(* IEC 61131-3 sources: PLC_FIFO_Optimization/build/OpenPLC Runtime v4/src, 1 file *)

(* ---- program.st ---- *)
FUNCTION_BLOCK Circular_queue
  VAR_INPUT
    XPush : BOOL;
    XPop : BOOL;
    iInputVal : INT;
  END_VAR
  VAR_OUTPUT
    iOutputVal : INT;
    iCount : INT;
    Operation_Cost : INT;
  END_VAR
  VAR
    Buffer : ARRAY [0..4999] OF INT;
    Head : INT;
    Tail : INT;
    MaxLen : INT;
    R_Trig_Push : R_TRIG;
    R_Trig_Pop : R_TRIG;
  END_VAR

  (* Edge Detection *)
  R_Trig_Push(CLK := xPush);
  R_Trig_Pop(CLK := xPop);

  (* initialize MaxLen if 0 (safety check) *)
  MaxLen := 5000;

  (* --- PUSH (Enqueue) --- *)
  IF R_Trig_Push.Q THEN
      (* Only push if not full (Optional safety, but good practice) *)
      IF iCount < MaxLen THEN
          Buffer[Head] := iInputVal;
          Head := Head + 1;
          IF Head >= MaxLen THEN Head := 0; END_IF;

          (* DIRECT COUNTING - The Fix *)
          iCount := iCount + 1;
      END_IF;
  END_IF;

  (* --- POP (Dequeue) --- *)
  IF R_Trig_Pop.Q AND iCount > 0 THEN
      iOutputVal := Buffer[Tail];
      Tail := Tail + 1;
      IF Tail >= MaxLen THEN Tail := 0; END_IF;

      (* DIRECT COUNTING - The Fix *)
      iCount := iCount - 1;
      Operation_Cost := 0;
  END_IF;
END_FUNCTION_BLOCK

FUNCTION_BLOCK FB_FIFO
  VAR_INPUT
    XPush : BOOL;
    XPop : BOOL;
    iInputVal : INT;
  END_VAR
  VAR_OUTPUT
    iOutputVal : INT;
    iCount : INT;
    Operation_Cost : INT;
  END_VAR
  VAR
    Buffer : ARRAY [0..4999] OF INT;
    i : INT;
    R_Trig_Push : R_TRIG;
    R_Trig_Pop : R_TRIG;
  END_VAR

  (* Edge Detection *)
  R_Trig_Push(CLK := xPush);
  R_Trig_Pop(CLK := xPop);

  (* --- PUSH (FFL) --- *)
  (* Simply add to the end. This part is actually fast (O(1)) *)
  IF R_Trig_Push.Q AND iCount < 5000 THEN
      Buffer[iCount] := iInputVal;
      iCount := iCount + 1;
  END_IF;

  (* --- POP (FFU) - THE EXPENSIVE PART --- *)
  (* This simulates the AB FFU shifting mechanism *)
  IF R_Trig_Pop.Q AND iCount > 0 THEN

      (* 1. Grab the value at Head (Index 0) *)
      iOutputVal := Buffer[0];

      (* 2. THE SHIFT LOOP (The "Bad" Part) *)
      (* We must physically move every item down one slot *)
      (* If you have 50 items, this loop runs 49 times! *)

      FOR i := 0 TO iCount - 2 DO
          Buffer[i] := Buffer[i+1]; (* Move data from i+1 to i *)

          (* Increment the "Cost" Counter to visualize the inefficiency *)
          Operation_Cost := Operation_Cost + 1;
      END_FOR;

      (* 3. Clear the last slot (optional, but clean) *)
      Buffer[iCount - 1] := 0;

      (* 4. Decrement Count *)
      iCount := iCount - 1;

  END_IF;
END_FUNCTION_BLOCK

PROGRAM main
  VAR
    My_Bad_FIFO : FB_FIFO;
    My_Good_FIFO : CIRCULAR_QUEUE;
    pb_Push : BOOL;
    pb_Pop : BOOL;
    Input_Data : INT;
    Auto_TImer : TON;
    Test_Step : INT := 0;
    Auto_Start : BOOL := FALSE;
    Fill_Queue_Now : BOOL := FALSE;
    i : INT := 0;
    Queue_Count_Good : INT := 0;
  END_VAR
  VAR
    Output_Bad AT %QW1 : INT;
    Output_Good AT %QW4 : INT;
    Test_value AT %QW5 : INT;
    Queue_Count AT %QW0 : INT;
    Shift_Counter AT %QW3 : INT;
    Shift_Counter_Good AT %QW2 : INT;
  END_VAR

  (* ============================================================= *)
  (* ZONE 1: THE STRESS TEST LOADER (Instant Fill) *)
  (* ============================================================= *)
  (* This logic only runs ONCE when you force 'Fill_Queue_Now' to TRUE. *)
  (* It pauses the scan cycle, stuffs 5,000 items into the queues, *)
  (* and then releases the PLC back to normal operation. *)

  IF Fill_Queue_Now THEN

      (* Loop from 1 to 5000 to fill the array completely *)
      FOR i := 1 TO 5000 DO

          (* 1. SIMULATE RISING EDGE (Push Button Press) *)
          (* We call the FBs directly here to force the data in *)
          My_Bad_FIFO(xPush := TRUE, xPop := FALSE, iInputVal := i);
          My_Good_FIFO(xPush := TRUE, xPop := FALSE, iInputVal := i);

          (* 2. SIMULATE FALLING EDGE (Push Button Release) *)
          (* We must call them again with FALSE to reset the trigger for the next loop iteration *)
          My_Bad_FIFO(xPush := FALSE, xPop := FALSE, iInputVal := i);
          My_Good_FIFO(xPush := FALSE, xPop := FALSE, iInputVal := i);

      END_FOR;

      (* Reset the trigger so it doesn't run forever *)
      Fill_Queue_Now := FALSE;

  END_IF;

  (* ============================================================= *)
  (* ZONE 2: NORMAL OPERATION (Manual Pop) *)
  (* ============================================================= *)
  (* This runs every single scan cycle. It listens to your manual *)
  (* 'pb_Pop' button so you can trigger the unloads when ready. *)

  (* Call the Bad FIFO (Linear Shift) *)
  My_Bad_FIFO(
      xPush := pb_Push,      (* Normal button control *)
      xPop := pb_Pop,        (* Normal button control *)
      iInputVal := Input_Data,
      iOutputVal => Output_Bad,
      iCount => Queue_Count,
      Operation_Cost => Shift_Counter
  );

  (* Call the Good FIFO (Circular Buffer) *)
  My_Good_FIFO(
      xPush := pb_Push,
      xPop := pb_Pop,
      iInputVal := Input_Data,
      iOutputVal => Output_Good,
      iCount => Queue_Count_Good,
      Operation_Cost => Shift_Counter_Good
  );
END_PROGRAM

CONFIGURATION Config0

  RESOURCE Res0 ON PLC
    TASK task0(INTERVAL := T#20ms,PRIORITY := 1);
    PROGRAM instance0 WITH task0 : main;
  END_RESOURCE
END_CONFIGURATION

(*DBG:char md5[] = "892a26d77c3caac8eb1d182cbc9cad2f";*)
(*DBG:/**)
(*DBG: * This file is part of OpenPLC Runtime*)
(*DBG: **)
(*DBG: * Copyright (C) 2023 Autonomy, GP Orcullo*)
(*DBG: * Based on the work by GP Orcullo on Beremiz for uC*)
(*DBG: **)
(*DBG: * This program is free software; you can redistribute it and/or*)
(*DBG: * modify it under the terms of the GNU General Public License*)
(*DBG: * as published by the Free Software Foundation; either version 2*)
(*DBG: * of the License, or (at your option) any later version.*)
(*DBG: **)
(*DBG: * This program is distributed in the hope that it will be useful,*)
(*DBG: * but WITHOUT ANY WARRANTY; without even the implied warranty of*)
(*DBG: * MERCHANTABILITY or FITNESS FOR A PARTICULAR PURPOSE.  See the*)
(*DBG: * GNU General Public License for more details.*)
(*DBG: **)
(*DBG: * You should have received a copy of the GNU General Public License*)
(*DBG: * along with this program; If not, see <http://www.gnu.org/licenses/>.*)
(*DBG: **)
(*DBG: */*)
(*DBG:*)
(*DBG:#include <stdbool.h>*)
(*DBG:*)
(*DBG:#include "iec_types_all.h"*)
(*DBG:#include "POUS.h"*)
(*DBG:*)
(*DBG:#define SAME_ENDIANNESS      0*)
(*DBG:#define REVERSE_ENDIANNESS   1*)
(*DBG:*)
(*DBG:char plc_program_md5[] = "892a26d77c3caac8eb1d182cbc9cad2f";*)
(*DBG:*)
(*DBG:uint8_t endianness;*)
(*DBG:*)
(*DBG:*)
(*DBG:extern MAIN RES0__INSTANCE0;*)
(*DBG:*)
(*DBG:static const struct {*)
(*DBG:    void *ptr;*)
(*DBG:    __IEC_types_enum type;*)
(*DBG:} debug_vars[] = {*)
(*DBG:    {&(RES0__INSTANCE0.MY_BAD_FIFO.EN), BOOL_ENUM},*)
(*DBG:    {&(RES0__INSTANCE0.MY_BAD_FIFO.ENO), BOOL_ENUM},*)
(*DBG:    {&(RES0__INSTANCE0.MY_BAD_FIFO.XPUSH), BOOL_ENUM},*)
(*DBG:    {&(RES0__INSTANCE0.MY_BAD_FIFO.XPOP), BOOL_ENUM},*)
(*DBG:    {&(RES0__INSTANCE0.MY_BAD_FIFO.IINPUTVAL), INT_ENUM},*)
(*DBG:    {&(RES0__INSTANCE0.MY_BAD_FIFO.IOUTPUTVAL), INT_ENUM},*)
(*DBG:    {&(RES0__INSTANCE0.MY_BAD_FIFO.ICOUNT), INT_ENUM},*)
(*DBG:    {&(RES0__INSTANCE0.MY_BAD_FIFO.OPERATION_COST), INT_ENUM},*)
(*DBG:    {&(RES0__INSTANCE0.MY_BAD_FIFO.BUFFER.value.table[0]), INT_ENUM},*)
(*DBG:    {&(RES0__INSTANCE0.MY_BAD_FIFO.BUFFER.value.table[1]), INT_ENUM},*)
(*DBG:    {&(RES0__INSTANCE0.MY_BAD_FIFO.BUFFER.value.table[2]), INT_ENUM},*)
(*DBG:    {&(RES0__INSTANCE0.MY_BAD_FIFO.BUFFER.value.table[3]), INT_ENUM},*)
(*DBG:    {&(RES0__INSTANCE0.MY_BAD_FIFO.BUFFER.value.table[4]), INT_ENUM},*)
(*DBG:    {&(RES0__INSTANCE0.MY_BAD_FIFO.BUFFER.value.table[5]), INT_ENUM},*)
(*DBG:    {&(RES0__INSTANCE0.MY_BAD_FIFO.BUFFER.value.table[6]), INT_ENUM},*)
(*DBG:    {&(RES0__INSTANCE0.MY_BAD_FIFO.BUFFER.value.table[7]), INT_ENUM},*)
(*DBG:    {&(RES0__INSTANCE0.MY_BAD_FIFO.BUFFER.value.table[8]), INT_ENUM},*)
(*DBG:    {&(RES0__INSTANCE0.MY_BAD_FIFO.BUFFER.value.table[9]), INT_ENUM},*)
(*DBG:    {&(RES0__INSTANCE0.MY_BAD_FIFO.BUFFER.value.table[10]), INT_ENUM},*)
(*DBG:    {&(RES0__INSTANCE0.MY_BAD_FIFO.BUFFER.value.table[11]), INT_ENUM},*)
(*DBG:    {&(RES0__INSTANCE0.MY_BAD_FIFO.BUFFER.value.table[12]), INT_ENUM},*)
(*DBG:    {&(RES0__INSTANCE0.MY_BAD_FIFO.BUFFER.value.table[13]), INT_ENUM},*)
(*DBG:    {&(RES0__INSTANCE0.MY_BAD_FIFO.BUFFER.value.table[14]), INT_ENUM},*)
(*DBG:    {&(RES0__INSTANCE0.MY_BAD_FIFO.BUFFER.value.table[15]), INT_ENUM},*)
(*DBG:    {&(RES0__INSTANCE0.MY_BAD_FIFO.BUFFER.value.table[16]), INT_ENUM},*)
(*DBG:    {&(RES0__INSTANCE0.MY_BAD_FIFO.BUFFER.value.table[17]), INT_ENUM},*)
(*DBG:    {&(RES0__INSTANCE0.MY_BAD_FIFO.BUFFER.value.table[18]), INT_ENUM},*)
(*DBG:    {&(RES0__INSTANCE0.MY_BAD_FIFO.BUFFER.value.table[19]), INT_ENUM},*)
(*DBG:    {&(RES0__INSTANCE0.MY_BAD_FIFO.BUFFER.value.table[20]), INT_ENUM},*)
(*DBG:    {&(RES0__INSTANCE0.MY_BAD_FIFO.BUFFER.value.table[21]), INT_ENUM},*)
(*DBG:    {&(RES0__INSTANCE0.MY_BAD_FIFO.BUFFER.value.table[22]), INT_ENUM},*)
(*DBG:    {&(RES0__INSTANCE0.MY_BAD_FIFO.BUFFER.value.table[23]), INT_ENUM},*)
(*DBG:    {&(RES0__INSTANCE0.MY_BAD_FIFO.BUFFER.value.table[24]), INT_ENUM},*)
(*DBG:    {&(RES0__INSTANCE0.MY_BAD_FIFO.BUFFER.value.table[25]), INT_ENUM},*)
(*DBG:    {&(RES0__INSTANCE0.MY_BAD_FIFO.BUFFER.value.table[26]), INT_ENUM},*)
(*DBG:    {&(RES0__INSTANCE0.MY_BAD_FIFO.BUFFER.value.table[27]), INT_ENUM},*)
(*DBG:    {&(RES0__INSTANCE0.MY_BAD_FIFO.BUFFER.value.table[28]), INT_ENUM},*)
(*DBG:    {&(RES0__INSTANCE0.MY_BAD_FIFO.BUFFER.value.table[29]), INT_ENUM},*)
(*DBG:    {&(RES0__INSTANCE0.MY_BAD_FIFO.BUFFER.value.table[30]), INT_ENUM},*)
(*DBG:    {&(RES0__INSTANCE0.MY_BAD_FIFO.BUFFER.value.table[31]), INT_ENUM},*)
(*DBG:    {&(RES0__INSTANCE0.MY_BAD_FIFO.BUFFER.value.table[32]), INT_ENUM},*)
(*DBG:    {&(RES0__INSTANCE0.MY_BAD_FIFO.BUFFER.value.table[33]), INT_ENUM},*)
(*DBG:    {&(RES0__INSTANCE0.MY_BAD_FIFO.BUFFER.value.table[34]), INT_ENUM},*)
(*DBG:    {&(RES0__INSTANCE0.MY_BAD_FIFO.BUFFER.value.table[35]), INT_ENUM},*)
(*DBG:    {&(RES0__INSTANCE0.MY_BAD_FIFO.BUFFER.value.table[36]), INT_ENUM},*)
(*DBG:    {&(RES0__INSTANCE0.MY_BAD_FIFO.BUFFER.value.table[37]), INT_ENUM},*)
(*DBG:    {&(RES0__INSTANCE0.MY_BAD_FIFO.BUFFER.value.table[38]), INT_ENUM},*)
(*DBG:    {&(RES0__INSTANCE0.MY_BAD_FIFO.BUFFER.value.table[39]), INT_ENUM},*)
(*DBG:    {&(RES0__INSTANCE0.MY_BAD_FIFO.BUFFER.value.table[40]), INT_ENUM},*)
(*DBG:    {&(RES0__INSTANCE0.MY_BAD_FIFO.BUFFER.value.table[41]), INT_ENUM},*)
(*DBG:    {&(RES0__INSTANCE0.MY_BAD_FIFO.BUFFER.value.table[42]), INT_ENUM},*)
(*DBG:    {&(RES0__INSTANCE0.MY_BAD_FIFO.BUFFER.value.table[43]), INT_ENUM},*)
(*DBG:    {&(RES0__INSTANCE0.MY_BAD_FIFO.BUFFER.value.table[44]), INT_ENUM},*)
(*DBG:    {&(RES0__INSTANCE0.MY_BAD_FIFO.BUFFER.value.table[45]), INT_ENUM},*)
(*DBG:    {&(RES0__INSTANCE0.MY_BAD_FIFO.BUFFER.value.table[46]), INT_ENUM},*)
(*DBG:    {&(RES0__INSTANCE0.MY_BAD_FIFO.BUFFER.value.table[47]), INT_ENUM},*)
(*DBG:    {&(RES0__INSTANCE0.MY_BAD_FIFO.BUFFER.value.table[48]), INT_ENUM},*)
(*DBG:    {&(RES0__INSTANCE0.MY_BAD_FIFO.BUFFER.value.table[49]), INT_ENUM},*)
(*DBG:    {&(RES0__INSTANCE0.MY_BAD_FIFO.BUFFER.value.table[50]), INT_ENUM},*)
(*DBG:    {&(RES0__INSTANCE0.MY_BAD_FIFO.BUFFER.value.table[51]), INT_ENUM},*)
(*DBG:    {&(RES0__INSTANCE0.MY_BAD_FIFO.BUFFER.value.table[52]), INT_ENUM},*)
(*DBG:    {&(RES0__INSTANCE0.MY_BAD_FIFO.BUFFER.value.table[53]), INT_ENUM},*)
(*DBG:    {&(RES0__INSTANCE0.MY_BAD_FIFO.BUFFER.value.table[54]), INT_ENUM},*)
(*DBG:    {&(RES0__INSTANCE0.MY_BAD_FIFO.BUFFER.value.table[55]), INT_ENUM},*)
(*DBG:    {&(RES0__INSTANCE0.MY_BAD_FIFO.BUFFER.value.table[56]), INT_ENUM},*)
(*DBG:    {&(RES0__INSTANCE0.MY_BAD_FIFO.BUFFER.value.table[57]), INT_ENUM},*)
(*DBG:    {&(RES0__INSTANCE0.MY_BAD_FIFO.BUFFER.value.table[58]), INT_ENUM},*)
(*DBG:    {&(RES0__INSTANCE0.MY_BAD_FIFO.BUFFER.value.table[59]), INT_ENUM},*)
(*DBG:    {&(RES0__INSTANCE0.MY_BAD_FIFO.BUFFER.value.table[60]), INT_ENUM},*)
(*DBG:    {&(RES0__INSTANCE0.MY_BAD_FIFO.BUFFER.value.table[61]), INT_ENUM},*)
(*DBG:    {&(RES0__INSTANCE0.MY_BAD_FIFO.BUFFER.value.table[62]), INT_ENUM},*)
(*DBG:    {&(RES0__INSTANCE0.MY_BAD_FIFO.BUFFER.value.table[63]), INT_ENUM},*)
(*DBG:    {&(RES0__INSTANCE0.MY_BAD_FIFO.BUFFER.value.table[64]), INT_ENUM},*)
(*DBG:    {&(RES0__INSTANCE0.MY_BAD_FIFO.BUFFER.value.table[65]), INT_ENUM},*)
(*DBG:    {&(RES0__INSTANCE0.MY_BAD_FIFO.BUFFER.value.table[66]), INT_ENUM},*)
(*DBG:    {&(RES0__INSTANCE0.MY_BAD_FIFO.BUFFER.value.table[67]), INT_ENUM},*)
(*DBG:    {&(RES0__INSTANCE0.MY_BAD_FIFO.BUFFER.value.table[68]), INT_ENUM},*)
(*DBG:    {&(RES0__INSTANCE0.MY_BAD_FIFO.BUFFER.value.table[69]), INT_ENUM},*)
(*DBG:    {&(RES0__INSTANCE0.MY_BAD_FIFO.BUFFER.value.table[70]), INT_ENUM},*)
(*DBG:    {&(RES0__INSTANCE0.MY_BAD_FIFO.BUFFER.value.table[71]), INT_ENUM},*)
(*DBG:    {&(RES0__INSTANCE0.MY_BAD_FIFO.BUFFER.value.table[72]), INT_ENUM},*)
(*DBG:    {&(RES0__INSTANCE0.MY_BAD_FIFO.BUFFER.value.table[73]), INT_ENUM},*)
(*DBG:    {&(RES0__INSTANCE0.MY_BAD_FIFO.BUFFER.value.table[74]), INT_ENUM},*)
(*DBG:    {&(RES0__INSTANCE0.MY_BAD_FIFO.BUFFER.value.table[75]), INT_ENUM},*)
(*DBG:    {&(RES0__INSTANCE0.MY_BAD_FIFO.BUFFER.value.table[76]), INT_ENUM},*)
(*DBG:    {&(RES0__INSTANCE0.MY_BAD_FIFO.BUFFER.value.table[77]), INT_ENUM},*)
(*DBG:    {&(RES0__INSTANCE0.MY_BAD_FIFO.BUFFER.value.table[78]), INT_ENUM},*)
(*DBG:    {&(RES0__INSTANCE0.MY_BAD_FIFO.BUFFER.value.table[79]), INT_ENUM},*)
(*DBG:    {&(RES0__INSTANCE0.MY_BAD_FIFO.BUFFER.value.table[80]), INT_ENUM},*)
(*DBG:    {&(RES0__INSTANCE0.MY_BAD_FIFO.BUFFER.value.table[81]), INT_ENUM},*)
(*DBG:    {&(RES0__INSTANCE0.MY_BAD_FIFO.BUFFER.value.table[82]), INT_ENUM},*)
(*DBG:    {&(RES0__INSTANCE0.MY_BAD_FIFO.BUFFER.value.table[83]), INT_ENUM},*)
(*DBG:    {&(RES0__INSTANCE0.MY_BAD_FIFO.BUFFER.value.table[84]), INT_ENUM},*)
(*DBG:    {&(RES0__INSTANCE0.MY_BAD_FIFO.BUFFER.value.table[85]), INT_ENUM},*)
(*DBG:    {&(RES0__INSTANCE0.MY_BAD_FIFO.BUFFER.value.table[86]), INT_ENUM},*)
(*DBG:    {&(RES0__INSTANCE0.MY_BAD_FIFO.BUFFER.value.table[87]), INT_ENUM},*)
(*DBG:    {&(RES0__INSTANCE0.MY_BAD_FIFO.BUFFER.value.table[88]), INT_ENUM},*)
(*DBG:    {&(RES0__INSTANCE0.MY_BAD_FIFO.BUFFER.value.table[89]), INT_ENUM},*)
(*DBG:    {&(RES0__INSTANCE0.MY_BAD_FIFO.BUFFER.value.table[90]), INT_ENUM},*)
(*DBG:    {&(RES0__INSTANCE0.MY_BAD_FIFO.BUFFER.value.table[91]), INT_ENUM},*)
(*DBG:    {&(RES0__INSTANCE0.MY_BAD_FIFO.BUFFER.value.table[92]), INT_ENUM},*)
(*DBG:    {&(RES0__INSTANCE0.MY_BAD_FIFO.BUFFER.value.table[93]), INT_ENUM},*)
(*DBG:    {&(RES0__INSTANCE0.MY_BAD_FIFO.BUFFER.value.table[94]), INT_ENUM},*)
(*DBG:    {&(RES0__INSTANCE0.MY_BAD_FIFO.BUFFER.value.table[95]), INT_ENUM},*)
(*DBG:    {&(RES0__INSTANCE0.MY_BAD_FIFO.BUFFER.value.table[96]), INT_ENUM},*)
(*DBG:    {&(RES0__INSTANCE0.MY_BAD_FIFO.BUFFER.value.table[97]), INT_ENUM},*)
(*DBG:    {&(RES0__INSTANCE0.MY_BAD_FIFO.BUFFER.value.table[98]), INT_ENUM},*)
(*DBG:    {&(RES0__INSTANCE0.MY_BAD_FIFO.BUFFER.value.table[99]), INT_ENUM},*)
(*DBG:    {&(RES0__INSTANCE0.MY_BAD_FIFO.BUFFER.value.table[100]), INT_ENUM},*)
(*DBG:    {&(RES0__INSTANCE0.MY_BAD_FIFO.BUFFER.value.table[101]), INT_ENUM},*)
(*DBG:    {&(RES0__INSTANCE0.MY_BAD_FIFO.BUFFER.value.table[102]), INT_ENUM},*)
(*DBG:    {&(RES0__INSTANCE0.MY_BAD_FIFO.BUFFER.value.table[103]), INT_ENUM},*)
(*DBG:    {&(RES0__INSTANCE0.MY_BAD_FIFO.BUFFER.value.table[104]), INT_ENUM},*)
(*DBG:    {&(RES0__INSTANCE0.MY_BAD_FIFO.BUFFER.value.table[105]), INT_ENUM},*)
(*DBG:    {&(RES0__INSTANCE0.MY_BAD_FIFO.BUFFER.value.table[106]), INT_ENUM},*)
(*DBG:    {&(RES0__INSTANCE0.MY_BAD_FIFO.BUFFER.value.table[107]), INT_ENUM},*)
(*DBG:    {&(RES0__INSTANCE0.MY_BAD_FIFO.BUFFER.value.table[108]), INT_ENUM},*)
(*DBG:    {&(RES0__INSTANCE0.MY_BAD_FIFO.BUFFER.value.table[109]), INT_ENUM},*)
(*DBG:    {&(RES0__INSTANCE0.MY_BAD_FIFO.BUFFER.value.table[110]), INT_ENUM},*)
(*DBG:    {&(RES0__INSTANCE0.MY_BAD_FIFO.BUFFER.value.table[111]), INT_ENUM},*)
(*DBG:    {&(RES0__INSTANCE0.MY_BAD_FIFO.BUFFER.value.table[112]), INT_ENUM},*)
(*DBG:    {&(RES0__INSTANCE0.MY_BAD_FIFO.BUFFER.value.table[113]), INT_ENUM},*)
(*DBG:    {&(RES0__INSTANCE0.MY_BAD_FIFO.BUFFER.value.table[114]), INT_ENUM},*)
(*DBG:    {&(RES0__INSTANCE0.MY_BAD_FIFO.BUFFER.value.table[115]), INT_ENUM},*)
(*DBG:    {&(RES0__INSTANCE0.MY_BAD_FIFO.BUFFER.value.table[116]), INT_ENUM},*)
(*DBG:    {&(RES0__INSTANCE0.MY_BAD_FIFO.BUFFER.value.table[117]), INT_ENUM},*)
(*DBG:    {&(RES0__INSTANCE0.MY_BAD_FIFO.BUFFER.value.table[118]), INT_ENUM},*)
(*DBG:    {&(RES0__INSTANCE0.MY_BAD_FIFO.BUFFER.value.table[119]), INT_ENUM},*)
(*DBG:    {&(RES0__INSTANCE0.MY_BAD_FIFO.BUFFER.value.table[120]), INT_ENUM},*)
(*DBG:    {&(RES0__INSTANCE0.MY_BAD_FIFO.BUFFER.value.table[121]), INT_ENUM},*)
(*DBG:    {&(RES0__INSTANCE0.MY_BAD_FIFO.BUFFER.value.table[122]), INT_ENUM},*)
(*DBG:    {&(RES0__INSTANCE0.MY_BAD_FIFO.BUFFER.value.table[123]), INT_ENUM},*)
(*DBG:    {&(RES0__INSTANCE0.MY_BAD_FIFO.BUFFER.value.table[124]), INT_ENUM},*)
(*DBG:    {&(RES0__INSTANCE0.MY_BAD_FIFO.BUFFER.value.table[125]), INT_ENUM},*)
(*DBG:    {&(RES0__INSTANCE0.MY_BAD_FIFO.BUFFER.value.table[126]), INT_ENUM},*)
(*DBG:    {&(RES0__INSTANCE0.MY_BAD_FIFO.BUFFER.value.table[127]), INT_ENUM},*)
(*DBG:    {&(RES0__INSTANCE0.MY_BAD_FIFO.BUFFER.value.table[128]), INT_ENUM},*)
(*DBG:    {&(RES0__INSTANCE0.MY_BAD_FIFO.BUFFER.value.table[129]), INT_ENUM},*)
(*DBG:    {&(RES0__INSTANCE0.MY_BAD_FIFO.BUFFER.value.table[130]), INT_ENUM},*)
(*DBG:    {&(RES0__INSTANCE0.MY_BAD_FIFO.BUFFER.value.table[131]), INT_ENUM},*)
(*DBG:    {&(RES0__INSTANCE0.MY_BAD_FIFO.BUFFER.value.table[132]), INT_ENUM},*)
(*DBG:    {&(RES0__INSTANCE0.MY_BAD_FIFO.BUFFER.value.table[133]), INT_ENUM},*)
(*DBG:    {&(RES0__INSTANCE0.MY_BAD_FIFO.BUFFER.value.table[134]), INT_ENUM},*)
(*DBG:    {&(RES0__INSTANCE0.MY_BAD_FIFO.BUFFER.value.table[135]), INT_ENUM},*)
(*DBG:    {&(RES0__INSTANCE0.MY_BAD_FIFO.BUFFER.value.table[136]), INT_ENUM},*)
(*DBG:    {&(RES0__INSTANCE0.MY_BAD_FIFO.BUFFER.value.table[137]), INT_ENUM},*)
(*DBG:    {&(RES0__INSTANCE0.MY_BAD_FIFO.BUFFER.value.table[138]), INT_ENUM},*)
(*DBG:    {&(RES0__INSTANCE0.MY_BAD_FIFO.BUFFER.value.table[139]), INT_ENUM},*)
(*DBG:    {&(RES0__INSTANCE0.MY_BAD_FIFO.BUFFER.value.table[140]), INT_ENUM},*)
(*DBG:    {&(RES0__INSTANCE0.MY_BAD_FIFO.BUFFER.value.table[141]), INT_ENUM},*)
(*DBG:    {&(RES0__INSTANCE0.MY_BAD_FIFO.BUFFER.value.table[142]), INT_ENUM},*)
(*DBG:    {&(RES0__INSTANCE0.MY_BAD_FIFO.BUFFER.value.table[143]), INT_ENUM},*)
(*DBG:    {&(RES0__INSTANCE0.MY_BAD_FIFO.BUFFER.value.table[144]), INT_ENUM},*)
(*DBG:    {&(RES0__INSTANCE0.MY_BAD_FIFO.BUFFER.value.table[145]), INT_ENUM},*)
(*DBG:    {&(RES0__INSTANCE0.MY_BAD_FIFO.BUFFER.value.table[146]), INT_ENUM},*)
(*DBG:    {&(RES0__INSTANCE0.MY_BAD_FIFO.BUFFER.value.table[147]), INT_ENUM},*)
(*DBG:    {&(RES0__INSTANCE0.MY_BAD_FIFO.BUFFER.value.table[148]), INT_ENUM},*)
(*DBG:    {&(RES0__INSTANCE0.MY_BAD_FIFO.BUFFER.value.table[149]), INT_ENUM},*)
(*DBG:    {&(RES0__INSTANCE0.MY_BAD_FIFO.BUFFER.value.table[150]), INT_ENUM},*)
(*DBG:    {&(RES0__INSTANCE0.MY_BAD_FIFO.BUFFER.value.table[151]), INT_ENUM},*)
(*DBG:    {&(RES0__INSTANCE0.MY_BAD_FIFO.BUFFER.value.table[152]), INT_ENUM},*)
(*DBG:    {&(RES0__INSTANCE0.MY_BAD_FIFO.BUFFER.value.table[153]), INT_ENUM},*)
(*DBG:    {&(RES0__INSTANCE0.MY_BAD_FIFO.BUFFER.value.table[154]), INT_ENUM},*)
(*DBG:    {&(RES0__INSTANCE0.MY_BAD_FIFO.BUFFER.value.table[155]), INT_ENUM},*)
(*DBG:    {&(RES0__INSTANCE0.MY_BAD_FIFO.BUFFER.value.table[156]), INT_ENUM},*)
(*DBG:    {&(RES0__INSTANCE0.MY_BAD_FIFO.BUFFER.value.table[157]), INT_ENUM},*)
(*DBG:    {&(RES0__INSTANCE0.MY_BAD_FIFO.BUFFER.value.table[158]), INT_ENUM},*)
(*DBG:    {&(RES0__INSTANCE0.MY_BAD_FIFO.BUFFER.value.table[159]), INT_ENUM},*)
(*DBG:    {&(RES0__INSTANCE0.MY_BAD_FIFO.BUFFER.value.table[160]), INT_ENUM},*)
(*DBG:    {&(RES0__INSTANCE0.MY_BAD_FIFO.BUFFER.value.table[161]), INT_ENUM},*)
(*DBG:    {&(RES0__INSTANCE0.MY_BAD_FIFO.BUFFER.value.table[162]), INT_ENUM},*)
(*DBG:    {&(RES0__INSTANCE0.MY_BAD_FIFO.BUFFER.value.table[163]), INT_ENUM},*)
(*DBG:    {&(RES0__INSTANCE0.MY_BAD_FIFO.BUFFER.value.table[164]), INT_ENUM},*)
(*DBG:    {&(RES0__INSTANCE0.MY_BAD_FIFO.BUFFER.value.table[165]), INT_ENUM},*)
(*DBG:    {&(RES0__INSTANCE0.MY_BAD_FIFO.BUFFER.value.table[166]), INT_ENUM},*)
(*DBG:    {&(RES0__INSTANCE0.MY_BAD_FIFO.BUFFER.value.table[167]), INT_ENUM},*)
(*DBG:    {&(RES0__INSTANCE0.MY_BAD_FIFO.BUFFER.value.table[168]), INT_ENUM},*)
(*DBG:    {&(RES0__INSTANCE0.MY_BAD_FIFO.BUFFER.value.table[169]), INT_ENUM},*)
(*DBG:    {&(RES0__INSTANCE0.MY_BAD_FIFO.BUFFER.value.table[170]), INT_ENUM},*)
(*DBG:    {&(RES0__INSTANCE0.MY_BAD_FIFO.BUFFER.value.table[171]), INT_ENUM},*)
(*DBG:    {&(RES0__INSTANCE0.MY_BAD_FIFO.BUFFER.value.table[172]), INT_ENUM},*)
(*DBG:    {&(RES0__INSTANCE0.MY_BAD_FIFO.BUFFER.value.table[173]), INT_ENUM},*)
(*DBG:    {&(RES0__INSTANCE0.MY_BAD_FIFO.BUFFER.value.table[174]), INT_ENUM},*)
(*DBG:    {&(RES0__INSTANCE0.MY_BAD_FIFO.BUFFER.value.table[175]), INT_ENUM},*)
(*DBG:    {&(RES0__INSTANCE0.MY_BAD_FIFO.BUFFER.value.table[176]), INT_ENUM},*)
(*DBG:    {&(RES0__INSTANCE0.MY_BAD_FIFO.BUFFER.value.table[177]), INT_ENUM},*)
(*DBG:    {&(RES0__INSTANCE0.MY_BAD_FIFO.BUFFER.value.table[178]), INT_ENUM},*)
(*DBG:    {&(RES0__INSTANCE0.MY_BAD_FIFO.BUFFER.value.table[179]), INT_ENUM},*)
(*DBG:    {&(RES0__INSTANCE0.MY_BAD_FIFO.BUFFER.value.table[180]), INT_ENUM},*)
(*DBG:    {&(RES0__INSTANCE0.MY_BAD_FIFO.BUFFER.value.table[181]), INT_ENUM},*)
(*DBG:    {&(RES0__INSTANCE0.MY_BAD_FIFO.BUFFER.value.table[182]), INT_ENUM},*)
(*DBG:    {&(RES0__INSTANCE0.MY_BAD_FIFO.BUFFER.value.table[183]), INT_ENUM},*)
(*DBG:    {&(RES0__INSTANCE0.MY_BAD_FIFO.BUFFER.value.table[184]), INT_ENUM},*)
(*DBG:    {&(RES0__INSTANCE0.MY_BAD_FIFO.BUFFER.value.table[185]), INT_ENUM},*)
(*DBG:    {&(RES0__INSTANCE0.MY_BAD_FIFO.BUFFER.value.table[186]), INT_ENUM},*)
(*DBG:    {&(RES0__INSTANCE0.MY_BAD_FIFO.BUFFER.value.table[187]), INT_ENUM},*)
(*DBG:    {&(RES0__INSTANCE0.MY_BAD_FIFO.BUFFER.value.table[188]), INT_ENUM},*)
(*DBG:    {&(RES0__INSTANCE0.MY_BAD_FIFO.BUFFER.value.table[189]), INT_ENUM},*)
(*DBG:    {&(RES0__INSTANCE0.MY_BAD_FIFO.BUFFER.value.table[190]), INT_ENUM},*)
(*DBG:    {&(RES0__INSTANCE0.MY_BAD_FIFO.BUFFER.value.table[191]), INT_ENUM},*)
(*DBG:    {&(RES0__INSTANCE0.MY_BAD_FIFO.BUFFER.value.table[192]), INT_ENUM},*)
(*DBG:    {&(RES0__INSTANCE0.MY_BAD_FIFO.BUFFER.value.table[193]), INT_ENUM},*)
(*DBG:    {&(RES0__INSTANCE0.MY_BAD_FIFO.BUFFER.value.table[194]), INT_ENUM},*)
(*DBG:    {&(RES0__INSTANCE0.MY_BAD_FIFO.BUFFER.value.table[195]), INT_ENUM},*)
(*DBG:    {&(RES0__INSTANCE0.MY_BAD_FIFO.BUFFER.value.table[196]), INT_ENUM},*)
(*DBG:    {&(RES0__INSTANCE0.MY_BAD_FIFO.BUFFER.value.table[197]), INT_ENUM},*)
(*DBG:    {&(RES0__INSTANCE0.MY_BAD_FIFO.BUFFER.value.table[198]), INT_ENUM},*)
(*DBG:    {&(RES0__INSTANCE0.MY_BAD_FIFO.BUFFER.value.table[199]), INT_ENUM},*)
(*DBG:    {&(RES0__INSTANCE0.MY_BAD_FIFO.BUFFER.value.table[200]), INT_ENUM},*)
(*DBG:    {&(RES0__INSTANCE0.MY_BAD_FIFO.BUFFER.value.table[201]), INT_ENUM},*)
(*DBG:    {&(RES0__INSTANCE0.MY_BAD_FIFO.BUFFER.value.table[202]), INT_ENUM},*)
(*DBG:    {&(RES0__INSTANCE0.MY_BAD_FIFO.BUFFER.value.table[203]), INT_ENUM},*)
(*DBG:    {&(RES0__INSTANCE0.MY_BAD_FIFO.BUFFER.value.table[204]), INT_ENUM},*)
(*DBG:    {&(RES0__INSTANCE0.MY_BAD_FIFO.BUFFER.value.table[205]), INT_ENUM},*)
(*DBG:    {&(RES0__INSTANCE0.MY_BAD_FIFO.BUFFER.value.table[206]), INT_ENUM},*)
(*DBG:    {&(RES0__INSTANCE0.MY_BAD_FIFO.BUFFER.value.table[207]), INT_ENUM},*)
(*DBG:    {&(RES0__INSTANCE0.MY_BAD_FIFO.BUFFER.value.table[208]), INT_ENUM},*)
(*DBG:    {&(RES0__INSTANCE0.MY_BAD_FIFO.BUFFER.value.table[209]), INT_ENUM},*)
(*DBG:    {&(RES0__INSTANCE0.MY_BAD_FIFO.BUFFER.value.table[210]), INT_ENUM},*)
(*DBG:    {&(RES0__INSTANCE0.MY_BAD_FIFO.BUFFER.value.table[211]), INT_ENUM},*)
(*DBG:    {&(RES0__INSTANCE0.MY_BAD_FIFO.BUFFER.value.table[212]), INT_ENUM},*)
(*DBG:    {&(RES0__INSTANCE0.MY_BAD_FIFO.BUFFER.value.table[213]), INT_ENUM},*)
(*DBG:    {&(RES0__INSTANCE0.MY_BAD_FIFO.BUFFER.value.table[214]), INT_ENUM},*)
(*DBG:    {&(RES0__INSTANCE0.MY_BAD_FIFO.BUFFER.value.table[215]), INT_ENUM},*)
(*DBG:    {&(RES0__INSTANCE0.MY_BAD_FIFO.BUFFER.value.table[216]), INT_ENUM},*)
(*DBG:    {&(RES0__INSTANCE0.MY_BAD_FIFO.BUFFER.value.table[217]), INT_ENUM},*)
(*DBG:    {&(RES0__INSTANCE0.MY_BAD_FIFO.BUFFER.value.table[218]), INT_ENUM},*)
(*DBG:    {&(RES0__INSTANCE0.MY_BAD_FIFO.BUFFER.value.table[219]), INT_ENUM},*)
(*DBG:    {&(RES0__INSTANCE0.MY_BAD_FIFO.BUFFER.value.table[220]), INT_ENUM},*)
(*DBG:    {&(RES0__INSTANCE0.MY_BAD_FIFO.BUFFER.value.table[221]), INT_ENUM},*)
(*DBG:    {&(RES0__INSTANCE0.MY_BAD_FIFO.BUFFER.value.table[222]), INT_ENUM},*)
(*DBG:    {&(RES0__INSTANCE0.MY_BAD_FIFO.BUFFER.value.table[223]), INT_ENUM},*)
(*DBG:    {&(RES0__INSTANCE0.MY_BAD_FIFO.BUFFER.value.table[224]), INT_ENUM},*)
(*DBG:    {&(RES0__INSTANCE0.MY_BAD_FIFO.BUFFER.value.table[225]), INT_ENUM},*)
(*DBG:    {&(RES0__INSTANCE0.MY_BAD_FIFO.BUFFER.value.table[226]), INT_ENUM},*)
(*DBG:    {&(RES0__INSTANCE0.MY_BAD_FIFO.BUFFER.value.table[227]), INT_ENUM},*)
(*DBG:    {&(RES0__INSTANCE0.MY_BAD_FIFO.BUFFER.value.table[228]), INT_ENUM},*)
(*DBG:    {&(RES0__INSTANCE0.MY_BAD_FIFO.BUFFER.value.table[229]), INT_ENUM},*)
(*DBG:    {&(RES0__INSTANCE0.MY_BAD_FIFO.BUFFER.value.table[230]), INT_ENUM},*)
(*DBG:    {&(RES0__INSTANCE0.MY_BAD_FIFO.BUFFER.value.table[231]), INT_ENUM},*)
(*DBG:    {&(RES0__INSTANCE0.MY_BAD_FIFO.BUFFER.value.table[232]), INT_ENUM},*)
(*DBG:    {&(RES0__INSTANCE0.MY_BAD_FIFO.BUFFER.value.table[233]), INT_ENUM},*)
(*DBG:    {&(RES0__INSTANCE0.MY_BAD_FIFO.BUFFER.value.table[234]), INT_ENUM},*)
(*DBG:    {&(RES0__INSTANCE0.MY_BAD_FIFO.BUFFER.value.table[235]), INT_ENUM},*)
(*DBG:    {&(RES0__INSTANCE0.MY_BAD_FIFO.BUFFER.value.table[236]), INT_ENUM},*)
(*DBG:    {&(RES0__INSTANCE0.MY_BAD_FIFO.BUFFER.value.table[237]), INT_ENUM},*)
(*DBG:    {&(RES0__INSTANCE0.MY_BAD_FIFO.BUFFER.value.table[238]), INT_ENUM},*)
(*DBG:    {&(RES0__INSTANCE0.MY_BAD_FIFO.BUFFER.value.table[239]), INT_ENUM},*)
(*DBG:    {&(RES0__INSTANCE0.MY_BAD_FIFO.BUFFER.value.table[240]), INT_ENUM},*)
(*DBG:    {&(RES0__INSTANCE0.MY_BAD_FIFO.BUFFER.value.table[241]), INT_ENUM},*)
(*DBG:    {&(RES0__INSTANCE0.MY_BAD_FIFO.BUFFER.value.table[242]), INT_ENUM},*)
(*DBG:    {&(RES0__INSTANCE0.MY_BAD_FIFO.BUFFER.value.table[243]), INT_ENUM},*)
(*DBG:    {&(RES0__INSTANCE0.MY_BAD_FIFO.BUFFER.value.table[244]), INT_ENUM},*)
(*DBG:    {&(RES0__INSTANCE0.MY_BAD_FIFO.BUFFER.value.table[245]), INT_ENUM},*)
(*DBG:    {&(RES0__INSTANCE0.MY_BAD_FIFO.BUFFER.value.table[246]), INT_ENUM},*)
(*DBG:    {&(RES0__INSTANCE0.MY_BAD_FIFO.BUFFER.value.table[247]), INT_ENUM},*)
(*DBG:    {&(RES0__INSTANCE0.MY_BAD_FIFO.BUFFER.value.table[248]), INT_ENUM},*)
(*DBG:    {&(RES0__INSTANCE0.MY_BAD_FIFO.BUFFER.value.table[249]), INT_ENUM},*)
(*DBG:    {&(RES0__INSTANCE0.MY_BAD_FIFO.BUFFER.value.table[250]), INT_ENUM},*)
(*DBG:    {&(RES0__INSTANCE0.MY_BAD_FIFO.BUFFER.value.table[251]), INT_ENUM},*)
(*DBG:    {&(RES0__INSTANCE0.MY_BAD_FIFO.BUFFER.value.table[252]), INT_ENUM},*)
(*DBG:    {&(RES0__INSTANCE0.MY_BAD_FIFO.BUFFER.value.table[253]), INT_ENUM},*)
(*DBG:    {&(RES0__INSTANCE0.MY_BAD_FIFO.BUFFER.value.table[254]), INT_ENUM},*)
(*DBG:    {&(RES0__INSTANCE0.MY_BAD_FIFO.BUFFER.value.table[255]), INT_ENUM},*)
(*DBG:    {&(RES0__INSTANCE0.MY_BAD_FIFO.BUFFER.value.table[256]), INT_ENUM},*)
(*DBG:    {&(RES0__INSTANCE0.MY_BAD_FIFO.BUFFER.value.table[257]), INT_ENUM},*)
(*DBG:    {&(RES0__INSTANCE0.MY_BAD_FIFO.BUFFER.value.table[258]), INT_ENUM},*)
(*DBG:    {&(RES0__INSTANCE0.MY_BAD_FIFO.BUFFER.value.table[259]), INT_ENUM},*)
(*DBG:    {&(RES0__INSTANCE0.MY_BAD_FIFO.BUFFER.value.table[260]), INT_ENUM},*)
(*DBG:    {&(RES0__INSTANCE0.MY_BAD_FIFO.BUFFER.value.table[261]), INT_ENUM},*)
(*DBG:    {&(RES0__INSTANCE0.MY_BAD_FIFO.BUFFER.value.table[262]), INT_ENUM},*)
(*DBG:    {&(RES0__INSTANCE0.MY_BAD_FIFO.BUFFER.value.table[263]), INT_ENUM},*)
(*DBG:    {&(RES0__INSTANCE0.MY_BAD_FIFO.BUFFER.value.table[264]), INT_ENUM},*)
(*DBG:    {&(RES0__INSTANCE0.MY_BAD_FIFO.BUFFER.value.table[265]), INT_ENUM},*)
(*DBG:    {&(RES0__INSTANCE0.MY_BAD_FIFO.BUFFER.value.table[266]), INT_ENUM},*)
(*DBG:    {&(RES0__INSTANCE0.MY_BAD_FIFO.BUFFER.value.table[267]), INT_ENUM},*)
(*DBG:    {&(RES0__INSTANCE0.MY_BAD_FIFO.BUFFER.value.table[268]), INT_ENUM},*)
(*DBG:    {&(RES0__INSTANCE0.MY_BAD_FIFO.BUFFER.value.table[269]), INT_ENUM},*)
(*DBG:    {&(RES0__INSTANCE0.MY_BAD_FIFO.BUFFER.value.table[270]), INT_ENUM},*)
(*DBG:    {&(RES0__INSTANCE0.MY_BAD_FIFO.BUFFER.value.table[271]), INT_ENUM},*)
(*DBG:    {&(RES0__INSTANCE0.MY_BAD_FIFO.BUFFER.value.table[272]), INT_ENUM},*)
(*DBG:    {&(RES0__INSTANCE0.MY_BAD_FIFO.BUFFER.value.table[273]), INT_ENUM},*)
(*DBG:    {&(RES0__INSTANCE0.MY_BAD_FIFO.BUFFER.value.table[274]), INT_ENUM},*)
(*DBG:    {&(RES0__INSTANCE0.MY_BAD_FIFO.BUFFER.value.table[275]), INT_ENUM},*)
(*DBG:    {&(RES0__INSTANCE0.MY_BAD_FIFO.BUFFER.value.table[276]), INT_ENUM},*)
(*DBG:    {&(RES0__INSTANCE0.MY_BAD_FIFO.BUFFER.value.table[277]), INT_ENUM},*)
(*DBG:    {&(RES0__INSTANCE0.MY_BAD_FIFO.BUFFER.value.table[278]), INT_ENUM},*)
(*DBG:    {&(RES0__INSTANCE0.MY_BAD_FIFO.BUFFER.value.table[279]), INT_ENUM},*)
(*DBG:    {&(RES0__INSTANCE0.MY_BAD_FIFO.BUFFER.value.table[280]), INT_ENUM},*)
(*DBG:    {&(RES0__INSTANCE0.MY_BAD_FIFO.BUFFER.value.table[281]), INT_ENUM},*)
(*DBG:    {&(RES0__INSTANCE0.MY_BAD_FIFO.BUFFER.value.table[282]), INT_ENUM},*)
(*DBG:    {&(RES0__INSTANCE0.MY_BAD_FIFO.BUFFER.value.table[283]), INT_ENUM},*)
(*DBG:    {&(RES0__INSTANCE0.MY_BAD_FIFO.BUFFER.value.table[284]), INT_ENUM},*)
(*DBG:    {&(RES0__INSTANCE0.MY_BAD_FIFO.BUFFER.value.table[285]), INT_ENUM},*)
(*DBG:    {&(RES0__INSTANCE0.MY_BAD_FIFO.BUFFER.value.table[286]), INT_ENUM},*)
(*DBG:    {&(RES0__INSTANCE0.MY_BAD_FIFO.BUFFER.value.table[287]), INT_ENUM},*)
(*DBG:    {&(RES0__INSTANCE0.MY_BAD_FIFO.BUFFER.value.table[288]), INT_ENUM},*)
(*DBG:    {&(RES0__INSTANCE0.MY_BAD_FIFO.BUFFER.value.table[289]), INT_ENUM},*)
(*DBG:    {&(RES0__INSTANCE0.MY_BAD_FIFO.BUFFER.value.table[290]), INT_ENUM},*)
(*DBG:    {&(RES0__INSTANCE0.MY_BAD_FIFO.BUFFER.value.table[291]), INT_ENUM},*)
(*DBG:    {&(RES0__INSTANCE0.MY_BAD_FIFO.BUFFER.value.table[292]), INT_ENUM},*)
(*DBG:    {&(RES0__INSTANCE0.MY_BAD_FIFO.BUFFER.value.table[293]), INT_ENUM},*)
(*DBG:    {&(RES0__INSTANCE0.MY_BAD_FIFO.BUFFER.value.table[294]), INT_ENUM},*)
(*DBG:    {&(RES0__INSTANCE0.MY_BAD_FIFO.BUFFER.value.table[295]), INT_ENUM},*)
(*DBG:    {&(RES0__INSTANCE0.MY_BAD_FIFO.BUFFER.value.table[296]), INT_ENUM},*)
(*DBG:    {&(RES0__INSTANCE0.MY_BAD_FIFO.BUFFER.value.table[297]), INT_ENUM},*)
(*DBG:    {&(RES0__INSTANCE0.MY_BAD_FIFO.BUFFER.value.table[298]), INT_ENUM},*)
(*DBG:    {&(RES0__INSTANCE0.MY_BAD_FIFO.BUFFER.value.table[299]), INT_ENUM},*)
(*DBG:    {&(RES0__INSTANCE0.MY_BAD_FIFO.BUFFER.value.table[300]), INT_ENUM},*)
(*DBG:    {&(RES0__INSTANCE0.MY_BAD_FIFO.BUFFER.value.table[301]), INT_ENUM},*)
(*DBG:    {&(RES0__INSTANCE0.MY_BAD_FIFO.BUFFER.value.table[302]), INT_ENUM},*)
(*DBG:    {&(RES0__INSTANCE0.MY_BAD_FIFO.BUFFER.value.table[303]), INT_ENUM},*)
(*DBG:    {&(RES0__INSTANCE0.MY_BAD_FIFO.BUFFER.value.table[304]), INT_ENUM},*)
(*DBG:    {&(RES0__INSTANCE0.MY_BAD_FIFO.BUFFER.value.table[305]), INT_ENUM},*)
(*DBG:    {&(RES0__INSTANCE0.MY_BAD_FIFO.BUFFER.value.table[306]), INT_ENUM},*)
(*DBG:    {&(RES0__INSTANCE0.MY_BAD_FIFO.BUFFER.value.table[307]), INT_ENUM},*)
(*DBG:    {&(RES0__INSTANCE0.MY_BAD_FIFO.BUFFER.value.table[308]), INT_ENUM},*)
(*DBG:    {&(RES0__INSTANCE0.MY_BAD_FIFO.BUFFER.value.table[309]), INT_ENUM},*)
(*DBG:    {&(RES0__INSTANCE0.MY_BAD_FIFO.BUFFER.value.table[310]), INT_ENUM},*)
(*DBG:    {&(RES0__INSTANCE0.MY_BAD_FIFO.BUFFER.value.table[311]), INT_ENUM},*)
(*DBG:    {&(RES0__INSTANCE0.MY_BAD_FIFO.BUFFER.value.table[312]), INT_ENUM},*)
(*DBG:    {&(RES0__INSTANCE0.MY_BAD_FIFO.BUFFER.value.table[313]), INT_ENUM},*)
(*DBG:    {&(RES0__INSTANCE0.MY_BAD_FIFO.BUFFER.value.table[314]), INT_ENUM},*)
(*DBG:    {&(RES0__INSTANCE0.MY_BAD_FIFO.BUFFER.value.table[315]), INT_ENUM},*)
(*DBG:    {&(RES0__INSTANCE0.MY_BAD_FIFO.BUFFER.value.table[316]), INT_ENUM},*)
(*DBG:    {&(RES0__INSTANCE0.MY_BAD_FIFO.BUFFER.value.table[317]), INT_ENUM},*)
(*DBG:    {&(RES0__INSTANCE0.MY_BAD_FIFO.BUFFER.value.table[318]), INT_ENUM},*)
(*DBG:    {&(RES0__INSTANCE0.MY_BAD_FIFO.BUFFER.value.table[319]), INT_ENUM},*)
(*DBG:    {&(RES0__INSTANCE0.MY_BAD_FIFO.BUFFER.value.table[320]), INT_ENUM},*)
(*DBG:    {&(RES0__INSTANCE0.MY_BAD_FIFO.BUFFER.value.table[321]), INT_ENUM},*)
(*DBG:    {&(RES0__INSTANCE0.MY_BAD_FIFO.BUFFER.value.table[322]), INT_ENUM},*)
(*DBG:    {&(RES0__INSTANCE0.MY_BAD_FIFO.BUFFER.value.table[323]), INT_ENUM},*)
(*DBG:    {&(RES0__INSTANCE0.MY_BAD_FIFO.BUFFER.value.table[324]), INT_ENUM},*)
(*DBG:    {&(RES0__INSTANCE0.MY_BAD_FIFO.BUFFER.value.table[325]), INT_ENUM},*)
(*DBG:    {&(RES0__INSTANCE0.MY_BAD_FIFO.BUFFER.value.table[326]), INT_ENUM},*)
(*DBG:    {&(RES0__INSTANCE0.MY_BAD_FIFO.BUFFER.value.table[327]), INT_ENUM},*)
(*DBG:    {&(RES0__INSTANCE0.MY_BAD_FIFO.BUFFER.value.table[328]), INT_ENUM},*)
(*DBG:    {&(RES0__INSTANCE0.MY_BAD_FIFO.BUFFER.value.table[329]), INT_ENUM},*)
(*DBG:    {&(RES0__INSTANCE0.MY_BAD_FIFO.BUFFER.value.table[330]), INT_ENUM},*)
(*DBG:    {&(RES0__INSTANCE0.MY_BAD_FIFO.BUFFER.value.table[331]), INT_ENUM},*)
(*DBG:    {&(RES0__INSTANCE0.MY_BAD_FIFO.BUFFER.value.table[332]), INT_ENUM},*)
(*DBG:    {&(RES0__INSTANCE0.MY_BAD_FIFO.BUFFER.value.table[333]), INT_ENUM},*)
(*DBG:    {&(RES0__INSTANCE0.MY_BAD_FIFO.BUFFER.value.table[334]), INT_ENUM},*)
(*DBG:    {&(RES0__INSTANCE0.MY_BAD_FIFO.BUFFER.value.table[335]), INT_ENUM},*)
(*DBG:    {&(RES0__INSTANCE0.MY_BAD_FIFO.BUFFER.value.table[336]), INT_ENUM},*)
(*DBG:    {&(RES0__INSTANCE0.MY_BAD_FIFO.BUFFER.value.table[337]), INT_ENUM},*)
(*DBG:    {&(RES0__INSTANCE0.MY_BAD_FIFO.BUFFER.value.table[338]), INT_ENUM},*)
(*DBG:    {&(RES0__INSTANCE0.MY_BAD_FIFO.BUFFER.value.table[339]), INT_ENUM},*)
(*DBG:    {&(RES0__INSTANCE0.MY_BAD_FIFO.BUFFER.value.table[340]), INT_ENUM},*)
(*DBG:    {&(RES0__INSTANCE0.MY_BAD_FIFO.BUFFER.value.table[341]), INT_ENUM},*)
(*DBG:    {&(RES0__INSTANCE0.MY_BAD_FIFO.BUFFER.value.table[342]), INT_ENUM},*)
(*DBG:    {&(RES0__INSTANCE0.MY_BAD_FIFO.BUFFER.value.table[343]), INT_ENUM},*)
(*DBG:    {&(RES0__INSTANCE0.MY_BAD_FIFO.BUFFER.value.table[344]), INT_ENUM},*)
(*DBG:    {&(RES0__INSTANCE0.MY_BAD_FIFO.BUFFER.value.table[345]), INT_ENUM},*)
(*DBG:    {&(RES0__INSTANCE0.MY_BAD_FIFO.BUFFER.value.table[346]), INT_ENUM},*)
(*DBG:    {&(RES0__INSTANCE0.MY_BAD_FIFO.BUFFER.value.table[347]), INT_ENUM},*)
(*DBG:    {&(RES0__INSTANCE0.MY_BAD_FIFO.BUFFER.value.table[348]), INT_ENUM},*)
(*DBG:    {&(RES0__INSTANCE0.MY_BAD_FIFO.BUFFER.value.table[349]), INT_ENUM},*)
(*DBG:    {&(RES0__INSTANCE0.MY_BAD_FIFO.BUFFER.value.table[350]), INT_ENUM},*)
(*DBG:    {&(RES0__INSTANCE0.MY_BAD_FIFO.BUFFER.value.table[351]), INT_ENUM},*)
(*DBG:    {&(RES0__INSTANCE0.MY_BAD_FIFO.BUFFER.value.table[352]), INT_ENUM},*)
(*DBG:    {&(RES0__INSTANCE0.MY_BAD_FIFO.BUFFER.value.table[353]), INT_ENUM},*)
(*DBG:    {&(RES0__INSTANCE0.MY_BAD_FIFO.BUFFER.value.table[354]), INT_ENUM},*)
(*DBG:    {&(RES0__INSTANCE0.MY_BAD_FIFO.BUFFER.value.table[355]), INT_ENUM},*)
(*DBG:    {&(RES0__INSTANCE0.MY_BAD_FIFO.BUFFER.value.table[356]), INT_ENUM},*)
(*DBG:    {&(RES0__INSTANCE0.MY_BAD_FIFO.BUFFER.value.table[357]), INT_ENUM},*)
(*DBG:    {&(RES0__INSTANCE0.MY_BAD_FIFO.BUFFER.value.table[358]), INT_ENUM},*)
(*DBG:    {&(RES0__INSTANCE0.MY_BAD_FIFO.BUFFER.value.table[359]), INT_ENUM},*)
(*DBG:    {&(RES0__INSTANCE0.MY_BAD_FIFO.BUFFER.value.table[360]), INT_ENUM},*)
(*DBG:    {&(RES0__INSTANCE0.MY_BAD_FIFO.BUFFER.value.table[361]), INT_ENUM},*)
(*DBG:    {&(RES0__INSTANCE0.MY_BAD_FIFO.BUFFER.value.table[362]), INT_ENUM},*)
(*DBG:    {&(RES0__INSTANCE0.MY_BAD_FIFO.BUFFER.value.table[363]), INT_ENUM},*)
(*DBG:    {&(RES0__INSTANCE0.MY_BAD_FIFO.BUFFER.value.table[364]), INT_ENUM},*)
(*DBG:    {&(RES0__INSTANCE0.MY_BAD_FIFO.BUFFER.value.table[365]), INT_ENUM},*)
(*DBG:    {&(RES0__INSTANCE0.MY_BAD_FIFO.BUFFER.value.table[366]), INT_ENUM},*)
(*DBG:    {&(RES0__INSTANCE0.MY_BAD_FIFO.BUFFER.value.table[367]), INT_ENUM},*)
(*DBG:    {&(RES0__INSTANCE0.MY_BAD_FIFO.BUFFER.value.table[368]), INT_ENUM},*)
(*DBG:    {&(RES0__INSTANCE0.MY_BAD_FIFO.BUFFER.value.table[369]), INT_ENUM},*)
(*DBG:    {&(RES0__INSTANCE0.MY_BAD_FIFO.BUFFER.value.table[370]), INT_ENUM},*)
(*DBG:    {&(RES0__INSTANCE0.MY_BAD_FIFO.BUFFER.value.table[371]), INT_ENUM},*)
(*DBG:    {&(RES0__INSTANCE0.MY_BAD_FIFO.BUFFER.value.table[372]), INT_ENUM},*)
(*DBG:    {&(RES0__INSTANCE0.MY_BAD_FIFO.BUFFER.value.table[373]), INT_ENUM},*)
(*DBG:    {&(RES0__INSTANCE0.MY_BAD_FIFO.BUFFER.value.table[374]), INT_ENUM},*)
(*DBG:    {&(RES0__INSTANCE0.MY_BAD_FIFO.BUFFER.value.table[375]), INT_ENUM},*)
(*DBG:    {&(RES0__INSTANCE0.MY_BAD_FIFO.BUFFER.value.table[376]), INT_ENUM},*)
(*DBG:    {&(RES0__INSTANCE0.MY_BAD_FIFO.BUFFER.value.table[377]), INT_ENUM},*)
(*DBG:    {&(RES0__INSTANCE0.MY_BAD_FIFO.BUFFER.value.table[378]), INT_ENUM},*)
(*DBG:    {&(RES0__INSTANCE0.MY_BAD_FIFO.BUFFER.value.table[379]), INT_ENUM},*)
(*DBG:    {&(RES0__INSTANCE0.MY_BAD_FIFO.BUFFER.value.table[380]), INT_ENUM},*)
(*DBG:    {&(RES0__INSTANCE0.MY_BAD_FIFO.BUFFER.value.table[381]), INT_ENUM},*)
(*DBG:    {&(RES0__INSTANCE0.MY_BAD_FIFO.BUFFER.value.table[382]), INT_ENUM},*)
(*DBG:    {&(RES0__INSTANCE0.MY_BAD_FIFO.BUFFER.value.table[383]), INT_ENUM},*)
(*DBG:    {&(RES0__INSTANCE0.MY_BAD_FIFO.BUFFER.value.table[384]), INT_ENUM},*)
(*DBG:    {&(RES0__INSTANCE0.MY_BAD_FIFO.BUFFER.value.table[385]), INT_ENUM},*)
(*DBG:    {&(RES0__INSTANCE0.MY_BAD_FIFO.BUFFER.value.table[386]), INT_ENUM},*)
(*DBG:    {&(RES0__INSTANCE0.MY_BAD_FIFO.BUFFER.value.table[387]), INT_ENUM},*)
(*DBG:    {&(RES0__INSTANCE0.MY_BAD_FIFO.BUFFER.value.table[388]), INT_ENUM},*)
(*DBG:    {&(RES0__INSTANCE0.MY_BAD_FIFO.BUFFER.value.table[389]), INT_ENUM},*)
(*DBG:    {&(RES0__INSTANCE0.MY_BAD_FIFO.BUFFER.value.table[390]), INT_ENUM},*)
(*DBG:    {&(RES0__INSTANCE0.MY_BAD_FIFO.BUFFER.value.table[391]), INT_ENUM},*)
(*DBG:    {&(RES0__INSTANCE0.MY_BAD_FIFO.BUFFER.value.table[392]), INT_ENUM},*)
(*DBG:    {&(RES0__INSTANCE0.MY_BAD_FIFO.BUFFER.value.table[393]), INT_ENUM},*)
(*DBG:    {&(RES0__INSTANCE0.MY_BAD_FIFO.BUFFER.value.table[394]), INT_ENUM},*)
(*DBG:    {&(RES0__INSTANCE0.MY_BAD_FIFO.BUFFER.value.table[395]), INT_ENUM},*)
(*DBG:    {&(RES0__INSTANCE0.MY_BAD_FIFO.BUFFER.value.table[396]), INT_ENUM},*)
(*DBG:    {&(RES0__INSTANCE0.MY_BAD_FIFO.BUFFER.value.table[397]), INT_ENUM},*)
(*DBG:    {&(RES0__INSTANCE0.MY_BAD_FIFO.BUFFER.value.table[398]), INT_ENUM},*)
(*DBG:    {&(RES0__INSTANCE0.MY_BAD_FIFO.BUFFER.value.table[399]), INT_ENUM},*)
(*DBG:    {&(RES0__INSTANCE0.MY_BAD_FIFO.BUFFER.value.table[400]), INT_ENUM},*)
(*DBG:    {&(RES0__INSTANCE0.MY_BAD_FIFO.BUFFER.value.table[401]), INT_ENUM},*)
(*DBG:    {&(RES0__INSTANCE0.MY_BAD_FIFO.BUFFER.value.table[402]), INT_ENUM},*)
(*DBG:    {&(RES0__INSTANCE0.MY_BAD_FIFO.BUFFER.value.table[403]), INT_ENUM},*)
(*DBG:    {&(RES0__INSTANCE0.MY_BAD_FIFO.BUFFER.value.table[404]), INT_ENUM},*)
(*DBG:    {&(RES0__INSTANCE0.MY_BAD_FIFO.BUFFER.value.table[405]), INT_ENUM},*)
(*DBG:    {&(RES0__INSTANCE0.MY_BAD_FIFO.BUFFER.value.table[406]), INT_ENUM},*)
(*DBG:    {&(RES0__INSTANCE0.MY_BAD_FIFO.BUFFER.value.table[407]), INT_ENUM},*)
(*DBG:    {&(RES0__INSTANCE0.MY_BAD_FIFO.BUFFER.value.table[408]), INT_ENUM},*)
(*DBG:    {&(RES0__INSTANCE0.MY_BAD_FIFO.BUFFER.value.table[409]), INT_ENUM},*)
(*DBG:    {&(RES0__INSTANCE0.MY_BAD_FIFO.BUFFER.value.table[410]), INT_ENUM},*)
(*DBG:    {&(RES0__INSTANCE0.MY_BAD_FIFO.BUFFER.value.table[411]), INT_ENUM},*)
(*DBG:    {&(RES0__INSTANCE0.MY_BAD_FIFO.BUFFER.value.table[412]), INT_ENUM},*)
(*DBG:    {&(RES0__INSTANCE0.MY_BAD_FIFO.BUFFER.value.table[413]), INT_ENUM},*)
(*DBG:    {&(RES0__INSTANCE0.MY_BAD_FIFO.BUFFER.value.table[414]), INT_ENUM},*)
(*DBG:    {&(RES0__INSTANCE0.MY_BAD_FIFO.BUFFER.value.table[415]), INT_ENUM},*)
(*DBG:    {&(RES0__INSTANCE0.MY_BAD_FIFO.BUFFER.value.table[416]), INT_ENUM},*)
(*DBG:    {&(RES0__INSTANCE0.MY_BAD_FIFO.BUFFER.value.table[417]), INT_ENUM},*)
(*DBG:    {&(RES0__INSTANCE0.MY_BAD_FIFO.BUFFER.value.table[418]), INT_ENUM},*)
(*DBG:    {&(RES0__INSTANCE0.MY_BAD_FIFO.BUFFER.value.table[419]), INT_ENUM},*)
(*DBG:    {&(RES0__INSTANCE0.MY_BAD_FIFO.BUFFER.value.table[420]), INT_ENUM},*)
(*DBG:    {&(RES0__INSTANCE0.MY_BAD_FIFO.BUFFER.value.table[421]), INT_ENUM},*)
(*DBG:    {&(RES0__INSTANCE0.MY_BAD_FIFO.BUFFER.value.table[422]), INT_ENUM},*)
(*DBG:    {&(RES0__INSTANCE0.MY_BAD_FIFO.BUFFER.value.table[423]), INT_ENUM},*)
(*DBG:    {&(RES0__INSTANCE0.MY_BAD_FIFO.BUFFER.value.table[424]), INT_ENUM},*)
(*DBG:    {&(RES0__INSTANCE0.MY_BAD_FIFO.BUFFER.value.table[425]), INT_ENUM},*)
(*DBG:    {&(RES0__INSTANCE0.MY_BAD_FIFO.BUFFER.value.table[426]), INT_ENUM},*)
(*DBG:    {&(RES0__INSTANCE0.MY_BAD_FIFO.BUFFER.value.table[427]), INT_ENUM},*)
(*DBG:    {&(RES0__INSTANCE0.MY_BAD_FIFO.BUFFER.value.table[428]), INT_ENUM},*)
(*DBG:    {&(RES0__INSTANCE0.MY_BAD_FIFO.BUFFER.value.table[429]), INT_ENUM},*)
(*DBG:    {&(RES0__INSTANCE0.MY_BAD_FIFO.BUFFER.value.table[430]), INT_ENUM},*)
(*DBG:    {&(RES0__INSTANCE0.MY_BAD_FIFO.BUFFER.value.table[431]), INT_ENUM},*)
(*DBG:    {&(RES0__INSTANCE0.MY_BAD_FIFO.BUFFER.value.table[432]), INT_ENUM},*)
(*DBG:    {&(RES0__INSTANCE0.MY_BAD_FIFO.BUFFER.value.table[433]), INT_ENUM},*)
(*DBG:    {&(RES0__INSTANCE0.MY_BAD_FIFO.BUFFER.value.table[434]), INT_ENUM},*)
(*DBG:    {&(RES0__INSTANCE0.MY_BAD_FIFO.BUFFER.value.table[435]), INT_ENUM},*)
(*DBG:    {&(RES0__INSTANCE0.MY_BAD_FIFO.BUFFER.value.table[436]), INT_ENUM},*)
(*DBG:    {&(RES0__INSTANCE0.MY_BAD_FIFO.BUFFER.value.table[437]), INT_ENUM},*)
(*DBG:    {&(RES0__INSTANCE0.MY_BAD_FIFO.BUFFER.value.table[438]), INT_ENUM},*)
(*DBG:    {&(RES0__INSTANCE0.MY_BAD_FIFO.BUFFER.value.table[439]), INT_ENUM},*)
(*DBG:    {&(RES0__INSTANCE0.MY_BAD_FIFO.BUFFER.value.table[440]), INT_ENUM},*)
(*DBG:    {&(RES0__INSTANCE0.MY_BAD_FIFO.BUFFER.value.table[441]), INT_ENUM},*)
(*DBG:    {&(RES0__INSTANCE0.MY_BAD_FIFO.BUFFER.value.table[442]), INT_ENUM},*)
(*DBG:    {&(RES0__INSTANCE0.MY_BAD_FIFO.BUFFER.value.table[443]), INT_ENUM},*)
(*DBG:    {&(RES0__INSTANCE0.MY_BAD_FIFO.BUFFER.value.table[444]), INT_ENUM},*)
(*DBG:    {&(RES0__INSTANCE0.MY_BAD_FIFO.BUFFER.value.table[445]), INT_ENUM},*)
(*DBG:    {&(RES0__INSTANCE0.MY_BAD_FIFO.BUFFER.value.table[446]), INT_ENUM},*)
(*DBG:    {&(RES0__INSTANCE0.MY_BAD_FIFO.BUFFER.value.table[447]), INT_ENUM},*)
(*DBG:    {&(RES0__INSTANCE0.MY_BAD_FIFO.BUFFER.value.table[448]), INT_ENUM},*)
(*DBG:    {&(RES0__INSTANCE0.MY_BAD_FIFO.BUFFER.value.table[449]), INT_ENUM},*)
(*DBG:    {&(RES0__INSTANCE0.MY_BAD_FIFO.BUFFER.value.table[450]), INT_ENUM},*)
(*DBG:    {&(RES0__INSTANCE0.MY_BAD_FIFO.BUFFER.value.table[451]), INT_ENUM},*)
(*DBG:    {&(RES0__INSTANCE0.MY_BAD_FIFO.BUFFER.value.table[452]), INT_ENUM},*)
(*DBG:    {&(RES0__INSTANCE0.MY_BAD_FIFO.BUFFER.value.table[453]), INT_ENUM},*)
(*DBG:    {&(RES0__INSTANCE0.MY_BAD_FIFO.BUFFER.value.table[454]), INT_ENUM},*)
(*DBG:    {&(RES0__INSTANCE0.MY_BAD_FIFO.BUFFER.value.table[455]), INT_ENUM},*)
(*DBG:    {&(RES0__INSTANCE0.MY_BAD_FIFO.BUFFER.value.table[456]), INT_ENUM},*)
(*DBG:    {&(RES0__INSTANCE0.MY_BAD_FIFO.BUFFER.value.table[457]), INT_ENUM},*)
(*DBG:    {&(RES0__INSTANCE0.MY_BAD_FIFO.BUFFER.value.table[458]), INT_ENUM},*)
(*DBG:    {&(RES0__INSTANCE0.MY_BAD_FIFO.BUFFER.value.table[459]), INT_ENUM},*)
(*DBG:    {&(RES0__INSTANCE0.MY_BAD_FIFO.BUFFER.value.table[460]), INT_ENUM},*)
(*DBG:    {&(RES0__INSTANCE0.MY_BAD_FIFO.BUFFER.value.table[461]), INT_ENUM},*)
(*DBG:    {&(RES0__INSTANCE0.MY_BAD_FIFO.BUFFER.value.table[462]), INT_ENUM},*)
(*DBG:    {&(RES0__INSTANCE0.MY_BAD_FIFO.BUFFER.value.table[463]), INT_ENUM},*)
(*DBG:    {&(RES0__INSTANCE0.MY_BAD_FIFO.BUFFER.value.table[464]), INT_ENUM},*)
(*DBG:    {&(RES0__INSTANCE0.MY_BAD_FIFO.BUFFER.value.table[465]), INT_ENUM},*)
(*DBG:    {&(RES0__INSTANCE0.MY_BAD_FIFO.BUFFER.value.table[466]), INT_ENUM},*)
(*DBG:    {&(RES0__INSTANCE0.MY_BAD_FIFO.BUFFER.value.table[467]), INT_ENUM},*)
(*DBG:    {&(RES0__INSTANCE0.MY_BAD_FIFO.BUFFER.value.table[468]), INT_ENUM},*)
(*DBG:    {&(RES0__INSTANCE0.MY_BAD_FIFO.BUFFER.value.table[469]), INT_ENUM},*)
(*DBG:    {&(RES0__INSTANCE0.MY_BAD_FIFO.BUFFER.value.table[470]), INT_ENUM},*)
(*DBG:    {&(RES0__INSTANCE0.MY_BAD_FIFO.BUFFER.value.table[471]), INT_ENUM},*)
(*DBG:    {&(RES0__INSTANCE0.MY_BAD_FIFO.BUFFER.value.table[472]), INT_ENUM},*)
(*DBG:    {&(RES0__INSTANCE0.MY_BAD_FIFO.BUFFER.value.table[473]), INT_ENUM},*)
(*DBG:    {&(RES0__INSTANCE0.MY_BAD_FIFO.BUFFER.value.table[474]), INT_ENUM},*)
(*DBG:    {&(RES0__INSTANCE0.MY_BAD_FIFO.BUFFER.value.table[475]), INT_ENUM},*)
(*DBG:    {&(RES0__INSTANCE0.MY_BAD_FIFO.BUFFER.value.table[476]), INT_ENUM},*)
(*DBG:    {&(RES0__INSTANCE0.MY_BAD_FIFO.BUFFER.value.table[477]), INT_ENUM},*)
(*DBG:    {&(RES0__INSTANCE0.MY_BAD_FIFO.BUFFER.value.table[478]), INT_ENUM},*)
(*DBG:    {&(RES0__INSTANCE0.MY_BAD_FIFO.BUFFER.value.table[479]), INT_ENUM},*)
(*DBG:    {&(RES0__INSTANCE0.MY_BAD_FIFO.BUFFER.value.table[480]), INT_ENUM},*)
(*DBG:    {&(RES0__INSTANCE0.MY_BAD_FIFO.BUFFER.value.table[481]), INT_ENUM},*)
(*DBG:    {&(RES0__INSTANCE0.MY_BAD_FIFO.BUFFER.value.table[482]), INT_ENUM},*)
(*DBG:    {&(RES0__INSTANCE0.MY_BAD_FIFO.BUFFER.value.table[483]), INT_ENUM},*)
(*DBG:    {&(RES0__INSTANCE0.MY_BAD_FIFO.BUFFER.value.table[484]), INT_ENUM},*)
(*DBG:    {&(RES0__INSTANCE0.MY_BAD_FIFO.BUFFER.value.table[485]), INT_ENUM},*)
(*DBG:    {&(RES0__INSTANCE0.MY_BAD_FIFO.BUFFER.value.table[486]), INT_ENUM},*)
(*DBG:    {&(RES0__INSTANCE0.MY_BAD_FIFO.BUFFER.value.table[487]), INT_ENUM},*)
(*DBG:    {&(RES0__INSTANCE0.MY_BAD_FIFO.BUFFER.value.table[488]), INT_ENUM},*)
(*DBG:    {&(RES0__INSTANCE0.MY_BAD_FIFO.BUFFER.value.table[489]), INT_ENUM},*)
(*DBG:    {&(RES0__INSTANCE0.MY_BAD_FIFO.BUFFER.value.table[490]), INT_ENUM},*)
(*DBG:    {&(RES0__INSTANCE0.MY_BAD_FIFO.BUFFER.value.table[491]), INT_ENUM},*)
(*DBG:    {&(RES0__INSTANCE0.MY_BAD_FIFO.BUFFER.value.table[492]), INT_ENUM},*)
(*DBG:    {&(RES0__INSTANCE0.MY_BAD_FIFO.BUFFER.value.table[493]), INT_ENUM},*)
(*DBG:    {&(RES0__INSTANCE0.MY_BAD_FIFO.BUFFER.value.table[494]), INT_ENUM},*)
(*DBG:    {&(RES0__INSTANCE0.MY_BAD_FIFO.BUFFER.value.table[495]), INT_ENUM},*)
(*DBG:    {&(RES0__INSTANCE0.MY_BAD_FIFO.BUFFER.value.table[496]), INT_ENUM},*)
(*DBG:    {&(RES0__INSTANCE0.MY_BAD_FIFO.BUFFER.value.table[497]), INT_ENUM},*)
(*DBG:    {&(RES0__INSTANCE0.MY_BAD_FIFO.BUFFER.value.table[498]), INT_ENUM},*)
(*DBG:    {&(RES0__INSTANCE0.MY_BAD_FIFO.BUFFER.value.table[499]), INT_ENUM},*)
(*DBG:    {&(RES0__INSTANCE0.MY_BAD_FIFO.BUFFER.value.table[500]), INT_ENUM},*)
(*DBG:    {&(RES0__INSTANCE0.MY_BAD_FIFO.BUFFER.value.table[501]), INT_ENUM},*)
(*DBG:    {&(RES0__INSTANCE0.MY_BAD_FIFO.BUFFER.value.table[502]), INT_ENUM},*)
(*DBG:    {&(RES0__INSTANCE0.MY_BAD_FIFO.BUFFER.value.table[503]), INT_ENUM},*)
(*DBG:    {&(RES0__INSTANCE0.MY_BAD_FIFO.BUFFER.value.table[504]), INT_ENUM},*)
(*DBG:    {&(RES0__INSTANCE0.MY_BAD_FIFO.BUFFER.value.table[505]), INT_ENUM},*)
(*DBG:    {&(RES0__INSTANCE0.MY_BAD_FIFO.BUFFER.value.table[506]), INT_ENUM},*)
(*DBG:    {&(RES0__INSTANCE0.MY_BAD_FIFO.BUFFER.value.table[507]), INT_ENUM},*)
(*DBG:    {&(RES0__INSTANCE0.MY_BAD_FIFO.BUFFER.value.table[508]), INT_ENUM},*)
(*DBG:    {&(RES0__INSTANCE0.MY_BAD_FIFO.BUFFER.value.table[509]), INT_ENUM},*)
(*DBG:    {&(RES0__INSTANCE0.MY_BAD_FIFO.BUFFER.value.table[510]), INT_ENUM},*)
(*DBG:    {&(RES0__INSTANCE0.MY_BAD_FIFO.BUFFER.value.table[511]), INT_ENUM},*)
(*DBG:    {&(RES0__INSTANCE0.MY_BAD_FIFO.BUFFER.value.table[512]), INT_ENUM},*)
(*DBG:    {&(RES0__INSTANCE0.MY_BAD_FIFO.BUFFER.value.table[513]), INT_ENUM},*)
(*DBG:    {&(RES0__INSTANCE0.MY_BAD_FIFO.BUFFER.value.table[514]), INT_ENUM},*)
(*DBG:    {&(RES0__INSTANCE0.MY_BAD_FIFO.BUFFER.value.table[515]), INT_ENUM},*)
(*DBG:    {&(RES0__INSTANCE0.MY_BAD_FIFO.BUFFER.value.table[516]), INT_ENUM},*)
(*DBG:    {&(RES0__INSTANCE0.MY_BAD_FIFO.BUFFER.value.table[517]), INT_ENUM},*)
(*DBG:    {&(RES0__INSTANCE0.MY_BAD_FIFO.BUFFER.value.table[518]), INT_ENUM},*)
(*DBG:    {&(RES0__INSTANCE0.MY_BAD_FIFO.BUFFER.value.table[519]), INT_ENUM},*)
(*DBG:    {&(RES0__INSTANCE0.MY_BAD_FIFO.BUFFER.value.table[520]), INT_ENUM},*)
(*DBG:    {&(RES0__INSTANCE0.MY_BAD_FIFO.BUFFER.value.table[521]), INT_ENUM},*)
(*DBG:    {&(RES0__INSTANCE0.MY_BAD_FIFO.BUFFER.value.table[522]), INT_ENUM},*)
(*DBG:    {&(RES0__INSTANCE0.MY_BAD_FIFO.BUFFER.value.table[523]), INT_ENUM},*)
(*DBG:    {&(RES0__INSTANCE0.MY_BAD_FIFO.BUFFER.value.table[524]), INT_ENUM},*)
(*DBG:    {&(RES0__INSTANCE0.MY_BAD_FIFO.BUFFER.value.table[525]), INT_ENUM},*)
(*DBG:    {&(RES0__INSTANCE0.MY_BAD_FIFO.BUFFER.value.table[526]), INT_ENUM},*)
(*DBG:    {&(RES0__INSTANCE0.MY_BAD_FIFO.BUFFER.value.table[527]), INT_ENUM},*)
(*DBG:    {&(RES0__INSTANCE0.MY_BAD_FIFO.BUFFER.value.table[528]), INT_ENUM},*)
(*DBG:    {&(RES0__INSTANCE0.MY_BAD_FIFO.BUFFER.value.table[529]), INT_ENUM},*)
(*DBG:    {&(RES0__INSTANCE0.MY_BAD_FIFO.BUFFER.value.table[530]), INT_ENUM},*)
(*DBG:    {&(RES0__INSTANCE0.MY_BAD_FIFO.BUFFER.value.table[531]), INT_ENUM},*)
(*DBG:    {&(RES0__INSTANCE0.MY_BAD_FIFO.BUFFER.value.table[532]), INT_ENUM},*)
(*DBG:    {&(RES0__INSTANCE0.MY_BAD_FIFO.BUFFER.value.table[533]), INT_ENUM},*)
(*DBG:    {&(RES0__INSTANCE0.MY_BAD_FIFO.BUFFER.value.table[534]), INT_ENUM},*)
(*DBG:    {&(RES0__INSTANCE0.MY_BAD_FIFO.BUFFER.value.table[535]), INT_ENUM},*)
(*DBG:    {&(RES0__INSTANCE0.MY_BAD_FIFO.BUFFER.value.table[536]), INT_ENUM},*)
(*DBG:    {&(RES0__INSTANCE0.MY_BAD_FIFO.BUFFER.value.table[537]), INT_ENUM},*)
(*DBG:    {&(RES0__INSTANCE0.MY_BAD_FIFO.BUFFER.value.table[538]), INT_ENUM},*)
(*DBG:    {&(RES0__INSTANCE0.MY_BAD_FIFO.BUFFER.value.table[539]), INT_ENUM},*)
(*DBG:    {&(RES0__INSTANCE0.MY_BAD_FIFO.BUFFER.value.table[540]), INT_ENUM},*)
(*DBG:    {&(RES0__INSTANCE0.MY_BAD_FIFO.BUFFER.value.table[541]), INT_ENUM},*)
(*DBG:    {&(RES0__INSTANCE0.MY_BAD_FIFO.BUFFER.value.table[542]), INT_ENUM},*)
(*DBG:    {&(RES0__INSTANCE0.MY_BAD_FIFO.BUFFER.value.table[543]), INT_ENUM},*)
(*DBG:    {&(RES0__INSTANCE0.MY_BAD_FIFO.BUFFER.value.table[544]), INT_ENUM},*)
(*DBG:    {&(RES0__INSTANCE0.MY_BAD_FIFO.BUFFER.value.table[545]), INT_ENUM},*)
(*DBG:    {&(RES0__INSTANCE0.MY_BAD_FIFO.BUFFER.value.table[546]), INT_ENUM},*)
(*DBG:    {&(RES0__INSTANCE0.MY_BAD_FIFO.BUFFER.value.table[547]), INT_ENUM},*)
(*DBG:    {&(RES0__INSTANCE0.MY_BAD_FIFO.BUFFER.value.table[548]), INT_ENUM},*)
(*DBG:    {&(RES0__INSTANCE0.MY_BAD_FIFO.BUFFER.value.table[549]), INT_ENUM},*)
(*DBG:    {&(RES0__INSTANCE0.MY_BAD_FIFO.BUFFER.value.table[550]), INT_ENUM},*)
(*DBG:    {&(RES0__INSTANCE0.MY_BAD_FIFO.BUFFER.value.table[551]), INT_ENUM},*)
(*DBG:    {&(RES0__INSTANCE0.MY_BAD_FIFO.BUFFER.value.table[552]), INT_ENUM},*)
(*DBG:    {&(RES0__INSTANCE0.MY_BAD_FIFO.BUFFER.value.table[553]), INT_ENUM},*)
(*DBG:    {&(RES0__INSTANCE0.MY_BAD_FIFO.BUFFER.value.table[554]), INT_ENUM},*)
(*DBG:    {&(RES0__INSTANCE0.MY_BAD_FIFO.BUFFER.value.table[555]), INT_ENUM},*)
(*DBG:    {&(RES0__INSTANCE0.MY_BAD_FIFO.BUFFER.value.table[556]), INT_ENUM},*)
(*DBG:    {&(RES0__INSTANCE0.MY_BAD_FIFO.BUFFER.value.table[557]), INT_ENUM},*)
(*DBG:    {&(RES0__INSTANCE0.MY_BAD_FIFO.BUFFER.value.table[558]), INT_ENUM},*)
(*DBG:    {&(RES0__INSTANCE0.MY_BAD_FIFO.BUFFER.value.table[559]), INT_ENUM},*)
(*DBG:    {&(RES0__INSTANCE0.MY_BAD_FIFO.BUFFER.value.table[560]), INT_ENUM},*)
(*DBG:    {&(RES0__INSTANCE0.MY_BAD_FIFO.BUFFER.value.table[561]), INT_ENUM},*)
(*DBG:    {&(RES0__INSTANCE0.MY_BAD_FIFO.BUFFER.value.table[562]), INT_ENUM},*)
(*DBG:    {&(RES0__INSTANCE0.MY_BAD_FIFO.BUFFER.value.table[563]), INT_ENUM},*)
(*DBG:    {&(RES0__INSTANCE0.MY_BAD_FIFO.BUFFER.value.table[564]), INT_ENUM},*)
(*DBG:    {&(RES0__INSTANCE0.MY_BAD_FIFO.BUFFER.value.table[565]), INT_ENUM},*)
(*DBG:    {&(RES0__INSTANCE0.MY_BAD_FIFO.BUFFER.value.table[566]), INT_ENUM},*)
(*DBG:    {&(RES0__INSTANCE0.MY_BAD_FIFO.BUFFER.value.table[567]), INT_ENUM},*)
(*DBG:    {&(RES0__INSTANCE0.MY_BAD_FIFO.BUFFER.value.table[568]), INT_ENUM},*)
(*DBG:    {&(RES0__INSTANCE0.MY_BAD_FIFO.BUFFER.value.table[569]), INT_ENUM},*)
(*DBG:    {&(RES0__INSTANCE0.MY_BAD_FIFO.BUFFER.value.table[570]), INT_ENUM},*)
(*DBG:    {&(RES0__INSTANCE0.MY_BAD_FIFO.BUFFER.value.table[571]), INT_ENUM},*)
(*DBG:    {&(RES0__INSTANCE0.MY_BAD_FIFO.BUFFER.value.table[572]), INT_ENUM},*)
(*DBG:    {&(RES0__INSTANCE0.MY_BAD_FIFO.BUFFER.value.table[573]), INT_ENUM},*)
(*DBG:    {&(RES0__INSTANCE0.MY_BAD_FIFO.BUFFER.value.table[574]), INT_ENUM},*)
(*DBG:    {&(RES0__INSTANCE0.MY_BAD_FIFO.BUFFER.value.table[575]), INT_ENUM},*)
(*DBG:    {&(RES0__INSTANCE0.MY_BAD_FIFO.BUFFER.value.table[576]), INT_ENUM},*)
(*DBG:    {&(RES0__INSTANCE0.MY_BAD_FIFO.BUFFER.value.table[577]), INT_ENUM},*)
(*DBG:    {&(RES0__INSTANCE0.MY_BAD_FIFO.BUFFER.value.table[578]), INT_ENUM},*)
(*DBG:    {&(RES0__INSTANCE0.MY_BAD_FIFO.BUFFER.value.table[579]), INT_ENUM},*)
(*DBG:    {&(RES0__INSTANCE0.MY_BAD_FIFO.BUFFER.value.table[580]), INT_ENUM},*)
(*DBG:    {&(RES0__INSTANCE0.MY_BAD_FIFO.BUFFER.value.table[581]), INT_ENUM},*)
(*DBG:    {&(RES0__INSTANCE0.MY_BAD_FIFO.BUFFER.value.table[582]), INT_ENUM},*)
(*DBG:    {&(RES0__INSTANCE0.MY_BAD_FIFO.BUFFER.value.table[583]), INT_ENUM},*)
(*DBG:    {&(RES0__INSTANCE0.MY_BAD_FIFO.BUFFER.value.table[584]), INT_ENUM},*)
(*DBG:    {&(RES0__INSTANCE0.MY_BAD_FIFO.BUFFER.value.table[585]), INT_ENUM},*)
(*DBG:    {&(RES0__INSTANCE0.MY_BAD_FIFO.BUFFER.value.table[586]), INT_ENUM},*)
(*DBG:    {&(RES0__INSTANCE0.MY_BAD_FIFO.BUFFER.value.table[587]), INT_ENUM},*)
(*DBG:    {&(RES0__INSTANCE0.MY_BAD_FIFO.BUFFER.value.table[588]), INT_ENUM},*)
(*DBG:    {&(RES0__INSTANCE0.MY_BAD_FIFO.BUFFER.value.table[589]), INT_ENUM},*)
(*DBG:    {&(RES0__INSTANCE0.MY_BAD_FIFO.BUFFER.value.table[590]), INT_ENUM},*)
(*DBG:    {&(RES0__INSTANCE0.MY_BAD_FIFO.BUFFER.value.table[591]), INT_ENUM},*)
(*DBG:    {&(RES0__INSTANCE0.MY_BAD_FIFO.BUFFER.value.table[592]), INT_ENUM},*)
(*DBG:    {&(RES0__INSTANCE0.MY_BAD_FIFO.BUFFER.value.table[593]), INT_ENUM},*)
(*DBG:    {&(RES0__INSTANCE0.MY_BAD_FIFO.BUFFER.value.table[594]), INT_ENUM},*)
(*DBG:    {&(RES0__INSTANCE0.MY_BAD_FIFO.BUFFER.value.table[595]), INT_ENUM},*)
(*DBG:    {&(RES0__INSTANCE0.MY_BAD_FIFO.BUFFER.value.table[596]), INT_ENUM},*)
(*DBG:    {&(RES0__INSTANCE0.MY_BAD_FIFO.BUFFER.value.table[597]), INT_ENUM},*)
(*DBG:    {&(RES0__INSTANCE0.MY_BAD_FIFO.BUFFER.value.table[598]), INT_ENUM},*)
(*DBG:    {&(RES0__INSTANCE0.MY_BAD_FIFO.BUFFER.value.table[599]), INT_ENUM},*)
(*DBG:    {&(RES0__INSTANCE0.MY_BAD_FIFO.BUFFER.value.table[600]), INT_ENUM},*)
(*DBG:    {&(RES0__INSTANCE0.MY_BAD_FIFO.BUFFER.value.table[601]), INT_ENUM},*)
(*DBG:    {&(RES0__INSTANCE0.MY_BAD_FIFO.BUFFER.value.table[602]), INT_ENUM},*)
(*DBG:    {&(RES0__INSTANCE0.MY_BAD_FIFO.BUFFER.value.table[603]), INT_ENUM},*)
(*DBG:    {&(RES0__INSTANCE0.MY_BAD_FIFO.BUFFER.value.table[604]), INT_ENUM},*)
(*DBG:    {&(RES0__INSTANCE0.MY_BAD_FIFO.BUFFER.value.table[605]), INT_ENUM},*)
(*DBG:    {&(RES0__INSTANCE0.MY_BAD_FIFO.BUFFER.value.table[606]), INT_ENUM},*)
(*DBG:    {&(RES0__INSTANCE0.MY_BAD_FIFO.BUFFER.value.table[607]), INT_ENUM},*)
(*DBG:    {&(RES0__INSTANCE0.MY_BAD_FIFO.BUFFER.value.table[608]), INT_ENUM},*)
(*DBG:    {&(RES0__INSTANCE0.MY_BAD_FIFO.BUFFER.value.table[609]), INT_ENUM},*)
(*DBG:    {&(RES0__INSTANCE0.MY_BAD_FIFO.BUFFER.value.table[610]), INT_ENUM},*)
(*DBG:    {&(RES0__INSTANCE0.MY_BAD_FIFO.BUFFER.value.table[611]), INT_ENUM},*)
(*DBG:    {&(RES0__INSTANCE0.MY_BAD_FIFO.BUFFER.value.table[612]), INT_ENUM},*)
(*DBG:    {&(RES0__INSTANCE0.MY_BAD_FIFO.BUFFER.value.table[613]), INT_ENUM},*)
(*DBG:    {&(RES0__INSTANCE0.MY_BAD_FIFO.BUFFER.value.table[614]), INT_ENUM},*)
(*DBG:    {&(RES0__INSTANCE0.MY_BAD_FIFO.BUFFER.value.table[615]), INT_ENUM},*)
(*DBG:    {&(RES0__INSTANCE0.MY_BAD_FIFO.BUFFER.value.table[616]), INT_ENUM},*)
(*DBG:    {&(RES0__INSTANCE0.MY_BAD_FIFO.BUFFER.value.table[617]), INT_ENUM},*)
(*DBG:    {&(RES0__INSTANCE0.MY_BAD_FIFO.BUFFER.value.table[618]), INT_ENUM},*)
(*DBG:    {&(RES0__INSTANCE0.MY_BAD_FIFO.BUFFER.value.table[619]), INT_ENUM},*)
(*DBG:    {&(RES0__INSTANCE0.MY_BAD_FIFO.BUFFER.value.table[620]), INT_ENUM},*)
(*DBG:    {&(RES0__INSTANCE0.MY_BAD_FIFO.BUFFER.value.table[621]), INT_ENUM},*)
(*DBG:    {&(RES0__INSTANCE0.MY_BAD_FIFO.BUFFER.value.table[622]), INT_ENUM},*)
(*DBG:    {&(RES0__INSTANCE0.MY_BAD_FIFO.BUFFER.value.table[623]), INT_ENUM},*)
(*DBG:    {&(RES0__INSTANCE0.MY_BAD_FIFO.BUFFER.value.table[624]), INT_ENUM},*)
(*DBG:    {&(RES0__INSTANCE0.MY_BAD_FIFO.BUFFER.value.table[625]), INT_ENUM},*)
(*DBG:    {&(RES0__INSTANCE0.MY_BAD_FIFO.BUFFER.value.table[626]), INT_ENUM},*)
(*DBG:    {&(RES0__INSTANCE0.MY_BAD_FIFO.BUFFER.value.table[627]), INT_ENUM},*)
(*DBG:    {&(RES0__INSTANCE0.MY_BAD_FIFO.BUFFER.value.table[628]), INT_ENUM},*)
(*DBG:    {&(RES0__INSTANCE0.MY_BAD_FIFO.BUFFER.value.table[629]), INT_ENUM},*)
(*DBG:    {&(RES0__INSTANCE0.MY_BAD_FIFO.BUFFER.value.table[630]), INT_ENUM},*)
(*DBG:    {&(RES0__INSTANCE0.MY_BAD_FIFO.BUFFER.value.table[631]), INT_ENUM},*)
(*DBG:    {&(RES0__INSTANCE0.MY_BAD_FIFO.BUFFER.value.table[632]), INT_ENUM},*)
(*DBG:    {&(RES0__INSTANCE0.MY_BAD_FIFO.BUFFER.value.table[633]), INT_ENUM},*)
(*DBG:    {&(RES0__INSTANCE0.MY_BAD_FIFO.BUFFER.value.table[634]), INT_ENUM},*)
(*DBG:    {&(RES0__INSTANCE0.MY_BAD_FIFO.BUFFER.value.table[635]), INT_ENUM},*)
(*DBG:    {&(RES0__INSTANCE0.MY_BAD_FIFO.BUFFER.value.table[636]), INT_ENUM},*)
(*DBG:    {&(RES0__INSTANCE0.MY_BAD_FIFO.BUFFER.value.table[637]), INT_ENUM},*)
(*DBG:    {&(RES0__INSTANCE0.MY_BAD_FIFO.BUFFER.value.table[638]), INT_ENUM},*)
(*DBG:    {&(RES0__INSTANCE0.MY_BAD_FIFO.BUFFER.value.table[639]), INT_ENUM},*)
(*DBG:    {&(RES0__INSTANCE0.MY_BAD_FIFO.BUFFER.value.table[640]), INT_ENUM},*)
(*DBG:    {&(RES0__INSTANCE0.MY_BAD_FIFO.BUFFER.value.table[641]), INT_ENUM},*)
(*DBG:    {&(RES0__INSTANCE0.MY_BAD_FIFO.BUFFER.value.table[642]), INT_ENUM},*)
(*DBG:    {&(RES0__INSTANCE0.MY_BAD_FIFO.BUFFER.value.table[643]), INT_ENUM},*)
(*DBG:    {&(RES0__INSTANCE0.MY_BAD_FIFO.BUFFER.value.table[644]), INT_ENUM},*)
(*DBG:    {&(RES0__INSTANCE0.MY_BAD_FIFO.BUFFER.value.table[645]), INT_ENUM},*)
(*DBG:    {&(RES0__INSTANCE0.MY_BAD_FIFO.BUFFER.value.table[646]), INT_ENUM},*)
(*DBG:    {&(RES0__INSTANCE0.MY_BAD_FIFO.BUFFER.value.table[647]), INT_ENUM},*)
(*DBG:    {&(RES0__INSTANCE0.MY_BAD_FIFO.BUFFER.value.table[648]), INT_ENUM},*)
(*DBG:    {&(RES0__INSTANCE0.MY_BAD_FIFO.BUFFER.value.table[649]), INT_ENUM},*)
(*DBG:    {&(RES0__INSTANCE0.MY_BAD_FIFO.BUFFER.value.table[650]), INT_ENUM},*)
(*DBG:    {&(RES0__INSTANCE0.MY_BAD_FIFO.BUFFER.value.table[651]), INT_ENUM},*)
(*DBG:    {&(RES0__INSTANCE0.MY_BAD_FIFO.BUFFER.value.table[652]), INT_ENUM},*)
(*DBG:    {&(RES0__INSTANCE0.MY_BAD_FIFO.BUFFER.value.table[653]), INT_ENUM},*)
(*DBG:    {&(RES0__INSTANCE0.MY_BAD_FIFO.BUFFER.value.table[654]), INT_ENUM},*)
(*DBG:    {&(RES0__INSTANCE0.MY_BAD_FIFO.BUFFER.value.table[655]), INT_ENUM},*)
(*DBG:    {&(RES0__INSTANCE0.MY_BAD_FIFO.BUFFER.value.table[656]), INT_ENUM},*)
(*DBG:    {&(RES0__INSTANCE0.MY_BAD_FIFO.BUFFER.value.table[657]), INT_ENUM},*)
(*DBG:    {&(RES0__INSTANCE0.MY_BAD_FIFO.BUFFER.value.table[658]), INT_ENUM},*)
(*DBG:    {&(RES0__INSTANCE0.MY_BAD_FIFO.BUFFER.value.table[659]), INT_ENUM},*)
(*DBG:    {&(RES0__INSTANCE0.MY_BAD_FIFO.BUFFER.value.table[660]), INT_ENUM},*)
(*DBG:    {&(RES0__INSTANCE0.MY_BAD_FIFO.BUFFER.value.table[661]), INT_ENUM},*)
(*DBG:    {&(RES0__INSTANCE0.MY_BAD_FIFO.BUFFER.value.table[662]), INT_ENUM},*)
(*DBG:    {&(RES0__INSTANCE0.MY_BAD_FIFO.BUFFER.value.table[663]), INT_ENUM},*)
(*DBG:    {&(RES0__INSTANCE0.MY_BAD_FIFO.BUFFER.value.table[664]), INT_ENUM},*)
(*DBG:    {&(RES0__INSTANCE0.MY_BAD_FIFO.BUFFER.value.table[665]), INT_ENUM},*)
(*DBG:    {&(RES0__INSTANCE0.MY_BAD_FIFO.BUFFER.value.table[666]), INT_ENUM},*)
(*DBG:    {&(RES0__INSTANCE0.MY_BAD_FIFO.BUFFER.value.table[667]), INT_ENUM},*)
(*DBG:    {&(RES0__INSTANCE0.MY_BAD_FIFO.BUFFER.value.table[668]), INT_ENUM},*)
(*DBG:    {&(RES0__INSTANCE0.MY_BAD_FIFO.BUFFER.value.table[669]), INT_ENUM},*)
(*DBG:    {&(RES0__INSTANCE0.MY_BAD_FIFO.BUFFER.value.table[670]), INT_ENUM},*)
(*DBG:    {&(RES0__INSTANCE0.MY_BAD_FIFO.BUFFER.value.table[671]), INT_ENUM},*)
(*DBG:    {&(RES0__INSTANCE0.MY_BAD_FIFO.BUFFER.value.table[672]), INT_ENUM},*)
(*DBG:    {&(RES0__INSTANCE0.MY_BAD_FIFO.BUFFER.value.table[673]), INT_ENUM},*)
(*DBG:    {&(RES0__INSTANCE0.MY_BAD_FIFO.BUFFER.value.table[674]), INT_ENUM},*)
(*DBG:    {&(RES0__INSTANCE0.MY_BAD_FIFO.BUFFER.value.table[675]), INT_ENUM},*)
(*DBG:    {&(RES0__INSTANCE0.MY_BAD_FIFO.BUFFER.value.table[676]), INT_ENUM},*)
(*DBG:    {&(RES0__INSTANCE0.MY_BAD_FIFO.BUFFER.value.table[677]), INT_ENUM},*)
(*DBG:    {&(RES0__INSTANCE0.MY_BAD_FIFO.BUFFER.value.table[678]), INT_ENUM},*)
(*DBG:    {&(RES0__INSTANCE0.MY_BAD_FIFO.BUFFER.value.table[679]), INT_ENUM},*)
(*DBG:    {&(RES0__INSTANCE0.MY_BAD_FIFO.BUFFER.value.table[680]), INT_ENUM},*)
(*DBG:    {&(RES0__INSTANCE0.MY_BAD_FIFO.BUFFER.value.table[681]), INT_ENUM},*)
(*DBG:    {&(RES0__INSTANCE0.MY_BAD_FIFO.BUFFER.value.table[682]), INT_ENUM},*)
(*DBG:    {&(RES0__INSTANCE0.MY_BAD_FIFO.BUFFER.value.table[683]), INT_ENUM},*)
(*DBG:    {&(RES0__INSTANCE0.MY_BAD_FIFO.BUFFER.value.table[684]), INT_ENUM},*)
(*DBG:    {&(RES0__INSTANCE0.MY_BAD_FIFO.BUFFER.value.table[685]), INT_ENUM},*)
(*DBG:    {&(RES0__INSTANCE0.MY_BAD_FIFO.BUFFER.value.table[686]), INT_ENUM},*)
(*DBG:    {&(RES0__INSTANCE0.MY_BAD_FIFO.BUFFER.value.table[687]), INT_ENUM},*)
(*DBG:    {&(RES0__INSTANCE0.MY_BAD_FIFO.BUFFER.value.table[688]), INT_ENUM},*)
(*DBG:    {&(RES0__INSTANCE0.MY_BAD_FIFO.BUFFER.value.table[689]), INT_ENUM},*)
(*DBG:    {&(RES0__INSTANCE0.MY_BAD_FIFO.BUFFER.value.table[690]), INT_ENUM},*)
(*DBG:    {&(RES0__INSTANCE0.MY_BAD_FIFO.BUFFER.value.table[691]), INT_ENUM},*)
(*DBG:    {&(RES0__INSTANCE0.MY_BAD_FIFO.BUFFER.value.table[692]), INT_ENUM},*)
(*DBG:    {&(RES0__INSTANCE0.MY_BAD_FIFO.BUFFER.value.table[693]), INT_ENUM},*)
(*DBG:    {&(RES0__INSTANCE0.MY_BAD_FIFO.BUFFER.value.table[694]), INT_ENUM},*)
(*DBG:    {&(RES0__INSTANCE0.MY_BAD_FIFO.BUFFER.value.table[695]), INT_ENUM},*)
(*DBG:    {&(RES0__INSTANCE0.MY_BAD_FIFO.BUFFER.value.table[696]), INT_ENUM},*)
(*DBG:    {&(RES0__INSTANCE0.MY_BAD_FIFO.BUFFER.value.table[697]), INT_ENUM},*)
(*DBG:    {&(RES0__INSTANCE0.MY_BAD_FIFO.BUFFER.value.table[698]), INT_ENUM},*)
(*DBG:    {&(RES0__INSTANCE0.MY_BAD_FIFO.BUFFER.value.table[699]), INT_ENUM},*)
(*DBG:    {&(RES0__INSTANCE0.MY_BAD_FIFO.BUFFER.value.table[700]), INT_ENUM},*)
(*DBG:    {&(RES0__INSTANCE0.MY_BAD_FIFO.BUFFER.value.table[701]), INT_ENUM},*)
(*DBG:    {&(RES0__INSTANCE0.MY_BAD_FIFO.BUFFER.value.table[702]), INT_ENUM},*)
(*DBG:    {&(RES0__INSTANCE0.MY_BAD_FIFO.BUFFER.value.table[703]), INT_ENUM},*)
(*DBG:    {&(RES0__INSTANCE0.MY_BAD_FIFO.BUFFER.value.table[704]), INT_ENUM},*)
(*DBG:    {&(RES0__INSTANCE0.MY_BAD_FIFO.BUFFER.value.table[705]), INT_ENUM},*)
(*DBG:    {&(RES0__INSTANCE0.MY_BAD_FIFO.BUFFER.value.table[706]), INT_ENUM},*)
(*DBG:    {&(RES0__INSTANCE0.MY_BAD_FIFO.BUFFER.value.table[707]), INT_ENUM},*)
(*DBG:    {&(RES0__INSTANCE0.MY_BAD_FIFO.BUFFER.value.table[708]), INT_ENUM},*)
(*DBG:    {&(RES0__INSTANCE0.MY_BAD_FIFO.BUFFER.value.table[709]), INT_ENUM},*)
(*DBG:    {&(RES0__INSTANCE0.MY_BAD_FIFO.BUFFER.value.table[710]), INT_ENUM},*)
(*DBG:    {&(RES0__INSTANCE0.MY_BAD_FIFO.BUFFER.value.table[711]), INT_ENUM},*)
(*DBG:    {&(RES0__INSTANCE0.MY_BAD_FIFO.BUFFER.value.table[712]), INT_ENUM},*)
(*DBG:    {&(RES0__INSTANCE0.MY_BAD_FIFO.BUFFER.value.table[713]), INT_ENUM},*)
(*DBG:    {&(RES0__INSTANCE0.MY_BAD_FIFO.BUFFER.value.table[714]), INT_ENUM},*)
(*DBG:    {&(RES0__INSTANCE0.MY_BAD_FIFO.BUFFER.value.table[715]), INT_ENUM},*)
(*DBG:    {&(RES0__INSTANCE0.MY_BAD_FIFO.BUFFER.value.table[716]), INT_ENUM},*)
(*DBG:    {&(RES0__INSTANCE0.MY_BAD_FIFO.BUFFER.value.table[717]), INT_ENUM},*)
(*DBG:    {&(RES0__INSTANCE0.MY_BAD_FIFO.BUFFER.value.table[718]), INT_ENUM},*)
(*DBG:    {&(RES0__INSTANCE0.MY_BAD_FIFO.BUFFER.value.table[719]), INT_ENUM},*)
(*DBG:    {&(RES0__INSTANCE0.MY_BAD_FIFO.BUFFER.value.table[720]), INT_ENUM},*)
(*DBG:    {&(RES0__INSTANCE0.MY_BAD_FIFO.BUFFER.value.table[721]), INT_ENUM},*)
(*DBG:    {&(RES0__INSTANCE0.MY_BAD_FIFO.BUFFER.value.table[722]), INT_ENUM},*)
(*DBG:    {&(RES0__INSTANCE0.MY_BAD_FIFO.BUFFER.value.table[723]), INT_ENUM},*)
(*DBG:    {&(RES0__INSTANCE0.MY_BAD_FIFO.BUFFER.value.table[724]), INT_ENUM},*)
(*DBG:    {&(RES0__INSTANCE0.MY_BAD_FIFO.BUFFER.value.table[725]), INT_ENUM},*)
(*DBG:    {&(RES0__INSTANCE0.MY_BAD_FIFO.BUFFER.value.table[726]), INT_ENUM},*)
(*DBG:    {&(RES0__INSTANCE0.MY_BAD_FIFO.BUFFER.value.table[727]), INT_ENUM},*)
(*DBG:    {&(RES0__INSTANCE0.MY_BAD_FIFO.BUFFER.value.table[728]), INT_ENUM},*)
(*DBG:    {&(RES0__INSTANCE0.MY_BAD_FIFO.BUFFER.value.table[729]), INT_ENUM},*)
(*DBG:    {&(RES0__INSTANCE0.MY_BAD_FIFO.BUFFER.value.table[730]), INT_ENUM},*)
(*DBG:    {&(RES0__INSTANCE0.MY_BAD_FIFO.BUFFER.value.table[731]), INT_ENUM},*)
(*DBG:    {&(RES0__INSTANCE0.MY_BAD_FIFO.BUFFER.value.table[732]), INT_ENUM},*)
(*DBG:    {&(RES0__INSTANCE0.MY_BAD_FIFO.BUFFER.value.table[733]), INT_ENUM},*)
(*DBG:    {&(RES0__INSTANCE0.MY_BAD_FIFO.BUFFER.value.table[734]), INT_ENUM},*)
(*DBG:    {&(RES0__INSTANCE0.MY_BAD_FIFO.BUFFER.value.table[735]), INT_ENUM},*)
(*DBG:    {&(RES0__INSTANCE0.MY_BAD_FIFO.BUFFER.value.table[736]), INT_ENUM},*)
(*DBG:    {&(RES0__INSTANCE0.MY_BAD_FIFO.BUFFER.value.table[737]), INT_ENUM},*)
(*DBG:    {&(RES0__INSTANCE0.MY_BAD_FIFO.BUFFER.value.table[738]), INT_ENUM},*)
(*DBG:    {&(RES0__INSTANCE0.MY_BAD_FIFO.BUFFER.value.table[739]), INT_ENUM},*)
(*DBG:    {&(RES0__INSTANCE0.MY_BAD_FIFO.BUFFER.value.table[740]), INT_ENUM},*)
(*DBG:    {&(RES0__INSTANCE0.MY_BAD_FIFO.BUFFER.value.table[741]), INT_ENUM},*)
(*DBG:    {&(RES0__INSTANCE0.MY_BAD_FIFO.BUFFER.value.table[742]), INT_ENUM},*)
(*DBG:    {&(RES0__INSTANCE0.MY_BAD_FIFO.BUFFER.value.table[743]), INT_ENUM},*)
(*DBG:    {&(RES0__INSTANCE0.MY_BAD_FIFO.BUFFER.value.table[744]), INT_ENUM},*)
(*DBG:    {&(RES0__INSTANCE0.MY_BAD_FIFO.BUFFER.value.table[745]), INT_ENUM},*)
(*DBG:    {&(RES0__INSTANCE0.MY_BAD_FIFO.BUFFER.value.table[746]), INT_ENUM},*)
(*DBG:    {&(RES0__INSTANCE0.MY_BAD_FIFO.BUFFER.value.table[747]), INT_ENUM},*)
(*DBG:    {&(RES0__INSTANCE0.MY_BAD_FIFO.BUFFER.value.table[748]), INT_ENUM},*)
(*DBG:    {&(RES0__INSTANCE0.MY_BAD_FIFO.BUFFER.value.table[749]), INT_ENUM},*)
(*DBG:    {&(RES0__INSTANCE0.MY_BAD_FIFO.BUFFER.value.table[750]), INT_ENUM},*)
(*DBG:    {&(RES0__INSTANCE0.MY_BAD_FIFO.BUFFER.value.table[751]), INT_ENUM},*)
(*DBG:    {&(RES0__INSTANCE0.MY_BAD_FIFO.BUFFER.value.table[752]), INT_ENUM},*)
(*DBG:    {&(RES0__INSTANCE0.MY_BAD_FIFO.BUFFER.value.table[753]), INT_ENUM},*)
(*DBG:    {&(RES0__INSTANCE0.MY_BAD_FIFO.BUFFER.value.table[754]), INT_ENUM},*)
(*DBG:    {&(RES0__INSTANCE0.MY_BAD_FIFO.BUFFER.value.table[755]), INT_ENUM},*)
(*DBG:    {&(RES0__INSTANCE0.MY_BAD_FIFO.BUFFER.value.table[756]), INT_ENUM},*)
(*DBG:    {&(RES0__INSTANCE0.MY_BAD_FIFO.BUFFER.value.table[757]), INT_ENUM},*)
(*DBG:    {&(RES0__INSTANCE0.MY_BAD_FIFO.BUFFER.value.table[758]), INT_ENUM},*)
(*DBG:    {&(RES0__INSTANCE0.MY_BAD_FIFO.BUFFER.value.table[759]), INT_ENUM},*)
(*DBG:    {&(RES0__INSTANCE0.MY_BAD_FIFO.BUFFER.value.table[760]), INT_ENUM},*)
(*DBG:    {&(RES0__INSTANCE0.MY_BAD_FIFO.BUFFER.value.table[761]), INT_ENUM},*)
(*DBG:    {&(RES0__INSTANCE0.MY_BAD_FIFO.BUFFER.value.table[762]), INT_ENUM},*)
(*DBG:    {&(RES0__INSTANCE0.MY_BAD_FIFO.BUFFER.value.table[763]), INT_ENUM},*)
(*DBG:    {&(RES0__INSTANCE0.MY_BAD_FIFO.BUFFER.value.table[764]), INT_ENUM},*)
(*DBG:    {&(RES0__INSTANCE0.MY_BAD_FIFO.BUFFER.value.table[765]), INT_ENUM},*)
(*DBG:    {&(RES0__INSTANCE0.MY_BAD_FIFO.BUFFER.value.table[766]), INT_ENUM},*)
(*DBG:    {&(RES0__INSTANCE0.MY_BAD_FIFO.BUFFER.value.table[767]), INT_ENUM},*)
(*DBG:    {&(RES0__INSTANCE0.MY_BAD_FIFO.BUFFER.value.table[768]), INT_ENUM},*)
(*DBG:    {&(RES0__INSTANCE0.MY_BAD_FIFO.BUFFER.value.table[769]), INT_ENUM},*)
(*DBG:    {&(RES0__INSTANCE0.MY_BAD_FIFO.BUFFER.value.table[770]), INT_ENUM},*)
(*DBG:    {&(RES0__INSTANCE0.MY_BAD_FIFO.BUFFER.value.table[771]), INT_ENUM},*)
(*DBG:    {&(RES0__INSTANCE0.MY_BAD_FIFO.BUFFER.value.table[772]), INT_ENUM},*)
(*DBG:    {&(RES0__INSTANCE0.MY_BAD_FIFO.BUFFER.value.table[773]), INT_ENUM},*)
(*DBG:    {&(RES0__INSTANCE0.MY_BAD_FIFO.BUFFER.value.table[774]), INT_ENUM},*)
(*DBG:    {&(RES0__INSTANCE0.MY_BAD_FIFO.BUFFER.value.table[775]), INT_ENUM},*)
(*DBG:    {&(RES0__INSTANCE0.MY_BAD_FIFO.BUFFER.value.table[776]), INT_ENUM},*)
(*DBG:    {&(RES0__INSTANCE0.MY_BAD_FIFO.BUFFER.value.table[777]), INT_ENUM},*)
(*DBG:    {&(RES0__INSTANCE0.MY_BAD_FIFO.BUFFER.value.table[778]), INT_ENUM},*)
(*DBG:    {&(RES0__INSTANCE0.MY_BAD_FIFO.BUFFER.value.table[779]), INT_ENUM},*)
(*DBG:    {&(RES0__INSTANCE0.MY_BAD_FIFO.BUFFER.value.table[780]), INT_ENUM},*)
(*DBG:    {&(RES0__INSTANCE0.MY_BAD_FIFO.BUFFER.value.table[781]), INT_ENUM},*)
(*DBG:    {&(RES0__INSTANCE0.MY_BAD_FIFO.BUFFER.value.table[782]), INT_ENUM},*)
(*DBG:    {&(RES0__INSTANCE0.MY_BAD_FIFO.BUFFER.value.table[783]), INT_ENUM},*)
(*DBG:    {&(RES0__INSTANCE0.MY_BAD_FIFO.BUFFER.value.table[784]), INT_ENUM},*)
(*DBG:    {&(RES0__INSTANCE0.MY_BAD_FIFO.BUFFER.value.table[785]), INT_ENUM},*)
(*DBG:    {&(RES0__INSTANCE0.MY_BAD_FIFO.BUFFER.value.table[786]), INT_ENUM},*)
(*DBG:    {&(RES0__INSTANCE0.MY_BAD_FIFO.BUFFER.value.table[787]), INT_ENUM},*)
(*DBG:    {&(RES0__INSTANCE0.MY_BAD_FIFO.BUFFER.value.table[788]), INT_ENUM},*)
(*DBG:    {&(RES0__INSTANCE0.MY_BAD_FIFO.BUFFER.value.table[789]), INT_ENUM},*)
(*DBG:    {&(RES0__INSTANCE0.MY_BAD_FIFO.BUFFER.value.table[790]), INT_ENUM},*)
(*DBG:    {&(RES0__INSTANCE0.MY_BAD_FIFO.BUFFER.value.table[791]), INT_ENUM},*)
(*DBG:    {&(RES0__INSTANCE0.MY_BAD_FIFO.BUFFER.value.table[792]), INT_ENUM},*)
(*DBG:    {&(RES0__INSTANCE0.MY_BAD_FIFO.BUFFER.value.table[793]), INT_ENUM},*)
(*DBG:    {&(RES0__INSTANCE0.MY_BAD_FIFO.BUFFER.value.table[794]), INT_ENUM},*)
(*DBG:    {&(RES0__INSTANCE0.MY_BAD_FIFO.BUFFER.value.table[795]), INT_ENUM},*)
(*DBG:    {&(RES0__INSTANCE0.MY_BAD_FIFO.BUFFER.value.table[796]), INT_ENUM},*)
(*DBG:    {&(RES0__INSTANCE0.MY_BAD_FIFO.BUFFER.value.table[797]), INT_ENUM},*)
(*DBG:    {&(RES0__INSTANCE0.MY_BAD_FIFO.BUFFER.value.table[798]), INT_ENUM},*)
(*DBG:    {&(RES0__INSTANCE0.MY_BAD_FIFO.BUFFER.value.table[799]), INT_ENUM},*)
(*DBG:    {&(RES0__INSTANCE0.MY_BAD_FIFO.BUFFER.value.table[800]), INT_ENUM},*)
(*DBG:    {&(RES0__INSTANCE0.MY_BAD_FIFO.BUFFER.value.table[801]), INT_ENUM},*)
(*DBG:    {&(RES0__INSTANCE0.MY_BAD_FIFO.BUFFER.value.table[802]), INT_ENUM},*)
(*DBG:    {&(RES0__INSTANCE0.MY_BAD_FIFO.BUFFER.value.table[803]), INT_ENUM},*)
(*DBG:    {&(RES0__INSTANCE0.MY_BAD_FIFO.BUFFER.value.table[804]), INT_ENUM},*)
(*DBG:    {&(RES0__INSTANCE0.MY_BAD_FIFO.BUFFER.value.table[805]), INT_ENUM},*)
(*DBG:    {&(RES0__INSTANCE0.MY_BAD_FIFO.BUFFER.value.table[806]), INT_ENUM},*)
(*DBG:    {&(RES0__INSTANCE0.MY_BAD_FIFO.BUFFER.value.table[807]), INT_ENUM},*)
(*DBG:    {&(RES0__INSTANCE0.MY_BAD_FIFO.BUFFER.value.table[808]), INT_ENUM},*)
(*DBG:    {&(RES0__INSTANCE0.MY_BAD_FIFO.BUFFER.value.table[809]), INT_ENUM},*)
(*DBG:    {&(RES0__INSTANCE0.MY_BAD_FIFO.BUFFER.value.table[810]), INT_ENUM},*)
(*DBG:    {&(RES0__INSTANCE0.MY_BAD_FIFO.BUFFER.value.table[811]), INT_ENUM},*)
(*DBG:    {&(RES0__INSTANCE0.MY_BAD_FIFO.BUFFER.value.table[812]), INT_ENUM},*)
(*DBG:    {&(RES0__INSTANCE0.MY_BAD_FIFO.BUFFER.value.table[813]), INT_ENUM},*)
(*DBG:    {&(RES0__INSTANCE0.MY_BAD_FIFO.BUFFER.value.table[814]), INT_ENUM},*)
(*DBG:    {&(RES0__INSTANCE0.MY_BAD_FIFO.BUFFER.value.table[815]), INT_ENUM},*)
(*DBG:    {&(RES0__INSTANCE0.MY_BAD_FIFO.BUFFER.value.table[816]), INT_ENUM},*)
(*DBG:    {&(RES0__INSTANCE0.MY_BAD_FIFO.BUFFER.value.table[817]), INT_ENUM},*)
(*DBG:    {&(RES0__INSTANCE0.MY_BAD_FIFO.BUFFER.value.table[818]), INT_ENUM},*)
(*DBG:    {&(RES0__INSTANCE0.MY_BAD_FIFO.BUFFER.value.table[819]), INT_ENUM},*)
(*DBG:    {&(RES0__INSTANCE0.MY_BAD_FIFO.BUFFER.value.table[820]), INT_ENUM},*)
(*DBG:    {&(RES0__INSTANCE0.MY_BAD_FIFO.BUFFER.value.table[821]), INT_ENUM},*)
(*DBG:    {&(RES0__INSTANCE0.MY_BAD_FIFO.BUFFER.value.table[822]), INT_ENUM},*)
(*DBG:    {&(RES0__INSTANCE0.MY_BAD_FIFO.BUFFER.value.table[823]), INT_ENUM},*)
(*DBG:    {&(RES0__INSTANCE0.MY_BAD_FIFO.BUFFER.value.table[824]), INT_ENUM},*)
(*DBG:    {&(RES0__INSTANCE0.MY_BAD_FIFO.BUFFER.value.table[825]), INT_ENUM},*)
(*DBG:    {&(RES0__INSTANCE0.MY_BAD_FIFO.BUFFER.value.table[826]), INT_ENUM},*)
(*DBG:    {&(RES0__INSTANCE0.MY_BAD_FIFO.BUFFER.value.table[827]), INT_ENUM},*)
(*DBG:    {&(RES0__INSTANCE0.MY_BAD_FIFO.BUFFER.value.table[828]), INT_ENUM},*)
(*DBG:    {&(RES0__INSTANCE0.MY_BAD_FIFO.BUFFER.value.table[829]), INT_ENUM},*)
(*DBG:    {&(RES0__INSTANCE0.MY_BAD_FIFO.BUFFER.value.table[830]), INT_ENUM},*)
(*DBG:    {&(RES0__INSTANCE0.MY_BAD_FIFO.BUFFER.value.table[831]), INT_ENUM},*)
(*DBG:    {&(RES0__INSTANCE0.MY_BAD_FIFO.BUFFER.value.table[832]), INT_ENUM},*)
(*DBG:    {&(RES0__INSTANCE0.MY_BAD_FIFO.BUFFER.value.table[833]), INT_ENUM},*)
(*DBG:    {&(RES0__INSTANCE0.MY_BAD_FIFO.BUFFER.value.table[834]), INT_ENUM},*)
(*DBG:    {&(RES0__INSTANCE0.MY_BAD_FIFO.BUFFER.value.table[835]), INT_ENUM},*)
(*DBG:    {&(RES0__INSTANCE0.MY_BAD_FIFO.BUFFER.value.table[836]), INT_ENUM},*)
(*DBG:    {&(RES0__INSTANCE0.MY_BAD_FIFO.BUFFER.value.table[837]), INT_ENUM},*)
(*DBG:    {&(RES0__INSTANCE0.MY_BAD_FIFO.BUFFER.value.table[838]), INT_ENUM},*)
(*DBG:    {&(RES0__INSTANCE0.MY_BAD_FIFO.BUFFER.value.table[839]), INT_ENUM},*)
(*DBG:    {&(RES0__INSTANCE0.MY_BAD_FIFO.BUFFER.value.table[840]), INT_ENUM},*)
(*DBG:    {&(RES0__INSTANCE0.MY_BAD_FIFO.BUFFER.value.table[841]), INT_ENUM},*)
(*DBG:    {&(RES0__INSTANCE0.MY_BAD_FIFO.BUFFER.value.table[842]), INT_ENUM},*)
(*DBG:    {&(RES0__INSTANCE0.MY_BAD_FIFO.BUFFER.value.table[843]), INT_ENUM},*)
(*DBG:    {&(RES0__INSTANCE0.MY_BAD_FIFO.BUFFER.value.table[844]), INT_ENUM},*)
(*DBG:    {&(RES0__INSTANCE0.MY_BAD_FIFO.BUFFER.value.table[845]), INT_ENUM},*)
(*DBG:    {&(RES0__INSTANCE0.MY_BAD_FIFO.BUFFER.value.table[846]), INT_ENUM},*)
(*DBG:    {&(RES0__INSTANCE0.MY_BAD_FIFO.BUFFER.value.table[847]), INT_ENUM},*)
(*DBG:    {&(RES0__INSTANCE0.MY_BAD_FIFO.BUFFER.value.table[848]), INT_ENUM},*)
(*DBG:    {&(RES0__INSTANCE0.MY_BAD_FIFO.BUFFER.value.table[849]), INT_ENUM},*)
(*DBG:    {&(RES0__INSTANCE0.MY_BAD_FIFO.BUFFER.value.table[850]), INT_ENUM},*)
(*DBG:    {&(RES0__INSTANCE0.MY_BAD_FIFO.BUFFER.value.table[851]), INT_ENUM},*)
(*DBG:    {&(RES0__INSTANCE0.MY_BAD_FIFO.BUFFER.value.table[852]), INT_ENUM},*)
(*DBG:    {&(RES0__INSTANCE0.MY_BAD_FIFO.BUFFER.value.table[853]), INT_ENUM},*)
(*DBG:    {&(RES0__INSTANCE0.MY_BAD_FIFO.BUFFER.value.table[854]), INT_ENUM},*)
(*DBG:    {&(RES0__INSTANCE0.MY_BAD_FIFO.BUFFER.value.table[855]), INT_ENUM},*)
(*DBG:    {&(RES0__INSTANCE0.MY_BAD_FIFO.BUFFER.value.table[856]), INT_ENUM},*)
(*DBG:    {&(RES0__INSTANCE0.MY_BAD_FIFO.BUFFER.value.table[857]), INT_ENUM},*)
(*DBG:    {&(RES0__INSTANCE0.MY_BAD_FIFO.BUFFER.value.table[858]), INT_ENUM},*)
(*DBG:    {&(RES0__INSTANCE0.MY_BAD_FIFO.BUFFER.value.table[859]), INT_ENUM},*)
(*DBG:    {&(RES0__INSTANCE0.MY_BAD_FIFO.BUFFER.value.table[860]), INT_ENUM},*)
(*DBG:    {&(RES0__INSTANCE0.MY_BAD_FIFO.BUFFER.value.table[861]), INT_ENUM},*)
(*DBG:    {&(RES0__INSTANCE0.MY_BAD_FIFO.BUFFER.value.table[862]), INT_ENUM},*)
(*DBG:    {&(RES0__INSTANCE0.MY_BAD_FIFO.BUFFER.value.table[863]), INT_ENUM},*)
(*DBG:    {&(RES0__INSTANCE0.MY_BAD_FIFO.BUFFER.value.table[864]), INT_ENUM},*)
(*DBG:    {&(RES0__INSTANCE0.MY_BAD_FIFO.BUFFER.value.table[865]), INT_ENUM},*)
(*DBG:    {&(RES0__INSTANCE0.MY_BAD_FIFO.BUFFER.value.table[866]), INT_ENUM},*)
(*DBG:    {&(RES0__INSTANCE0.MY_BAD_FIFO.BUFFER.value.table[867]), INT_ENUM},*)
(*DBG:    {&(RES0__INSTANCE0.MY_BAD_FIFO.BUFFER.value.table[868]), INT_ENUM},*)
(*DBG:    {&(RES0__INSTANCE0.MY_BAD_FIFO.BUFFER.value.table[869]), INT_ENUM},*)
(*DBG:    {&(RES0__INSTANCE0.MY_BAD_FIFO.BUFFER.value.table[870]), INT_ENUM},*)
(*DBG:    {&(RES0__INSTANCE0.MY_BAD_FIFO.BUFFER.value.table[871]), INT_ENUM},*)
(*DBG:    {&(RES0__INSTANCE0.MY_BAD_FIFO.BUFFER.value.table[872]), INT_ENUM},*)
(*DBG:    {&(RES0__INSTANCE0.MY_BAD_FIFO.BUFFER.value.table[873]), INT_ENUM},*)
(*DBG:    {&(RES0__INSTANCE0.MY_BAD_FIFO.BUFFER.value.table[874]), INT_ENUM},*)
(*DBG:    {&(RES0__INSTANCE0.MY_BAD_FIFO.BUFFER.value.table[875]), INT_ENUM},*)
(*DBG:    {&(RES0__INSTANCE0.MY_BAD_FIFO.BUFFER.value.table[876]), INT_ENUM},*)
(*DBG:    {&(RES0__INSTANCE0.MY_BAD_FIFO.BUFFER.value.table[877]), INT_ENUM},*)
(*DBG:    {&(RES0__INSTANCE0.MY_BAD_FIFO.BUFFER.value.table[878]), INT_ENUM},*)
(*DBG:    {&(RES0__INSTANCE0.MY_BAD_FIFO.BUFFER.value.table[879]), INT_ENUM},*)
(*DBG:    {&(RES0__INSTANCE0.MY_BAD_FIFO.BUFFER.value.table[880]), INT_ENUM},*)
(*DBG:    {&(RES0__INSTANCE0.MY_BAD_FIFO.BUFFER.value.table[881]), INT_ENUM},*)
(*DBG:    {&(RES0__INSTANCE0.MY_BAD_FIFO.BUFFER.value.table[882]), INT_ENUM},*)
(*DBG:    {&(RES0__INSTANCE0.MY_BAD_FIFO.BUFFER.value.table[883]), INT_ENUM},*)
(*DBG:    {&(RES0__INSTANCE0.MY_BAD_FIFO.BUFFER.value.table[884]), INT_ENUM},*)
(*DBG:    {&(RES0__INSTANCE0.MY_BAD_FIFO.BUFFER.value.table[885]), INT_ENUM},*)
(*DBG:    {&(RES0__INSTANCE0.MY_BAD_FIFO.BUFFER.value.table[886]), INT_ENUM},*)
(*DBG:    {&(RES0__INSTANCE0.MY_BAD_FIFO.BUFFER.value.table[887]), INT_ENUM},*)
(*DBG:    {&(RES0__INSTANCE0.MY_BAD_FIFO.BUFFER.value.table[888]), INT_ENUM},*)
(*DBG:    {&(RES0__INSTANCE0.MY_BAD_FIFO.BUFFER.value.table[889]), INT_ENUM},*)
(*DBG:    {&(RES0__INSTANCE0.MY_BAD_FIFO.BUFFER.value.table[890]), INT_ENUM},*)
(*DBG:    {&(RES0__INSTANCE0.MY_BAD_FIFO.BUFFER.value.table[891]), INT_ENUM},*)
(*DBG:    {&(RES0__INSTANCE0.MY_BAD_FIFO.BUFFER.value.table[892]), INT_ENUM},*)
(*DBG:    {&(RES0__INSTANCE0.MY_BAD_FIFO.BUFFER.value.table[893]), INT_ENUM},*)
(*DBG:    {&(RES0__INSTANCE0.MY_BAD_FIFO.BUFFER.value.table[894]), INT_ENUM},*)
(*DBG:    {&(RES0__INSTANCE0.MY_BAD_FIFO.BUFFER.value.table[895]), INT_ENUM},*)
(*DBG:    {&(RES0__INSTANCE0.MY_BAD_FIFO.BUFFER.value.table[896]), INT_ENUM},*)
(*DBG:    {&(RES0__INSTANCE0.MY_BAD_FIFO.BUFFER.value.table[897]), INT_ENUM},*)
(*DBG:    {&(RES0__INSTANCE0.MY_BAD_FIFO.BUFFER.value.table[898]), INT_ENUM},*)
(*DBG:    {&(RES0__INSTANCE0.MY_BAD_FIFO.BUFFER.value.table[899]), INT_ENUM},*)
(*DBG:    {&(RES0__INSTANCE0.MY_BAD_FIFO.BUFFER.value.table[900]), INT_ENUM},*)
(*DBG:    {&(RES0__INSTANCE0.MY_BAD_FIFO.BUFFER.value.table[901]), INT_ENUM},*)
(*DBG:    {&(RES0__INSTANCE0.MY_BAD_FIFO.BUFFER.value.table[902]), INT_ENUM},*)
(*DBG:    {&(RES0__INSTANCE0.MY_BAD_FIFO.BUFFER.value.table[903]), INT_ENUM},*)
(*DBG:    {&(RES0__INSTANCE0.MY_BAD_FIFO.BUFFER.value.table[904]), INT_ENUM},*)
(*DBG:    {&(RES0__INSTANCE0.MY_BAD_FIFO.BUFFER.value.table[905]), INT_ENUM},*)
(*DBG:    {&(RES0__INSTANCE0.MY_BAD_FIFO.BUFFER.value.table[906]), INT_ENUM},*)
(*DBG:    {&(RES0__INSTANCE0.MY_BAD_FIFO.BUFFER.value.table[907]), INT_ENUM},*)
(*DBG:    {&(RES0__INSTANCE0.MY_BAD_FIFO.BUFFER.value.table[908]), INT_ENUM},*)
(*DBG:    {&(RES0__INSTANCE0.MY_BAD_FIFO.BUFFER.value.table[909]), INT_ENUM},*)
(*DBG:    {&(RES0__INSTANCE0.MY_BAD_FIFO.BUFFER.value.table[910]), INT_ENUM},*)
(*DBG:    {&(RES0__INSTANCE0.MY_BAD_FIFO.BUFFER.value.table[911]), INT_ENUM},*)
(*DBG:    {&(RES0__INSTANCE0.MY_BAD_FIFO.BUFFER.value.table[912]), INT_ENUM},*)
(*DBG:    {&(RES0__INSTANCE0.MY_BAD_FIFO.BUFFER.value.table[913]), INT_ENUM},*)
(*DBG:    {&(RES0__INSTANCE0.MY_BAD_FIFO.BUFFER.value.table[914]), INT_ENUM},*)
(*DBG:    {&(RES0__INSTANCE0.MY_BAD_FIFO.BUFFER.value.table[915]), INT_ENUM},*)
(*DBG:    {&(RES0__INSTANCE0.MY_BAD_FIFO.BUFFER.value.table[916]), INT_ENUM},*)
(*DBG:    {&(RES0__INSTANCE0.MY_BAD_FIFO.BUFFER.value.table[917]), INT_ENUM},*)
(*DBG:    {&(RES0__INSTANCE0.MY_BAD_FIFO.BUFFER.value.table[918]), INT_ENUM},*)
(*DBG:    {&(RES0__INSTANCE0.MY_BAD_FIFO.BUFFER.value.table[919]), INT_ENUM},*)
(*DBG:    {&(RES0__INSTANCE0.MY_BAD_FIFO.BUFFER.value.table[920]), INT_ENUM},*)
(*DBG:    {&(RES0__INSTANCE0.MY_BAD_FIFO.BUFFER.value.table[921]), INT_ENUM},*)
(*DBG:    {&(RES0__INSTANCE0.MY_BAD_FIFO.BUFFER.value.table[922]), INT_ENUM},*)
(*DBG:    {&(RES0__INSTANCE0.MY_BAD_FIFO.BUFFER.value.table[923]), INT_ENUM},*)
(*DBG:    {&(RES0__INSTANCE0.MY_BAD_FIFO.BUFFER.value.table[924]), INT_ENUM},*)
(*DBG:    {&(RES0__INSTANCE0.MY_BAD_FIFO.BUFFER.value.table[925]), INT_ENUM},*)
(*DBG:    {&(RES0__INSTANCE0.MY_BAD_FIFO.BUFFER.value.table[926]), INT_ENUM},*)
(*DBG:    {&(RES0__INSTANCE0.MY_BAD_FIFO.BUFFER.value.table[927]), INT_ENUM},*)
(*DBG:    {&(RES0__INSTANCE0.MY_BAD_FIFO.BUFFER.value.table[928]), INT_ENUM},*)
(*DBG:    {&(RES0__INSTANCE0.MY_BAD_FIFO.BUFFER.value.table[929]), INT_ENUM},*)
(*DBG:    {&(RES0__INSTANCE0.MY_BAD_FIFO.BUFFER.value.table[930]), INT_ENUM},*)
(*DBG:    {&(RES0__INSTANCE0.MY_BAD_FIFO.BUFFER.value.table[931]), INT_ENUM},*)
(*DBG:    {&(RES0__INSTANCE0.MY_BAD_FIFO.BUFFER.value.table[932]), INT_ENUM},*)
(*DBG:    {&(RES0__INSTANCE0.MY_BAD_FIFO.BUFFER.value.table[933]), INT_ENUM},*)
(*DBG:    {&(RES0__INSTANCE0.MY_BAD_FIFO.BUFFER.value.table[934]), INT_ENUM},*)
(*DBG:    {&(RES0__INSTANCE0.MY_BAD_FIFO.BUFFER.value.table[935]), INT_ENUM},*)
(*DBG:    {&(RES0__INSTANCE0.MY_BAD_FIFO.BUFFER.value.table[936]), INT_ENUM},*)
(*DBG:    {&(RES0__INSTANCE0.MY_BAD_FIFO.BUFFER.value.table[937]), INT_ENUM},*)
(*DBG:    {&(RES0__INSTANCE0.MY_BAD_FIFO.BUFFER.value.table[938]), INT_ENUM},*)
(*DBG:    {&(RES0__INSTANCE0.MY_BAD_FIFO.BUFFER.value.table[939]), INT_ENUM},*)
(*DBG:    {&(RES0__INSTANCE0.MY_BAD_FIFO.BUFFER.value.table[940]), INT_ENUM},*)
(*DBG:    {&(RES0__INSTANCE0.MY_BAD_FIFO.BUFFER.value.table[941]), INT_ENUM},*)
(*DBG:    {&(RES0__INSTANCE0.MY_BAD_FIFO.BUFFER.value.table[942]), INT_ENUM},*)
(*DBG:    {&(RES0__INSTANCE0.MY_BAD_FIFO.BUFFER.value.table[943]), INT_ENUM},*)
(*DBG:    {&(RES0__INSTANCE0.MY_BAD_FIFO.BUFFER.value.table[944]), INT_ENUM},*)
(*DBG:    {&(RES0__INSTANCE0.MY_BAD_FIFO.BUFFER.value.table[945]), INT_ENUM},*)
(*DBG:    {&(RES0__INSTANCE0.MY_BAD_FIFO.BUFFER.value.table[946]), INT_ENUM},*)
(*DBG:    {&(RES0__INSTANCE0.MY_BAD_FIFO.BUFFER.value.table[947]), INT_ENUM},*)
(*DBG:    {&(RES0__INSTANCE0.MY_BAD_FIFO.BUFFER.value.table[948]), INT_ENUM},*)
(*DBG:    {&(RES0__INSTANCE0.MY_BAD_FIFO.BUFFER.value.table[949]), INT_ENUM},*)
(*DBG:    {&(RES0__INSTANCE0.MY_BAD_FIFO.BUFFER.value.table[950]), INT_ENUM},*)
(*DBG:    {&(RES0__INSTANCE0.MY_BAD_FIFO.BUFFER.value.table[951]), INT_ENUM},*)
(*DBG:    {&(RES0__INSTANCE0.MY_BAD_FIFO.BUFFER.value.table[952]), INT_ENUM},*)
(*DBG:    {&(RES0__INSTANCE0.MY_BAD_FIFO.BUFFER.value.table[953]), INT_ENUM},*)
(*DBG:    {&(RES0__INSTANCE0.MY_BAD_FIFO.BUFFER.value.table[954]), INT_ENUM},*)
(*DBG:    {&(RES0__INSTANCE0.MY_BAD_FIFO.BUFFER.value.table[955]), INT_ENUM},*)
(*DBG:    {&(RES0__INSTANCE0.MY_BAD_FIFO.BUFFER.value.table[956]), INT_ENUM},*)
(*DBG:    {&(RES0__INSTANCE0.MY_BAD_FIFO.BUFFER.value.table[957]), INT_ENUM},*)
(*DBG:    {&(RES0__INSTANCE0.MY_BAD_FIFO.BUFFER.value.table[958]), INT_ENUM},*)
(*DBG:    {&(RES0__INSTANCE0.MY_BAD_FIFO.BUFFER.value.table[959]), INT_ENUM},*)
(*DBG:    {&(RES0__INSTANCE0.MY_BAD_FIFO.BUFFER.value.table[960]), INT_ENUM},*)
(*DBG:    {&(RES0__INSTANCE0.MY_BAD_FIFO.BUFFER.value.table[961]), INT_ENUM},*)
(*DBG:    {&(RES0__INSTANCE0.MY_BAD_FIFO.BUFFER.value.table[962]), INT_ENUM},*)
(*DBG:    {&(RES0__INSTANCE0.MY_BAD_FIFO.BUFFER.value.table[963]), INT_ENUM},*)
(*DBG:    {&(RES0__INSTANCE0.MY_BAD_FIFO.BUFFER.value.table[964]), INT_ENUM},*)
(*DBG:    {&(RES0__INSTANCE0.MY_BAD_FIFO.BUFFER.value.table[965]), INT_ENUM},*)
(*DBG:    {&(RES0__INSTANCE0.MY_BAD_FIFO.BUFFER.value.table[966]), INT_ENUM},*)
(*DBG:    {&(RES0__INSTANCE0.MY_BAD_FIFO.BUFFER.value.table[967]), INT_ENUM},*)
(*DBG:    {&(RES0__INSTANCE0.MY_BAD_FIFO.BUFFER.value.table[968]), INT_ENUM},*)
(*DBG:    {&(RES0__INSTANCE0.MY_BAD_FIFO.BUFFER.value.table[969]), INT_ENUM},*)
(*DBG:    {&(RES0__INSTANCE0.MY_BAD_FIFO.BUFFER.value.table[970]), INT_ENUM},*)
(*DBG:    {&(RES0__INSTANCE0.MY_BAD_FIFO.BUFFER.value.table[971]), INT_ENUM},*)
(*DBG:    {&(RES0__INSTANCE0.MY_BAD_FIFO.BUFFER.value.table[972]), INT_ENUM},*)
(*DBG:    {&(RES0__INSTANCE0.MY_BAD_FIFO.BUFFER.value.table[973]), INT_ENUM},*)
(*DBG:    {&(RES0__INSTANCE0.MY_BAD_FIFO.BUFFER.value.table[974]), INT_ENUM},*)
(*DBG:    {&(RES0__INSTANCE0.MY_BAD_FIFO.BUFFER.value.table[975]), INT_ENUM},*)
(*DBG:    {&(RES0__INSTANCE0.MY_BAD_FIFO.BUFFER.value.table[976]), INT_ENUM},*)
(*DBG:    {&(RES0__INSTANCE0.MY_BAD_FIFO.BUFFER.value.table[977]), INT_ENUM},*)
(*DBG:    {&(RES0__INSTANCE0.MY_BAD_FIFO.BUFFER.value.table[978]), INT_ENUM},*)
(*DBG:    {&(RES0__INSTANCE0.MY_BAD_FIFO.BUFFER.value.table[979]), INT_ENUM},*)
(*DBG:    {&(RES0__INSTANCE0.MY_BAD_FIFO.BUFFER.value.table[980]), INT_ENUM},*)
(*DBG:    {&(RES0__INSTANCE0.MY_BAD_FIFO.BUFFER.value.table[981]), INT_ENUM},*)
(*DBG:    {&(RES0__INSTANCE0.MY_BAD_FIFO.BUFFER.value.table[982]), INT_ENUM},*)
(*DBG:    {&(RES0__INSTANCE0.MY_BAD_FIFO.BUFFER.value.table[983]), INT_ENUM},*)
(*DBG:    {&(RES0__INSTANCE0.MY_BAD_FIFO.BUFFER.value.table[984]), INT_ENUM},*)
(*DBG:    {&(RES0__INSTANCE0.MY_BAD_FIFO.BUFFER.value.table[985]), INT_ENUM},*)
(*DBG:    {&(RES0__INSTANCE0.MY_BAD_FIFO.BUFFER.value.table[986]), INT_ENUM},*)
(*DBG:    {&(RES0__INSTANCE0.MY_BAD_FIFO.BUFFER.value.table[987]), INT_ENUM},*)
(*DBG:    {&(RES0__INSTANCE0.MY_BAD_FIFO.BUFFER.value.table[988]), INT_ENUM},*)
(*DBG:    {&(RES0__INSTANCE0.MY_BAD_FIFO.BUFFER.value.table[989]), INT_ENUM},*)
(*DBG:    {&(RES0__INSTANCE0.MY_BAD_FIFO.BUFFER.value.table[990]), INT_ENUM},*)
(*DBG:    {&(RES0__INSTANCE0.MY_BAD_FIFO.BUFFER.value.table[991]), INT_ENUM},*)
(*DBG:    {&(RES0__INSTANCE0.MY_BAD_FIFO.BUFFER.value.table[992]), INT_ENUM},*)
(*DBG:    {&(RES0__INSTANCE0.MY_BAD_FIFO.BUFFER.value.table[993]), INT_ENUM},*)
(*DBG:    {&(RES0__INSTANCE0.MY_BAD_FIFO.BUFFER.value.table[994]), INT_ENUM},*)
(*DBG:    {&(RES0__INSTANCE0.MY_BAD_FIFO.BUFFER.value.table[995]), INT_ENUM},*)
(*DBG:    {&(RES0__INSTANCE0.MY_BAD_FIFO.BUFFER.value.table[996]), INT_ENUM},*)
(*DBG:    {&(RES0__INSTANCE0.MY_BAD_FIFO.BUFFER.value.table[997]), INT_ENUM},*)
(*DBG:    {&(RES0__INSTANCE0.MY_BAD_FIFO.BUFFER.value.table[998]), INT_ENUM},*)
(*DBG:    {&(RES0__INSTANCE0.MY_BAD_FIFO.BUFFER.value.table[999]), INT_ENUM},*)
(*DBG:    {&(RES0__INSTANCE0.MY_BAD_FIFO.BUFFER.value.table[1000]), INT_ENUM},*)
(*DBG:    {&(RES0__INSTANCE0.MY_BAD_FIFO.BUFFER.value.table[1001]), INT_ENUM},*)
(*DBG:    {&(RES0__INSTANCE0.MY_BAD_FIFO.BUFFER.value.table[1002]), INT_ENUM},*)
(*DBG:    {&(RES0__INSTANCE0.MY_BAD_FIFO.BUFFER.value.table[1003]), INT_ENUM},*)
(*DBG:    {&(RES0__INSTANCE0.MY_BAD_FIFO.BUFFER.value.table[1004]), INT_ENUM},*)
(*DBG:    {&(RES0__INSTANCE0.MY_BAD_FIFO.BUFFER.value.table[1005]), INT_ENUM},*)
(*DBG:    {&(RES0__INSTANCE0.MY_BAD_FIFO.BUFFER.value.table[1006]), INT_ENUM},*)
(*DBG:    {&(RES0__INSTANCE0.MY_BAD_FIFO.BUFFER.value.table[1007]), INT_ENUM},*)
(*DBG:    {&(RES0__INSTANCE0.MY_BAD_FIFO.BUFFER.value.table[1008]), INT_ENUM},*)
(*DBG:    {&(RES0__INSTANCE0.MY_BAD_FIFO.BUFFER.value.table[1009]), INT_ENUM},*)
(*DBG:    {&(RES0__INSTANCE0.MY_BAD_FIFO.BUFFER.value.table[1010]), INT_ENUM},*)
(*DBG:    {&(RES0__INSTANCE0.MY_BAD_FIFO.BUFFER.value.table[1011]), INT_ENUM},*)
(*DBG:    {&(RES0__INSTANCE0.MY_BAD_FIFO.BUFFER.value.table[1012]), INT_ENUM},*)
(*DBG:    {&(RES0__INSTANCE0.MY_BAD_FIFO.BUFFER.value.table[1013]), INT_ENUM},*)
(*DBG:    {&(RES0__INSTANCE0.MY_BAD_FIFO.BUFFER.value.table[1014]), INT_ENUM},*)
(*DBG:    {&(RES0__INSTANCE0.MY_BAD_FIFO.BUFFER.value.table[1015]), INT_ENUM},*)
(*DBG:    {&(RES0__INSTANCE0.MY_BAD_FIFO.BUFFER.value.table[1016]), INT_ENUM},*)
(*DBG:    {&(RES0__INSTANCE0.MY_BAD_FIFO.BUFFER.value.table[1017]), INT_ENUM},*)
(*DBG:    {&(RES0__INSTANCE0.MY_BAD_FIFO.BUFFER.value.table[1018]), INT_ENUM},*)
(*DBG:    {&(RES0__INSTANCE0.MY_BAD_FIFO.BUFFER.value.table[1019]), INT_ENUM},*)
(*DBG:    {&(RES0__INSTANCE0.MY_BAD_FIFO.BUFFER.value.table[1020]), INT_ENUM},*)
(*DBG:    {&(RES0__INSTANCE0.MY_BAD_FIFO.BUFFER.value.table[1021]), INT_ENUM},*)
(*DBG:    {&(RES0__INSTANCE0.MY_BAD_FIFO.BUFFER.value.table[1022]), INT_ENUM},*)
(*DBG:    {&(RES0__INSTANCE0.MY_BAD_FIFO.BUFFER.value.table[1023]), INT_ENUM},*)
(*DBG:    {&(RES0__INSTANCE0.MY_BAD_FIFO.BUFFER.value.table[1024]), INT_ENUM},*)
(*DBG:    {&(RES0__INSTANCE0.MY_BAD_FIFO.BUFFER.value.table[1025]), INT_ENUM},*)
(*DBG:    {&(RES0__INSTANCE0.MY_BAD_FIFO.BUFFER.value.table[1026]), INT_ENUM},*)
(*DBG:    {&(RES0__INSTANCE0.MY_BAD_FIFO.BUFFER.value.table[1027]), INT_ENUM},*)
(*DBG:    {&(RES0__INSTANCE0.MY_BAD_FIFO.BUFFER.value.table[1028]), INT_ENUM},*)
(*DBG:    {&(RES0__INSTANCE0.MY_BAD_FIFO.BUFFER.value.table[1029]), INT_ENUM},*)
(*DBG:    {&(RES0__INSTANCE0.MY_BAD_FIFO.BUFFER.value.table[1030]), INT_ENUM},*)
(*DBG:    {&(RES0__INSTANCE0.MY_BAD_FIFO.BUFFER.value.table[1031]), INT_ENUM},*)
(*DBG:    {&(RES0__INSTANCE0.MY_BAD_FIFO.BUFFER.value.table[1032]), INT_ENUM},*)
(*DBG:    {&(RES0__INSTANCE0.MY_BAD_FIFO.BUFFER.value.table[1033]), INT_ENUM},*)
(*DBG:    {&(RES0__INSTANCE0.MY_BAD_FIFO.BUFFER.value.table[1034]), INT_ENUM},*)
(*DBG:    {&(RES0__INSTANCE0.MY_BAD_FIFO.BUFFER.value.table[1035]), INT_ENUM},*)
(*DBG:    {&(RES0__INSTANCE0.MY_BAD_FIFO.BUFFER.value.table[1036]), INT_ENUM},*)
(*DBG:    {&(RES0__INSTANCE0.MY_BAD_FIFO.BUFFER.value.table[1037]), INT_ENUM},*)
(*DBG:    {&(RES0__INSTANCE0.MY_BAD_FIFO.BUFFER.value.table[1038]), INT_ENUM},*)
(*DBG:    {&(RES0__INSTANCE0.MY_BAD_FIFO.BUFFER.value.table[1039]), INT_ENUM},*)
(*DBG:    {&(RES0__INSTANCE0.MY_BAD_FIFO.BUFFER.value.table[1040]), INT_ENUM},*)
(*DBG:    {&(RES0__INSTANCE0.MY_BAD_FIFO.BUFFER.value.table[1041]), INT_ENUM},*)
(*DBG:    {&(RES0__INSTANCE0.MY_BAD_FIFO.BUFFER.value.table[1042]), INT_ENUM},*)
(*DBG:    {&(RES0__INSTANCE0.MY_BAD_FIFO.BUFFER.value.table[1043]), INT_ENUM},*)
(*DBG:    {&(RES0__INSTANCE0.MY_BAD_FIFO.BUFFER.value.table[1044]), INT_ENUM},*)
(*DBG:    {&(RES0__INSTANCE0.MY_BAD_FIFO.BUFFER.value.table[1045]), INT_ENUM},*)
(*DBG:    {&(RES0__INSTANCE0.MY_BAD_FIFO.BUFFER.value.table[1046]), INT_ENUM},*)
(*DBG:    {&(RES0__INSTANCE0.MY_BAD_FIFO.BUFFER.value.table[1047]), INT_ENUM},*)
(*DBG:    {&(RES0__INSTANCE0.MY_BAD_FIFO.BUFFER.value.table[1048]), INT_ENUM},*)
(*DBG:    {&(RES0__INSTANCE0.MY_BAD_FIFO.BUFFER.value.table[1049]), INT_ENUM},*)
(*DBG:    {&(RES0__INSTANCE0.MY_BAD_FIFO.BUFFER.value.table[1050]), INT_ENUM},*)
(*DBG:    {&(RES0__INSTANCE0.MY_BAD_FIFO.BUFFER.value.table[1051]), INT_ENUM},*)
(*DBG:    {&(RES0__INSTANCE0.MY_BAD_FIFO.BUFFER.value.table[1052]), INT_ENUM},*)
(*DBG:    {&(RES0__INSTANCE0.MY_BAD_FIFO.BUFFER.value.table[1053]), INT_ENUM},*)
(*DBG:    {&(RES0__INSTANCE0.MY_BAD_FIFO.BUFFER.value.table[1054]), INT_ENUM},*)
(*DBG:    {&(RES0__INSTANCE0.MY_BAD_FIFO.BUFFER.value.table[1055]), INT_ENUM},*)
(*DBG:    {&(RES0__INSTANCE0.MY_BAD_FIFO.BUFFER.value.table[1056]), INT_ENUM},*)
(*DBG:    {&(RES0__INSTANCE0.MY_BAD_FIFO.BUFFER.value.table[1057]), INT_ENUM},*)
(*DBG:    {&(RES0__INSTANCE0.MY_BAD_FIFO.BUFFER.value.table[1058]), INT_ENUM},*)
(*DBG:    {&(RES0__INSTANCE0.MY_BAD_FIFO.BUFFER.value.table[1059]), INT_ENUM},*)
(*DBG:    {&(RES0__INSTANCE0.MY_BAD_FIFO.BUFFER.value.table[1060]), INT_ENUM},*)
(*DBG:    {&(RES0__INSTANCE0.MY_BAD_FIFO.BUFFER.value.table[1061]), INT_ENUM},*)
(*DBG:    {&(RES0__INSTANCE0.MY_BAD_FIFO.BUFFER.value.table[1062]), INT_ENUM},*)
(*DBG:    {&(RES0__INSTANCE0.MY_BAD_FIFO.BUFFER.value.table[1063]), INT_ENUM},*)
(*DBG:    {&(RES0__INSTANCE0.MY_BAD_FIFO.BUFFER.value.table[1064]), INT_ENUM},*)
(*DBG:    {&(RES0__INSTANCE0.MY_BAD_FIFO.BUFFER.value.table[1065]), INT_ENUM},*)
(*DBG:    {&(RES0__INSTANCE0.MY_BAD_FIFO.BUFFER.value.table[1066]), INT_ENUM},*)
(*DBG:    {&(RES0__INSTANCE0.MY_BAD_FIFO.BUFFER.value.table[1067]), INT_ENUM},*)
(*DBG:    {&(RES0__INSTANCE0.MY_BAD_FIFO.BUFFER.value.table[1068]), INT_ENUM},*)
(*DBG:    {&(RES0__INSTANCE0.MY_BAD_FIFO.BUFFER.value.table[1069]), INT_ENUM},*)
(*DBG:    {&(RES0__INSTANCE0.MY_BAD_FIFO.BUFFER.value.table[1070]), INT_ENUM},*)
(*DBG:    {&(RES0__INSTANCE0.MY_BAD_FIFO.BUFFER.value.table[1071]), INT_ENUM},*)
(*DBG:    {&(RES0__INSTANCE0.MY_BAD_FIFO.BUFFER.value.table[1072]), INT_ENUM},*)
(*DBG:    {&(RES0__INSTANCE0.MY_BAD_FIFO.BUFFER.value.table[1073]), INT_ENUM},*)
(*DBG:    {&(RES0__INSTANCE0.MY_BAD_FIFO.BUFFER.value.table[1074]), INT_ENUM},*)
(*DBG:    {&(RES0__INSTANCE0.MY_BAD_FIFO.BUFFER.value.table[1075]), INT_ENUM},*)
(*DBG:    {&(RES0__INSTANCE0.MY_BAD_FIFO.BUFFER.value.table[1076]), INT_ENUM},*)
(*DBG:    {&(RES0__INSTANCE0.MY_BAD_FIFO.BUFFER.value.table[1077]), INT_ENUM},*)
(*DBG:    {&(RES0__INSTANCE0.MY_BAD_FIFO.BUFFER.value.table[1078]), INT_ENUM},*)
(*DBG:    {&(RES0__INSTANCE0.MY_BAD_FIFO.BUFFER.value.table[1079]), INT_ENUM},*)
(*DBG:    {&(RES0__INSTANCE0.MY_BAD_FIFO.BUFFER.value.table[1080]), INT_ENUM},*)
(*DBG:    {&(RES0__INSTANCE0.MY_BAD_FIFO.BUFFER.value.table[1081]), INT_ENUM},*)
(*DBG:    {&(RES0__INSTANCE0.MY_BAD_FIFO.BUFFER.value.table[1082]), INT_ENUM},*)
(*DBG:    {&(RES0__INSTANCE0.MY_BAD_FIFO.BUFFER.value.table[1083]), INT_ENUM},*)
(*DBG:    {&(RES0__INSTANCE0.MY_BAD_FIFO.BUFFER.value.table[1084]), INT_ENUM},*)
(*DBG:    {&(RES0__INSTANCE0.MY_BAD_FIFO.BUFFER.value.table[1085]), INT_ENUM},*)
(*DBG:    {&(RES0__INSTANCE0.MY_BAD_FIFO.BUFFER.value.table[1086]), INT_ENUM},*)
(*DBG:    {&(RES0__INSTANCE0.MY_BAD_FIFO.BUFFER.value.table[1087]), INT_ENUM},*)
(*DBG:    {&(RES0__INSTANCE0.MY_BAD_FIFO.BUFFER.value.table[1088]), INT_ENUM},*)
(*DBG:    {&(RES0__INSTANCE0.MY_BAD_FIFO.BUFFER.value.table[1089]), INT_ENUM},*)
(*DBG:    {&(RES0__INSTANCE0.MY_BAD_FIFO.BUFFER.value.table[1090]), INT_ENUM},*)
(*DBG:    {&(RES0__INSTANCE0.MY_BAD_FIFO.BUFFER.value.table[1091]), INT_ENUM},*)
(*DBG:    {&(RES0__INSTANCE0.MY_BAD_FIFO.BUFFER.value.table[1092]), INT_ENUM},*)
(*DBG:    {&(RES0__INSTANCE0.MY_BAD_FIFO.BUFFER.value.table[1093]), INT_ENUM},*)
(*DBG:    {&(RES0__INSTANCE0.MY_BAD_FIFO.BUFFER.value.table[1094]), INT_ENUM},*)
(*DBG:    {&(RES0__INSTANCE0.MY_BAD_FIFO.BUFFER.value.table[1095]), INT_ENUM},*)
(*DBG:    {&(RES0__INSTANCE0.MY_BAD_FIFO.BUFFER.value.table[1096]), INT_ENUM},*)
(*DBG:    {&(RES0__INSTANCE0.MY_BAD_FIFO.BUFFER.value.table[1097]), INT_ENUM},*)
(*DBG:    {&(RES0__INSTANCE0.MY_BAD_FIFO.BUFFER.value.table[1098]), INT_ENUM},*)
(*DBG:    {&(RES0__INSTANCE0.MY_BAD_FIFO.BUFFER.value.table[1099]), INT_ENUM},*)
(*DBG:    {&(RES0__INSTANCE0.MY_BAD_FIFO.BUFFER.value.table[1100]), INT_ENUM},*)
(*DBG:    {&(RES0__INSTANCE0.MY_BAD_FIFO.BUFFER.value.table[1101]), INT_ENUM},*)
(*DBG:    {&(RES0__INSTANCE0.MY_BAD_FIFO.BUFFER.value.table[1102]), INT_ENUM},*)
(*DBG:    {&(RES0__INSTANCE0.MY_BAD_FIFO.BUFFER.value.table[1103]), INT_ENUM},*)
(*DBG:    {&(RES0__INSTANCE0.MY_BAD_FIFO.BUFFER.value.table[1104]), INT_ENUM},*)
(*DBG:    {&(RES0__INSTANCE0.MY_BAD_FIFO.BUFFER.value.table[1105]), INT_ENUM},*)
(*DBG:    {&(RES0__INSTANCE0.MY_BAD_FIFO.BUFFER.value.table[1106]), INT_ENUM},*)
(*DBG:    {&(RES0__INSTANCE0.MY_BAD_FIFO.BUFFER.value.table[1107]), INT_ENUM},*)
(*DBG:    {&(RES0__INSTANCE0.MY_BAD_FIFO.BUFFER.value.table[1108]), INT_ENUM},*)
(*DBG:    {&(RES0__INSTANCE0.MY_BAD_FIFO.BUFFER.value.table[1109]), INT_ENUM},*)
(*DBG:    {&(RES0__INSTANCE0.MY_BAD_FIFO.BUFFER.value.table[1110]), INT_ENUM},*)
(*DBG:    {&(RES0__INSTANCE0.MY_BAD_FIFO.BUFFER.value.table[1111]), INT_ENUM},*)
(*DBG:    {&(RES0__INSTANCE0.MY_BAD_FIFO.BUFFER.value.table[1112]), INT_ENUM},*)
(*DBG:    {&(RES0__INSTANCE0.MY_BAD_FIFO.BUFFER.value.table[1113]), INT_ENUM},*)
(*DBG:    {&(RES0__INSTANCE0.MY_BAD_FIFO.BUFFER.value.table[1114]), INT_ENUM},*)
(*DBG:    {&(RES0__INSTANCE0.MY_BAD_FIFO.BUFFER.value.table[1115]), INT_ENUM},*)
(*DBG:    {&(RES0__INSTANCE0.MY_BAD_FIFO.BUFFER.value.table[1116]), INT_ENUM},*)
(*DBG:    {&(RES0__INSTANCE0.MY_BAD_FIFO.BUFFER.value.table[1117]), INT_ENUM},*)
(*DBG:    {&(RES0__INSTANCE0.MY_BAD_FIFO.BUFFER.value.table[1118]), INT_ENUM},*)
(*DBG:    {&(RES0__INSTANCE0.MY_BAD_FIFO.BUFFER.value.table[1119]), INT_ENUM},*)
(*DBG:    {&(RES0__INSTANCE0.MY_BAD_FIFO.BUFFER.value.table[1120]), INT_ENUM},*)
(*DBG:    {&(RES0__INSTANCE0.MY_BAD_FIFO.BUFFER.value.table[1121]), INT_ENUM},*)
(*DBG:    {&(RES0__INSTANCE0.MY_BAD_FIFO.BUFFER.value.table[1122]), INT_ENUM},*)
(*DBG:    {&(RES0__INSTANCE0.MY_BAD_FIFO.BUFFER.value.table[1123]), INT_ENUM},*)
(*DBG:    {&(RES0__INSTANCE0.MY_BAD_FIFO.BUFFER.value.table[1124]), INT_ENUM},*)
(*DBG:    {&(RES0__INSTANCE0.MY_BAD_FIFO.BUFFER.value.table[1125]), INT_ENUM},*)
(*DBG:    {&(RES0__INSTANCE0.MY_BAD_FIFO.BUFFER.value.table[1126]), INT_ENUM},*)
(*DBG:    {&(RES0__INSTANCE0.MY_BAD_FIFO.BUFFER.value.table[1127]), INT_ENUM},*)
(*DBG:    {&(RES0__INSTANCE0.MY_BAD_FIFO.BUFFER.value.table[1128]), INT_ENUM},*)
(*DBG:    {&(RES0__INSTANCE0.MY_BAD_FIFO.BUFFER.value.table[1129]), INT_ENUM},*)
(*DBG:    {&(RES0__INSTANCE0.MY_BAD_FIFO.BUFFER.value.table[1130]), INT_ENUM},*)
(*DBG:    {&(RES0__INSTANCE0.MY_BAD_FIFO.BUFFER.value.table[1131]), INT_ENUM},*)
(*DBG:    {&(RES0__INSTANCE0.MY_BAD_FIFO.BUFFER.value.table[1132]), INT_ENUM},*)
(*DBG:    {&(RES0__INSTANCE0.MY_BAD_FIFO.BUFFER.value.table[1133]), INT_ENUM},*)
(*DBG:    {&(RES0__INSTANCE0.MY_BAD_FIFO.BUFFER.value.table[1134]), INT_ENUM},*)
(*DBG:    {&(RES0__INSTANCE0.MY_BAD_FIFO.BUFFER.value.table[1135]), INT_ENUM},*)
(*DBG:    {&(RES0__INSTANCE0.MY_BAD_FIFO.BUFFER.value.table[1136]), INT_ENUM},*)
(*DBG:    {&(RES0__INSTANCE0.MY_BAD_FIFO.BUFFER.value.table[1137]), INT_ENUM},*)
(*DBG:    {&(RES0__INSTANCE0.MY_BAD_FIFO.BUFFER.value.table[1138]), INT_ENUM},*)
(*DBG:    {&(RES0__INSTANCE0.MY_BAD_FIFO.BUFFER.value.table[1139]), INT_ENUM},*)
(*DBG:    {&(RES0__INSTANCE0.MY_BAD_FIFO.BUFFER.value.table[1140]), INT_ENUM},*)
(*DBG:    {&(RES0__INSTANCE0.MY_BAD_FIFO.BUFFER.value.table[1141]), INT_ENUM},*)
(*DBG:    {&(RES0__INSTANCE0.MY_BAD_FIFO.BUFFER.value.table[1142]), INT_ENUM},*)
(*DBG:    {&(RES0__INSTANCE0.MY_BAD_FIFO.BUFFER.value.table[1143]), INT_ENUM},*)
(*DBG:    {&(RES0__INSTANCE0.MY_BAD_FIFO.BUFFER.value.table[1144]), INT_ENUM},*)
(*DBG:    {&(RES0__INSTANCE0.MY_BAD_FIFO.BUFFER.value.table[1145]), INT_ENUM},*)
(*DBG:    {&(RES0__INSTANCE0.MY_BAD_FIFO.BUFFER.value.table[1146]), INT_ENUM},*)
(*DBG:    {&(RES0__INSTANCE0.MY_BAD_FIFO.BUFFER.value.table[1147]), INT_ENUM},*)
(*DBG:    {&(RES0__INSTANCE0.MY_BAD_FIFO.BUFFER.value.table[1148]), INT_ENUM},*)
(*DBG:    {&(RES0__INSTANCE0.MY_BAD_FIFO.BUFFER.value.table[1149]), INT_ENUM},*)
(*DBG:    {&(RES0__INSTANCE0.MY_BAD_FIFO.BUFFER.value.table[1150]), INT_ENUM},*)
(*DBG:    {&(RES0__INSTANCE0.MY_BAD_FIFO.BUFFER.value.table[1151]), INT_ENUM},*)
(*DBG:    {&(RES0__INSTANCE0.MY_BAD_FIFO.BUFFER.value.table[1152]), INT_ENUM},*)
(*DBG:    {&(RES0__INSTANCE0.MY_BAD_FIFO.BUFFER.value.table[1153]), INT_ENUM},*)
(*DBG:    {&(RES0__INSTANCE0.MY_BAD_FIFO.BUFFER.value.table[1154]), INT_ENUM},*)
(*DBG:    {&(RES0__INSTANCE0.MY_BAD_FIFO.BUFFER.value.table[1155]), INT_ENUM},*)
(*DBG:    {&(RES0__INSTANCE0.MY_BAD_FIFO.BUFFER.value.table[1156]), INT_ENUM},*)
(*DBG:    {&(RES0__INSTANCE0.MY_BAD_FIFO.BUFFER.value.table[1157]), INT_ENUM},*)
(*DBG:    {&(RES0__INSTANCE0.MY_BAD_FIFO.BUFFER.value.table[1158]), INT_ENUM},*)
(*DBG:    {&(RES0__INSTANCE0.MY_BAD_FIFO.BUFFER.value.table[1159]), INT_ENUM},*)
(*DBG:    {&(RES0__INSTANCE0.MY_BAD_FIFO.BUFFER.value.table[1160]), INT_ENUM},*)
(*DBG:    {&(RES0__INSTANCE0.MY_BAD_FIFO.BUFFER.value.table[1161]), INT_ENUM},*)
(*DBG:    {&(RES0__INSTANCE0.MY_BAD_FIFO.BUFFER.value.table[1162]), INT_ENUM},*)
(*DBG:    {&(RES0__INSTANCE0.MY_BAD_FIFO.BUFFER.value.table[1163]), INT_ENUM},*)
(*DBG:    {&(RES0__INSTANCE0.MY_BAD_FIFO.BUFFER.value.table[1164]), INT_ENUM},*)
(*DBG:    {&(RES0__INSTANCE0.MY_BAD_FIFO.BUFFER.value.table[1165]), INT_ENUM},*)
(*DBG:    {&(RES0__INSTANCE0.MY_BAD_FIFO.BUFFER.value.table[1166]), INT_ENUM},*)
(*DBG:    {&(RES0__INSTANCE0.MY_BAD_FIFO.BUFFER.value.table[1167]), INT_ENUM},*)
(*DBG:    {&(RES0__INSTANCE0.MY_BAD_FIFO.BUFFER.value.table[1168]), INT_ENUM},*)
(*DBG:    {&(RES0__INSTANCE0.MY_BAD_FIFO.BUFFER.value.table[1169]), INT_ENUM},*)
(*DBG:    {&(RES0__INSTANCE0.MY_BAD_FIFO.BUFFER.value.table[1170]), INT_ENUM},*)
(*DBG:    {&(RES0__INSTANCE0.MY_BAD_FIFO.BUFFER.value.table[1171]), INT_ENUM},*)
(*DBG:    {&(RES0__INSTANCE0.MY_BAD_FIFO.BUFFER.value.table[1172]), INT_ENUM},*)
(*DBG:    {&(RES0__INSTANCE0.MY_BAD_FIFO.BUFFER.value.table[1173]), INT_ENUM},*)
(*DBG:    {&(RES0__INSTANCE0.MY_BAD_FIFO.BUFFER.value.table[1174]), INT_ENUM},*)
(*DBG:    {&(RES0__INSTANCE0.MY_BAD_FIFO.BUFFER.value.table[1175]), INT_ENUM},*)
(*DBG:    {&(RES0__INSTANCE0.MY_BAD_FIFO.BUFFER.value.table[1176]), INT_ENUM},*)
(*DBG:    {&(RES0__INSTANCE0.MY_BAD_FIFO.BUFFER.value.table[1177]), INT_ENUM},*)
(*DBG:    {&(RES0__INSTANCE0.MY_BAD_FIFO.BUFFER.value.table[1178]), INT_ENUM},*)
(*DBG:    {&(RES0__INSTANCE0.MY_BAD_FIFO.BUFFER.value.table[1179]), INT_ENUM},*)
(*DBG:    {&(RES0__INSTANCE0.MY_BAD_FIFO.BUFFER.value.table[1180]), INT_ENUM},*)
(*DBG:    {&(RES0__INSTANCE0.MY_BAD_FIFO.BUFFER.value.table[1181]), INT_ENUM},*)
(*DBG:    {&(RES0__INSTANCE0.MY_BAD_FIFO.BUFFER.value.table[1182]), INT_ENUM},*)
(*DBG:    {&(RES0__INSTANCE0.MY_BAD_FIFO.BUFFER.value.table[1183]), INT_ENUM},*)
(*DBG:    {&(RES0__INSTANCE0.MY_BAD_FIFO.BUFFER.value.table[1184]), INT_ENUM},*)
(*DBG:    {&(RES0__INSTANCE0.MY_BAD_FIFO.BUFFER.value.table[1185]), INT_ENUM},*)
(*DBG:    {&(RES0__INSTANCE0.MY_BAD_FIFO.BUFFER.value.table[1186]), INT_ENUM},*)
(*DBG:    {&(RES0__INSTANCE0.MY_BAD_FIFO.BUFFER.value.table[1187]), INT_ENUM},*)
(*DBG:    {&(RES0__INSTANCE0.MY_BAD_FIFO.BUFFER.value.table[1188]), INT_ENUM},*)
(*DBG:    {&(RES0__INSTANCE0.MY_BAD_FIFO.BUFFER.value.table[1189]), INT_ENUM},*)
(*DBG:    {&(RES0__INSTANCE0.MY_BAD_FIFO.BUFFER.value.table[1190]), INT_ENUM},*)
(*DBG:    {&(RES0__INSTANCE0.MY_BAD_FIFO.BUFFER.value.table[1191]), INT_ENUM},*)
(*DBG:    {&(RES0__INSTANCE0.MY_BAD_FIFO.BUFFER.value.table[1192]), INT_ENUM},*)
(*DBG:    {&(RES0__INSTANCE0.MY_BAD_FIFO.BUFFER.value.table[1193]), INT_ENUM},*)
(*DBG:    {&(RES0__INSTANCE0.MY_BAD_FIFO.BUFFER.value.table[1194]), INT_ENUM},*)
(*DBG:    {&(RES0__INSTANCE0.MY_BAD_FIFO.BUFFER.value.table[1195]), INT_ENUM},*)
(*DBG:    {&(RES0__INSTANCE0.MY_BAD_FIFO.BUFFER.value.table[1196]), INT_ENUM},*)
(*DBG:    {&(RES0__INSTANCE0.MY_BAD_FIFO.BUFFER.value.table[1197]), INT_ENUM},*)
(*DBG:    {&(RES0__INSTANCE0.MY_BAD_FIFO.BUFFER.value.table[1198]), INT_ENUM},*)
(*DBG:    {&(RES0__INSTANCE0.MY_BAD_FIFO.BUFFER.value.table[1199]), INT_ENUM},*)
(*DBG:    {&(RES0__INSTANCE0.MY_BAD_FIFO.BUFFER.value.table[1200]), INT_ENUM},*)
(*DBG:    {&(RES0__INSTANCE0.MY_BAD_FIFO.BUFFER.value.table[1201]), INT_ENUM},*)
(*DBG:    {&(RES0__INSTANCE0.MY_BAD_FIFO.BUFFER.value.table[1202]), INT_ENUM},*)
(*DBG:    {&(RES0__INSTANCE0.MY_BAD_FIFO.BUFFER.value.table[1203]), INT_ENUM},*)
(*DBG:    {&(RES0__INSTANCE0.MY_BAD_FIFO.BUFFER.value.table[1204]), INT_ENUM},*)
(*DBG:    {&(RES0__INSTANCE0.MY_BAD_FIFO.BUFFER.value.table[1205]), INT_ENUM},*)
(*DBG:    {&(RES0__INSTANCE0.MY_BAD_FIFO.BUFFER.value.table[1206]), INT_ENUM},*)
(*DBG:    {&(RES0__INSTANCE0.MY_BAD_FIFO.BUFFER.value.table[1207]), INT_ENUM},*)
(*DBG:    {&(RES0__INSTANCE0.MY_BAD_FIFO.BUFFER.value.table[1208]), INT_ENUM},*)
(*DBG:    {&(RES0__INSTANCE0.MY_BAD_FIFO.BUFFER.value.table[1209]), INT_ENUM},*)
(*DBG:    {&(RES0__INSTANCE0.MY_BAD_FIFO.BUFFER.value.table[1210]), INT_ENUM},*)
(*DBG:    {&(RES0__INSTANCE0.MY_BAD_FIFO.BUFFER.value.table[1211]), INT_ENUM},*)
(*DBG:    {&(RES0__INSTANCE0.MY_BAD_FIFO.BUFFER.value.table[1212]), INT_ENUM},*)
(*DBG:    {&(RES0__INSTANCE0.MY_BAD_FIFO.BUFFER.value.table[1213]), INT_ENUM},*)
(*DBG:    {&(RES0__INSTANCE0.MY_BAD_FIFO.BUFFER.value.table[1214]), INT_ENUM},*)
(*DBG:    {&(RES0__INSTANCE0.MY_BAD_FIFO.BUFFER.value.table[1215]), INT_ENUM},*)
(*DBG:    {&(RES0__INSTANCE0.MY_BAD_FIFO.BUFFER.value.table[1216]), INT_ENUM},*)
(*DBG:    {&(RES0__INSTANCE0.MY_BAD_FIFO.BUFFER.value.table[1217]), INT_ENUM},*)
(*DBG:    {&(RES0__INSTANCE0.MY_BAD_FIFO.BUFFER.value.table[1218]), INT_ENUM},*)
(*DBG:    {&(RES0__INSTANCE0.MY_BAD_FIFO.BUFFER.value.table[1219]), INT_ENUM},*)
(*DBG:    {&(RES0__INSTANCE0.MY_BAD_FIFO.BUFFER.value.table[1220]), INT_ENUM},*)
(*DBG:    {&(RES0__INSTANCE0.MY_BAD_FIFO.BUFFER.value.table[1221]), INT_ENUM},*)
(*DBG:    {&(RES0__INSTANCE0.MY_BAD_FIFO.BUFFER.value.table[1222]), INT_ENUM},*)
(*DBG:    {&(RES0__INSTANCE0.MY_BAD_FIFO.BUFFER.value.table[1223]), INT_ENUM},*)
(*DBG:    {&(RES0__INSTANCE0.MY_BAD_FIFO.BUFFER.value.table[1224]), INT_ENUM},*)
(*DBG:    {&(RES0__INSTANCE0.MY_BAD_FIFO.BUFFER.value.table[1225]), INT_ENUM},*)
(*DBG:    {&(RES0__INSTANCE0.MY_BAD_FIFO.BUFFER.value.table[1226]), INT_ENUM},*)
(*DBG:    {&(RES0__INSTANCE0.MY_BAD_FIFO.BUFFER.value.table[1227]), INT_ENUM},*)
(*DBG:    {&(RES0__INSTANCE0.MY_BAD_FIFO.BUFFER.value.table[1228]), INT_ENUM},*)
(*DBG:    {&(RES0__INSTANCE0.MY_BAD_FIFO.BUFFER.value.table[1229]), INT_ENUM},*)
(*DBG:    {&(RES0__INSTANCE0.MY_BAD_FIFO.BUFFER.value.table[1230]), INT_ENUM},*)
(*DBG:    {&(RES0__INSTANCE0.MY_BAD_FIFO.BUFFER.value.table[1231]), INT_ENUM},*)
(*DBG:    {&(RES0__INSTANCE0.MY_BAD_FIFO.BUFFER.value.table[1232]), INT_ENUM},*)
(*DBG:    {&(RES0__INSTANCE0.MY_BAD_FIFO.BUFFER.value.table[1233]), INT_ENUM},*)
(*DBG:    {&(RES0__INSTANCE0.MY_BAD_FIFO.BUFFER.value.table[1234]), INT_ENUM},*)
(*DBG:    {&(RES0__INSTANCE0.MY_BAD_FIFO.BUFFER.value.table[1235]), INT_ENUM},*)
(*DBG:    {&(RES0__INSTANCE0.MY_BAD_FIFO.BUFFER.value.table[1236]), INT_ENUM},*)
(*DBG:    {&(RES0__INSTANCE0.MY_BAD_FIFO.BUFFER.value.table[1237]), INT_ENUM},*)
(*DBG:    {&(RES0__INSTANCE0.MY_BAD_FIFO.BUFFER.value.table[1238]), INT_ENUM},*)
(*DBG:    {&(RES0__INSTANCE0.MY_BAD_FIFO.BUFFER.value.table[1239]), INT_ENUM},*)
(*DBG:    {&(RES0__INSTANCE0.MY_BAD_FIFO.BUFFER.value.table[1240]), INT_ENUM},*)
(*DBG:    {&(RES0__INSTANCE0.MY_BAD_FIFO.BUFFER.value.table[1241]), INT_ENUM},*)
(*DBG:    {&(RES0__INSTANCE0.MY_BAD_FIFO.BUFFER.value.table[1242]), INT_ENUM},*)
(*DBG:    {&(RES0__INSTANCE0.MY_BAD_FIFO.BUFFER.value.table[1243]), INT_ENUM},*)
(*DBG:    {&(RES0__INSTANCE0.MY_BAD_FIFO.BUFFER.value.table[1244]), INT_ENUM},*)
(*DBG:    {&(RES0__INSTANCE0.MY_BAD_FIFO.BUFFER.value.table[1245]), INT_ENUM},*)
(*DBG:    {&(RES0__INSTANCE0.MY_BAD_FIFO.BUFFER.value.table[1246]), INT_ENUM},*)
(*DBG:    {&(RES0__INSTANCE0.MY_BAD_FIFO.BUFFER.value.table[1247]), INT_ENUM},*)
(*DBG:    {&(RES0__INSTANCE0.MY_BAD_FIFO.BUFFER.value.table[1248]), INT_ENUM},*)
(*DBG:    {&(RES0__INSTANCE0.MY_BAD_FIFO.BUFFER.value.table[1249]), INT_ENUM},*)
(*DBG:    {&(RES0__INSTANCE0.MY_BAD_FIFO.BUFFER.value.table[1250]), INT_ENUM},*)
(*DBG:    {&(RES0__INSTANCE0.MY_BAD_FIFO.BUFFER.value.table[1251]), INT_ENUM},*)
(*DBG:    {&(RES0__INSTANCE0.MY_BAD_FIFO.BUFFER.value.table[1252]), INT_ENUM},*)
(*DBG:    {&(RES0__INSTANCE0.MY_BAD_FIFO.BUFFER.value.table[1253]), INT_ENUM},*)
(*DBG:    {&(RES0__INSTANCE0.MY_BAD_FIFO.BUFFER.value.table[1254]), INT_ENUM},*)
(*DBG:    {&(RES0__INSTANCE0.MY_BAD_FIFO.BUFFER.value.table[1255]), INT_ENUM},*)
(*DBG:    {&(RES0__INSTANCE0.MY_BAD_FIFO.BUFFER.value.table[1256]), INT_ENUM},*)
(*DBG:    {&(RES0__INSTANCE0.MY_BAD_FIFO.BUFFER.value.table[1257]), INT_ENUM},*)
(*DBG:    {&(RES0__INSTANCE0.MY_BAD_FIFO.BUFFER.value.table[1258]), INT_ENUM},*)
(*DBG:    {&(RES0__INSTANCE0.MY_BAD_FIFO.BUFFER.value.table[1259]), INT_ENUM},*)
(*DBG:    {&(RES0__INSTANCE0.MY_BAD_FIFO.BUFFER.value.table[1260]), INT_ENUM},*)
(*DBG:    {&(RES0__INSTANCE0.MY_BAD_FIFO.BUFFER.value.table[1261]), INT_ENUM},*)
(*DBG:    {&(RES0__INSTANCE0.MY_BAD_FIFO.BUFFER.value.table[1262]), INT_ENUM},*)
(*DBG:    {&(RES0__INSTANCE0.MY_BAD_FIFO.BUFFER.value.table[1263]), INT_ENUM},*)
(*DBG:    {&(RES0__INSTANCE0.MY_BAD_FIFO.BUFFER.value.table[1264]), INT_ENUM},*)
(*DBG:    {&(RES0__INSTANCE0.MY_BAD_FIFO.BUFFER.value.table[1265]), INT_ENUM},*)
(*DBG:    {&(RES0__INSTANCE0.MY_BAD_FIFO.BUFFER.value.table[1266]), INT_ENUM},*)
(*DBG:    {&(RES0__INSTANCE0.MY_BAD_FIFO.BUFFER.value.table[1267]), INT_ENUM},*)
(*DBG:    {&(RES0__INSTANCE0.MY_BAD_FIFO.BUFFER.value.table[1268]), INT_ENUM},*)
(*DBG:    {&(RES0__INSTANCE0.MY_BAD_FIFO.BUFFER.value.table[1269]), INT_ENUM},*)
(*DBG:    {&(RES0__INSTANCE0.MY_BAD_FIFO.BUFFER.value.table[1270]), INT_ENUM},*)
(*DBG:    {&(RES0__INSTANCE0.MY_BAD_FIFO.BUFFER.value.table[1271]), INT_ENUM},*)
(*DBG:    {&(RES0__INSTANCE0.MY_BAD_FIFO.BUFFER.value.table[1272]), INT_ENUM},*)
(*DBG:    {&(RES0__INSTANCE0.MY_BAD_FIFO.BUFFER.value.table[1273]), INT_ENUM},*)
(*DBG:    {&(RES0__INSTANCE0.MY_BAD_FIFO.BUFFER.value.table[1274]), INT_ENUM},*)
(*DBG:    {&(RES0__INSTANCE0.MY_BAD_FIFO.BUFFER.value.table[1275]), INT_ENUM},*)
(*DBG:    {&(RES0__INSTANCE0.MY_BAD_FIFO.BUFFER.value.table[1276]), INT_ENUM},*)
(*DBG:    {&(RES0__INSTANCE0.MY_BAD_FIFO.BUFFER.value.table[1277]), INT_ENUM},*)
(*DBG:    {&(RES0__INSTANCE0.MY_BAD_FIFO.BUFFER.value.table[1278]), INT_ENUM},*)
(*DBG:    {&(RES0__INSTANCE0.MY_BAD_FIFO.BUFFER.value.table[1279]), INT_ENUM},*)
(*DBG:    {&(RES0__INSTANCE0.MY_BAD_FIFO.BUFFER.value.table[1280]), INT_ENUM},*)
(*DBG:    {&(RES0__INSTANCE0.MY_BAD_FIFO.BUFFER.value.table[1281]), INT_ENUM},*)
(*DBG:    {&(RES0__INSTANCE0.MY_BAD_FIFO.BUFFER.value.table[1282]), INT_ENUM},*)
(*DBG:    {&(RES0__INSTANCE0.MY_BAD_FIFO.BUFFER.value.table[1283]), INT_ENUM},*)
(*DBG:    {&(RES0__INSTANCE0.MY_BAD_FIFO.BUFFER.value.table[1284]), INT_ENUM},*)
(*DBG:    {&(RES0__INSTANCE0.MY_BAD_FIFO.BUFFER.value.table[1285]), INT_ENUM},*)
(*DBG:    {&(RES0__INSTANCE0.MY_BAD_FIFO.BUFFER.value.table[1286]), INT_ENUM},*)
(*DBG:    {&(RES0__INSTANCE0.MY_BAD_FIFO.BUFFER.value.table[1287]), INT_ENUM},*)
(*DBG:    {&(RES0__INSTANCE0.MY_BAD_FIFO.BUFFER.value.table[1288]), INT_ENUM},*)
(*DBG:    {&(RES0__INSTANCE0.MY_BAD_FIFO.BUFFER.value.table[1289]), INT_ENUM},*)
(*DBG:    {&(RES0__INSTANCE0.MY_BAD_FIFO.BUFFER.value.table[1290]), INT_ENUM},*)
(*DBG:    {&(RES0__INSTANCE0.MY_BAD_FIFO.BUFFER.value.table[1291]), INT_ENUM},*)
(*DBG:    {&(RES0__INSTANCE0.MY_BAD_FIFO.BUFFER.value.table[1292]), INT_ENUM},*)
(*DBG:    {&(RES0__INSTANCE0.MY_BAD_FIFO.BUFFER.value.table[1293]), INT_ENUM},*)
(*DBG:    {&(RES0__INSTANCE0.MY_BAD_FIFO.BUFFER.value.table[1294]), INT_ENUM},*)
(*DBG:    {&(RES0__INSTANCE0.MY_BAD_FIFO.BUFFER.value.table[1295]), INT_ENUM},*)
(*DBG:    {&(RES0__INSTANCE0.MY_BAD_FIFO.BUFFER.value.table[1296]), INT_ENUM},*)
(*DBG:    {&(RES0__INSTANCE0.MY_BAD_FIFO.BUFFER.value.table[1297]), INT_ENUM},*)
(*DBG:    {&(RES0__INSTANCE0.MY_BAD_FIFO.BUFFER.value.table[1298]), INT_ENUM},*)
(*DBG:    {&(RES0__INSTANCE0.MY_BAD_FIFO.BUFFER.value.table[1299]), INT_ENUM},*)
(*DBG:    {&(RES0__INSTANCE0.MY_BAD_FIFO.BUFFER.value.table[1300]), INT_ENUM},*)
(*DBG:    {&(RES0__INSTANCE0.MY_BAD_FIFO.BUFFER.value.table[1301]), INT_ENUM},*)
(*DBG:    {&(RES0__INSTANCE0.MY_BAD_FIFO.BUFFER.value.table[1302]), INT_ENUM},*)
(*DBG:    {&(RES0__INSTANCE0.MY_BAD_FIFO.BUFFER.value.table[1303]), INT_ENUM},*)
(*DBG:    {&(RES0__INSTANCE0.MY_BAD_FIFO.BUFFER.value.table[1304]), INT_ENUM},*)
(*DBG:    {&(RES0__INSTANCE0.MY_BAD_FIFO.BUFFER.value.table[1305]), INT_ENUM},*)
(*DBG:    {&(RES0__INSTANCE0.MY_BAD_FIFO.BUFFER.value.table[1306]), INT_ENUM},*)
(*DBG:    {&(RES0__INSTANCE0.MY_BAD_FIFO.BUFFER.value.table[1307]), INT_ENUM},*)
(*DBG:    {&(RES0__INSTANCE0.MY_BAD_FIFO.BUFFER.value.table[1308]), INT_ENUM},*)
(*DBG:    {&(RES0__INSTANCE0.MY_BAD_FIFO.BUFFER.value.table[1309]), INT_ENUM},*)
(*DBG:    {&(RES0__INSTANCE0.MY_BAD_FIFO.BUFFER.value.table[1310]), INT_ENUM},*)
(*DBG:    {&(RES0__INSTANCE0.MY_BAD_FIFO.BUFFER.value.table[1311]), INT_ENUM},*)
(*DBG:    {&(RES0__INSTANCE0.MY_BAD_FIFO.BUFFER.value.table[1312]), INT_ENUM},*)
(*DBG:    {&(RES0__INSTANCE0.MY_BAD_FIFO.BUFFER.value.table[1313]), INT_ENUM},*)
(*DBG:    {&(RES0__INSTANCE0.MY_BAD_FIFO.BUFFER.value.table[1314]), INT_ENUM},*)
(*DBG:    {&(RES0__INSTANCE0.MY_BAD_FIFO.BUFFER.value.table[1315]), INT_ENUM},*)
(*DBG:    {&(RES0__INSTANCE0.MY_BAD_FIFO.BUFFER.value.table[1316]), INT_ENUM},*)
(*DBG:    {&(RES0__INSTANCE0.MY_BAD_FIFO.BUFFER.value.table[1317]), INT_ENUM},*)
(*DBG:    {&(RES0__INSTANCE0.MY_BAD_FIFO.BUFFER.value.table[1318]), INT_ENUM},*)
(*DBG:    {&(RES0__INSTANCE0.MY_BAD_FIFO.BUFFER.value.table[1319]), INT_ENUM},*)
(*DBG:    {&(RES0__INSTANCE0.MY_BAD_FIFO.BUFFER.value.table[1320]), INT_ENUM},*)
(*DBG:    {&(RES0__INSTANCE0.MY_BAD_FIFO.BUFFER.value.table[1321]), INT_ENUM},*)
(*DBG:    {&(RES0__INSTANCE0.MY_BAD_FIFO.BUFFER.value.table[1322]), INT_ENUM},*)
(*DBG:    {&(RES0__INSTANCE0.MY_BAD_FIFO.BUFFER.value.table[1323]), INT_ENUM},*)
(*DBG:    {&(RES0__INSTANCE0.MY_BAD_FIFO.BUFFER.value.table[1324]), INT_ENUM},*)
(*DBG:    {&(RES0__INSTANCE0.MY_BAD_FIFO.BUFFER.value.table[1325]), INT_ENUM},*)
(*DBG:    {&(RES0__INSTANCE0.MY_BAD_FIFO.BUFFER.value.table[1326]), INT_ENUM},*)
(*DBG:    {&(RES0__INSTANCE0.MY_BAD_FIFO.BUFFER.value.table[1327]), INT_ENUM},*)
(*DBG:    {&(RES0__INSTANCE0.MY_BAD_FIFO.BUFFER.value.table[1328]), INT_ENUM},*)
(*DBG:    {&(RES0__INSTANCE0.MY_BAD_FIFO.BUFFER.value.table[1329]), INT_ENUM},*)
(*DBG:    {&(RES0__INSTANCE0.MY_BAD_FIFO.BUFFER.value.table[1330]), INT_ENUM},*)
(*DBG:    {&(RES0__INSTANCE0.MY_BAD_FIFO.BUFFER.value.table[1331]), INT_ENUM},*)
(*DBG:    {&(RES0__INSTANCE0.MY_BAD_FIFO.BUFFER.value.table[1332]), INT_ENUM},*)
(*DBG:    {&(RES0__INSTANCE0.MY_BAD_FIFO.BUFFER.value.table[1333]), INT_ENUM},*)
(*DBG:    {&(RES0__INSTANCE0.MY_BAD_FIFO.BUFFER.value.table[1334]), INT_ENUM},*)
(*DBG:    {&(RES0__INSTANCE0.MY_BAD_FIFO.BUFFER.value.table[1335]), INT_ENUM},*)
(*DBG:    {&(RES0__INSTANCE0.MY_BAD_FIFO.BUFFER.value.table[1336]), INT_ENUM},*)
(*DBG:    {&(RES0__INSTANCE0.MY_BAD_FIFO.BUFFER.value.table[1337]), INT_ENUM},*)
(*DBG:    {&(RES0__INSTANCE0.MY_BAD_FIFO.BUFFER.value.table[1338]), INT_ENUM},*)
(*DBG:    {&(RES0__INSTANCE0.MY_BAD_FIFO.BUFFER.value.table[1339]), INT_ENUM},*)
(*DBG:    {&(RES0__INSTANCE0.MY_BAD_FIFO.BUFFER.value.table[1340]), INT_ENUM},*)
(*DBG:    {&(RES0__INSTANCE0.MY_BAD_FIFO.BUFFER.value.table[1341]), INT_ENUM},*)
(*DBG:    {&(RES0__INSTANCE0.MY_BAD_FIFO.BUFFER.value.table[1342]), INT_ENUM},*)
(*DBG:    {&(RES0__INSTANCE0.MY_BAD_FIFO.BUFFER.value.table[1343]), INT_ENUM},*)
(*DBG:    {&(RES0__INSTANCE0.MY_BAD_FIFO.BUFFER.value.table[1344]), INT_ENUM},*)
(*DBG:    {&(RES0__INSTANCE0.MY_BAD_FIFO.BUFFER.value.table[1345]), INT_ENUM},*)
(*DBG:    {&(RES0__INSTANCE0.MY_BAD_FIFO.BUFFER.value.table[1346]), INT_ENUM},*)
(*DBG:    {&(RES0__INSTANCE0.MY_BAD_FIFO.BUFFER.value.table[1347]), INT_ENUM},*)
(*DBG:    {&(RES0__INSTANCE0.MY_BAD_FIFO.BUFFER.value.table[1348]), INT_ENUM},*)
(*DBG:    {&(RES0__INSTANCE0.MY_BAD_FIFO.BUFFER.value.table[1349]), INT_ENUM},*)
(*DBG:    {&(RES0__INSTANCE0.MY_BAD_FIFO.BUFFER.value.table[1350]), INT_ENUM},*)
(*DBG:    {&(RES0__INSTANCE0.MY_BAD_FIFO.BUFFER.value.table[1351]), INT_ENUM},*)
(*DBG:    {&(RES0__INSTANCE0.MY_BAD_FIFO.BUFFER.value.table[1352]), INT_ENUM},*)
(*DBG:    {&(RES0__INSTANCE0.MY_BAD_FIFO.BUFFER.value.table[1353]), INT_ENUM},*)
(*DBG:    {&(RES0__INSTANCE0.MY_BAD_FIFO.BUFFER.value.table[1354]), INT_ENUM},*)
(*DBG:    {&(RES0__INSTANCE0.MY_BAD_FIFO.BUFFER.value.table[1355]), INT_ENUM},*)
(*DBG:    {&(RES0__INSTANCE0.MY_BAD_FIFO.BUFFER.value.table[1356]), INT_ENUM},*)
(*DBG:    {&(RES0__INSTANCE0.MY_BAD_FIFO.BUFFER.value.table[1357]), INT_ENUM},*)
(*DBG:    {&(RES0__INSTANCE0.MY_BAD_FIFO.BUFFER.value.table[1358]), INT_ENUM},*)
(*DBG:    {&(RES0__INSTANCE0.MY_BAD_FIFO.BUFFER.value.table[1359]), INT_ENUM},*)
(*DBG:    {&(RES0__INSTANCE0.MY_BAD_FIFO.BUFFER.value.table[1360]), INT_ENUM},*)
(*DBG:    {&(RES0__INSTANCE0.MY_BAD_FIFO.BUFFER.value.table[1361]), INT_ENUM},*)
(*DBG:    {&(RES0__INSTANCE0.MY_BAD_FIFO.BUFFER.value.table[1362]), INT_ENUM},*)
(*DBG:    {&(RES0__INSTANCE0.MY_BAD_FIFO.BUFFER.value.table[1363]), INT_ENUM},*)
(*DBG:    {&(RES0__INSTANCE0.MY_BAD_FIFO.BUFFER.value.table[1364]), INT_ENUM},*)
(*DBG:    {&(RES0__INSTANCE0.MY_BAD_FIFO.BUFFER.value.table[1365]), INT_ENUM},*)
(*DBG:    {&(RES0__INSTANCE0.MY_BAD_FIFO.BUFFER.value.table[1366]), INT_ENUM},*)
(*DBG:    {&(RES0__INSTANCE0.MY_BAD_FIFO.BUFFER.value.table[1367]), INT_ENUM},*)
(*DBG:    {&(RES0__INSTANCE0.MY_BAD_FIFO.BUFFER.value.table[1368]), INT_ENUM},*)
(*DBG:    {&(RES0__INSTANCE0.MY_BAD_FIFO.BUFFER.value.table[1369]), INT_ENUM},*)
(*DBG:    {&(RES0__INSTANCE0.MY_BAD_FIFO.BUFFER.value.table[1370]), INT_ENUM},*)
(*DBG:    {&(RES0__INSTANCE0.MY_BAD_FIFO.BUFFER.value.table[1371]), INT_ENUM},*)
(*DBG:    {&(RES0__INSTANCE0.MY_BAD_FIFO.BUFFER.value.table[1372]), INT_ENUM},*)
(*DBG:    {&(RES0__INSTANCE0.MY_BAD_FIFO.BUFFER.value.table[1373]), INT_ENUM},*)
(*DBG:    {&(RES0__INSTANCE0.MY_BAD_FIFO.BUFFER.value.table[1374]), INT_ENUM},*)
(*DBG:    {&(RES0__INSTANCE0.MY_BAD_FIFO.BUFFER.value.table[1375]), INT_ENUM},*)
(*DBG:    {&(RES0__INSTANCE0.MY_BAD_FIFO.BUFFER.value.table[1376]), INT_ENUM},*)
(*DBG:    {&(RES0__INSTANCE0.MY_BAD_FIFO.BUFFER.value.table[1377]), INT_ENUM},*)
(*DBG:    {&(RES0__INSTANCE0.MY_BAD_FIFO.BUFFER.value.table[1378]), INT_ENUM},*)
(*DBG:    {&(RES0__INSTANCE0.MY_BAD_FIFO.BUFFER.value.table[1379]), INT_ENUM},*)
(*DBG:    {&(RES0__INSTANCE0.MY_BAD_FIFO.BUFFER.value.table[1380]), INT_ENUM},*)
(*DBG:    {&(RES0__INSTANCE0.MY_BAD_FIFO.BUFFER.value.table[1381]), INT_ENUM},*)
(*DBG:    {&(RES0__INSTANCE0.MY_BAD_FIFO.BUFFER.value.table[1382]), INT_ENUM},*)
(*DBG:    {&(RES0__INSTANCE0.MY_BAD_FIFO.BUFFER.value.table[1383]), INT_ENUM},*)
(*DBG:    {&(RES0__INSTANCE0.MY_BAD_FIFO.BUFFER.value.table[1384]), INT_ENUM},*)
(*DBG:    {&(RES0__INSTANCE0.MY_BAD_FIFO.BUFFER.value.table[1385]), INT_ENUM},*)
(*DBG:    {&(RES0__INSTANCE0.MY_BAD_FIFO.BUFFER.value.table[1386]), INT_ENUM},*)
(*DBG:    {&(RES0__INSTANCE0.MY_BAD_FIFO.BUFFER.value.table[1387]), INT_ENUM},*)
(*DBG:    {&(RES0__INSTANCE0.MY_BAD_FIFO.BUFFER.value.table[1388]), INT_ENUM},*)
(*DBG:    {&(RES0__INSTANCE0.MY_BAD_FIFO.BUFFER.value.table[1389]), INT_ENUM},*)
(*DBG:    {&(RES0__INSTANCE0.MY_BAD_FIFO.BUFFER.value.table[1390]), INT_ENUM},*)
(*DBG:    {&(RES0__INSTANCE0.MY_BAD_FIFO.BUFFER.value.table[1391]), INT_ENUM},*)
(*DBG:    {&(RES0__INSTANCE0.MY_BAD_FIFO.BUFFER.value.table[1392]), INT_ENUM},*)
(*DBG:    {&(RES0__INSTANCE0.MY_BAD_FIFO.BUFFER.value.table[1393]), INT_ENUM},*)
(*DBG:    {&(RES0__INSTANCE0.MY_BAD_FIFO.BUFFER.value.table[1394]), INT_ENUM},*)
(*DBG:    {&(RES0__INSTANCE0.MY_BAD_FIFO.BUFFER.value.table[1395]), INT_ENUM},*)
(*DBG:    {&(RES0__INSTANCE0.MY_BAD_FIFO.BUFFER.value.table[1396]), INT_ENUM},*)
(*DBG:    {&(RES0__INSTANCE0.MY_BAD_FIFO.BUFFER.value.table[1397]), INT_ENUM},*)
(*DBG:    {&(RES0__INSTANCE0.MY_BAD_FIFO.BUFFER.value.table[1398]), INT_ENUM},*)
(*DBG:    {&(RES0__INSTANCE0.MY_BAD_FIFO.BUFFER.value.table[1399]), INT_ENUM},*)
(*DBG:    {&(RES0__INSTANCE0.MY_BAD_FIFO.BUFFER.value.table[1400]), INT_ENUM},*)
(*DBG:    {&(RES0__INSTANCE0.MY_BAD_FIFO.BUFFER.value.table[1401]), INT_ENUM},*)
(*DBG:    {&(RES0__INSTANCE0.MY_BAD_FIFO.BUFFER.value.table[1402]), INT_ENUM},*)
(*DBG:    {&(RES0__INSTANCE0.MY_BAD_FIFO.BUFFER.value.table[1403]), INT_ENUM},*)
(*DBG:    {&(RES0__INSTANCE0.MY_BAD_FIFO.BUFFER.value.table[1404]), INT_ENUM},*)
(*DBG:    {&(RES0__INSTANCE0.MY_BAD_FIFO.BUFFER.value.table[1405]), INT_ENUM},*)
(*DBG:    {&(RES0__INSTANCE0.MY_BAD_FIFO.BUFFER.value.table[1406]), INT_ENUM},*)
(*DBG:    {&(RES0__INSTANCE0.MY_BAD_FIFO.BUFFER.value.table[1407]), INT_ENUM},*)
(*DBG:    {&(RES0__INSTANCE0.MY_BAD_FIFO.BUFFER.value.table[1408]), INT_ENUM},*)
(*DBG:    {&(RES0__INSTANCE0.MY_BAD_FIFO.BUFFER.value.table[1409]), INT_ENUM},*)
(*DBG:    {&(RES0__INSTANCE0.MY_BAD_FIFO.BUFFER.value.table[1410]), INT_ENUM},*)
(*DBG:    {&(RES0__INSTANCE0.MY_BAD_FIFO.BUFFER.value.table[1411]), INT_ENUM},*)
(*DBG:    {&(RES0__INSTANCE0.MY_BAD_FIFO.BUFFER.value.table[1412]), INT_ENUM},*)
(*DBG:    {&(RES0__INSTANCE0.MY_BAD_FIFO.BUFFER.value.table[1413]), INT_ENUM},*)
(*DBG:    {&(RES0__INSTANCE0.MY_BAD_FIFO.BUFFER.value.table[1414]), INT_ENUM},*)
(*DBG:    {&(RES0__INSTANCE0.MY_BAD_FIFO.BUFFER.value.table[1415]), INT_ENUM},*)
(*DBG:    {&(RES0__INSTANCE0.MY_BAD_FIFO.BUFFER.value.table[1416]), INT_ENUM},*)
(*DBG:    {&(RES0__INSTANCE0.MY_BAD_FIFO.BUFFER.value.table[1417]), INT_ENUM},*)
(*DBG:    {&(RES0__INSTANCE0.MY_BAD_FIFO.BUFFER.value.table[1418]), INT_ENUM},*)
(*DBG:    {&(RES0__INSTANCE0.MY_BAD_FIFO.BUFFER.value.table[1419]), INT_ENUM},*)
(*DBG:    {&(RES0__INSTANCE0.MY_BAD_FIFO.BUFFER.value.table[1420]), INT_ENUM},*)
(*DBG:    {&(RES0__INSTANCE0.MY_BAD_FIFO.BUFFER.value.table[1421]), INT_ENUM},*)
(*DBG:    {&(RES0__INSTANCE0.MY_BAD_FIFO.BUFFER.value.table[1422]), INT_ENUM},*)
(*DBG:    {&(RES0__INSTANCE0.MY_BAD_FIFO.BUFFER.value.table[1423]), INT_ENUM},*)
(*DBG:    {&(RES0__INSTANCE0.MY_BAD_FIFO.BUFFER.value.table[1424]), INT_ENUM},*)
(*DBG:    {&(RES0__INSTANCE0.MY_BAD_FIFO.BUFFER.value.table[1425]), INT_ENUM},*)
(*DBG:    {&(RES0__INSTANCE0.MY_BAD_FIFO.BUFFER.value.table[1426]), INT_ENUM},*)
(*DBG:    {&(RES0__INSTANCE0.MY_BAD_FIFO.BUFFER.value.table[1427]), INT_ENUM},*)
(*DBG:    {&(RES0__INSTANCE0.MY_BAD_FIFO.BUFFER.value.table[1428]), INT_ENUM},*)
(*DBG:    {&(RES0__INSTANCE0.MY_BAD_FIFO.BUFFER.value.table[1429]), INT_ENUM},*)
(*DBG:    {&(RES0__INSTANCE0.MY_BAD_FIFO.BUFFER.value.table[1430]), INT_ENUM},*)
(*DBG:    {&(RES0__INSTANCE0.MY_BAD_FIFO.BUFFER.value.table[1431]), INT_ENUM},*)
(*DBG:    {&(RES0__INSTANCE0.MY_BAD_FIFO.BUFFER.value.table[1432]), INT_ENUM},*)
(*DBG:    {&(RES0__INSTANCE0.MY_BAD_FIFO.BUFFER.value.table[1433]), INT_ENUM},*)
(*DBG:    {&(RES0__INSTANCE0.MY_BAD_FIFO.BUFFER.value.table[1434]), INT_ENUM},*)
(*DBG:    {&(RES0__INSTANCE0.MY_BAD_FIFO.BUFFER.value.table[1435]), INT_ENUM},*)
(*DBG:    {&(RES0__INSTANCE0.MY_BAD_FIFO.BUFFER.value.table[1436]), INT_ENUM},*)
(*DBG:    {&(RES0__INSTANCE0.MY_BAD_FIFO.BUFFER.value.table[1437]), INT_ENUM},*)
(*DBG:    {&(RES0__INSTANCE0.MY_BAD_FIFO.BUFFER.value.table[1438]), INT_ENUM},*)
(*DBG:    {&(RES0__INSTANCE0.MY_BAD_FIFO.BUFFER.value.table[1439]), INT_ENUM},*)
(*DBG:    {&(RES0__INSTANCE0.MY_BAD_FIFO.BUFFER.value.table[1440]), INT_ENUM},*)
(*DBG:    {&(RES0__INSTANCE0.MY_BAD_FIFO.BUFFER.value.table[1441]), INT_ENUM},*)
(*DBG:    {&(RES0__INSTANCE0.MY_BAD_FIFO.BUFFER.value.table[1442]), INT_ENUM},*)
(*DBG:    {&(RES0__INSTANCE0.MY_BAD_FIFO.BUFFER.value.table[1443]), INT_ENUM},*)
(*DBG:    {&(RES0__INSTANCE0.MY_BAD_FIFO.BUFFER.value.table[1444]), INT_ENUM},*)
(*DBG:    {&(RES0__INSTANCE0.MY_BAD_FIFO.BUFFER.value.table[1445]), INT_ENUM},*)
(*DBG:    {&(RES0__INSTANCE0.MY_BAD_FIFO.BUFFER.value.table[1446]), INT_ENUM},*)
(*DBG:    {&(RES0__INSTANCE0.MY_BAD_FIFO.BUFFER.value.table[1447]), INT_ENUM},*)
(*DBG:    {&(RES0__INSTANCE0.MY_BAD_FIFO.BUFFER.value.table[1448]), INT_ENUM},*)
(*DBG:    {&(RES0__INSTANCE0.MY_BAD_FIFO.BUFFER.value.table[1449]), INT_ENUM},*)
(*DBG:    {&(RES0__INSTANCE0.MY_BAD_FIFO.BUFFER.value.table[1450]), INT_ENUM},*)
(*DBG:    {&(RES0__INSTANCE0.MY_BAD_FIFO.BUFFER.value.table[1451]), INT_ENUM},*)
(*DBG:    {&(RES0__INSTANCE0.MY_BAD_FIFO.BUFFER.value.table[1452]), INT_ENUM},*)
(*DBG:    {&(RES0__INSTANCE0.MY_BAD_FIFO.BUFFER.value.table[1453]), INT_ENUM},*)
(*DBG:    {&(RES0__INSTANCE0.MY_BAD_FIFO.BUFFER.value.table[1454]), INT_ENUM},*)
(*DBG:    {&(RES0__INSTANCE0.MY_BAD_FIFO.BUFFER.value.table[1455]), INT_ENUM},*)
(*DBG:    {&(RES0__INSTANCE0.MY_BAD_FIFO.BUFFER.value.table[1456]), INT_ENUM},*)
(*DBG:    {&(RES0__INSTANCE0.MY_BAD_FIFO.BUFFER.value.table[1457]), INT_ENUM},*)
(*DBG:    {&(RES0__INSTANCE0.MY_BAD_FIFO.BUFFER.value.table[1458]), INT_ENUM},*)
(*DBG:    {&(RES0__INSTANCE0.MY_BAD_FIFO.BUFFER.value.table[1459]), INT_ENUM},*)
(*DBG:    {&(RES0__INSTANCE0.MY_BAD_FIFO.BUFFER.value.table[1460]), INT_ENUM},*)
(*DBG:    {&(RES0__INSTANCE0.MY_BAD_FIFO.BUFFER.value.table[1461]), INT_ENUM},*)
(*DBG:    {&(RES0__INSTANCE0.MY_BAD_FIFO.BUFFER.value.table[1462]), INT_ENUM},*)
(*DBG:    {&(RES0__INSTANCE0.MY_BAD_FIFO.BUFFER.value.table[1463]), INT_ENUM},*)
(*DBG:    {&(RES0__INSTANCE0.MY_BAD_FIFO.BUFFER.value.table[1464]), INT_ENUM},*)
(*DBG:    {&(RES0__INSTANCE0.MY_BAD_FIFO.BUFFER.value.table[1465]), INT_ENUM},*)
(*DBG:    {&(RES0__INSTANCE0.MY_BAD_FIFO.BUFFER.value.table[1466]), INT_ENUM},*)
(*DBG:    {&(RES0__INSTANCE0.MY_BAD_FIFO.BUFFER.value.table[1467]), INT_ENUM},*)
(*DBG:    {&(RES0__INSTANCE0.MY_BAD_FIFO.BUFFER.value.table[1468]), INT_ENUM},*)
(*DBG:    {&(RES0__INSTANCE0.MY_BAD_FIFO.BUFFER.value.table[1469]), INT_ENUM},*)
(*DBG:    {&(RES0__INSTANCE0.MY_BAD_FIFO.BUFFER.value.table[1470]), INT_ENUM},*)
(*DBG:    {&(RES0__INSTANCE0.MY_BAD_FIFO.BUFFER.value.table[1471]), INT_ENUM},*)
(*DBG:    {&(RES0__INSTANCE0.MY_BAD_FIFO.BUFFER.value.table[1472]), INT_ENUM},*)
(*DBG:    {&(RES0__INSTANCE0.MY_BAD_FIFO.BUFFER.value.table[1473]), INT_ENUM},*)
(*DBG:    {&(RES0__INSTANCE0.MY_BAD_FIFO.BUFFER.value.table[1474]), INT_ENUM},*)
(*DBG:    {&(RES0__INSTANCE0.MY_BAD_FIFO.BUFFER.value.table[1475]), INT_ENUM},*)
(*DBG:    {&(RES0__INSTANCE0.MY_BAD_FIFO.BUFFER.value.table[1476]), INT_ENUM},*)
(*DBG:    {&(RES0__INSTANCE0.MY_BAD_FIFO.BUFFER.value.table[1477]), INT_ENUM},*)
(*DBG:    {&(RES0__INSTANCE0.MY_BAD_FIFO.BUFFER.value.table[1478]), INT_ENUM},*)
(*DBG:    {&(RES0__INSTANCE0.MY_BAD_FIFO.BUFFER.value.table[1479]), INT_ENUM},*)
(*DBG:    {&(RES0__INSTANCE0.MY_BAD_FIFO.BUFFER.value.table[1480]), INT_ENUM},*)
(*DBG:    {&(RES0__INSTANCE0.MY_BAD_FIFO.BUFFER.value.table[1481]), INT_ENUM},*)
(*DBG:    {&(RES0__INSTANCE0.MY_BAD_FIFO.BUFFER.value.table[1482]), INT_ENUM},*)
(*DBG:    {&(RES0__INSTANCE0.MY_BAD_FIFO.BUFFER.value.table[1483]), INT_ENUM},*)
(*DBG:    {&(RES0__INSTANCE0.MY_BAD_FIFO.BUFFER.value.table[1484]), INT_ENUM},*)
(*DBG:    {&(RES0__INSTANCE0.MY_BAD_FIFO.BUFFER.value.table[1485]), INT_ENUM},*)
(*DBG:    {&(RES0__INSTANCE0.MY_BAD_FIFO.BUFFER.value.table[1486]), INT_ENUM},*)
(*DBG:    {&(RES0__INSTANCE0.MY_BAD_FIFO.BUFFER.value.table[1487]), INT_ENUM},*)
(*DBG:    {&(RES0__INSTANCE0.MY_BAD_FIFO.BUFFER.value.table[1488]), INT_ENUM},*)
(*DBG:    {&(RES0__INSTANCE0.MY_BAD_FIFO.BUFFER.value.table[1489]), INT_ENUM},*)
(*DBG:    {&(RES0__INSTANCE0.MY_BAD_FIFO.BUFFER.value.table[1490]), INT_ENUM},*)
(*DBG:    {&(RES0__INSTANCE0.MY_BAD_FIFO.BUFFER.value.table[1491]), INT_ENUM},*)
(*DBG:    {&(RES0__INSTANCE0.MY_BAD_FIFO.BUFFER.value.table[1492]), INT_ENUM},*)
(*DBG:    {&(RES0__INSTANCE0.MY_BAD_FIFO.BUFFER.value.table[1493]), INT_ENUM},*)
(*DBG:    {&(RES0__INSTANCE0.MY_BAD_FIFO.BUFFER.value.table[1494]), INT_ENUM},*)
(*DBG:    {&(RES0__INSTANCE0.MY_BAD_FIFO.BUFFER.value.table[1495]), INT_ENUM},*)
(*DBG:    {&(RES0__INSTANCE0.MY_BAD_FIFO.BUFFER.value.table[1496]), INT_ENUM},*)
(*DBG:    {&(RES0__INSTANCE0.MY_BAD_FIFO.BUFFER.value.table[1497]), INT_ENUM},*)
(*DBG:    {&(RES0__INSTANCE0.MY_BAD_FIFO.BUFFER.value.table[1498]), INT_ENUM},*)
(*DBG:    {&(RES0__INSTANCE0.MY_BAD_FIFO.BUFFER.value.table[1499]), INT_ENUM},*)
(*DBG:    {&(RES0__INSTANCE0.MY_BAD_FIFO.BUFFER.value.table[1500]), INT_ENUM},*)
(*DBG:    {&(RES0__INSTANCE0.MY_BAD_FIFO.BUFFER.value.table[1501]), INT_ENUM},*)
(*DBG:    {&(RES0__INSTANCE0.MY_BAD_FIFO.BUFFER.value.table[1502]), INT_ENUM},*)
(*DBG:    {&(RES0__INSTANCE0.MY_BAD_FIFO.BUFFER.value.table[1503]), INT_ENUM},*)
(*DBG:    {&(RES0__INSTANCE0.MY_BAD_FIFO.BUFFER.value.table[1504]), INT_ENUM},*)
(*DBG:    {&(RES0__INSTANCE0.MY_BAD_FIFO.BUFFER.value.table[1505]), INT_ENUM},*)
(*DBG:    {&(RES0__INSTANCE0.MY_BAD_FIFO.BUFFER.value.table[1506]), INT_ENUM},*)
(*DBG:    {&(RES0__INSTANCE0.MY_BAD_FIFO.BUFFER.value.table[1507]), INT_ENUM},*)
(*DBG:    {&(RES0__INSTANCE0.MY_BAD_FIFO.BUFFER.value.table[1508]), INT_ENUM},*)
(*DBG:    {&(RES0__INSTANCE0.MY_BAD_FIFO.BUFFER.value.table[1509]), INT_ENUM},*)
(*DBG:    {&(RES0__INSTANCE0.MY_BAD_FIFO.BUFFER.value.table[1510]), INT_ENUM},*)
(*DBG:    {&(RES0__INSTANCE0.MY_BAD_FIFO.BUFFER.value.table[1511]), INT_ENUM},*)
(*DBG:    {&(RES0__INSTANCE0.MY_BAD_FIFO.BUFFER.value.table[1512]), INT_ENUM},*)
(*DBG:    {&(RES0__INSTANCE0.MY_BAD_FIFO.BUFFER.value.table[1513]), INT_ENUM},*)
(*DBG:    {&(RES0__INSTANCE0.MY_BAD_FIFO.BUFFER.value.table[1514]), INT_ENUM},*)
(*DBG:    {&(RES0__INSTANCE0.MY_BAD_FIFO.BUFFER.value.table[1515]), INT_ENUM},*)
(*DBG:    {&(RES0__INSTANCE0.MY_BAD_FIFO.BUFFER.value.table[1516]), INT_ENUM},*)
(*DBG:    {&(RES0__INSTANCE0.MY_BAD_FIFO.BUFFER.value.table[1517]), INT_ENUM},*)
(*DBG:    {&(RES0__INSTANCE0.MY_BAD_FIFO.BUFFER.value.table[1518]), INT_ENUM},*)
(*DBG:    {&(RES0__INSTANCE0.MY_BAD_FIFO.BUFFER.value.table[1519]), INT_ENUM},*)
(*DBG:    {&(RES0__INSTANCE0.MY_BAD_FIFO.BUFFER.value.table[1520]), INT_ENUM},*)
(*DBG:    {&(RES0__INSTANCE0.MY_BAD_FIFO.BUFFER.value.table[1521]), INT_ENUM},*)
(*DBG:    {&(RES0__INSTANCE0.MY_BAD_FIFO.BUFFER.value.table[1522]), INT_ENUM},*)
(*DBG:    {&(RES0__INSTANCE0.MY_BAD_FIFO.BUFFER.value.table[1523]), INT_ENUM},*)
(*DBG:    {&(RES0__INSTANCE0.MY_BAD_FIFO.BUFFER.value.table[1524]), INT_ENUM},*)
(*DBG:    {&(RES0__INSTANCE0.MY_BAD_FIFO.BUFFER.value.table[1525]), INT_ENUM},*)
(*DBG:    {&(RES0__INSTANCE0.MY_BAD_FIFO.BUFFER.value.table[1526]), INT_ENUM},*)
(*DBG:    {&(RES0__INSTANCE0.MY_BAD_FIFO.BUFFER.value.table[1527]), INT_ENUM},*)
(*DBG:    {&(RES0__INSTANCE0.MY_BAD_FIFO.BUFFER.value.table[1528]), INT_ENUM},*)
(*DBG:    {&(RES0__INSTANCE0.MY_BAD_FIFO.BUFFER.value.table[1529]), INT_ENUM},*)
(*DBG:    {&(RES0__INSTANCE0.MY_BAD_FIFO.BUFFER.value.table[1530]), INT_ENUM},*)
(*DBG:    {&(RES0__INSTANCE0.MY_BAD_FIFO.BUFFER.value.table[1531]), INT_ENUM},*)
(*DBG:    {&(RES0__INSTANCE0.MY_BAD_FIFO.BUFFER.value.table[1532]), INT_ENUM},*)
(*DBG:    {&(RES0__INSTANCE0.MY_BAD_FIFO.BUFFER.value.table[1533]), INT_ENUM},*)
(*DBG:    {&(RES0__INSTANCE0.MY_BAD_FIFO.BUFFER.value.table[1534]), INT_ENUM},*)
(*DBG:    {&(RES0__INSTANCE0.MY_BAD_FIFO.BUFFER.value.table[1535]), INT_ENUM},*)
(*DBG:    {&(RES0__INSTANCE0.MY_BAD_FIFO.BUFFER.value.table[1536]), INT_ENUM},*)
(*DBG:    {&(RES0__INSTANCE0.MY_BAD_FIFO.BUFFER.value.table[1537]), INT_ENUM},*)
(*DBG:    {&(RES0__INSTANCE0.MY_BAD_FIFO.BUFFER.value.table[1538]), INT_ENUM},*)
(*DBG:    {&(RES0__INSTANCE0.MY_BAD_FIFO.BUFFER.value.table[1539]), INT_ENUM},*)
(*DBG:    {&(RES0__INSTANCE0.MY_BAD_FIFO.BUFFER.value.table[1540]), INT_ENUM},*)
(*DBG:    {&(RES0__INSTANCE0.MY_BAD_FIFO.BUFFER.value.table[1541]), INT_ENUM},*)
(*DBG:    {&(RES0__INSTANCE0.MY_BAD_FIFO.BUFFER.value.table[1542]), INT_ENUM},*)
(*DBG:    {&(RES0__INSTANCE0.MY_BAD_FIFO.BUFFER.value.table[1543]), INT_ENUM},*)
(*DBG:    {&(RES0__INSTANCE0.MY_BAD_FIFO.BUFFER.value.table[1544]), INT_ENUM},*)
(*DBG:    {&(RES0__INSTANCE0.MY_BAD_FIFO.BUFFER.value.table[1545]), INT_ENUM},*)
(*DBG:    {&(RES0__INSTANCE0.MY_BAD_FIFO.BUFFER.value.table[1546]), INT_ENUM},*)
(*DBG:    {&(RES0__INSTANCE0.MY_BAD_FIFO.BUFFER.value.table[1547]), INT_ENUM},*)
(*DBG:    {&(RES0__INSTANCE0.MY_BAD_FIFO.BUFFER.value.table[1548]), INT_ENUM},*)
(*DBG:    {&(RES0__INSTANCE0.MY_BAD_FIFO.BUFFER.value.table[1549]), INT_ENUM},*)
(*DBG:    {&(RES0__INSTANCE0.MY_BAD_FIFO.BUFFER.value.table[1550]), INT_ENUM},*)
(*DBG:    {&(RES0__INSTANCE0.MY_BAD_FIFO.BUFFER.value.table[1551]), INT_ENUM},*)
(*DBG:    {&(RES0__INSTANCE0.MY_BAD_FIFO.BUFFER.value.table[1552]), INT_ENUM},*)
(*DBG:    {&(RES0__INSTANCE0.MY_BAD_FIFO.BUFFER.value.table[1553]), INT_ENUM},*)
(*DBG:    {&(RES0__INSTANCE0.MY_BAD_FIFO.BUFFER.value.table[1554]), INT_ENUM},*)
(*DBG:    {&(RES0__INSTANCE0.MY_BAD_FIFO.BUFFER.value.table[1555]), INT_ENUM},*)
(*DBG:    {&(RES0__INSTANCE0.MY_BAD_FIFO.BUFFER.value.table[1556]), INT_ENUM},*)
(*DBG:    {&(RES0__INSTANCE0.MY_BAD_FIFO.BUFFER.value.table[1557]), INT_ENUM},*)
(*DBG:    {&(RES0__INSTANCE0.MY_BAD_FIFO.BUFFER.value.table[1558]), INT_ENUM},*)
(*DBG:    {&(RES0__INSTANCE0.MY_BAD_FIFO.BUFFER.value.table[1559]), INT_ENUM},*)
(*DBG:    {&(RES0__INSTANCE0.MY_BAD_FIFO.BUFFER.value.table[1560]), INT_ENUM},*)
(*DBG:    {&(RES0__INSTANCE0.MY_BAD_FIFO.BUFFER.value.table[1561]), INT_ENUM},*)
(*DBG:    {&(RES0__INSTANCE0.MY_BAD_FIFO.BUFFER.value.table[1562]), INT_ENUM},*)
(*DBG:    {&(RES0__INSTANCE0.MY_BAD_FIFO.BUFFER.value.table[1563]), INT_ENUM},*)
(*DBG:    {&(RES0__INSTANCE0.MY_BAD_FIFO.BUFFER.value.table[1564]), INT_ENUM},*)
(*DBG:    {&(RES0__INSTANCE0.MY_BAD_FIFO.BUFFER.value.table[1565]), INT_ENUM},*)
(*DBG:    {&(RES0__INSTANCE0.MY_BAD_FIFO.BUFFER.value.table[1566]), INT_ENUM},*)
(*DBG:    {&(RES0__INSTANCE0.MY_BAD_FIFO.BUFFER.value.table[1567]), INT_ENUM},*)
(*DBG:    {&(RES0__INSTANCE0.MY_BAD_FIFO.BUFFER.value.table[1568]), INT_ENUM},*)
(*DBG:    {&(RES0__INSTANCE0.MY_BAD_FIFO.BUFFER.value.table[1569]), INT_ENUM},*)
(*DBG:    {&(RES0__INSTANCE0.MY_BAD_FIFO.BUFFER.value.table[1570]), INT_ENUM},*)
(*DBG:    {&(RES0__INSTANCE0.MY_BAD_FIFO.BUFFER.value.table[1571]), INT_ENUM},*)
(*DBG:    {&(RES0__INSTANCE0.MY_BAD_FIFO.BUFFER.value.table[1572]), INT_ENUM},*)
(*DBG:    {&(RES0__INSTANCE0.MY_BAD_FIFO.BUFFER.value.table[1573]), INT_ENUM},*)
(*DBG:    {&(RES0__INSTANCE0.MY_BAD_FIFO.BUFFER.value.table[1574]), INT_ENUM},*)
(*DBG:    {&(RES0__INSTANCE0.MY_BAD_FIFO.BUFFER.value.table[1575]), INT_ENUM},*)
(*DBG:    {&(RES0__INSTANCE0.MY_BAD_FIFO.BUFFER.value.table[1576]), INT_ENUM},*)
(*DBG:    {&(RES0__INSTANCE0.MY_BAD_FIFO.BUFFER.value.table[1577]), INT_ENUM},*)
(*DBG:    {&(RES0__INSTANCE0.MY_BAD_FIFO.BUFFER.value.table[1578]), INT_ENUM},*)
(*DBG:    {&(RES0__INSTANCE0.MY_BAD_FIFO.BUFFER.value.table[1579]), INT_ENUM},*)
(*DBG:    {&(RES0__INSTANCE0.MY_BAD_FIFO.BUFFER.value.table[1580]), INT_ENUM},*)
(*DBG:    {&(RES0__INSTANCE0.MY_BAD_FIFO.BUFFER.value.table[1581]), INT_ENUM},*)
(*DBG:    {&(RES0__INSTANCE0.MY_BAD_FIFO.BUFFER.value.table[1582]), INT_ENUM},*)
(*DBG:    {&(RES0__INSTANCE0.MY_BAD_FIFO.BUFFER.value.table[1583]), INT_ENUM},*)
(*DBG:    {&(RES0__INSTANCE0.MY_BAD_FIFO.BUFFER.value.table[1584]), INT_ENUM},*)
(*DBG:    {&(RES0__INSTANCE0.MY_BAD_FIFO.BUFFER.value.table[1585]), INT_ENUM},*)
(*DBG:    {&(RES0__INSTANCE0.MY_BAD_FIFO.BUFFER.value.table[1586]), INT_ENUM},*)
(*DBG:    {&(RES0__INSTANCE0.MY_BAD_FIFO.BUFFER.value.table[1587]), INT_ENUM},*)
(*DBG:    {&(RES0__INSTANCE0.MY_BAD_FIFO.BUFFER.value.table[1588]), INT_ENUM},*)
(*DBG:    {&(RES0__INSTANCE0.MY_BAD_FIFO.BUFFER.value.table[1589]), INT_ENUM},*)
(*DBG:    {&(RES0__INSTANCE0.MY_BAD_FIFO.BUFFER.value.table[1590]), INT_ENUM},*)
(*DBG:    {&(RES0__INSTANCE0.MY_BAD_FIFO.BUFFER.value.table[1591]), INT_ENUM},*)
(*DBG:    {&(RES0__INSTANCE0.MY_BAD_FIFO.BUFFER.value.table[1592]), INT_ENUM},*)
(*DBG:    {&(RES0__INSTANCE0.MY_BAD_FIFO.BUFFER.value.table[1593]), INT_ENUM},*)
(*DBG:    {&(RES0__INSTANCE0.MY_BAD_FIFO.BUFFER.value.table[1594]), INT_ENUM},*)
(*DBG:    {&(RES0__INSTANCE0.MY_BAD_FIFO.BUFFER.value.table[1595]), INT_ENUM},*)
(*DBG:    {&(RES0__INSTANCE0.MY_BAD_FIFO.BUFFER.value.table[1596]), INT_ENUM},*)
(*DBG:    {&(RES0__INSTANCE0.MY_BAD_FIFO.BUFFER.value.table[1597]), INT_ENUM},*)
(*DBG:    {&(RES0__INSTANCE0.MY_BAD_FIFO.BUFFER.value.table[1598]), INT_ENUM},*)
(*DBG:    {&(RES0__INSTANCE0.MY_BAD_FIFO.BUFFER.value.table[1599]), INT_ENUM},*)
(*DBG:    {&(RES0__INSTANCE0.MY_BAD_FIFO.BUFFER.value.table[1600]), INT_ENUM},*)
(*DBG:    {&(RES0__INSTANCE0.MY_BAD_FIFO.BUFFER.value.table[1601]), INT_ENUM},*)
(*DBG:    {&(RES0__INSTANCE0.MY_BAD_FIFO.BUFFER.value.table[1602]), INT_ENUM},*)
(*DBG:    {&(RES0__INSTANCE0.MY_BAD_FIFO.BUFFER.value.table[1603]), INT_ENUM},*)
(*DBG:    {&(RES0__INSTANCE0.MY_BAD_FIFO.BUFFER.value.table[1604]), INT_ENUM},*)
(*DBG:    {&(RES0__INSTANCE0.MY_BAD_FIFO.BUFFER.value.table[1605]), INT_ENUM},*)
(*DBG:    {&(RES0__INSTANCE0.MY_BAD_FIFO.BUFFER.value.table[1606]), INT_ENUM},*)
(*DBG:    {&(RES0__INSTANCE0.MY_BAD_FIFO.BUFFER.value.table[1607]), INT_ENUM},*)
(*DBG:    {&(RES0__INSTANCE0.MY_BAD_FIFO.BUFFER.value.table[1608]), INT_ENUM},*)
(*DBG:    {&(RES0__INSTANCE0.MY_BAD_FIFO.BUFFER.value.table[1609]), INT_ENUM},*)
(*DBG:    {&(RES0__INSTANCE0.MY_BAD_FIFO.BUFFER.value.table[1610]), INT_ENUM},*)
(*DBG:    {&(RES0__INSTANCE0.MY_BAD_FIFO.BUFFER.value.table[1611]), INT_ENUM},*)
(*DBG:    {&(RES0__INSTANCE0.MY_BAD_FIFO.BUFFER.value.table[1612]), INT_ENUM},*)
(*DBG:    {&(RES0__INSTANCE0.MY_BAD_FIFO.BUFFER.value.table[1613]), INT_ENUM},*)
(*DBG:    {&(RES0__INSTANCE0.MY_BAD_FIFO.BUFFER.value.table[1614]), INT_ENUM},*)
(*DBG:    {&(RES0__INSTANCE0.MY_BAD_FIFO.BUFFER.value.table[1615]), INT_ENUM},*)
(*DBG:    {&(RES0__INSTANCE0.MY_BAD_FIFO.BUFFER.value.table[1616]), INT_ENUM},*)
(*DBG:    {&(RES0__INSTANCE0.MY_BAD_FIFO.BUFFER.value.table[1617]), INT_ENUM},*)
(*DBG:    {&(RES0__INSTANCE0.MY_BAD_FIFO.BUFFER.value.table[1618]), INT_ENUM},*)
(*DBG:    {&(RES0__INSTANCE0.MY_BAD_FIFO.BUFFER.value.table[1619]), INT_ENUM},*)
(*DBG:    {&(RES0__INSTANCE0.MY_BAD_FIFO.BUFFER.value.table[1620]), INT_ENUM},*)
(*DBG:    {&(RES0__INSTANCE0.MY_BAD_FIFO.BUFFER.value.table[1621]), INT_ENUM},*)
(*DBG:    {&(RES0__INSTANCE0.MY_BAD_FIFO.BUFFER.value.table[1622]), INT_ENUM},*)
(*DBG:    {&(RES0__INSTANCE0.MY_BAD_FIFO.BUFFER.value.table[1623]), INT_ENUM},*)
(*DBG:    {&(RES0__INSTANCE0.MY_BAD_FIFO.BUFFER.value.table[1624]), INT_ENUM},*)
(*DBG:    {&(RES0__INSTANCE0.MY_BAD_FIFO.BUFFER.value.table[1625]), INT_ENUM},*)
(*DBG:    {&(RES0__INSTANCE0.MY_BAD_FIFO.BUFFER.value.table[1626]), INT_ENUM},*)
(*DBG:    {&(RES0__INSTANCE0.MY_BAD_FIFO.BUFFER.value.table[1627]), INT_ENUM},*)
(*DBG:    {&(RES0__INSTANCE0.MY_BAD_FIFO.BUFFER.value.table[1628]), INT_ENUM},*)
(*DBG:    {&(RES0__INSTANCE0.MY_BAD_FIFO.BUFFER.value.table[1629]), INT_ENUM},*)
(*DBG:    {&(RES0__INSTANCE0.MY_BAD_FIFO.BUFFER.value.table[1630]), INT_ENUM},*)
(*DBG:    {&(RES0__INSTANCE0.MY_BAD_FIFO.BUFFER.value.table[1631]), INT_ENUM},*)
(*DBG:    {&(RES0__INSTANCE0.MY_BAD_FIFO.BUFFER.value.table[1632]), INT_ENUM},*)
(*DBG:    {&(RES0__INSTANCE0.MY_BAD_FIFO.BUFFER.value.table[1633]), INT_ENUM},*)
(*DBG:    {&(RES0__INSTANCE0.MY_BAD_FIFO.BUFFER.value.table[1634]), INT_ENUM},*)
(*DBG:    {&(RES0__INSTANCE0.MY_BAD_FIFO.BUFFER.value.table[1635]), INT_ENUM},*)
(*DBG:    {&(RES0__INSTANCE0.MY_BAD_FIFO.BUFFER.value.table[1636]), INT_ENUM},*)
(*DBG:    {&(RES0__INSTANCE0.MY_BAD_FIFO.BUFFER.value.table[1637]), INT_ENUM},*)
(*DBG:    {&(RES0__INSTANCE0.MY_BAD_FIFO.BUFFER.value.table[1638]), INT_ENUM},*)
(*DBG:    {&(RES0__INSTANCE0.MY_BAD_FIFO.BUFFER.value.table[1639]), INT_ENUM},*)
(*DBG:    {&(RES0__INSTANCE0.MY_BAD_FIFO.BUFFER.value.table[1640]), INT_ENUM},*)
(*DBG:    {&(RES0__INSTANCE0.MY_BAD_FIFO.BUFFER.value.table[1641]), INT_ENUM},*)
(*DBG:    {&(RES0__INSTANCE0.MY_BAD_FIFO.BUFFER.value.table[1642]), INT_ENUM},*)
(*DBG:    {&(RES0__INSTANCE0.MY_BAD_FIFO.BUFFER.value.table[1643]), INT_ENUM},*)
(*DBG:    {&(RES0__INSTANCE0.MY_BAD_FIFO.BUFFER.value.table[1644]), INT_ENUM},*)
(*DBG:    {&(RES0__INSTANCE0.MY_BAD_FIFO.BUFFER.value.table[1645]), INT_ENUM},*)
(*DBG:    {&(RES0__INSTANCE0.MY_BAD_FIFO.BUFFER.value.table[1646]), INT_ENUM},*)
(*DBG:    {&(RES0__INSTANCE0.MY_BAD_FIFO.BUFFER.value.table[1647]), INT_ENUM},*)
(*DBG:    {&(RES0__INSTANCE0.MY_BAD_FIFO.BUFFER.value.table[1648]), INT_ENUM},*)
(*DBG:    {&(RES0__INSTANCE0.MY_BAD_FIFO.BUFFER.value.table[1649]), INT_ENUM},*)
(*DBG:    {&(RES0__INSTANCE0.MY_BAD_FIFO.BUFFER.value.table[1650]), INT_ENUM},*)
(*DBG:    {&(RES0__INSTANCE0.MY_BAD_FIFO.BUFFER.value.table[1651]), INT_ENUM},*)
(*DBG:    {&(RES0__INSTANCE0.MY_BAD_FIFO.BUFFER.value.table[1652]), INT_ENUM},*)
(*DBG:    {&(RES0__INSTANCE0.MY_BAD_FIFO.BUFFER.value.table[1653]), INT_ENUM},*)
(*DBG:    {&(RES0__INSTANCE0.MY_BAD_FIFO.BUFFER.value.table[1654]), INT_ENUM},*)
(*DBG:    {&(RES0__INSTANCE0.MY_BAD_FIFO.BUFFER.value.table[1655]), INT_ENUM},*)
(*DBG:    {&(RES0__INSTANCE0.MY_BAD_FIFO.BUFFER.value.table[1656]), INT_ENUM},*)
(*DBG:    {&(RES0__INSTANCE0.MY_BAD_FIFO.BUFFER.value.table[1657]), INT_ENUM},*)
(*DBG:    {&(RES0__INSTANCE0.MY_BAD_FIFO.BUFFER.value.table[1658]), INT_ENUM},*)
(*DBG:    {&(RES0__INSTANCE0.MY_BAD_FIFO.BUFFER.value.table[1659]), INT_ENUM},*)
(*DBG:    {&(RES0__INSTANCE0.MY_BAD_FIFO.BUFFER.value.table[1660]), INT_ENUM},*)
(*DBG:    {&(RES0__INSTANCE0.MY_BAD_FIFO.BUFFER.value.table[1661]), INT_ENUM},*)
(*DBG:    {&(RES0__INSTANCE0.MY_BAD_FIFO.BUFFER.value.table[1662]), INT_ENUM},*)
(*DBG:    {&(RES0__INSTANCE0.MY_BAD_FIFO.BUFFER.value.table[1663]), INT_ENUM},*)
(*DBG:    {&(RES0__INSTANCE0.MY_BAD_FIFO.BUFFER.value.table[1664]), INT_ENUM},*)
(*DBG:    {&(RES0__INSTANCE0.MY_BAD_FIFO.BUFFER.value.table[1665]), INT_ENUM},*)
(*DBG:    {&(RES0__INSTANCE0.MY_BAD_FIFO.BUFFER.value.table[1666]), INT_ENUM},*)
(*DBG:    {&(RES0__INSTANCE0.MY_BAD_FIFO.BUFFER.value.table[1667]), INT_ENUM},*)
(*DBG:    {&(RES0__INSTANCE0.MY_BAD_FIFO.BUFFER.value.table[1668]), INT_ENUM},*)
(*DBG:    {&(RES0__INSTANCE0.MY_BAD_FIFO.BUFFER.value.table[1669]), INT_ENUM},*)
(*DBG:    {&(RES0__INSTANCE0.MY_BAD_FIFO.BUFFER.value.table[1670]), INT_ENUM},*)
(*DBG:    {&(RES0__INSTANCE0.MY_BAD_FIFO.BUFFER.value.table[1671]), INT_ENUM},*)
(*DBG:    {&(RES0__INSTANCE0.MY_BAD_FIFO.BUFFER.value.table[1672]), INT_ENUM},*)
(*DBG:    {&(RES0__INSTANCE0.MY_BAD_FIFO.BUFFER.value.table[1673]), INT_ENUM},*)
(*DBG:    {&(RES0__INSTANCE0.MY_BAD_FIFO.BUFFER.value.table[1674]), INT_ENUM},*)
(*DBG:    {&(RES0__INSTANCE0.MY_BAD_FIFO.BUFFER.value.table[1675]), INT_ENUM},*)
(*DBG:    {&(RES0__INSTANCE0.MY_BAD_FIFO.BUFFER.value.table[1676]), INT_ENUM},*)
(*DBG:    {&(RES0__INSTANCE0.MY_BAD_FIFO.BUFFER.value.table[1677]), INT_ENUM},*)
(*DBG:    {&(RES0__INSTANCE0.MY_BAD_FIFO.BUFFER.value.table[1678]), INT_ENUM},*)
(*DBG:    {&(RES0__INSTANCE0.MY_BAD_FIFO.BUFFER.value.table[1679]), INT_ENUM},*)
(*DBG:    {&(RES0__INSTANCE0.MY_BAD_FIFO.BUFFER.value.table[1680]), INT_ENUM},*)
(*DBG:    {&(RES0__INSTANCE0.MY_BAD_FIFO.BUFFER.value.table[1681]), INT_ENUM},*)
(*DBG:    {&(RES0__INSTANCE0.MY_BAD_FIFO.BUFFER.value.table[1682]), INT_ENUM},*)
(*DBG:    {&(RES0__INSTANCE0.MY_BAD_FIFO.BUFFER.value.table[1683]), INT_ENUM},*)
(*DBG:    {&(RES0__INSTANCE0.MY_BAD_FIFO.BUFFER.value.table[1684]), INT_ENUM},*)
(*DBG:    {&(RES0__INSTANCE0.MY_BAD_FIFO.BUFFER.value.table[1685]), INT_ENUM},*)
(*DBG:    {&(RES0__INSTANCE0.MY_BAD_FIFO.BUFFER.value.table[1686]), INT_ENUM},*)
(*DBG:    {&(RES0__INSTANCE0.MY_BAD_FIFO.BUFFER.value.table[1687]), INT_ENUM},*)
(*DBG:    {&(RES0__INSTANCE0.MY_BAD_FIFO.BUFFER.value.table[1688]), INT_ENUM},*)
(*DBG:    {&(RES0__INSTANCE0.MY_BAD_FIFO.BUFFER.value.table[1689]), INT_ENUM},*)
(*DBG:    {&(RES0__INSTANCE0.MY_BAD_FIFO.BUFFER.value.table[1690]), INT_ENUM},*)
(*DBG:    {&(RES0__INSTANCE0.MY_BAD_FIFO.BUFFER.value.table[1691]), INT_ENUM},*)
(*DBG:    {&(RES0__INSTANCE0.MY_BAD_FIFO.BUFFER.value.table[1692]), INT_ENUM},*)
(*DBG:    {&(RES0__INSTANCE0.MY_BAD_FIFO.BUFFER.value.table[1693]), INT_ENUM},*)
(*DBG:    {&(RES0__INSTANCE0.MY_BAD_FIFO.BUFFER.value.table[1694]), INT_ENUM},*)
(*DBG:    {&(RES0__INSTANCE0.MY_BAD_FIFO.BUFFER.value.table[1695]), INT_ENUM},*)
(*DBG:    {&(RES0__INSTANCE0.MY_BAD_FIFO.BUFFER.value.table[1696]), INT_ENUM},*)
(*DBG:    {&(RES0__INSTANCE0.MY_BAD_FIFO.BUFFER.value.table[1697]), INT_ENUM},*)
(*DBG:    {&(RES0__INSTANCE0.MY_BAD_FIFO.BUFFER.value.table[1698]), INT_ENUM},*)
(*DBG:    {&(RES0__INSTANCE0.MY_BAD_FIFO.BUFFER.value.table[1699]), INT_ENUM},*)
(*DBG:    {&(RES0__INSTANCE0.MY_BAD_FIFO.BUFFER.value.table[1700]), INT_ENUM},*)
(*DBG:    {&(RES0__INSTANCE0.MY_BAD_FIFO.BUFFER.value.table[1701]), INT_ENUM},*)
(*DBG:    {&(RES0__INSTANCE0.MY_BAD_FIFO.BUFFER.value.table[1702]), INT_ENUM},*)
(*DBG:    {&(RES0__INSTANCE0.MY_BAD_FIFO.BUFFER.value.table[1703]), INT_ENUM},*)
(*DBG:    {&(RES0__INSTANCE0.MY_BAD_FIFO.BUFFER.value.table[1704]), INT_ENUM},*)
(*DBG:    {&(RES0__INSTANCE0.MY_BAD_FIFO.BUFFER.value.table[1705]), INT_ENUM},*)
(*DBG:    {&(RES0__INSTANCE0.MY_BAD_FIFO.BUFFER.value.table[1706]), INT_ENUM},*)
(*DBG:    {&(RES0__INSTANCE0.MY_BAD_FIFO.BUFFER.value.table[1707]), INT_ENUM},*)
(*DBG:    {&(RES0__INSTANCE0.MY_BAD_FIFO.BUFFER.value.table[1708]), INT_ENUM},*)
(*DBG:    {&(RES0__INSTANCE0.MY_BAD_FIFO.BUFFER.value.table[1709]), INT_ENUM},*)
(*DBG:    {&(RES0__INSTANCE0.MY_BAD_FIFO.BUFFER.value.table[1710]), INT_ENUM},*)
(*DBG:    {&(RES0__INSTANCE0.MY_BAD_FIFO.BUFFER.value.table[1711]), INT_ENUM},*)
(*DBG:    {&(RES0__INSTANCE0.MY_BAD_FIFO.BUFFER.value.table[1712]), INT_ENUM},*)
(*DBG:    {&(RES0__INSTANCE0.MY_BAD_FIFO.BUFFER.value.table[1713]), INT_ENUM},*)
(*DBG:    {&(RES0__INSTANCE0.MY_BAD_FIFO.BUFFER.value.table[1714]), INT_ENUM},*)
(*DBG:    {&(RES0__INSTANCE0.MY_BAD_FIFO.BUFFER.value.table[1715]), INT_ENUM},*)
(*DBG:    {&(RES0__INSTANCE0.MY_BAD_FIFO.BUFFER.value.table[1716]), INT_ENUM},*)
(*DBG:    {&(RES0__INSTANCE0.MY_BAD_FIFO.BUFFER.value.table[1717]), INT_ENUM},*)
(*DBG:    {&(RES0__INSTANCE0.MY_BAD_FIFO.BUFFER.value.table[1718]), INT_ENUM},*)
(*DBG:    {&(RES0__INSTANCE0.MY_BAD_FIFO.BUFFER.value.table[1719]), INT_ENUM},*)
(*DBG:    {&(RES0__INSTANCE0.MY_BAD_FIFO.BUFFER.value.table[1720]), INT_ENUM},*)
(*DBG:    {&(RES0__INSTANCE0.MY_BAD_FIFO.BUFFER.value.table[1721]), INT_ENUM},*)
(*DBG:    {&(RES0__INSTANCE0.MY_BAD_FIFO.BUFFER.value.table[1722]), INT_ENUM},*)
(*DBG:    {&(RES0__INSTANCE0.MY_BAD_FIFO.BUFFER.value.table[1723]), INT_ENUM},*)
(*DBG:    {&(RES0__INSTANCE0.MY_BAD_FIFO.BUFFER.value.table[1724]), INT_ENUM},*)
(*DBG:    {&(RES0__INSTANCE0.MY_BAD_FIFO.BUFFER.value.table[1725]), INT_ENUM},*)
(*DBG:    {&(RES0__INSTANCE0.MY_BAD_FIFO.BUFFER.value.table[1726]), INT_ENUM},*)
(*DBG:    {&(RES0__INSTANCE0.MY_BAD_FIFO.BUFFER.value.table[1727]), INT_ENUM},*)
(*DBG:    {&(RES0__INSTANCE0.MY_BAD_FIFO.BUFFER.value.table[1728]), INT_ENUM},*)
(*DBG:    {&(RES0__INSTANCE0.MY_BAD_FIFO.BUFFER.value.table[1729]), INT_ENUM},*)
(*DBG:    {&(RES0__INSTANCE0.MY_BAD_FIFO.BUFFER.value.table[1730]), INT_ENUM},*)
(*DBG:    {&(RES0__INSTANCE0.MY_BAD_FIFO.BUFFER.value.table[1731]), INT_ENUM},*)
(*DBG:    {&(RES0__INSTANCE0.MY_BAD_FIFO.BUFFER.value.table[1732]), INT_ENUM},*)
(*DBG:    {&(RES0__INSTANCE0.MY_BAD_FIFO.BUFFER.value.table[1733]), INT_ENUM},*)
(*DBG:    {&(RES0__INSTANCE0.MY_BAD_FIFO.BUFFER.value.table[1734]), INT_ENUM},*)
(*DBG:    {&(RES0__INSTANCE0.MY_BAD_FIFO.BUFFER.value.table[1735]), INT_ENUM},*)
(*DBG:    {&(RES0__INSTANCE0.MY_BAD_FIFO.BUFFER.value.table[1736]), INT_ENUM},*)
(*DBG:    {&(RES0__INSTANCE0.MY_BAD_FIFO.BUFFER.value.table[1737]), INT_ENUM},*)
(*DBG:    {&(RES0__INSTANCE0.MY_BAD_FIFO.BUFFER.value.table[1738]), INT_ENUM},*)
(*DBG:    {&(RES0__INSTANCE0.MY_BAD_FIFO.BUFFER.value.table[1739]), INT_ENUM},*)
(*DBG:    {&(RES0__INSTANCE0.MY_BAD_FIFO.BUFFER.value.table[1740]), INT_ENUM},*)
(*DBG:    {&(RES0__INSTANCE0.MY_BAD_FIFO.BUFFER.value.table[1741]), INT_ENUM},*)
(*DBG:    {&(RES0__INSTANCE0.MY_BAD_FIFO.BUFFER.value.table[1742]), INT_ENUM},*)
(*DBG:    {&(RES0__INSTANCE0.MY_BAD_FIFO.BUFFER.value.table[1743]), INT_ENUM},*)
(*DBG:    {&(RES0__INSTANCE0.MY_BAD_FIFO.BUFFER.value.table[1744]), INT_ENUM},*)
(*DBG:    {&(RES0__INSTANCE0.MY_BAD_FIFO.BUFFER.value.table[1745]), INT_ENUM},*)
(*DBG:    {&(RES0__INSTANCE0.MY_BAD_FIFO.BUFFER.value.table[1746]), INT_ENUM},*)
(*DBG:    {&(RES0__INSTANCE0.MY_BAD_FIFO.BUFFER.value.table[1747]), INT_ENUM},*)
(*DBG:    {&(RES0__INSTANCE0.MY_BAD_FIFO.BUFFER.value.table[1748]), INT_ENUM},*)
(*DBG:    {&(RES0__INSTANCE0.MY_BAD_FIFO.BUFFER.value.table[1749]), INT_ENUM},*)
(*DBG:    {&(RES0__INSTANCE0.MY_BAD_FIFO.BUFFER.value.table[1750]), INT_ENUM},*)
(*DBG:    {&(RES0__INSTANCE0.MY_BAD_FIFO.BUFFER.value.table[1751]), INT_ENUM},*)
(*DBG:    {&(RES0__INSTANCE0.MY_BAD_FIFO.BUFFER.value.table[1752]), INT_ENUM},*)
(*DBG:    {&(RES0__INSTANCE0.MY_BAD_FIFO.BUFFER.value.table[1753]), INT_ENUM},*)
(*DBG:    {&(RES0__INSTANCE0.MY_BAD_FIFO.BUFFER.value.table[1754]), INT_ENUM},*)
(*DBG:    {&(RES0__INSTANCE0.MY_BAD_FIFO.BUFFER.value.table[1755]), INT_ENUM},*)
(*DBG:    {&(RES0__INSTANCE0.MY_BAD_FIFO.BUFFER.value.table[1756]), INT_ENUM},*)
(*DBG:    {&(RES0__INSTANCE0.MY_BAD_FIFO.BUFFER.value.table[1757]), INT_ENUM},*)
(*DBG:    {&(RES0__INSTANCE0.MY_BAD_FIFO.BUFFER.value.table[1758]), INT_ENUM},*)
(*DBG:    {&(RES0__INSTANCE0.MY_BAD_FIFO.BUFFER.value.table[1759]), INT_ENUM},*)
(*DBG:    {&(RES0__INSTANCE0.MY_BAD_FIFO.BUFFER.value.table[1760]), INT_ENUM},*)
(*DBG:    {&(RES0__INSTANCE0.MY_BAD_FIFO.BUFFER.value.table[1761]), INT_ENUM},*)
(*DBG:    {&(RES0__INSTANCE0.MY_BAD_FIFO.BUFFER.value.table[1762]), INT_ENUM},*)
(*DBG:    {&(RES0__INSTANCE0.MY_BAD_FIFO.BUFFER.value.table[1763]), INT_ENUM},*)
(*DBG:    {&(RES0__INSTANCE0.MY_BAD_FIFO.BUFFER.value.table[1764]), INT_ENUM},*)
(*DBG:    {&(RES0__INSTANCE0.MY_BAD_FIFO.BUFFER.value.table[1765]), INT_ENUM},*)
(*DBG:    {&(RES0__INSTANCE0.MY_BAD_FIFO.BUFFER.value.table[1766]), INT_ENUM},*)
(*DBG:    {&(RES0__INSTANCE0.MY_BAD_FIFO.BUFFER.value.table[1767]), INT_ENUM},*)
(*DBG:    {&(RES0__INSTANCE0.MY_BAD_FIFO.BUFFER.value.table[1768]), INT_ENUM},*)
(*DBG:    {&(RES0__INSTANCE0.MY_BAD_FIFO.BUFFER.value.table[1769]), INT_ENUM},*)
(*DBG:    {&(RES0__INSTANCE0.MY_BAD_FIFO.BUFFER.value.table[1770]), INT_ENUM},*)
(*DBG:    {&(RES0__INSTANCE0.MY_BAD_FIFO.BUFFER.value.table[1771]), INT_ENUM},*)
(*DBG:    {&(RES0__INSTANCE0.MY_BAD_FIFO.BUFFER.value.table[1772]), INT_ENUM},*)
(*DBG:    {&(RES0__INSTANCE0.MY_BAD_FIFO.BUFFER.value.table[1773]), INT_ENUM},*)
(*DBG:    {&(RES0__INSTANCE0.MY_BAD_FIFO.BUFFER.value.table[1774]), INT_ENUM},*)
(*DBG:    {&(RES0__INSTANCE0.MY_BAD_FIFO.BUFFER.value.table[1775]), INT_ENUM},*)
(*DBG:    {&(RES0__INSTANCE0.MY_BAD_FIFO.BUFFER.value.table[1776]), INT_ENUM},*)
(*DBG:    {&(RES0__INSTANCE0.MY_BAD_FIFO.BUFFER.value.table[1777]), INT_ENUM},*)
(*DBG:    {&(RES0__INSTANCE0.MY_BAD_FIFO.BUFFER.value.table[1778]), INT_ENUM},*)
(*DBG:    {&(RES0__INSTANCE0.MY_BAD_FIFO.BUFFER.value.table[1779]), INT_ENUM},*)
(*DBG:    {&(RES0__INSTANCE0.MY_BAD_FIFO.BUFFER.value.table[1780]), INT_ENUM},*)
(*DBG:    {&(RES0__INSTANCE0.MY_BAD_FIFO.BUFFER.value.table[1781]), INT_ENUM},*)
(*DBG:    {&(RES0__INSTANCE0.MY_BAD_FIFO.BUFFER.value.table[1782]), INT_ENUM},*)
(*DBG:    {&(RES0__INSTANCE0.MY_BAD_FIFO.BUFFER.value.table[1783]), INT_ENUM},*)
(*DBG:    {&(RES0__INSTANCE0.MY_BAD_FIFO.BUFFER.value.table[1784]), INT_ENUM},*)
(*DBG:    {&(RES0__INSTANCE0.MY_BAD_FIFO.BUFFER.value.table[1785]), INT_ENUM},*)
(*DBG:    {&(RES0__INSTANCE0.MY_BAD_FIFO.BUFFER.value.table[1786]), INT_ENUM},*)
(*DBG:    {&(RES0__INSTANCE0.MY_BAD_FIFO.BUFFER.value.table[1787]), INT_ENUM},*)
(*DBG:    {&(RES0__INSTANCE0.MY_BAD_FIFO.BUFFER.value.table[1788]), INT_ENUM},*)
(*DBG:    {&(RES0__INSTANCE0.MY_BAD_FIFO.BUFFER.value.table[1789]), INT_ENUM},*)
(*DBG:    {&(RES0__INSTANCE0.MY_BAD_FIFO.BUFFER.value.table[1790]), INT_ENUM},*)
(*DBG:    {&(RES0__INSTANCE0.MY_BAD_FIFO.BUFFER.value.table[1791]), INT_ENUM},*)
(*DBG:    {&(RES0__INSTANCE0.MY_BAD_FIFO.BUFFER.value.table[1792]), INT_ENUM},*)
(*DBG:    {&(RES0__INSTANCE0.MY_BAD_FIFO.BUFFER.value.table[1793]), INT_ENUM},*)
(*DBG:    {&(RES0__INSTANCE0.MY_BAD_FIFO.BUFFER.value.table[1794]), INT_ENUM},*)
(*DBG:    {&(RES0__INSTANCE0.MY_BAD_FIFO.BUFFER.value.table[1795]), INT_ENUM},*)
(*DBG:    {&(RES0__INSTANCE0.MY_BAD_FIFO.BUFFER.value.table[1796]), INT_ENUM},*)
(*DBG:    {&(RES0__INSTANCE0.MY_BAD_FIFO.BUFFER.value.table[1797]), INT_ENUM},*)
(*DBG:    {&(RES0__INSTANCE0.MY_BAD_FIFO.BUFFER.value.table[1798]), INT_ENUM},*)
(*DBG:    {&(RES0__INSTANCE0.MY_BAD_FIFO.BUFFER.value.table[1799]), INT_ENUM},*)
(*DBG:    {&(RES0__INSTANCE0.MY_BAD_FIFO.BUFFER.value.table[1800]), INT_ENUM},*)
(*DBG:    {&(RES0__INSTANCE0.MY_BAD_FIFO.BUFFER.value.table[1801]), INT_ENUM},*)
(*DBG:    {&(RES0__INSTANCE0.MY_BAD_FIFO.BUFFER.value.table[1802]), INT_ENUM},*)
(*DBG:    {&(RES0__INSTANCE0.MY_BAD_FIFO.BUFFER.value.table[1803]), INT_ENUM},*)
(*DBG:    {&(RES0__INSTANCE0.MY_BAD_FIFO.BUFFER.value.table[1804]), INT_ENUM},*)
(*DBG:    {&(RES0__INSTANCE0.MY_BAD_FIFO.BUFFER.value.table[1805]), INT_ENUM},*)
(*DBG:    {&(RES0__INSTANCE0.MY_BAD_FIFO.BUFFER.value.table[1806]), INT_ENUM},*)
(*DBG:    {&(RES0__INSTANCE0.MY_BAD_FIFO.BUFFER.value.table[1807]), INT_ENUM},*)
(*DBG:    {&(RES0__INSTANCE0.MY_BAD_FIFO.BUFFER.value.table[1808]), INT_ENUM},*)
(*DBG:    {&(RES0__INSTANCE0.MY_BAD_FIFO.BUFFER.value.table[1809]), INT_ENUM},*)
(*DBG:    {&(RES0__INSTANCE0.MY_BAD_FIFO.BUFFER.value.table[1810]), INT_ENUM},*)
(*DBG:    {&(RES0__INSTANCE0.MY_BAD_FIFO.BUFFER.value.table[1811]), INT_ENUM},*)
(*DBG:    {&(RES0__INSTANCE0.MY_BAD_FIFO.BUFFER.value.table[1812]), INT_ENUM},*)
(*DBG:    {&(RES0__INSTANCE0.MY_BAD_FIFO.BUFFER.value.table[1813]), INT_ENUM},*)
(*DBG:    {&(RES0__INSTANCE0.MY_BAD_FIFO.BUFFER.value.table[1814]), INT_ENUM},*)
(*DBG:    {&(RES0__INSTANCE0.MY_BAD_FIFO.BUFFER.value.table[1815]), INT_ENUM},*)
(*DBG:    {&(RES0__INSTANCE0.MY_BAD_FIFO.BUFFER.value.table[1816]), INT_ENUM},*)
(*DBG:    {&(RES0__INSTANCE0.MY_BAD_FIFO.BUFFER.value.table[1817]), INT_ENUM},*)
(*DBG:    {&(RES0__INSTANCE0.MY_BAD_FIFO.BUFFER.value.table[1818]), INT_ENUM},*)
(*DBG:    {&(RES0__INSTANCE0.MY_BAD_FIFO.BUFFER.value.table[1819]), INT_ENUM},*)
(*DBG:    {&(RES0__INSTANCE0.MY_BAD_FIFO.BUFFER.value.table[1820]), INT_ENUM},*)
(*DBG:    {&(RES0__INSTANCE0.MY_BAD_FIFO.BUFFER.value.table[1821]), INT_ENUM},*)
(*DBG:    {&(RES0__INSTANCE0.MY_BAD_FIFO.BUFFER.value.table[1822]), INT_ENUM},*)
(*DBG:    {&(RES0__INSTANCE0.MY_BAD_FIFO.BUFFER.value.table[1823]), INT_ENUM},*)
(*DBG:    {&(RES0__INSTANCE0.MY_BAD_FIFO.BUFFER.value.table[1824]), INT_ENUM},*)
(*DBG:    {&(RES0__INSTANCE0.MY_BAD_FIFO.BUFFER.value.table[1825]), INT_ENUM},*)
(*DBG:    {&(RES0__INSTANCE0.MY_BAD_FIFO.BUFFER.value.table[1826]), INT_ENUM},*)
(*DBG:    {&(RES0__INSTANCE0.MY_BAD_FIFO.BUFFER.value.table[1827]), INT_ENUM},*)
(*DBG:    {&(RES0__INSTANCE0.MY_BAD_FIFO.BUFFER.value.table[1828]), INT_ENUM},*)
(*DBG:    {&(RES0__INSTANCE0.MY_BAD_FIFO.BUFFER.value.table[1829]), INT_ENUM},*)
(*DBG:    {&(RES0__INSTANCE0.MY_BAD_FIFO.BUFFER.value.table[1830]), INT_ENUM},*)
(*DBG:    {&(RES0__INSTANCE0.MY_BAD_FIFO.BUFFER.value.table[1831]), INT_ENUM},*)
(*DBG:    {&(RES0__INSTANCE0.MY_BAD_FIFO.BUFFER.value.table[1832]), INT_ENUM},*)
(*DBG:    {&(RES0__INSTANCE0.MY_BAD_FIFO.BUFFER.value.table[1833]), INT_ENUM},*)
(*DBG:    {&(RES0__INSTANCE0.MY_BAD_FIFO.BUFFER.value.table[1834]), INT_ENUM},*)
(*DBG:    {&(RES0__INSTANCE0.MY_BAD_FIFO.BUFFER.value.table[1835]), INT_ENUM},*)
(*DBG:    {&(RES0__INSTANCE0.MY_BAD_FIFO.BUFFER.value.table[1836]), INT_ENUM},*)
(*DBG:    {&(RES0__INSTANCE0.MY_BAD_FIFO.BUFFER.value.table[1837]), INT_ENUM},*)
(*DBG:    {&(RES0__INSTANCE0.MY_BAD_FIFO.BUFFER.value.table[1838]), INT_ENUM},*)
(*DBG:    {&(RES0__INSTANCE0.MY_BAD_FIFO.BUFFER.value.table[1839]), INT_ENUM},*)
(*DBG:    {&(RES0__INSTANCE0.MY_BAD_FIFO.BUFFER.value.table[1840]), INT_ENUM},*)
(*DBG:    {&(RES0__INSTANCE0.MY_BAD_FIFO.BUFFER.value.table[1841]), INT_ENUM},*)
(*DBG:    {&(RES0__INSTANCE0.MY_BAD_FIFO.BUFFER.value.table[1842]), INT_ENUM},*)
(*DBG:    {&(RES0__INSTANCE0.MY_BAD_FIFO.BUFFER.value.table[1843]), INT_ENUM},*)
(*DBG:    {&(RES0__INSTANCE0.MY_BAD_FIFO.BUFFER.value.table[1844]), INT_ENUM},*)
(*DBG:    {&(RES0__INSTANCE0.MY_BAD_FIFO.BUFFER.value.table[1845]), INT_ENUM},*)
(*DBG:    {&(RES0__INSTANCE0.MY_BAD_FIFO.BUFFER.value.table[1846]), INT_ENUM},*)
(*DBG:    {&(RES0__INSTANCE0.MY_BAD_FIFO.BUFFER.value.table[1847]), INT_ENUM},*)
(*DBG:    {&(RES0__INSTANCE0.MY_BAD_FIFO.BUFFER.value.table[1848]), INT_ENUM},*)
(*DBG:    {&(RES0__INSTANCE0.MY_BAD_FIFO.BUFFER.value.table[1849]), INT_ENUM},*)
(*DBG:    {&(RES0__INSTANCE0.MY_BAD_FIFO.BUFFER.value.table[1850]), INT_ENUM},*)
(*DBG:    {&(RES0__INSTANCE0.MY_BAD_FIFO.BUFFER.value.table[1851]), INT_ENUM},*)
(*DBG:    {&(RES0__INSTANCE0.MY_BAD_FIFO.BUFFER.value.table[1852]), INT_ENUM},*)
(*DBG:    {&(RES0__INSTANCE0.MY_BAD_FIFO.BUFFER.value.table[1853]), INT_ENUM},*)
(*DBG:    {&(RES0__INSTANCE0.MY_BAD_FIFO.BUFFER.value.table[1854]), INT_ENUM},*)
(*DBG:    {&(RES0__INSTANCE0.MY_BAD_FIFO.BUFFER.value.table[1855]), INT_ENUM},*)
(*DBG:    {&(RES0__INSTANCE0.MY_BAD_FIFO.BUFFER.value.table[1856]), INT_ENUM},*)
(*DBG:    {&(RES0__INSTANCE0.MY_BAD_FIFO.BUFFER.value.table[1857]), INT_ENUM},*)
(*DBG:    {&(RES0__INSTANCE0.MY_BAD_FIFO.BUFFER.value.table[1858]), INT_ENUM},*)
(*DBG:    {&(RES0__INSTANCE0.MY_BAD_FIFO.BUFFER.value.table[1859]), INT_ENUM},*)
(*DBG:    {&(RES0__INSTANCE0.MY_BAD_FIFO.BUFFER.value.table[1860]), INT_ENUM},*)
(*DBG:    {&(RES0__INSTANCE0.MY_BAD_FIFO.BUFFER.value.table[1861]), INT_ENUM},*)
(*DBG:    {&(RES0__INSTANCE0.MY_BAD_FIFO.BUFFER.value.table[1862]), INT_ENUM},*)
(*DBG:    {&(RES0__INSTANCE0.MY_BAD_FIFO.BUFFER.value.table[1863]), INT_ENUM},*)
(*DBG:    {&(RES0__INSTANCE0.MY_BAD_FIFO.BUFFER.value.table[1864]), INT_ENUM},*)
(*DBG:    {&(RES0__INSTANCE0.MY_BAD_FIFO.BUFFER.value.table[1865]), INT_ENUM},*)
(*DBG:    {&(RES0__INSTANCE0.MY_BAD_FIFO.BUFFER.value.table[1866]), INT_ENUM},*)
(*DBG:    {&(RES0__INSTANCE0.MY_BAD_FIFO.BUFFER.value.table[1867]), INT_ENUM},*)
(*DBG:    {&(RES0__INSTANCE0.MY_BAD_FIFO.BUFFER.value.table[1868]), INT_ENUM},*)
(*DBG:    {&(RES0__INSTANCE0.MY_BAD_FIFO.BUFFER.value.table[1869]), INT_ENUM},*)
(*DBG:    {&(RES0__INSTANCE0.MY_BAD_FIFO.BUFFER.value.table[1870]), INT_ENUM},*)
(*DBG:    {&(RES0__INSTANCE0.MY_BAD_FIFO.BUFFER.value.table[1871]), INT_ENUM},*)
(*DBG:    {&(RES0__INSTANCE0.MY_BAD_FIFO.BUFFER.value.table[1872]), INT_ENUM},*)
(*DBG:    {&(RES0__INSTANCE0.MY_BAD_FIFO.BUFFER.value.table[1873]), INT_ENUM},*)
(*DBG:    {&(RES0__INSTANCE0.MY_BAD_FIFO.BUFFER.value.table[1874]), INT_ENUM},*)
(*DBG:    {&(RES0__INSTANCE0.MY_BAD_FIFO.BUFFER.value.table[1875]), INT_ENUM},*)
(*DBG:    {&(RES0__INSTANCE0.MY_BAD_FIFO.BUFFER.value.table[1876]), INT_ENUM},*)
(*DBG:    {&(RES0__INSTANCE0.MY_BAD_FIFO.BUFFER.value.table[1877]), INT_ENUM},*)
(*DBG:    {&(RES0__INSTANCE0.MY_BAD_FIFO.BUFFER.value.table[1878]), INT_ENUM},*)
(*DBG:    {&(RES0__INSTANCE0.MY_BAD_FIFO.BUFFER.value.table[1879]), INT_ENUM},*)
(*DBG:    {&(RES0__INSTANCE0.MY_BAD_FIFO.BUFFER.value.table[1880]), INT_ENUM},*)
(*DBG:    {&(RES0__INSTANCE0.MY_BAD_FIFO.BUFFER.value.table[1881]), INT_ENUM},*)
(*DBG:    {&(RES0__INSTANCE0.MY_BAD_FIFO.BUFFER.value.table[1882]), INT_ENUM},*)
(*DBG:    {&(RES0__INSTANCE0.MY_BAD_FIFO.BUFFER.value.table[1883]), INT_ENUM},*)
(*DBG:    {&(RES0__INSTANCE0.MY_BAD_FIFO.BUFFER.value.table[1884]), INT_ENUM},*)
(*DBG:    {&(RES0__INSTANCE0.MY_BAD_FIFO.BUFFER.value.table[1885]), INT_ENUM},*)
(*DBG:    {&(RES0__INSTANCE0.MY_BAD_FIFO.BUFFER.value.table[1886]), INT_ENUM},*)
(*DBG:    {&(RES0__INSTANCE0.MY_BAD_FIFO.BUFFER.value.table[1887]), INT_ENUM},*)
(*DBG:    {&(RES0__INSTANCE0.MY_BAD_FIFO.BUFFER.value.table[1888]), INT_ENUM},*)
(*DBG:    {&(RES0__INSTANCE0.MY_BAD_FIFO.BUFFER.value.table[1889]), INT_ENUM},*)
(*DBG:    {&(RES0__INSTANCE0.MY_BAD_FIFO.BUFFER.value.table[1890]), INT_ENUM},*)
(*DBG:    {&(RES0__INSTANCE0.MY_BAD_FIFO.BUFFER.value.table[1891]), INT_ENUM},*)
(*DBG:    {&(RES0__INSTANCE0.MY_BAD_FIFO.BUFFER.value.table[1892]), INT_ENUM},*)
(*DBG:    {&(RES0__INSTANCE0.MY_BAD_FIFO.BUFFER.value.table[1893]), INT_ENUM},*)
(*DBG:    {&(RES0__INSTANCE0.MY_BAD_FIFO.BUFFER.value.table[1894]), INT_ENUM},*)
(*DBG:    {&(RES0__INSTANCE0.MY_BAD_FIFO.BUFFER.value.table[1895]), INT_ENUM},*)
(*DBG:    {&(RES0__INSTANCE0.MY_BAD_FIFO.BUFFER.value.table[1896]), INT_ENUM},*)
(*DBG:    {&(RES0__INSTANCE0.MY_BAD_FIFO.BUFFER.value.table[1897]), INT_ENUM},*)
(*DBG:    {&(RES0__INSTANCE0.MY_BAD_FIFO.BUFFER.value.table[1898]), INT_ENUM},*)
(*DBG:    {&(RES0__INSTANCE0.MY_BAD_FIFO.BUFFER.value.table[1899]), INT_ENUM},*)
(*DBG:    {&(RES0__INSTANCE0.MY_BAD_FIFO.BUFFER.value.table[1900]), INT_ENUM},*)
(*DBG:    {&(RES0__INSTANCE0.MY_BAD_FIFO.BUFFER.value.table[1901]), INT_ENUM},*)
(*DBG:    {&(RES0__INSTANCE0.MY_BAD_FIFO.BUFFER.value.table[1902]), INT_ENUM},*)
(*DBG:    {&(RES0__INSTANCE0.MY_BAD_FIFO.BUFFER.value.table[1903]), INT_ENUM},*)
(*DBG:    {&(RES0__INSTANCE0.MY_BAD_FIFO.BUFFER.value.table[1904]), INT_ENUM},*)
(*DBG:    {&(RES0__INSTANCE0.MY_BAD_FIFO.BUFFER.value.table[1905]), INT_ENUM},*)
(*DBG:    {&(RES0__INSTANCE0.MY_BAD_FIFO.BUFFER.value.table[1906]), INT_ENUM},*)
(*DBG:    {&(RES0__INSTANCE0.MY_BAD_FIFO.BUFFER.value.table[1907]), INT_ENUM},*)
(*DBG:    {&(RES0__INSTANCE0.MY_BAD_FIFO.BUFFER.value.table[1908]), INT_ENUM},*)
(*DBG:    {&(RES0__INSTANCE0.MY_BAD_FIFO.BUFFER.value.table[1909]), INT_ENUM},*)
(*DBG:    {&(RES0__INSTANCE0.MY_BAD_FIFO.BUFFER.value.table[1910]), INT_ENUM},*)
(*DBG:    {&(RES0__INSTANCE0.MY_BAD_FIFO.BUFFER.value.table[1911]), INT_ENUM},*)
(*DBG:    {&(RES0__INSTANCE0.MY_BAD_FIFO.BUFFER.value.table[1912]), INT_ENUM},*)
(*DBG:    {&(RES0__INSTANCE0.MY_BAD_FIFO.BUFFER.value.table[1913]), INT_ENUM},*)
(*DBG:    {&(RES0__INSTANCE0.MY_BAD_FIFO.BUFFER.value.table[1914]), INT_ENUM},*)
(*DBG:    {&(RES0__INSTANCE0.MY_BAD_FIFO.BUFFER.value.table[1915]), INT_ENUM},*)
(*DBG:    {&(RES0__INSTANCE0.MY_BAD_FIFO.BUFFER.value.table[1916]), INT_ENUM},*)
(*DBG:    {&(RES0__INSTANCE0.MY_BAD_FIFO.BUFFER.value.table[1917]), INT_ENUM},*)
(*DBG:    {&(RES0__INSTANCE0.MY_BAD_FIFO.BUFFER.value.table[1918]), INT_ENUM},*)
(*DBG:    {&(RES0__INSTANCE0.MY_BAD_FIFO.BUFFER.value.table[1919]), INT_ENUM},*)
(*DBG:    {&(RES0__INSTANCE0.MY_BAD_FIFO.BUFFER.value.table[1920]), INT_ENUM},*)
(*DBG:    {&(RES0__INSTANCE0.MY_BAD_FIFO.BUFFER.value.table[1921]), INT_ENUM},*)
(*DBG:    {&(RES0__INSTANCE0.MY_BAD_FIFO.BUFFER.value.table[1922]), INT_ENUM},*)
(*DBG:    {&(RES0__INSTANCE0.MY_BAD_FIFO.BUFFER.value.table[1923]), INT_ENUM},*)
(*DBG:    {&(RES0__INSTANCE0.MY_BAD_FIFO.BUFFER.value.table[1924]), INT_ENUM},*)
(*DBG:    {&(RES0__INSTANCE0.MY_BAD_FIFO.BUFFER.value.table[1925]), INT_ENUM},*)
(*DBG:    {&(RES0__INSTANCE0.MY_BAD_FIFO.BUFFER.value.table[1926]), INT_ENUM},*)
(*DBG:    {&(RES0__INSTANCE0.MY_BAD_FIFO.BUFFER.value.table[1927]), INT_ENUM},*)
(*DBG:    {&(RES0__INSTANCE0.MY_BAD_FIFO.BUFFER.value.table[1928]), INT_ENUM},*)
(*DBG:    {&(RES0__INSTANCE0.MY_BAD_FIFO.BUFFER.value.table[1929]), INT_ENUM},*)
(*DBG:    {&(RES0__INSTANCE0.MY_BAD_FIFO.BUFFER.value.table[1930]), INT_ENUM},*)
(*DBG:    {&(RES0__INSTANCE0.MY_BAD_FIFO.BUFFER.value.table[1931]), INT_ENUM},*)
(*DBG:    {&(RES0__INSTANCE0.MY_BAD_FIFO.BUFFER.value.table[1932]), INT_ENUM},*)
(*DBG:    {&(RES0__INSTANCE0.MY_BAD_FIFO.BUFFER.value.table[1933]), INT_ENUM},*)
(*DBG:    {&(RES0__INSTANCE0.MY_BAD_FIFO.BUFFER.value.table[1934]), INT_ENUM},*)
(*DBG:    {&(RES0__INSTANCE0.MY_BAD_FIFO.BUFFER.value.table[1935]), INT_ENUM},*)
(*DBG:    {&(RES0__INSTANCE0.MY_BAD_FIFO.BUFFER.value.table[1936]), INT_ENUM},*)
(*DBG:    {&(RES0__INSTANCE0.MY_BAD_FIFO.BUFFER.value.table[1937]), INT_ENUM},*)
(*DBG:    {&(RES0__INSTANCE0.MY_BAD_FIFO.BUFFER.value.table[1938]), INT_ENUM},*)
(*DBG:    {&(RES0__INSTANCE0.MY_BAD_FIFO.BUFFER.value.table[1939]), INT_ENUM},*)
(*DBG:    {&(RES0__INSTANCE0.MY_BAD_FIFO.BUFFER.value.table[1940]), INT_ENUM},*)
(*DBG:    {&(RES0__INSTANCE0.MY_BAD_FIFO.BUFFER.value.table[1941]), INT_ENUM},*)
(*DBG:    {&(RES0__INSTANCE0.MY_BAD_FIFO.BUFFER.value.table[1942]), INT_ENUM},*)
(*DBG:    {&(RES0__INSTANCE0.MY_BAD_FIFO.BUFFER.value.table[1943]), INT_ENUM},*)
(*DBG:    {&(RES0__INSTANCE0.MY_BAD_FIFO.BUFFER.value.table[1944]), INT_ENUM},*)
(*DBG:    {&(RES0__INSTANCE0.MY_BAD_FIFO.BUFFER.value.table[1945]), INT_ENUM},*)
(*DBG:    {&(RES0__INSTANCE0.MY_BAD_FIFO.BUFFER.value.table[1946]), INT_ENUM},*)
(*DBG:    {&(RES0__INSTANCE0.MY_BAD_FIFO.BUFFER.value.table[1947]), INT_ENUM},*)
(*DBG:    {&(RES0__INSTANCE0.MY_BAD_FIFO.BUFFER.value.table[1948]), INT_ENUM},*)
(*DBG:    {&(RES0__INSTANCE0.MY_BAD_FIFO.BUFFER.value.table[1949]), INT_ENUM},*)
(*DBG:    {&(RES0__INSTANCE0.MY_BAD_FIFO.BUFFER.value.table[1950]), INT_ENUM},*)
(*DBG:    {&(RES0__INSTANCE0.MY_BAD_FIFO.BUFFER.value.table[1951]), INT_ENUM},*)
(*DBG:    {&(RES0__INSTANCE0.MY_BAD_FIFO.BUFFER.value.table[1952]), INT_ENUM},*)
(*DBG:    {&(RES0__INSTANCE0.MY_BAD_FIFO.BUFFER.value.table[1953]), INT_ENUM},*)
(*DBG:    {&(RES0__INSTANCE0.MY_BAD_FIFO.BUFFER.value.table[1954]), INT_ENUM},*)
(*DBG:    {&(RES0__INSTANCE0.MY_BAD_FIFO.BUFFER.value.table[1955]), INT_ENUM},*)
(*DBG:    {&(RES0__INSTANCE0.MY_BAD_FIFO.BUFFER.value.table[1956]), INT_ENUM},*)
(*DBG:    {&(RES0__INSTANCE0.MY_BAD_FIFO.BUFFER.value.table[1957]), INT_ENUM},*)
(*DBG:    {&(RES0__INSTANCE0.MY_BAD_FIFO.BUFFER.value.table[1958]), INT_ENUM},*)
(*DBG:    {&(RES0__INSTANCE0.MY_BAD_FIFO.BUFFER.value.table[1959]), INT_ENUM},*)
(*DBG:    {&(RES0__INSTANCE0.MY_BAD_FIFO.BUFFER.value.table[1960]), INT_ENUM},*)
(*DBG:    {&(RES0__INSTANCE0.MY_BAD_FIFO.BUFFER.value.table[1961]), INT_ENUM},*)
(*DBG:    {&(RES0__INSTANCE0.MY_BAD_FIFO.BUFFER.value.table[1962]), INT_ENUM},*)
(*DBG:    {&(RES0__INSTANCE0.MY_BAD_FIFO.BUFFER.value.table[1963]), INT_ENUM},*)
(*DBG:    {&(RES0__INSTANCE0.MY_BAD_FIFO.BUFFER.value.table[1964]), INT_ENUM},*)
(*DBG:    {&(RES0__INSTANCE0.MY_BAD_FIFO.BUFFER.value.table[1965]), INT_ENUM},*)
(*DBG:    {&(RES0__INSTANCE0.MY_BAD_FIFO.BUFFER.value.table[1966]), INT_ENUM},*)
(*DBG:    {&(RES0__INSTANCE0.MY_BAD_FIFO.BUFFER.value.table[1967]), INT_ENUM},*)
(*DBG:    {&(RES0__INSTANCE0.MY_BAD_FIFO.BUFFER.value.table[1968]), INT_ENUM},*)
(*DBG:    {&(RES0__INSTANCE0.MY_BAD_FIFO.BUFFER.value.table[1969]), INT_ENUM},*)
(*DBG:    {&(RES0__INSTANCE0.MY_BAD_FIFO.BUFFER.value.table[1970]), INT_ENUM},*)
(*DBG:    {&(RES0__INSTANCE0.MY_BAD_FIFO.BUFFER.value.table[1971]), INT_ENUM},*)
(*DBG:    {&(RES0__INSTANCE0.MY_BAD_FIFO.BUFFER.value.table[1972]), INT_ENUM},*)
(*DBG:    {&(RES0__INSTANCE0.MY_BAD_FIFO.BUFFER.value.table[1973]), INT_ENUM},*)
(*DBG:    {&(RES0__INSTANCE0.MY_BAD_FIFO.BUFFER.value.table[1974]), INT_ENUM},*)
(*DBG:    {&(RES0__INSTANCE0.MY_BAD_FIFO.BUFFER.value.table[1975]), INT_ENUM},*)
(*DBG:    {&(RES0__INSTANCE0.MY_BAD_FIFO.BUFFER.value.table[1976]), INT_ENUM},*)
(*DBG:    {&(RES0__INSTANCE0.MY_BAD_FIFO.BUFFER.value.table[1977]), INT_ENUM},*)
(*DBG:    {&(RES0__INSTANCE0.MY_BAD_FIFO.BUFFER.value.table[1978]), INT_ENUM},*)
(*DBG:    {&(RES0__INSTANCE0.MY_BAD_FIFO.BUFFER.value.table[1979]), INT_ENUM},*)
(*DBG:    {&(RES0__INSTANCE0.MY_BAD_FIFO.BUFFER.value.table[1980]), INT_ENUM},*)
(*DBG:    {&(RES0__INSTANCE0.MY_BAD_FIFO.BUFFER.value.table[1981]), INT_ENUM},*)
(*DBG:    {&(RES0__INSTANCE0.MY_BAD_FIFO.BUFFER.value.table[1982]), INT_ENUM},*)
(*DBG:    {&(RES0__INSTANCE0.MY_BAD_FIFO.BUFFER.value.table[1983]), INT_ENUM},*)
(*DBG:    {&(RES0__INSTANCE0.MY_BAD_FIFO.BUFFER.value.table[1984]), INT_ENUM},*)
(*DBG:    {&(RES0__INSTANCE0.MY_BAD_FIFO.BUFFER.value.table[1985]), INT_ENUM},*)
(*DBG:    {&(RES0__INSTANCE0.MY_BAD_FIFO.BUFFER.value.table[1986]), INT_ENUM},*)
(*DBG:    {&(RES0__INSTANCE0.MY_BAD_FIFO.BUFFER.value.table[1987]), INT_ENUM},*)
(*DBG:    {&(RES0__INSTANCE0.MY_BAD_FIFO.BUFFER.value.table[1988]), INT_ENUM},*)
(*DBG:    {&(RES0__INSTANCE0.MY_BAD_FIFO.BUFFER.value.table[1989]), INT_ENUM},*)
(*DBG:    {&(RES0__INSTANCE0.MY_BAD_FIFO.BUFFER.value.table[1990]), INT_ENUM},*)
(*DBG:    {&(RES0__INSTANCE0.MY_BAD_FIFO.BUFFER.value.table[1991]), INT_ENUM},*)
(*DBG:    {&(RES0__INSTANCE0.MY_BAD_FIFO.BUFFER.value.table[1992]), INT_ENUM},*)
(*DBG:    {&(RES0__INSTANCE0.MY_BAD_FIFO.BUFFER.value.table[1993]), INT_ENUM},*)
(*DBG:    {&(RES0__INSTANCE0.MY_BAD_FIFO.BUFFER.value.table[1994]), INT_ENUM},*)
(*DBG:    {&(RES0__INSTANCE0.MY_BAD_FIFO.BUFFER.value.table[1995]), INT_ENUM},*)
(*DBG:    {&(RES0__INSTANCE0.MY_BAD_FIFO.BUFFER.value.table[1996]), INT_ENUM},*)
(*DBG:    {&(RES0__INSTANCE0.MY_BAD_FIFO.BUFFER.value.table[1997]), INT_ENUM},*)
(*DBG:    {&(RES0__INSTANCE0.MY_BAD_FIFO.BUFFER.value.table[1998]), INT_ENUM},*)
(*DBG:    {&(RES0__INSTANCE0.MY_BAD_FIFO.BUFFER.value.table[1999]), INT_ENUM},*)
(*DBG:    {&(RES0__INSTANCE0.MY_BAD_FIFO.BUFFER.value.table[2000]), INT_ENUM},*)
(*DBG:    {&(RES0__INSTANCE0.MY_BAD_FIFO.BUFFER.value.table[2001]), INT_ENUM},*)
(*DBG:    {&(RES0__INSTANCE0.MY_BAD_FIFO.BUFFER.value.table[2002]), INT_ENUM},*)
(*DBG:    {&(RES0__INSTANCE0.MY_BAD_FIFO.BUFFER.value.table[2003]), INT_ENUM},*)
(*DBG:    {&(RES0__INSTANCE0.MY_BAD_FIFO.BUFFER.value.table[2004]), INT_ENUM},*)
(*DBG:    {&(RES0__INSTANCE0.MY_BAD_FIFO.BUFFER.value.table[2005]), INT_ENUM},*)
(*DBG:    {&(RES0__INSTANCE0.MY_BAD_FIFO.BUFFER.value.table[2006]), INT_ENUM},*)
(*DBG:    {&(RES0__INSTANCE0.MY_BAD_FIFO.BUFFER.value.table[2007]), INT_ENUM},*)
(*DBG:    {&(RES0__INSTANCE0.MY_BAD_FIFO.BUFFER.value.table[2008]), INT_ENUM},*)
(*DBG:    {&(RES0__INSTANCE0.MY_BAD_FIFO.BUFFER.value.table[2009]), INT_ENUM},*)
(*DBG:    {&(RES0__INSTANCE0.MY_BAD_FIFO.BUFFER.value.table[2010]), INT_ENUM},*)
(*DBG:    {&(RES0__INSTANCE0.MY_BAD_FIFO.BUFFER.value.table[2011]), INT_ENUM},*)
(*DBG:    {&(RES0__INSTANCE0.MY_BAD_FIFO.BUFFER.value.table[2012]), INT_ENUM},*)
(*DBG:    {&(RES0__INSTANCE0.MY_BAD_FIFO.BUFFER.value.table[2013]), INT_ENUM},*)
(*DBG:    {&(RES0__INSTANCE0.MY_BAD_FIFO.BUFFER.value.table[2014]), INT_ENUM},*)
(*DBG:    {&(RES0__INSTANCE0.MY_BAD_FIFO.BUFFER.value.table[2015]), INT_ENUM},*)
(*DBG:    {&(RES0__INSTANCE0.MY_BAD_FIFO.BUFFER.value.table[2016]), INT_ENUM},*)
(*DBG:    {&(RES0__INSTANCE0.MY_BAD_FIFO.BUFFER.value.table[2017]), INT_ENUM},*)
(*DBG:    {&(RES0__INSTANCE0.MY_BAD_FIFO.BUFFER.value.table[2018]), INT_ENUM},*)
(*DBG:    {&(RES0__INSTANCE0.MY_BAD_FIFO.BUFFER.value.table[2019]), INT_ENUM},*)
(*DBG:    {&(RES0__INSTANCE0.MY_BAD_FIFO.BUFFER.value.table[2020]), INT_ENUM},*)
(*DBG:    {&(RES0__INSTANCE0.MY_BAD_FIFO.BUFFER.value.table[2021]), INT_ENUM},*)
(*DBG:    {&(RES0__INSTANCE0.MY_BAD_FIFO.BUFFER.value.table[2022]), INT_ENUM},*)
(*DBG:    {&(RES0__INSTANCE0.MY_BAD_FIFO.BUFFER.value.table[2023]), INT_ENUM},*)
(*DBG:    {&(RES0__INSTANCE0.MY_BAD_FIFO.BUFFER.value.table[2024]), INT_ENUM},*)
(*DBG:    {&(RES0__INSTANCE0.MY_BAD_FIFO.BUFFER.value.table[2025]), INT_ENUM},*)
(*DBG:    {&(RES0__INSTANCE0.MY_BAD_FIFO.BUFFER.value.table[2026]), INT_ENUM},*)
(*DBG:    {&(RES0__INSTANCE0.MY_BAD_FIFO.BUFFER.value.table[2027]), INT_ENUM},*)
(*DBG:    {&(RES0__INSTANCE0.MY_BAD_FIFO.BUFFER.value.table[2028]), INT_ENUM},*)
(*DBG:    {&(RES0__INSTANCE0.MY_BAD_FIFO.BUFFER.value.table[2029]), INT_ENUM},*)
(*DBG:    {&(RES0__INSTANCE0.MY_BAD_FIFO.BUFFER.value.table[2030]), INT_ENUM},*)
(*DBG:    {&(RES0__INSTANCE0.MY_BAD_FIFO.BUFFER.value.table[2031]), INT_ENUM},*)
(*DBG:    {&(RES0__INSTANCE0.MY_BAD_FIFO.BUFFER.value.table[2032]), INT_ENUM},*)
(*DBG:    {&(RES0__INSTANCE0.MY_BAD_FIFO.BUFFER.value.table[2033]), INT_ENUM},*)
(*DBG:    {&(RES0__INSTANCE0.MY_BAD_FIFO.BUFFER.value.table[2034]), INT_ENUM},*)
(*DBG:    {&(RES0__INSTANCE0.MY_BAD_FIFO.BUFFER.value.table[2035]), INT_ENUM},*)
(*DBG:    {&(RES0__INSTANCE0.MY_BAD_FIFO.BUFFER.value.table[2036]), INT_ENUM},*)
(*DBG:    {&(RES0__INSTANCE0.MY_BAD_FIFO.BUFFER.value.table[2037]), INT_ENUM},*)
(*DBG:    {&(RES0__INSTANCE0.MY_BAD_FIFO.BUFFER.value.table[2038]), INT_ENUM},*)
(*DBG:    {&(RES0__INSTANCE0.MY_BAD_FIFO.BUFFER.value.table[2039]), INT_ENUM},*)
(*DBG:    {&(RES0__INSTANCE0.MY_BAD_FIFO.BUFFER.value.table[2040]), INT_ENUM},*)
(*DBG:    {&(RES0__INSTANCE0.MY_BAD_FIFO.BUFFER.value.table[2041]), INT_ENUM},*)
(*DBG:    {&(RES0__INSTANCE0.MY_BAD_FIFO.BUFFER.value.table[2042]), INT_ENUM},*)
(*DBG:    {&(RES0__INSTANCE0.MY_BAD_FIFO.BUFFER.value.table[2043]), INT_ENUM},*)
(*DBG:    {&(RES0__INSTANCE0.MY_BAD_FIFO.BUFFER.value.table[2044]), INT_ENUM},*)
(*DBG:    {&(RES0__INSTANCE0.MY_BAD_FIFO.BUFFER.value.table[2045]), INT_ENUM},*)
(*DBG:    {&(RES0__INSTANCE0.MY_BAD_FIFO.BUFFER.value.table[2046]), INT_ENUM},*)
(*DBG:    {&(RES0__INSTANCE0.MY_BAD_FIFO.BUFFER.value.table[2047]), INT_ENUM},*)
(*DBG:    {&(RES0__INSTANCE0.MY_BAD_FIFO.BUFFER.value.table[2048]), INT_ENUM},*)
(*DBG:    {&(RES0__INSTANCE0.MY_BAD_FIFO.BUFFER.value.table[2049]), INT_ENUM},*)
(*DBG:    {&(RES0__INSTANCE0.MY_BAD_FIFO.BUFFER.value.table[2050]), INT_ENUM},*)
(*DBG:    {&(RES0__INSTANCE0.MY_BAD_FIFO.BUFFER.value.table[2051]), INT_ENUM},*)
(*DBG:    {&(RES0__INSTANCE0.MY_BAD_FIFO.BUFFER.value.table[2052]), INT_ENUM},*)
(*DBG:    {&(RES0__INSTANCE0.MY_BAD_FIFO.BUFFER.value.table[2053]), INT_ENUM},*)
(*DBG:    {&(RES0__INSTANCE0.MY_BAD_FIFO.BUFFER.value.table[2054]), INT_ENUM},*)
(*DBG:    {&(RES0__INSTANCE0.MY_BAD_FIFO.BUFFER.value.table[2055]), INT_ENUM},*)
(*DBG:    {&(RES0__INSTANCE0.MY_BAD_FIFO.BUFFER.value.table[2056]), INT_ENUM},*)
(*DBG:    {&(RES0__INSTANCE0.MY_BAD_FIFO.BUFFER.value.table[2057]), INT_ENUM},*)
(*DBG:    {&(RES0__INSTANCE0.MY_BAD_FIFO.BUFFER.value.table[2058]), INT_ENUM},*)
(*DBG:    {&(RES0__INSTANCE0.MY_BAD_FIFO.BUFFER.value.table[2059]), INT_ENUM},*)
(*DBG:    {&(RES0__INSTANCE0.MY_BAD_FIFO.BUFFER.value.table[2060]), INT_ENUM},*)
(*DBG:    {&(RES0__INSTANCE0.MY_BAD_FIFO.BUFFER.value.table[2061]), INT_ENUM},*)
(*DBG:    {&(RES0__INSTANCE0.MY_BAD_FIFO.BUFFER.value.table[2062]), INT_ENUM},*)
(*DBG:    {&(RES0__INSTANCE0.MY_BAD_FIFO.BUFFER.value.table[2063]), INT_ENUM},*)
(*DBG:    {&(RES0__INSTANCE0.MY_BAD_FIFO.BUFFER.value.table[2064]), INT_ENUM},*)
(*DBG:    {&(RES0__INSTANCE0.MY_BAD_FIFO.BUFFER.value.table[2065]), INT_ENUM},*)
(*DBG:    {&(RES0__INSTANCE0.MY_BAD_FIFO.BUFFER.value.table[2066]), INT_ENUM},*)
(*DBG:    {&(RES0__INSTANCE0.MY_BAD_FIFO.BUFFER.value.table[2067]), INT_ENUM},*)
(*DBG:    {&(RES0__INSTANCE0.MY_BAD_FIFO.BUFFER.value.table[2068]), INT_ENUM},*)
(*DBG:    {&(RES0__INSTANCE0.MY_BAD_FIFO.BUFFER.value.table[2069]), INT_ENUM},*)
(*DBG:    {&(RES0__INSTANCE0.MY_BAD_FIFO.BUFFER.value.table[2070]), INT_ENUM},*)
(*DBG:    {&(RES0__INSTANCE0.MY_BAD_FIFO.BUFFER.value.table[2071]), INT_ENUM},*)
(*DBG:    {&(RES0__INSTANCE0.MY_BAD_FIFO.BUFFER.value.table[2072]), INT_ENUM},*)
(*DBG:    {&(RES0__INSTANCE0.MY_BAD_FIFO.BUFFER.value.table[2073]), INT_ENUM},*)
(*DBG:    {&(RES0__INSTANCE0.MY_BAD_FIFO.BUFFER.value.table[2074]), INT_ENUM},*)
(*DBG:    {&(RES0__INSTANCE0.MY_BAD_FIFO.BUFFER.value.table[2075]), INT_ENUM},*)
(*DBG:    {&(RES0__INSTANCE0.MY_BAD_FIFO.BUFFER.value.table[2076]), INT_ENUM},*)
(*DBG:    {&(RES0__INSTANCE0.MY_BAD_FIFO.BUFFER.value.table[2077]), INT_ENUM},*)
(*DBG:    {&(RES0__INSTANCE0.MY_BAD_FIFO.BUFFER.value.table[2078]), INT_ENUM},*)
(*DBG:    {&(RES0__INSTANCE0.MY_BAD_FIFO.BUFFER.value.table[2079]), INT_ENUM},*)
(*DBG:    {&(RES0__INSTANCE0.MY_BAD_FIFO.BUFFER.value.table[2080]), INT_ENUM},*)
(*DBG:    {&(RES0__INSTANCE0.MY_BAD_FIFO.BUFFER.value.table[2081]), INT_ENUM},*)
(*DBG:    {&(RES0__INSTANCE0.MY_BAD_FIFO.BUFFER.value.table[2082]), INT_ENUM},*)
(*DBG:    {&(RES0__INSTANCE0.MY_BAD_FIFO.BUFFER.value.table[2083]), INT_ENUM},*)
(*DBG:    {&(RES0__INSTANCE0.MY_BAD_FIFO.BUFFER.value.table[2084]), INT_ENUM},*)
(*DBG:    {&(RES0__INSTANCE0.MY_BAD_FIFO.BUFFER.value.table[2085]), INT_ENUM},*)
(*DBG:    {&(RES0__INSTANCE0.MY_BAD_FIFO.BUFFER.value.table[2086]), INT_ENUM},*)
(*DBG:    {&(RES0__INSTANCE0.MY_BAD_FIFO.BUFFER.value.table[2087]), INT_ENUM},*)
(*DBG:    {&(RES0__INSTANCE0.MY_BAD_FIFO.BUFFER.value.table[2088]), INT_ENUM},*)
(*DBG:    {&(RES0__INSTANCE0.MY_BAD_FIFO.BUFFER.value.table[2089]), INT_ENUM},*)
(*DBG:    {&(RES0__INSTANCE0.MY_BAD_FIFO.BUFFER.value.table[2090]), INT_ENUM},*)
(*DBG:    {&(RES0__INSTANCE0.MY_BAD_FIFO.BUFFER.value.table[2091]), INT_ENUM},*)
(*DBG:    {&(RES0__INSTANCE0.MY_BAD_FIFO.BUFFER.value.table[2092]), INT_ENUM},*)
(*DBG:    {&(RES0__INSTANCE0.MY_BAD_FIFO.BUFFER.value.table[2093]), INT_ENUM},*)
(*DBG:    {&(RES0__INSTANCE0.MY_BAD_FIFO.BUFFER.value.table[2094]), INT_ENUM},*)
(*DBG:    {&(RES0__INSTANCE0.MY_BAD_FIFO.BUFFER.value.table[2095]), INT_ENUM},*)
(*DBG:    {&(RES0__INSTANCE0.MY_BAD_FIFO.BUFFER.value.table[2096]), INT_ENUM},*)
(*DBG:    {&(RES0__INSTANCE0.MY_BAD_FIFO.BUFFER.value.table[2097]), INT_ENUM},*)
(*DBG:    {&(RES0__INSTANCE0.MY_BAD_FIFO.BUFFER.value.table[2098]), INT_ENUM},*)
(*DBG:    {&(RES0__INSTANCE0.MY_BAD_FIFO.BUFFER.value.table[2099]), INT_ENUM},*)
(*DBG:    {&(RES0__INSTANCE0.MY_BAD_FIFO.BUFFER.value.table[2100]), INT_ENUM},*)
(*DBG:    {&(RES0__INSTANCE0.MY_BAD_FIFO.BUFFER.value.table[2101]), INT_ENUM},*)
(*DBG:    {&(RES0__INSTANCE0.MY_BAD_FIFO.BUFFER.value.table[2102]), INT_ENUM},*)
(*DBG:    {&(RES0__INSTANCE0.MY_BAD_FIFO.BUFFER.value.table[2103]), INT_ENUM},*)
(*DBG:    {&(RES0__INSTANCE0.MY_BAD_FIFO.BUFFER.value.table[2104]), INT_ENUM},*)
(*DBG:    {&(RES0__INSTANCE0.MY_BAD_FIFO.BUFFER.value.table[2105]), INT_ENUM},*)
(*DBG:    {&(RES0__INSTANCE0.MY_BAD_FIFO.BUFFER.value.table[2106]), INT_ENUM},*)
(*DBG:    {&(RES0__INSTANCE0.MY_BAD_FIFO.BUFFER.value.table[2107]), INT_ENUM},*)
(*DBG:    {&(RES0__INSTANCE0.MY_BAD_FIFO.BUFFER.value.table[2108]), INT_ENUM},*)
(*DBG:    {&(RES0__INSTANCE0.MY_BAD_FIFO.BUFFER.value.table[2109]), INT_ENUM},*)
(*DBG:    {&(RES0__INSTANCE0.MY_BAD_FIFO.BUFFER.value.table[2110]), INT_ENUM},*)
(*DBG:    {&(RES0__INSTANCE0.MY_BAD_FIFO.BUFFER.value.table[2111]), INT_ENUM},*)
(*DBG:    {&(RES0__INSTANCE0.MY_BAD_FIFO.BUFFER.value.table[2112]), INT_ENUM},*)
(*DBG:    {&(RES0__INSTANCE0.MY_BAD_FIFO.BUFFER.value.table[2113]), INT_ENUM},*)
(*DBG:    {&(RES0__INSTANCE0.MY_BAD_FIFO.BUFFER.value.table[2114]), INT_ENUM},*)
(*DBG:    {&(RES0__INSTANCE0.MY_BAD_FIFO.BUFFER.value.table[2115]), INT_ENUM},*)
(*DBG:    {&(RES0__INSTANCE0.MY_BAD_FIFO.BUFFER.value.table[2116]), INT_ENUM},*)
(*DBG:    {&(RES0__INSTANCE0.MY_BAD_FIFO.BUFFER.value.table[2117]), INT_ENUM},*)
(*DBG:    {&(RES0__INSTANCE0.MY_BAD_FIFO.BUFFER.value.table[2118]), INT_ENUM},*)
(*DBG:    {&(RES0__INSTANCE0.MY_BAD_FIFO.BUFFER.value.table[2119]), INT_ENUM},*)
(*DBG:    {&(RES0__INSTANCE0.MY_BAD_FIFO.BUFFER.value.table[2120]), INT_ENUM},*)
(*DBG:    {&(RES0__INSTANCE0.MY_BAD_FIFO.BUFFER.value.table[2121]), INT_ENUM},*)
(*DBG:    {&(RES0__INSTANCE0.MY_BAD_FIFO.BUFFER.value.table[2122]), INT_ENUM},*)
(*DBG:    {&(RES0__INSTANCE0.MY_BAD_FIFO.BUFFER.value.table[2123]), INT_ENUM},*)
(*DBG:    {&(RES0__INSTANCE0.MY_BAD_FIFO.BUFFER.value.table[2124]), INT_ENUM},*)
(*DBG:    {&(RES0__INSTANCE0.MY_BAD_FIFO.BUFFER.value.table[2125]), INT_ENUM},*)
(*DBG:    {&(RES0__INSTANCE0.MY_BAD_FIFO.BUFFER.value.table[2126]), INT_ENUM},*)
(*DBG:    {&(RES0__INSTANCE0.MY_BAD_FIFO.BUFFER.value.table[2127]), INT_ENUM},*)
(*DBG:    {&(RES0__INSTANCE0.MY_BAD_FIFO.BUFFER.value.table[2128]), INT_ENUM},*)
(*DBG:    {&(RES0__INSTANCE0.MY_BAD_FIFO.BUFFER.value.table[2129]), INT_ENUM},*)
(*DBG:    {&(RES0__INSTANCE0.MY_BAD_FIFO.BUFFER.value.table[2130]), INT_ENUM},*)
(*DBG:    {&(RES0__INSTANCE0.MY_BAD_FIFO.BUFFER.value.table[2131]), INT_ENUM},*)
(*DBG:    {&(RES0__INSTANCE0.MY_BAD_FIFO.BUFFER.value.table[2132]), INT_ENUM},*)
(*DBG:    {&(RES0__INSTANCE0.MY_BAD_FIFO.BUFFER.value.table[2133]), INT_ENUM},*)
(*DBG:    {&(RES0__INSTANCE0.MY_BAD_FIFO.BUFFER.value.table[2134]), INT_ENUM},*)
(*DBG:    {&(RES0__INSTANCE0.MY_BAD_FIFO.BUFFER.value.table[2135]), INT_ENUM},*)
(*DBG:    {&(RES0__INSTANCE0.MY_BAD_FIFO.BUFFER.value.table[2136]), INT_ENUM},*)
(*DBG:    {&(RES0__INSTANCE0.MY_BAD_FIFO.BUFFER.value.table[2137]), INT_ENUM},*)
(*DBG:    {&(RES0__INSTANCE0.MY_BAD_FIFO.BUFFER.value.table[2138]), INT_ENUM},*)
(*DBG:    {&(RES0__INSTANCE0.MY_BAD_FIFO.BUFFER.value.table[2139]), INT_ENUM},*)
(*DBG:    {&(RES0__INSTANCE0.MY_BAD_FIFO.BUFFER.value.table[2140]), INT_ENUM},*)
(*DBG:    {&(RES0__INSTANCE0.MY_BAD_FIFO.BUFFER.value.table[2141]), INT_ENUM},*)
(*DBG:    {&(RES0__INSTANCE0.MY_BAD_FIFO.BUFFER.value.table[2142]), INT_ENUM},*)
(*DBG:    {&(RES0__INSTANCE0.MY_BAD_FIFO.BUFFER.value.table[2143]), INT_ENUM},*)
(*DBG:    {&(RES0__INSTANCE0.MY_BAD_FIFO.BUFFER.value.table[2144]), INT_ENUM},*)
(*DBG:    {&(RES0__INSTANCE0.MY_BAD_FIFO.BUFFER.value.table[2145]), INT_ENUM},*)
(*DBG:    {&(RES0__INSTANCE0.MY_BAD_FIFO.BUFFER.value.table[2146]), INT_ENUM},*)
(*DBG:    {&(RES0__INSTANCE0.MY_BAD_FIFO.BUFFER.value.table[2147]), INT_ENUM},*)
(*DBG:    {&(RES0__INSTANCE0.MY_BAD_FIFO.BUFFER.value.table[2148]), INT_ENUM},*)
(*DBG:    {&(RES0__INSTANCE0.MY_BAD_FIFO.BUFFER.value.table[2149]), INT_ENUM},*)
(*DBG:    {&(RES0__INSTANCE0.MY_BAD_FIFO.BUFFER.value.table[2150]), INT_ENUM},*)
(*DBG:    {&(RES0__INSTANCE0.MY_BAD_FIFO.BUFFER.value.table[2151]), INT_ENUM},*)
(*DBG:    {&(RES0__INSTANCE0.MY_BAD_FIFO.BUFFER.value.table[2152]), INT_ENUM},*)
(*DBG:    {&(RES0__INSTANCE0.MY_BAD_FIFO.BUFFER.value.table[2153]), INT_ENUM},*)
(*DBG:    {&(RES0__INSTANCE0.MY_BAD_FIFO.BUFFER.value.table[2154]), INT_ENUM},*)
(*DBG:    {&(RES0__INSTANCE0.MY_BAD_FIFO.BUFFER.value.table[2155]), INT_ENUM},*)
(*DBG:    {&(RES0__INSTANCE0.MY_BAD_FIFO.BUFFER.value.table[2156]), INT_ENUM},*)
(*DBG:    {&(RES0__INSTANCE0.MY_BAD_FIFO.BUFFER.value.table[2157]), INT_ENUM},*)
(*DBG:    {&(RES0__INSTANCE0.MY_BAD_FIFO.BUFFER.value.table[2158]), INT_ENUM},*)
(*DBG:    {&(RES0__INSTANCE0.MY_BAD_FIFO.BUFFER.value.table[2159]), INT_ENUM},*)
(*DBG:    {&(RES0__INSTANCE0.MY_BAD_FIFO.BUFFER.value.table[2160]), INT_ENUM},*)
(*DBG:    {&(RES0__INSTANCE0.MY_BAD_FIFO.BUFFER.value.table[2161]), INT_ENUM},*)
(*DBG:    {&(RES0__INSTANCE0.MY_BAD_FIFO.BUFFER.value.table[2162]), INT_ENUM},*)
(*DBG:    {&(RES0__INSTANCE0.MY_BAD_FIFO.BUFFER.value.table[2163]), INT_ENUM},*)
(*DBG:    {&(RES0__INSTANCE0.MY_BAD_FIFO.BUFFER.value.table[2164]), INT_ENUM},*)
(*DBG:    {&(RES0__INSTANCE0.MY_BAD_FIFO.BUFFER.value.table[2165]), INT_ENUM},*)
(*DBG:    {&(RES0__INSTANCE0.MY_BAD_FIFO.BUFFER.value.table[2166]), INT_ENUM},*)
(*DBG:    {&(RES0__INSTANCE0.MY_BAD_FIFO.BUFFER.value.table[2167]), INT_ENUM},*)
(*DBG:    {&(RES0__INSTANCE0.MY_BAD_FIFO.BUFFER.value.table[2168]), INT_ENUM},*)
(*DBG:    {&(RES0__INSTANCE0.MY_BAD_FIFO.BUFFER.value.table[2169]), INT_ENUM},*)
(*DBG:    {&(RES0__INSTANCE0.MY_BAD_FIFO.BUFFER.value.table[2170]), INT_ENUM},*)
(*DBG:    {&(RES0__INSTANCE0.MY_BAD_FIFO.BUFFER.value.table[2171]), INT_ENUM},*)
(*DBG:    {&(RES0__INSTANCE0.MY_BAD_FIFO.BUFFER.value.table[2172]), INT_ENUM},*)
(*DBG:    {&(RES0__INSTANCE0.MY_BAD_FIFO.BUFFER.value.table[2173]), INT_ENUM},*)
(*DBG:    {&(RES0__INSTANCE0.MY_BAD_FIFO.BUFFER.value.table[2174]), INT_ENUM},*)
(*DBG:    {&(RES0__INSTANCE0.MY_BAD_FIFO.BUFFER.value.table[2175]), INT_ENUM},*)
(*DBG:    {&(RES0__INSTANCE0.MY_BAD_FIFO.BUFFER.value.table[2176]), INT_ENUM},*)
(*DBG:    {&(RES0__INSTANCE0.MY_BAD_FIFO.BUFFER.value.table[2177]), INT_ENUM},*)
(*DBG:    {&(RES0__INSTANCE0.MY_BAD_FIFO.BUFFER.value.table[2178]), INT_ENUM},*)
(*DBG:    {&(RES0__INSTANCE0.MY_BAD_FIFO.BUFFER.value.table[2179]), INT_ENUM},*)
(*DBG:    {&(RES0__INSTANCE0.MY_BAD_FIFO.BUFFER.value.table[2180]), INT_ENUM},*)
(*DBG:    {&(RES0__INSTANCE0.MY_BAD_FIFO.BUFFER.value.table[2181]), INT_ENUM},*)
(*DBG:    {&(RES0__INSTANCE0.MY_BAD_FIFO.BUFFER.value.table[2182]), INT_ENUM},*)
(*DBG:    {&(RES0__INSTANCE0.MY_BAD_FIFO.BUFFER.value.table[2183]), INT_ENUM},*)
(*DBG:    {&(RES0__INSTANCE0.MY_BAD_FIFO.BUFFER.value.table[2184]), INT_ENUM},*)
(*DBG:    {&(RES0__INSTANCE0.MY_BAD_FIFO.BUFFER.value.table[2185]), INT_ENUM},*)
(*DBG:    {&(RES0__INSTANCE0.MY_BAD_FIFO.BUFFER.value.table[2186]), INT_ENUM},*)
(*DBG:    {&(RES0__INSTANCE0.MY_BAD_FIFO.BUFFER.value.table[2187]), INT_ENUM},*)
(*DBG:    {&(RES0__INSTANCE0.MY_BAD_FIFO.BUFFER.value.table[2188]), INT_ENUM},*)
(*DBG:    {&(RES0__INSTANCE0.MY_BAD_FIFO.BUFFER.value.table[2189]), INT_ENUM},*)
(*DBG:    {&(RES0__INSTANCE0.MY_BAD_FIFO.BUFFER.value.table[2190]), INT_ENUM},*)
(*DBG:    {&(RES0__INSTANCE0.MY_BAD_FIFO.BUFFER.value.table[2191]), INT_ENUM},*)
(*DBG:    {&(RES0__INSTANCE0.MY_BAD_FIFO.BUFFER.value.table[2192]), INT_ENUM},*)
(*DBG:    {&(RES0__INSTANCE0.MY_BAD_FIFO.BUFFER.value.table[2193]), INT_ENUM},*)
(*DBG:    {&(RES0__INSTANCE0.MY_BAD_FIFO.BUFFER.value.table[2194]), INT_ENUM},*)
(*DBG:    {&(RES0__INSTANCE0.MY_BAD_FIFO.BUFFER.value.table[2195]), INT_ENUM},*)
(*DBG:    {&(RES0__INSTANCE0.MY_BAD_FIFO.BUFFER.value.table[2196]), INT_ENUM},*)
(*DBG:    {&(RES0__INSTANCE0.MY_BAD_FIFO.BUFFER.value.table[2197]), INT_ENUM},*)
(*DBG:    {&(RES0__INSTANCE0.MY_BAD_FIFO.BUFFER.value.table[2198]), INT_ENUM},*)
(*DBG:    {&(RES0__INSTANCE0.MY_BAD_FIFO.BUFFER.value.table[2199]), INT_ENUM},*)
(*DBG:    {&(RES0__INSTANCE0.MY_BAD_FIFO.BUFFER.value.table[2200]), INT_ENUM},*)
(*DBG:    {&(RES0__INSTANCE0.MY_BAD_FIFO.BUFFER.value.table[2201]), INT_ENUM},*)
(*DBG:    {&(RES0__INSTANCE0.MY_BAD_FIFO.BUFFER.value.table[2202]), INT_ENUM},*)
(*DBG:    {&(RES0__INSTANCE0.MY_BAD_FIFO.BUFFER.value.table[2203]), INT_ENUM},*)
(*DBG:    {&(RES0__INSTANCE0.MY_BAD_FIFO.BUFFER.value.table[2204]), INT_ENUM},*)
(*DBG:    {&(RES0__INSTANCE0.MY_BAD_FIFO.BUFFER.value.table[2205]), INT_ENUM},*)
(*DBG:    {&(RES0__INSTANCE0.MY_BAD_FIFO.BUFFER.value.table[2206]), INT_ENUM},*)
(*DBG:    {&(RES0__INSTANCE0.MY_BAD_FIFO.BUFFER.value.table[2207]), INT_ENUM},*)
(*DBG:    {&(RES0__INSTANCE0.MY_BAD_FIFO.BUFFER.value.table[2208]), INT_ENUM},*)
(*DBG:    {&(RES0__INSTANCE0.MY_BAD_FIFO.BUFFER.value.table[2209]), INT_ENUM},*)
(*DBG:    {&(RES0__INSTANCE0.MY_BAD_FIFO.BUFFER.value.table[2210]), INT_ENUM},*)
(*DBG:    {&(RES0__INSTANCE0.MY_BAD_FIFO.BUFFER.value.table[2211]), INT_ENUM},*)
(*DBG:    {&(RES0__INSTANCE0.MY_BAD_FIFO.BUFFER.value.table[2212]), INT_ENUM},*)
(*DBG:    {&(RES0__INSTANCE0.MY_BAD_FIFO.BUFFER.value.table[2213]), INT_ENUM},*)
(*DBG:    {&(RES0__INSTANCE0.MY_BAD_FIFO.BUFFER.value.table[2214]), INT_ENUM},*)
(*DBG:    {&(RES0__INSTANCE0.MY_BAD_FIFO.BUFFER.value.table[2215]), INT_ENUM},*)
(*DBG:    {&(RES0__INSTANCE0.MY_BAD_FIFO.BUFFER.value.table[2216]), INT_ENUM},*)
(*DBG:    {&(RES0__INSTANCE0.MY_BAD_FIFO.BUFFER.value.table[2217]), INT_ENUM},*)
(*DBG:    {&(RES0__INSTANCE0.MY_BAD_FIFO.BUFFER.value.table[2218]), INT_ENUM},*)
(*DBG:    {&(RES0__INSTANCE0.MY_BAD_FIFO.BUFFER.value.table[2219]), INT_ENUM},*)
(*DBG:    {&(RES0__INSTANCE0.MY_BAD_FIFO.BUFFER.value.table[2220]), INT_ENUM},*)
(*DBG:    {&(RES0__INSTANCE0.MY_BAD_FIFO.BUFFER.value.table[2221]), INT_ENUM},*)
(*DBG:    {&(RES0__INSTANCE0.MY_BAD_FIFO.BUFFER.value.table[2222]), INT_ENUM},*)
(*DBG:    {&(RES0__INSTANCE0.MY_BAD_FIFO.BUFFER.value.table[2223]), INT_ENUM},*)
(*DBG:    {&(RES0__INSTANCE0.MY_BAD_FIFO.BUFFER.value.table[2224]), INT_ENUM},*)
(*DBG:    {&(RES0__INSTANCE0.MY_BAD_FIFO.BUFFER.value.table[2225]), INT_ENUM},*)
(*DBG:    {&(RES0__INSTANCE0.MY_BAD_FIFO.BUFFER.value.table[2226]), INT_ENUM},*)
(*DBG:    {&(RES0__INSTANCE0.MY_BAD_FIFO.BUFFER.value.table[2227]), INT_ENUM},*)
(*DBG:    {&(RES0__INSTANCE0.MY_BAD_FIFO.BUFFER.value.table[2228]), INT_ENUM},*)
(*DBG:    {&(RES0__INSTANCE0.MY_BAD_FIFO.BUFFER.value.table[2229]), INT_ENUM},*)
(*DBG:    {&(RES0__INSTANCE0.MY_BAD_FIFO.BUFFER.value.table[2230]), INT_ENUM},*)
(*DBG:    {&(RES0__INSTANCE0.MY_BAD_FIFO.BUFFER.value.table[2231]), INT_ENUM},*)
(*DBG:    {&(RES0__INSTANCE0.MY_BAD_FIFO.BUFFER.value.table[2232]), INT_ENUM},*)
(*DBG:    {&(RES0__INSTANCE0.MY_BAD_FIFO.BUFFER.value.table[2233]), INT_ENUM},*)
(*DBG:    {&(RES0__INSTANCE0.MY_BAD_FIFO.BUFFER.value.table[2234]), INT_ENUM},*)
(*DBG:    {&(RES0__INSTANCE0.MY_BAD_FIFO.BUFFER.value.table[2235]), INT_ENUM},*)
(*DBG:    {&(RES0__INSTANCE0.MY_BAD_FIFO.BUFFER.value.table[2236]), INT_ENUM},*)
(*DBG:    {&(RES0__INSTANCE0.MY_BAD_FIFO.BUFFER.value.table[2237]), INT_ENUM},*)
(*DBG:    {&(RES0__INSTANCE0.MY_BAD_FIFO.BUFFER.value.table[2238]), INT_ENUM},*)
(*DBG:    {&(RES0__INSTANCE0.MY_BAD_FIFO.BUFFER.value.table[2239]), INT_ENUM},*)
(*DBG:    {&(RES0__INSTANCE0.MY_BAD_FIFO.BUFFER.value.table[2240]), INT_ENUM},*)
(*DBG:    {&(RES0__INSTANCE0.MY_BAD_FIFO.BUFFER.value.table[2241]), INT_ENUM},*)
(*DBG:    {&(RES0__INSTANCE0.MY_BAD_FIFO.BUFFER.value.table[2242]), INT_ENUM},*)
(*DBG:    {&(RES0__INSTANCE0.MY_BAD_FIFO.BUFFER.value.table[2243]), INT_ENUM},*)
(*DBG:    {&(RES0__INSTANCE0.MY_BAD_FIFO.BUFFER.value.table[2244]), INT_ENUM},*)
(*DBG:    {&(RES0__INSTANCE0.MY_BAD_FIFO.BUFFER.value.table[2245]), INT_ENUM},*)
(*DBG:    {&(RES0__INSTANCE0.MY_BAD_FIFO.BUFFER.value.table[2246]), INT_ENUM},*)
(*DBG:    {&(RES0__INSTANCE0.MY_BAD_FIFO.BUFFER.value.table[2247]), INT_ENUM},*)
(*DBG:    {&(RES0__INSTANCE0.MY_BAD_FIFO.BUFFER.value.table[2248]), INT_ENUM},*)
(*DBG:    {&(RES0__INSTANCE0.MY_BAD_FIFO.BUFFER.value.table[2249]), INT_ENUM},*)
(*DBG:    {&(RES0__INSTANCE0.MY_BAD_FIFO.BUFFER.value.table[2250]), INT_ENUM},*)
(*DBG:    {&(RES0__INSTANCE0.MY_BAD_FIFO.BUFFER.value.table[2251]), INT_ENUM},*)
(*DBG:    {&(RES0__INSTANCE0.MY_BAD_FIFO.BUFFER.value.table[2252]), INT_ENUM},*)
(*DBG:    {&(RES0__INSTANCE0.MY_BAD_FIFO.BUFFER.value.table[2253]), INT_ENUM},*)
(*DBG:    {&(RES0__INSTANCE0.MY_BAD_FIFO.BUFFER.value.table[2254]), INT_ENUM},*)
(*DBG:    {&(RES0__INSTANCE0.MY_BAD_FIFO.BUFFER.value.table[2255]), INT_ENUM},*)
(*DBG:    {&(RES0__INSTANCE0.MY_BAD_FIFO.BUFFER.value.table[2256]), INT_ENUM},*)
(*DBG:    {&(RES0__INSTANCE0.MY_BAD_FIFO.BUFFER.value.table[2257]), INT_ENUM},*)
(*DBG:    {&(RES0__INSTANCE0.MY_BAD_FIFO.BUFFER.value.table[2258]), INT_ENUM},*)
(*DBG:    {&(RES0__INSTANCE0.MY_BAD_FIFO.BUFFER.value.table[2259]), INT_ENUM},*)
(*DBG:    {&(RES0__INSTANCE0.MY_BAD_FIFO.BUFFER.value.table[2260]), INT_ENUM},*)
(*DBG:    {&(RES0__INSTANCE0.MY_BAD_FIFO.BUFFER.value.table[2261]), INT_ENUM},*)
(*DBG:    {&(RES0__INSTANCE0.MY_BAD_FIFO.BUFFER.value.table[2262]), INT_ENUM},*)
(*DBG:    {&(RES0__INSTANCE0.MY_BAD_FIFO.BUFFER.value.table[2263]), INT_ENUM},*)
(*DBG:    {&(RES0__INSTANCE0.MY_BAD_FIFO.BUFFER.value.table[2264]), INT_ENUM},*)
(*DBG:    {&(RES0__INSTANCE0.MY_BAD_FIFO.BUFFER.value.table[2265]), INT_ENUM},*)
(*DBG:    {&(RES0__INSTANCE0.MY_BAD_FIFO.BUFFER.value.table[2266]), INT_ENUM},*)
(*DBG:    {&(RES0__INSTANCE0.MY_BAD_FIFO.BUFFER.value.table[2267]), INT_ENUM},*)
(*DBG:    {&(RES0__INSTANCE0.MY_BAD_FIFO.BUFFER.value.table[2268]), INT_ENUM},*)
(*DBG:    {&(RES0__INSTANCE0.MY_BAD_FIFO.BUFFER.value.table[2269]), INT_ENUM},*)
(*DBG:    {&(RES0__INSTANCE0.MY_BAD_FIFO.BUFFER.value.table[2270]), INT_ENUM},*)
(*DBG:    {&(RES0__INSTANCE0.MY_BAD_FIFO.BUFFER.value.table[2271]), INT_ENUM},*)
(*DBG:    {&(RES0__INSTANCE0.MY_BAD_FIFO.BUFFER.value.table[2272]), INT_ENUM},*)
(*DBG:    {&(RES0__INSTANCE0.MY_BAD_FIFO.BUFFER.value.table[2273]), INT_ENUM},*)
(*DBG:    {&(RES0__INSTANCE0.MY_BAD_FIFO.BUFFER.value.table[2274]), INT_ENUM},*)
(*DBG:    {&(RES0__INSTANCE0.MY_BAD_FIFO.BUFFER.value.table[2275]), INT_ENUM},*)
(*DBG:    {&(RES0__INSTANCE0.MY_BAD_FIFO.BUFFER.value.table[2276]), INT_ENUM},*)
(*DBG:    {&(RES0__INSTANCE0.MY_BAD_FIFO.BUFFER.value.table[2277]), INT_ENUM},*)
(*DBG:    {&(RES0__INSTANCE0.MY_BAD_FIFO.BUFFER.value.table[2278]), INT_ENUM},*)
(*DBG:    {&(RES0__INSTANCE0.MY_BAD_FIFO.BUFFER.value.table[2279]), INT_ENUM},*)
(*DBG:    {&(RES0__INSTANCE0.MY_BAD_FIFO.BUFFER.value.table[2280]), INT_ENUM},*)
(*DBG:    {&(RES0__INSTANCE0.MY_BAD_FIFO.BUFFER.value.table[2281]), INT_ENUM},*)
(*DBG:    {&(RES0__INSTANCE0.MY_BAD_FIFO.BUFFER.value.table[2282]), INT_ENUM},*)
(*DBG:    {&(RES0__INSTANCE0.MY_BAD_FIFO.BUFFER.value.table[2283]), INT_ENUM},*)
(*DBG:    {&(RES0__INSTANCE0.MY_BAD_FIFO.BUFFER.value.table[2284]), INT_ENUM},*)
(*DBG:    {&(RES0__INSTANCE0.MY_BAD_FIFO.BUFFER.value.table[2285]), INT_ENUM},*)
(*DBG:    {&(RES0__INSTANCE0.MY_BAD_FIFO.BUFFER.value.table[2286]), INT_ENUM},*)
(*DBG:    {&(RES0__INSTANCE0.MY_BAD_FIFO.BUFFER.value.table[2287]), INT_ENUM},*)
(*DBG:    {&(RES0__INSTANCE0.MY_BAD_FIFO.BUFFER.value.table[2288]), INT_ENUM},*)
(*DBG:    {&(RES0__INSTANCE0.MY_BAD_FIFO.BUFFER.value.table[2289]), INT_ENUM},*)
(*DBG:    {&(RES0__INSTANCE0.MY_BAD_FIFO.BUFFER.value.table[2290]), INT_ENUM},*)
(*DBG:    {&(RES0__INSTANCE0.MY_BAD_FIFO.BUFFER.value.table[2291]), INT_ENUM},*)
(*DBG:    {&(RES0__INSTANCE0.MY_BAD_FIFO.BUFFER.value.table[2292]), INT_ENUM},*)
(*DBG:    {&(RES0__INSTANCE0.MY_BAD_FIFO.BUFFER.value.table[2293]), INT_ENUM},*)
(*DBG:    {&(RES0__INSTANCE0.MY_BAD_FIFO.BUFFER.value.table[2294]), INT_ENUM},*)
(*DBG:    {&(RES0__INSTANCE0.MY_BAD_FIFO.BUFFER.value.table[2295]), INT_ENUM},*)
(*DBG:    {&(RES0__INSTANCE0.MY_BAD_FIFO.BUFFER.value.table[2296]), INT_ENUM},*)
(*DBG:    {&(RES0__INSTANCE0.MY_BAD_FIFO.BUFFER.value.table[2297]), INT_ENUM},*)
(*DBG:    {&(RES0__INSTANCE0.MY_BAD_FIFO.BUFFER.value.table[2298]), INT_ENUM},*)
(*DBG:    {&(RES0__INSTANCE0.MY_BAD_FIFO.BUFFER.value.table[2299]), INT_ENUM},*)
(*DBG:    {&(RES0__INSTANCE0.MY_BAD_FIFO.BUFFER.value.table[2300]), INT_ENUM},*)
(*DBG:    {&(RES0__INSTANCE0.MY_BAD_FIFO.BUFFER.value.table[2301]), INT_ENUM},*)
(*DBG:    {&(RES0__INSTANCE0.MY_BAD_FIFO.BUFFER.value.table[2302]), INT_ENUM},*)
(*DBG:    {&(RES0__INSTANCE0.MY_BAD_FIFO.BUFFER.value.table[2303]), INT_ENUM},*)
(*DBG:    {&(RES0__INSTANCE0.MY_BAD_FIFO.BUFFER.value.table[2304]), INT_ENUM},*)
(*DBG:    {&(RES0__INSTANCE0.MY_BAD_FIFO.BUFFER.value.table[2305]), INT_ENUM},*)
(*DBG:    {&(RES0__INSTANCE0.MY_BAD_FIFO.BUFFER.value.table[2306]), INT_ENUM},*)
(*DBG:    {&(RES0__INSTANCE0.MY_BAD_FIFO.BUFFER.value.table[2307]), INT_ENUM},*)
(*DBG:    {&(RES0__INSTANCE0.MY_BAD_FIFO.BUFFER.value.table[2308]), INT_ENUM},*)
(*DBG:    {&(RES0__INSTANCE0.MY_BAD_FIFO.BUFFER.value.table[2309]), INT_ENUM},*)
(*DBG:    {&(RES0__INSTANCE0.MY_BAD_FIFO.BUFFER.value.table[2310]), INT_ENUM},*)
(*DBG:    {&(RES0__INSTANCE0.MY_BAD_FIFO.BUFFER.value.table[2311]), INT_ENUM},*)
(*DBG:    {&(RES0__INSTANCE0.MY_BAD_FIFO.BUFFER.value.table[2312]), INT_ENUM},*)
(*DBG:    {&(RES0__INSTANCE0.MY_BAD_FIFO.BUFFER.value.table[2313]), INT_ENUM},*)
(*DBG:    {&(RES0__INSTANCE0.MY_BAD_FIFO.BUFFER.value.table[2314]), INT_ENUM},*)
(*DBG:    {&(RES0__INSTANCE0.MY_BAD_FIFO.BUFFER.value.table[2315]), INT_ENUM},*)
(*DBG:    {&(RES0__INSTANCE0.MY_BAD_FIFO.BUFFER.value.table[2316]), INT_ENUM},*)
(*DBG:    {&(RES0__INSTANCE0.MY_BAD_FIFO.BUFFER.value.table[2317]), INT_ENUM},*)
(*DBG:    {&(RES0__INSTANCE0.MY_BAD_FIFO.BUFFER.value.table[2318]), INT_ENUM},*)
(*DBG:    {&(RES0__INSTANCE0.MY_BAD_FIFO.BUFFER.value.table[2319]), INT_ENUM},*)
(*DBG:    {&(RES0__INSTANCE0.MY_BAD_FIFO.BUFFER.value.table[2320]), INT_ENUM},*)
(*DBG:    {&(RES0__INSTANCE0.MY_BAD_FIFO.BUFFER.value.table[2321]), INT_ENUM},*)
(*DBG:    {&(RES0__INSTANCE0.MY_BAD_FIFO.BUFFER.value.table[2322]), INT_ENUM},*)
(*DBG:    {&(RES0__INSTANCE0.MY_BAD_FIFO.BUFFER.value.table[2323]), INT_ENUM},*)
(*DBG:    {&(RES0__INSTANCE0.MY_BAD_FIFO.BUFFER.value.table[2324]), INT_ENUM},*)
(*DBG:    {&(RES0__INSTANCE0.MY_BAD_FIFO.BUFFER.value.table[2325]), INT_ENUM},*)
(*DBG:    {&(RES0__INSTANCE0.MY_BAD_FIFO.BUFFER.value.table[2326]), INT_ENUM},*)
(*DBG:    {&(RES0__INSTANCE0.MY_BAD_FIFO.BUFFER.value.table[2327]), INT_ENUM},*)
(*DBG:    {&(RES0__INSTANCE0.MY_BAD_FIFO.BUFFER.value.table[2328]), INT_ENUM},*)
(*DBG:    {&(RES0__INSTANCE0.MY_BAD_FIFO.BUFFER.value.table[2329]), INT_ENUM},*)
(*DBG:    {&(RES0__INSTANCE0.MY_BAD_FIFO.BUFFER.value.table[2330]), INT_ENUM},*)
(*DBG:    {&(RES0__INSTANCE0.MY_BAD_FIFO.BUFFER.value.table[2331]), INT_ENUM},*)
(*DBG:    {&(RES0__INSTANCE0.MY_BAD_FIFO.BUFFER.value.table[2332]), INT_ENUM},*)
(*DBG:    {&(RES0__INSTANCE0.MY_BAD_FIFO.BUFFER.value.table[2333]), INT_ENUM},*)
(*DBG:    {&(RES0__INSTANCE0.MY_BAD_FIFO.BUFFER.value.table[2334]), INT_ENUM},*)
(*DBG:    {&(RES0__INSTANCE0.MY_BAD_FIFO.BUFFER.value.table[2335]), INT_ENUM},*)
(*DBG:    {&(RES0__INSTANCE0.MY_BAD_FIFO.BUFFER.value.table[2336]), INT_ENUM},*)
(*DBG:    {&(RES0__INSTANCE0.MY_BAD_FIFO.BUFFER.value.table[2337]), INT_ENUM},*)
(*DBG:    {&(RES0__INSTANCE0.MY_BAD_FIFO.BUFFER.value.table[2338]), INT_ENUM},*)
(*DBG:    {&(RES0__INSTANCE0.MY_BAD_FIFO.BUFFER.value.table[2339]), INT_ENUM},*)
(*DBG:    {&(RES0__INSTANCE0.MY_BAD_FIFO.BUFFER.value.table[2340]), INT_ENUM},*)
(*DBG:    {&(RES0__INSTANCE0.MY_BAD_FIFO.BUFFER.value.table[2341]), INT_ENUM},*)
(*DBG:    {&(RES0__INSTANCE0.MY_BAD_FIFO.BUFFER.value.table[2342]), INT_ENUM},*)
(*DBG:    {&(RES0__INSTANCE0.MY_BAD_FIFO.BUFFER.value.table[2343]), INT_ENUM},*)
(*DBG:    {&(RES0__INSTANCE0.MY_BAD_FIFO.BUFFER.value.table[2344]), INT_ENUM},*)
(*DBG:    {&(RES0__INSTANCE0.MY_BAD_FIFO.BUFFER.value.table[2345]), INT_ENUM},*)
(*DBG:    {&(RES0__INSTANCE0.MY_BAD_FIFO.BUFFER.value.table[2346]), INT_ENUM},*)
(*DBG:    {&(RES0__INSTANCE0.MY_BAD_FIFO.BUFFER.value.table[2347]), INT_ENUM},*)
(*DBG:    {&(RES0__INSTANCE0.MY_BAD_FIFO.BUFFER.value.table[2348]), INT_ENUM},*)
(*DBG:    {&(RES0__INSTANCE0.MY_BAD_FIFO.BUFFER.value.table[2349]), INT_ENUM},*)
(*DBG:    {&(RES0__INSTANCE0.MY_BAD_FIFO.BUFFER.value.table[2350]), INT_ENUM},*)
(*DBG:    {&(RES0__INSTANCE0.MY_BAD_FIFO.BUFFER.value.table[2351]), INT_ENUM},*)
(*DBG:    {&(RES0__INSTANCE0.MY_BAD_FIFO.BUFFER.value.table[2352]), INT_ENUM},*)
(*DBG:    {&(RES0__INSTANCE0.MY_BAD_FIFO.BUFFER.value.table[2353]), INT_ENUM},*)
(*DBG:    {&(RES0__INSTANCE0.MY_BAD_FIFO.BUFFER.value.table[2354]), INT_ENUM},*)
(*DBG:    {&(RES0__INSTANCE0.MY_BAD_FIFO.BUFFER.value.table[2355]), INT_ENUM},*)
(*DBG:    {&(RES0__INSTANCE0.MY_BAD_FIFO.BUFFER.value.table[2356]), INT_ENUM},*)
(*DBG:    {&(RES0__INSTANCE0.MY_BAD_FIFO.BUFFER.value.table[2357]), INT_ENUM},*)
(*DBG:    {&(RES0__INSTANCE0.MY_BAD_FIFO.BUFFER.value.table[2358]), INT_ENUM},*)
(*DBG:    {&(RES0__INSTANCE0.MY_BAD_FIFO.BUFFER.value.table[2359]), INT_ENUM},*)
(*DBG:    {&(RES0__INSTANCE0.MY_BAD_FIFO.BUFFER.value.table[2360]), INT_ENUM},*)
(*DBG:    {&(RES0__INSTANCE0.MY_BAD_FIFO.BUFFER.value.table[2361]), INT_ENUM},*)
(*DBG:    {&(RES0__INSTANCE0.MY_BAD_FIFO.BUFFER.value.table[2362]), INT_ENUM},*)
(*DBG:    {&(RES0__INSTANCE0.MY_BAD_FIFO.BUFFER.value.table[2363]), INT_ENUM},*)
(*DBG:    {&(RES0__INSTANCE0.MY_BAD_FIFO.BUFFER.value.table[2364]), INT_ENUM},*)
(*DBG:    {&(RES0__INSTANCE0.MY_BAD_FIFO.BUFFER.value.table[2365]), INT_ENUM},*)
(*DBG:    {&(RES0__INSTANCE0.MY_BAD_FIFO.BUFFER.value.table[2366]), INT_ENUM},*)
(*DBG:    {&(RES0__INSTANCE0.MY_BAD_FIFO.BUFFER.value.table[2367]), INT_ENUM},*)
(*DBG:    {&(RES0__INSTANCE0.MY_BAD_FIFO.BUFFER.value.table[2368]), INT_ENUM},*)
(*DBG:    {&(RES0__INSTANCE0.MY_BAD_FIFO.BUFFER.value.table[2369]), INT_ENUM},*)
(*DBG:    {&(RES0__INSTANCE0.MY_BAD_FIFO.BUFFER.value.table[2370]), INT_ENUM},*)
(*DBG:    {&(RES0__INSTANCE0.MY_BAD_FIFO.BUFFER.value.table[2371]), INT_ENUM},*)
(*DBG:    {&(RES0__INSTANCE0.MY_BAD_FIFO.BUFFER.value.table[2372]), INT_ENUM},*)
(*DBG:    {&(RES0__INSTANCE0.MY_BAD_FIFO.BUFFER.value.table[2373]), INT_ENUM},*)
(*DBG:    {&(RES0__INSTANCE0.MY_BAD_FIFO.BUFFER.value.table[2374]), INT_ENUM},*)
(*DBG:    {&(RES0__INSTANCE0.MY_BAD_FIFO.BUFFER.value.table[2375]), INT_ENUM},*)
(*DBG:    {&(RES0__INSTANCE0.MY_BAD_FIFO.BUFFER.value.table[2376]), INT_ENUM},*)
(*DBG:    {&(RES0__INSTANCE0.MY_BAD_FIFO.BUFFER.value.table[2377]), INT_ENUM},*)
(*DBG:    {&(RES0__INSTANCE0.MY_BAD_FIFO.BUFFER.value.table[2378]), INT_ENUM},*)
(*DBG:    {&(RES0__INSTANCE0.MY_BAD_FIFO.BUFFER.value.table[2379]), INT_ENUM},*)
(*DBG:    {&(RES0__INSTANCE0.MY_BAD_FIFO.BUFFER.value.table[2380]), INT_ENUM},*)
(*DBG:    {&(RES0__INSTANCE0.MY_BAD_FIFO.BUFFER.value.table[2381]), INT_ENUM},*)
(*DBG:    {&(RES0__INSTANCE0.MY_BAD_FIFO.BUFFER.value.table[2382]), INT_ENUM},*)
(*DBG:    {&(RES0__INSTANCE0.MY_BAD_FIFO.BUFFER.value.table[2383]), INT_ENUM},*)
(*DBG:    {&(RES0__INSTANCE0.MY_BAD_FIFO.BUFFER.value.table[2384]), INT_ENUM},*)
(*DBG:    {&(RES0__INSTANCE0.MY_BAD_FIFO.BUFFER.value.table[2385]), INT_ENUM},*)
(*DBG:    {&(RES0__INSTANCE0.MY_BAD_FIFO.BUFFER.value.table[2386]), INT_ENUM},*)
(*DBG:    {&(RES0__INSTANCE0.MY_BAD_FIFO.BUFFER.value.table[2387]), INT_ENUM},*)
(*DBG:    {&(RES0__INSTANCE0.MY_BAD_FIFO.BUFFER.value.table[2388]), INT_ENUM},*)
(*DBG:    {&(RES0__INSTANCE0.MY_BAD_FIFO.BUFFER.value.table[2389]), INT_ENUM},*)
(*DBG:    {&(RES0__INSTANCE0.MY_BAD_FIFO.BUFFER.value.table[2390]), INT_ENUM},*)
(*DBG:    {&(RES0__INSTANCE0.MY_BAD_FIFO.BUFFER.value.table[2391]), INT_ENUM},*)
(*DBG:    {&(RES0__INSTANCE0.MY_BAD_FIFO.BUFFER.value.table[2392]), INT_ENUM},*)
(*DBG:    {&(RES0__INSTANCE0.MY_BAD_FIFO.BUFFER.value.table[2393]), INT_ENUM},*)
(*DBG:    {&(RES0__INSTANCE0.MY_BAD_FIFO.BUFFER.value.table[2394]), INT_ENUM},*)
(*DBG:    {&(RES0__INSTANCE0.MY_BAD_FIFO.BUFFER.value.table[2395]), INT_ENUM},*)
(*DBG:    {&(RES0__INSTANCE0.MY_BAD_FIFO.BUFFER.value.table[2396]), INT_ENUM},*)
(*DBG:    {&(RES0__INSTANCE0.MY_BAD_FIFO.BUFFER.value.table[2397]), INT_ENUM},*)
(*DBG:    {&(RES0__INSTANCE0.MY_BAD_FIFO.BUFFER.value.table[2398]), INT_ENUM},*)
(*DBG:    {&(RES0__INSTANCE0.MY_BAD_FIFO.BUFFER.value.table[2399]), INT_ENUM},*)
(*DBG:    {&(RES0__INSTANCE0.MY_BAD_FIFO.BUFFER.value.table[2400]), INT_ENUM},*)
(*DBG:    {&(RES0__INSTANCE0.MY_BAD_FIFO.BUFFER.value.table[2401]), INT_ENUM},*)
(*DBG:    {&(RES0__INSTANCE0.MY_BAD_FIFO.BUFFER.value.table[2402]), INT_ENUM},*)
(*DBG:    {&(RES0__INSTANCE0.MY_BAD_FIFO.BUFFER.value.table[2403]), INT_ENUM},*)
(*DBG:    {&(RES0__INSTANCE0.MY_BAD_FIFO.BUFFER.value.table[2404]), INT_ENUM},*)
(*DBG:    {&(RES0__INSTANCE0.MY_BAD_FIFO.BUFFER.value.table[2405]), INT_ENUM},*)
(*DBG:    {&(RES0__INSTANCE0.MY_BAD_FIFO.BUFFER.value.table[2406]), INT_ENUM},*)
(*DBG:    {&(RES0__INSTANCE0.MY_BAD_FIFO.BUFFER.value.table[2407]), INT_ENUM},*)
(*DBG:    {&(RES0__INSTANCE0.MY_BAD_FIFO.BUFFER.value.table[2408]), INT_ENUM},*)
(*DBG:    {&(RES0__INSTANCE0.MY_BAD_FIFO.BUFFER.value.table[2409]), INT_ENUM},*)
(*DBG:    {&(RES0__INSTANCE0.MY_BAD_FIFO.BUFFER.value.table[2410]), INT_ENUM},*)
(*DBG:    {&(RES0__INSTANCE0.MY_BAD_FIFO.BUFFER.value.table[2411]), INT_ENUM},*)
(*DBG:    {&(RES0__INSTANCE0.MY_BAD_FIFO.BUFFER.value.table[2412]), INT_ENUM},*)
(*DBG:    {&(RES0__INSTANCE0.MY_BAD_FIFO.BUFFER.value.table[2413]), INT_ENUM},*)
(*DBG:    {&(RES0__INSTANCE0.MY_BAD_FIFO.BUFFER.value.table[2414]), INT_ENUM},*)
(*DBG:    {&(RES0__INSTANCE0.MY_BAD_FIFO.BUFFER.value.table[2415]), INT_ENUM},*)
(*DBG:    {&(RES0__INSTANCE0.MY_BAD_FIFO.BUFFER.value.table[2416]), INT_ENUM},*)
(*DBG:    {&(RES0__INSTANCE0.MY_BAD_FIFO.BUFFER.value.table[2417]), INT_ENUM},*)
(*DBG:    {&(RES0__INSTANCE0.MY_BAD_FIFO.BUFFER.value.table[2418]), INT_ENUM},*)
(*DBG:    {&(RES0__INSTANCE0.MY_BAD_FIFO.BUFFER.value.table[2419]), INT_ENUM},*)
(*DBG:    {&(RES0__INSTANCE0.MY_BAD_FIFO.BUFFER.value.table[2420]), INT_ENUM},*)
(*DBG:    {&(RES0__INSTANCE0.MY_BAD_FIFO.BUFFER.value.table[2421]), INT_ENUM},*)
(*DBG:    {&(RES0__INSTANCE0.MY_BAD_FIFO.BUFFER.value.table[2422]), INT_ENUM},*)
(*DBG:    {&(RES0__INSTANCE0.MY_BAD_FIFO.BUFFER.value.table[2423]), INT_ENUM},*)
(*DBG:    {&(RES0__INSTANCE0.MY_BAD_FIFO.BUFFER.value.table[2424]), INT_ENUM},*)
(*DBG:    {&(RES0__INSTANCE0.MY_BAD_FIFO.BUFFER.value.table[2425]), INT_ENUM},*)
(*DBG:    {&(RES0__INSTANCE0.MY_BAD_FIFO.BUFFER.value.table[2426]), INT_ENUM},*)
(*DBG:    {&(RES0__INSTANCE0.MY_BAD_FIFO.BUFFER.value.table[2427]), INT_ENUM},*)
(*DBG:    {&(RES0__INSTANCE0.MY_BAD_FIFO.BUFFER.value.table[2428]), INT_ENUM},*)
(*DBG:    {&(RES0__INSTANCE0.MY_BAD_FIFO.BUFFER.value.table[2429]), INT_ENUM},*)
(*DBG:    {&(RES0__INSTANCE0.MY_BAD_FIFO.BUFFER.value.table[2430]), INT_ENUM},*)
(*DBG:    {&(RES0__INSTANCE0.MY_BAD_FIFO.BUFFER.value.table[2431]), INT_ENUM},*)
(*DBG:    {&(RES0__INSTANCE0.MY_BAD_FIFO.BUFFER.value.table[2432]), INT_ENUM},*)
(*DBG:    {&(RES0__INSTANCE0.MY_BAD_FIFO.BUFFER.value.table[2433]), INT_ENUM},*)
(*DBG:    {&(RES0__INSTANCE0.MY_BAD_FIFO.BUFFER.value.table[2434]), INT_ENUM},*)
(*DBG:    {&(RES0__INSTANCE0.MY_BAD_FIFO.BUFFER.value.table[2435]), INT_ENUM},*)
(*DBG:    {&(RES0__INSTANCE0.MY_BAD_FIFO.BUFFER.value.table[2436]), INT_ENUM},*)
(*DBG:    {&(RES0__INSTANCE0.MY_BAD_FIFO.BUFFER.value.table[2437]), INT_ENUM},*)
(*DBG:    {&(RES0__INSTANCE0.MY_BAD_FIFO.BUFFER.value.table[2438]), INT_ENUM},*)
(*DBG:    {&(RES0__INSTANCE0.MY_BAD_FIFO.BUFFER.value.table[2439]), INT_ENUM},*)
(*DBG:    {&(RES0__INSTANCE0.MY_BAD_FIFO.BUFFER.value.table[2440]), INT_ENUM},*)
(*DBG:    {&(RES0__INSTANCE0.MY_BAD_FIFO.BUFFER.value.table[2441]), INT_ENUM},*)
(*DBG:    {&(RES0__INSTANCE0.MY_BAD_FIFO.BUFFER.value.table[2442]), INT_ENUM},*)
(*DBG:    {&(RES0__INSTANCE0.MY_BAD_FIFO.BUFFER.value.table[2443]), INT_ENUM},*)
(*DBG:    {&(RES0__INSTANCE0.MY_BAD_FIFO.BUFFER.value.table[2444]), INT_ENUM},*)
(*DBG:    {&(RES0__INSTANCE0.MY_BAD_FIFO.BUFFER.value.table[2445]), INT_ENUM},*)
(*DBG:    {&(RES0__INSTANCE0.MY_BAD_FIFO.BUFFER.value.table[2446]), INT_ENUM},*)
(*DBG:    {&(RES0__INSTANCE0.MY_BAD_FIFO.BUFFER.value.table[2447]), INT_ENUM},*)
(*DBG:    {&(RES0__INSTANCE0.MY_BAD_FIFO.BUFFER.value.table[2448]), INT_ENUM},*)
(*DBG:    {&(RES0__INSTANCE0.MY_BAD_FIFO.BUFFER.value.table[2449]), INT_ENUM},*)
(*DBG:    {&(RES0__INSTANCE0.MY_BAD_FIFO.BUFFER.value.table[2450]), INT_ENUM},*)
(*DBG:    {&(RES0__INSTANCE0.MY_BAD_FIFO.BUFFER.value.table[2451]), INT_ENUM},*)
(*DBG:    {&(RES0__INSTANCE0.MY_BAD_FIFO.BUFFER.value.table[2452]), INT_ENUM},*)
(*DBG:    {&(RES0__INSTANCE0.MY_BAD_FIFO.BUFFER.value.table[2453]), INT_ENUM},*)
(*DBG:    {&(RES0__INSTANCE0.MY_BAD_FIFO.BUFFER.value.table[2454]), INT_ENUM},*)
(*DBG:    {&(RES0__INSTANCE0.MY_BAD_FIFO.BUFFER.value.table[2455]), INT_ENUM},*)
(*DBG:    {&(RES0__INSTANCE0.MY_BAD_FIFO.BUFFER.value.table[2456]), INT_ENUM},*)
(*DBG:    {&(RES0__INSTANCE0.MY_BAD_FIFO.BUFFER.value.table[2457]), INT_ENUM},*)
(*DBG:    {&(RES0__INSTANCE0.MY_BAD_FIFO.BUFFER.value.table[2458]), INT_ENUM},*)
(*DBG:    {&(RES0__INSTANCE0.MY_BAD_FIFO.BUFFER.value.table[2459]), INT_ENUM},*)
(*DBG:    {&(RES0__INSTANCE0.MY_BAD_FIFO.BUFFER.value.table[2460]), INT_ENUM},*)
(*DBG:    {&(RES0__INSTANCE0.MY_BAD_FIFO.BUFFER.value.table[2461]), INT_ENUM},*)
(*DBG:    {&(RES0__INSTANCE0.MY_BAD_FIFO.BUFFER.value.table[2462]), INT_ENUM},*)
(*DBG:    {&(RES0__INSTANCE0.MY_BAD_FIFO.BUFFER.value.table[2463]), INT_ENUM},*)
(*DBG:    {&(RES0__INSTANCE0.MY_BAD_FIFO.BUFFER.value.table[2464]), INT_ENUM},*)
(*DBG:    {&(RES0__INSTANCE0.MY_BAD_FIFO.BUFFER.value.table[2465]), INT_ENUM},*)
(*DBG:    {&(RES0__INSTANCE0.MY_BAD_FIFO.BUFFER.value.table[2466]), INT_ENUM},*)
(*DBG:    {&(RES0__INSTANCE0.MY_BAD_FIFO.BUFFER.value.table[2467]), INT_ENUM},*)
(*DBG:    {&(RES0__INSTANCE0.MY_BAD_FIFO.BUFFER.value.table[2468]), INT_ENUM},*)
(*DBG:    {&(RES0__INSTANCE0.MY_BAD_FIFO.BUFFER.value.table[2469]), INT_ENUM},*)
(*DBG:    {&(RES0__INSTANCE0.MY_BAD_FIFO.BUFFER.value.table[2470]), INT_ENUM},*)
(*DBG:    {&(RES0__INSTANCE0.MY_BAD_FIFO.BUFFER.value.table[2471]), INT_ENUM},*)
(*DBG:    {&(RES0__INSTANCE0.MY_BAD_FIFO.BUFFER.value.table[2472]), INT_ENUM},*)
(*DBG:    {&(RES0__INSTANCE0.MY_BAD_FIFO.BUFFER.value.table[2473]), INT_ENUM},*)
(*DBG:    {&(RES0__INSTANCE0.MY_BAD_FIFO.BUFFER.value.table[2474]), INT_ENUM},*)
(*DBG:    {&(RES0__INSTANCE0.MY_BAD_FIFO.BUFFER.value.table[2475]), INT_ENUM},*)
(*DBG:    {&(RES0__INSTANCE0.MY_BAD_FIFO.BUFFER.value.table[2476]), INT_ENUM},*)
(*DBG:    {&(RES0__INSTANCE0.MY_BAD_FIFO.BUFFER.value.table[2477]), INT_ENUM},*)
(*DBG:    {&(RES0__INSTANCE0.MY_BAD_FIFO.BUFFER.value.table[2478]), INT_ENUM},*)
(*DBG:    {&(RES0__INSTANCE0.MY_BAD_FIFO.BUFFER.value.table[2479]), INT_ENUM},*)
(*DBG:    {&(RES0__INSTANCE0.MY_BAD_FIFO.BUFFER.value.table[2480]), INT_ENUM},*)
(*DBG:    {&(RES0__INSTANCE0.MY_BAD_FIFO.BUFFER.value.table[2481]), INT_ENUM},*)
(*DBG:    {&(RES0__INSTANCE0.MY_BAD_FIFO.BUFFER.value.table[2482]), INT_ENUM},*)
(*DBG:    {&(RES0__INSTANCE0.MY_BAD_FIFO.BUFFER.value.table[2483]), INT_ENUM},*)
(*DBG:    {&(RES0__INSTANCE0.MY_BAD_FIFO.BUFFER.value.table[2484]), INT_ENUM},*)
(*DBG:    {&(RES0__INSTANCE0.MY_BAD_FIFO.BUFFER.value.table[2485]), INT_ENUM},*)
(*DBG:    {&(RES0__INSTANCE0.MY_BAD_FIFO.BUFFER.value.table[2486]), INT_ENUM},*)
(*DBG:    {&(RES0__INSTANCE0.MY_BAD_FIFO.BUFFER.value.table[2487]), INT_ENUM},*)
(*DBG:    {&(RES0__INSTANCE0.MY_BAD_FIFO.BUFFER.value.table[2488]), INT_ENUM},*)
(*DBG:    {&(RES0__INSTANCE0.MY_BAD_FIFO.BUFFER.value.table[2489]), INT_ENUM},*)
(*DBG:    {&(RES0__INSTANCE0.MY_BAD_FIFO.BUFFER.value.table[2490]), INT_ENUM},*)
(*DBG:    {&(RES0__INSTANCE0.MY_BAD_FIFO.BUFFER.value.table[2491]), INT_ENUM},*)
(*DBG:    {&(RES0__INSTANCE0.MY_BAD_FIFO.BUFFER.value.table[2492]), INT_ENUM},*)
(*DBG:    {&(RES0__INSTANCE0.MY_BAD_FIFO.BUFFER.value.table[2493]), INT_ENUM},*)
(*DBG:    {&(RES0__INSTANCE0.MY_BAD_FIFO.BUFFER.value.table[2494]), INT_ENUM},*)
(*DBG:    {&(RES0__INSTANCE0.MY_BAD_FIFO.BUFFER.value.table[2495]), INT_ENUM},*)
(*DBG:    {&(RES0__INSTANCE0.MY_BAD_FIFO.BUFFER.value.table[2496]), INT_ENUM},*)
(*DBG:    {&(RES0__INSTANCE0.MY_BAD_FIFO.BUFFER.value.table[2497]), INT_ENUM},*)
(*DBG:    {&(RES0__INSTANCE0.MY_BAD_FIFO.BUFFER.value.table[2498]), INT_ENUM},*)
(*DBG:    {&(RES0__INSTANCE0.MY_BAD_FIFO.BUFFER.value.table[2499]), INT_ENUM},*)
(*DBG:    {&(RES0__INSTANCE0.MY_BAD_FIFO.BUFFER.value.table[2500]), INT_ENUM},*)
(*DBG:    {&(RES0__INSTANCE0.MY_BAD_FIFO.BUFFER.value.table[2501]), INT_ENUM},*)
(*DBG:    {&(RES0__INSTANCE0.MY_BAD_FIFO.BUFFER.value.table[2502]), INT_ENUM},*)
(*DBG:    {&(RES0__INSTANCE0.MY_BAD_FIFO.BUFFER.value.table[2503]), INT_ENUM},*)
(*DBG:    {&(RES0__INSTANCE0.MY_BAD_FIFO.BUFFER.value.table[2504]), INT_ENUM},*)
(*DBG:    {&(RES0__INSTANCE0.MY_BAD_FIFO.BUFFER.value.table[2505]), INT_ENUM},*)
(*DBG:    {&(RES0__INSTANCE0.MY_BAD_FIFO.BUFFER.value.table[2506]), INT_ENUM},*)
(*DBG:    {&(RES0__INSTANCE0.MY_BAD_FIFO.BUFFER.value.table[2507]), INT_ENUM},*)
(*DBG:    {&(RES0__INSTANCE0.MY_BAD_FIFO.BUFFER.value.table[2508]), INT_ENUM},*)
(*DBG:    {&(RES0__INSTANCE0.MY_BAD_FIFO.BUFFER.value.table[2509]), INT_ENUM},*)
(*DBG:    {&(RES0__INSTANCE0.MY_BAD_FIFO.BUFFER.value.table[2510]), INT_ENUM},*)
(*DBG:    {&(RES0__INSTANCE0.MY_BAD_FIFO.BUFFER.value.table[2511]), INT_ENUM},*)
(*DBG:    {&(RES0__INSTANCE0.MY_BAD_FIFO.BUFFER.value.table[2512]), INT_ENUM},*)
(*DBG:    {&(RES0__INSTANCE0.MY_BAD_FIFO.BUFFER.value.table[2513]), INT_ENUM},*)
(*DBG:    {&(RES0__INSTANCE0.MY_BAD_FIFO.BUFFER.value.table[2514]), INT_ENUM},*)
(*DBG:    {&(RES0__INSTANCE0.MY_BAD_FIFO.BUFFER.value.table[2515]), INT_ENUM},*)
(*DBG:    {&(RES0__INSTANCE0.MY_BAD_FIFO.BUFFER.value.table[2516]), INT_ENUM},*)
(*DBG:    {&(RES0__INSTANCE0.MY_BAD_FIFO.BUFFER.value.table[2517]), INT_ENUM},*)
(*DBG:    {&(RES0__INSTANCE0.MY_BAD_FIFO.BUFFER.value.table[2518]), INT_ENUM},*)
(*DBG:    {&(RES0__INSTANCE0.MY_BAD_FIFO.BUFFER.value.table[2519]), INT_ENUM},*)
(*DBG:    {&(RES0__INSTANCE0.MY_BAD_FIFO.BUFFER.value.table[2520]), INT_ENUM},*)
(*DBG:    {&(RES0__INSTANCE0.MY_BAD_FIFO.BUFFER.value.table[2521]), INT_ENUM},*)
(*DBG:    {&(RES0__INSTANCE0.MY_BAD_FIFO.BUFFER.value.table[2522]), INT_ENUM},*)
(*DBG:    {&(RES0__INSTANCE0.MY_BAD_FIFO.BUFFER.value.table[2523]), INT_ENUM},*)
(*DBG:    {&(RES0__INSTANCE0.MY_BAD_FIFO.BUFFER.value.table[2524]), INT_ENUM},*)
(*DBG:    {&(RES0__INSTANCE0.MY_BAD_FIFO.BUFFER.value.table[2525]), INT_ENUM},*)
(*DBG:    {&(RES0__INSTANCE0.MY_BAD_FIFO.BUFFER.value.table[2526]), INT_ENUM},*)
(*DBG:    {&(RES0__INSTANCE0.MY_BAD_FIFO.BUFFER.value.table[2527]), INT_ENUM},*)
(*DBG:    {&(RES0__INSTANCE0.MY_BAD_FIFO.BUFFER.value.table[2528]), INT_ENUM},*)
(*DBG:    {&(RES0__INSTANCE0.MY_BAD_FIFO.BUFFER.value.table[2529]), INT_ENUM},*)
(*DBG:    {&(RES0__INSTANCE0.MY_BAD_FIFO.BUFFER.value.table[2530]), INT_ENUM},*)
(*DBG:    {&(RES0__INSTANCE0.MY_BAD_FIFO.BUFFER.value.table[2531]), INT_ENUM},*)
(*DBG:    {&(RES0__INSTANCE0.MY_BAD_FIFO.BUFFER.value.table[2532]), INT_ENUM},*)
(*DBG:    {&(RES0__INSTANCE0.MY_BAD_FIFO.BUFFER.value.table[2533]), INT_ENUM},*)
(*DBG:    {&(RES0__INSTANCE0.MY_BAD_FIFO.BUFFER.value.table[2534]), INT_ENUM},*)
(*DBG:    {&(RES0__INSTANCE0.MY_BAD_FIFO.BUFFER.value.table[2535]), INT_ENUM},*)
(*DBG:    {&(RES0__INSTANCE0.MY_BAD_FIFO.BUFFER.value.table[2536]), INT_ENUM},*)
(*DBG:    {&(RES0__INSTANCE0.MY_BAD_FIFO.BUFFER.value.table[2537]), INT_ENUM},*)
(*DBG:    {&(RES0__INSTANCE0.MY_BAD_FIFO.BUFFER.value.table[2538]), INT_ENUM},*)
(*DBG:    {&(RES0__INSTANCE0.MY_BAD_FIFO.BUFFER.value.table[2539]), INT_ENUM},*)
(*DBG:    {&(RES0__INSTANCE0.MY_BAD_FIFO.BUFFER.value.table[2540]), INT_ENUM},*)
(*DBG:    {&(RES0__INSTANCE0.MY_BAD_FIFO.BUFFER.value.table[2541]), INT_ENUM},*)
(*DBG:    {&(RES0__INSTANCE0.MY_BAD_FIFO.BUFFER.value.table[2542]), INT_ENUM},*)
(*DBG:    {&(RES0__INSTANCE0.MY_BAD_FIFO.BUFFER.value.table[2543]), INT_ENUM},*)
(*DBG:    {&(RES0__INSTANCE0.MY_BAD_FIFO.BUFFER.value.table[2544]), INT_ENUM},*)
(*DBG:    {&(RES0__INSTANCE0.MY_BAD_FIFO.BUFFER.value.table[2545]), INT_ENUM},*)
(*DBG:    {&(RES0__INSTANCE0.MY_BAD_FIFO.BUFFER.value.table[2546]), INT_ENUM},*)
(*DBG:    {&(RES0__INSTANCE0.MY_BAD_FIFO.BUFFER.value.table[2547]), INT_ENUM},*)
(*DBG:    {&(RES0__INSTANCE0.MY_BAD_FIFO.BUFFER.value.table[2548]), INT_ENUM},*)
(*DBG:    {&(RES0__INSTANCE0.MY_BAD_FIFO.BUFFER.value.table[2549]), INT_ENUM},*)
(*DBG:    {&(RES0__INSTANCE0.MY_BAD_FIFO.BUFFER.value.table[2550]), INT_ENUM},*)
(*DBG:    {&(RES0__INSTANCE0.MY_BAD_FIFO.BUFFER.value.table[2551]), INT_ENUM},*)
(*DBG:    {&(RES0__INSTANCE0.MY_BAD_FIFO.BUFFER.value.table[2552]), INT_ENUM},*)
(*DBG:    {&(RES0__INSTANCE0.MY_BAD_FIFO.BUFFER.value.table[2553]), INT_ENUM},*)
(*DBG:    {&(RES0__INSTANCE0.MY_BAD_FIFO.BUFFER.value.table[2554]), INT_ENUM},*)
(*DBG:    {&(RES0__INSTANCE0.MY_BAD_FIFO.BUFFER.value.table[2555]), INT_ENUM},*)
(*DBG:    {&(RES0__INSTANCE0.MY_BAD_FIFO.BUFFER.value.table[2556]), INT_ENUM},*)
(*DBG:    {&(RES0__INSTANCE0.MY_BAD_FIFO.BUFFER.value.table[2557]), INT_ENUM},*)
(*DBG:    {&(RES0__INSTANCE0.MY_BAD_FIFO.BUFFER.value.table[2558]), INT_ENUM},*)
(*DBG:    {&(RES0__INSTANCE0.MY_BAD_FIFO.BUFFER.value.table[2559]), INT_ENUM},*)
(*DBG:    {&(RES0__INSTANCE0.MY_BAD_FIFO.BUFFER.value.table[2560]), INT_ENUM},*)
(*DBG:    {&(RES0__INSTANCE0.MY_BAD_FIFO.BUFFER.value.table[2561]), INT_ENUM},*)
(*DBG:    {&(RES0__INSTANCE0.MY_BAD_FIFO.BUFFER.value.table[2562]), INT_ENUM},*)
(*DBG:    {&(RES0__INSTANCE0.MY_BAD_FIFO.BUFFER.value.table[2563]), INT_ENUM},*)
(*DBG:    {&(RES0__INSTANCE0.MY_BAD_FIFO.BUFFER.value.table[2564]), INT_ENUM},*)
(*DBG:    {&(RES0__INSTANCE0.MY_BAD_FIFO.BUFFER.value.table[2565]), INT_ENUM},*)
(*DBG:    {&(RES0__INSTANCE0.MY_BAD_FIFO.BUFFER.value.table[2566]), INT_ENUM},*)
(*DBG:    {&(RES0__INSTANCE0.MY_BAD_FIFO.BUFFER.value.table[2567]), INT_ENUM},*)
(*DBG:    {&(RES0__INSTANCE0.MY_BAD_FIFO.BUFFER.value.table[2568]), INT_ENUM},*)
(*DBG:    {&(RES0__INSTANCE0.MY_BAD_FIFO.BUFFER.value.table[2569]), INT_ENUM},*)
(*DBG:    {&(RES0__INSTANCE0.MY_BAD_FIFO.BUFFER.value.table[2570]), INT_ENUM},*)
(*DBG:    {&(RES0__INSTANCE0.MY_BAD_FIFO.BUFFER.value.table[2571]), INT_ENUM},*)
(*DBG:    {&(RES0__INSTANCE0.MY_BAD_FIFO.BUFFER.value.table[2572]), INT_ENUM},*)
(*DBG:    {&(RES0__INSTANCE0.MY_BAD_FIFO.BUFFER.value.table[2573]), INT_ENUM},*)
(*DBG:    {&(RES0__INSTANCE0.MY_BAD_FIFO.BUFFER.value.table[2574]), INT_ENUM},*)
(*DBG:    {&(RES0__INSTANCE0.MY_BAD_FIFO.BUFFER.value.table[2575]), INT_ENUM},*)
(*DBG:    {&(RES0__INSTANCE0.MY_BAD_FIFO.BUFFER.value.table[2576]), INT_ENUM},*)
(*DBG:    {&(RES0__INSTANCE0.MY_BAD_FIFO.BUFFER.value.table[2577]), INT_ENUM},*)
(*DBG:    {&(RES0__INSTANCE0.MY_BAD_FIFO.BUFFER.value.table[2578]), INT_ENUM},*)
(*DBG:    {&(RES0__INSTANCE0.MY_BAD_FIFO.BUFFER.value.table[2579]), INT_ENUM},*)
(*DBG:    {&(RES0__INSTANCE0.MY_BAD_FIFO.BUFFER.value.table[2580]), INT_ENUM},*)
(*DBG:    {&(RES0__INSTANCE0.MY_BAD_FIFO.BUFFER.value.table[2581]), INT_ENUM},*)
(*DBG:    {&(RES0__INSTANCE0.MY_BAD_FIFO.BUFFER.value.table[2582]), INT_ENUM},*)
(*DBG:    {&(RES0__INSTANCE0.MY_BAD_FIFO.BUFFER.value.table[2583]), INT_ENUM},*)
(*DBG:    {&(RES0__INSTANCE0.MY_BAD_FIFO.BUFFER.value.table[2584]), INT_ENUM},*)
(*DBG:    {&(RES0__INSTANCE0.MY_BAD_FIFO.BUFFER.value.table[2585]), INT_ENUM},*)
(*DBG:    {&(RES0__INSTANCE0.MY_BAD_FIFO.BUFFER.value.table[2586]), INT_ENUM},*)
(*DBG:    {&(RES0__INSTANCE0.MY_BAD_FIFO.BUFFER.value.table[2587]), INT_ENUM},*)
(*DBG:    {&(RES0__INSTANCE0.MY_BAD_FIFO.BUFFER.value.table[2588]), INT_ENUM},*)
(*DBG:    {&(RES0__INSTANCE0.MY_BAD_FIFO.BUFFER.value.table[2589]), INT_ENUM},*)
(*DBG:    {&(RES0__INSTANCE0.MY_BAD_FIFO.BUFFER.value.table[2590]), INT_ENUM},*)
(*DBG:    {&(RES0__INSTANCE0.MY_BAD_FIFO.BUFFER.value.table[2591]), INT_ENUM},*)
(*DBG:    {&(RES0__INSTANCE0.MY_BAD_FIFO.BUFFER.value.table[2592]), INT_ENUM},*)
(*DBG:    {&(RES0__INSTANCE0.MY_BAD_FIFO.BUFFER.value.table[2593]), INT_ENUM},*)
(*DBG:    {&(RES0__INSTANCE0.MY_BAD_FIFO.BUFFER.value.table[2594]), INT_ENUM},*)
(*DBG:    {&(RES0__INSTANCE0.MY_BAD_FIFO.BUFFER.value.table[2595]), INT_ENUM},*)
(*DBG:    {&(RES0__INSTANCE0.MY_BAD_FIFO.BUFFER.value.table[2596]), INT_ENUM},*)
(*DBG:    {&(RES0__INSTANCE0.MY_BAD_FIFO.BUFFER.value.table[2597]), INT_ENUM},*)
(*DBG:    {&(RES0__INSTANCE0.MY_BAD_FIFO.BUFFER.value.table[2598]), INT_ENUM},*)
(*DBG:    {&(RES0__INSTANCE0.MY_BAD_FIFO.BUFFER.value.table[2599]), INT_ENUM},*)
(*DBG:    {&(RES0__INSTANCE0.MY_BAD_FIFO.BUFFER.value.table[2600]), INT_ENUM},*)
(*DBG:    {&(RES0__INSTANCE0.MY_BAD_FIFO.BUFFER.value.table[2601]), INT_ENUM},*)
(*DBG:    {&(RES0__INSTANCE0.MY_BAD_FIFO.BUFFER.value.table[2602]), INT_ENUM},*)
(*DBG:    {&(RES0__INSTANCE0.MY_BAD_FIFO.BUFFER.value.table[2603]), INT_ENUM},*)
(*DBG:    {&(RES0__INSTANCE0.MY_BAD_FIFO.BUFFER.value.table[2604]), INT_ENUM},*)
(*DBG:    {&(RES0__INSTANCE0.MY_BAD_FIFO.BUFFER.value.table[2605]), INT_ENUM},*)
(*DBG:    {&(RES0__INSTANCE0.MY_BAD_FIFO.BUFFER.value.table[2606]), INT_ENUM},*)
(*DBG:    {&(RES0__INSTANCE0.MY_BAD_FIFO.BUFFER.value.table[2607]), INT_ENUM},*)
(*DBG:    {&(RES0__INSTANCE0.MY_BAD_FIFO.BUFFER.value.table[2608]), INT_ENUM},*)
(*DBG:    {&(RES0__INSTANCE0.MY_BAD_FIFO.BUFFER.value.table[2609]), INT_ENUM},*)
(*DBG:    {&(RES0__INSTANCE0.MY_BAD_FIFO.BUFFER.value.table[2610]), INT_ENUM},*)
(*DBG:    {&(RES0__INSTANCE0.MY_BAD_FIFO.BUFFER.value.table[2611]), INT_ENUM},*)
(*DBG:    {&(RES0__INSTANCE0.MY_BAD_FIFO.BUFFER.value.table[2612]), INT_ENUM},*)
(*DBG:    {&(RES0__INSTANCE0.MY_BAD_FIFO.BUFFER.value.table[2613]), INT_ENUM},*)
(*DBG:    {&(RES0__INSTANCE0.MY_BAD_FIFO.BUFFER.value.table[2614]), INT_ENUM},*)
(*DBG:    {&(RES0__INSTANCE0.MY_BAD_FIFO.BUFFER.value.table[2615]), INT_ENUM},*)
(*DBG:    {&(RES0__INSTANCE0.MY_BAD_FIFO.BUFFER.value.table[2616]), INT_ENUM},*)
(*DBG:    {&(RES0__INSTANCE0.MY_BAD_FIFO.BUFFER.value.table[2617]), INT_ENUM},*)
(*DBG:    {&(RES0__INSTANCE0.MY_BAD_FIFO.BUFFER.value.table[2618]), INT_ENUM},*)
(*DBG:    {&(RES0__INSTANCE0.MY_BAD_FIFO.BUFFER.value.table[2619]), INT_ENUM},*)
(*DBG:    {&(RES0__INSTANCE0.MY_BAD_FIFO.BUFFER.value.table[2620]), INT_ENUM},*)
(*DBG:    {&(RES0__INSTANCE0.MY_BAD_FIFO.BUFFER.value.table[2621]), INT_ENUM},*)
(*DBG:    {&(RES0__INSTANCE0.MY_BAD_FIFO.BUFFER.value.table[2622]), INT_ENUM},*)
(*DBG:    {&(RES0__INSTANCE0.MY_BAD_FIFO.BUFFER.value.table[2623]), INT_ENUM},*)
(*DBG:    {&(RES0__INSTANCE0.MY_BAD_FIFO.BUFFER.value.table[2624]), INT_ENUM},*)
(*DBG:    {&(RES0__INSTANCE0.MY_BAD_FIFO.BUFFER.value.table[2625]), INT_ENUM},*)
(*DBG:    {&(RES0__INSTANCE0.MY_BAD_FIFO.BUFFER.value.table[2626]), INT_ENUM},*)
(*DBG:    {&(RES0__INSTANCE0.MY_BAD_FIFO.BUFFER.value.table[2627]), INT_ENUM},*)
(*DBG:    {&(RES0__INSTANCE0.MY_BAD_FIFO.BUFFER.value.table[2628]), INT_ENUM},*)
(*DBG:    {&(RES0__INSTANCE0.MY_BAD_FIFO.BUFFER.value.table[2629]), INT_ENUM},*)
(*DBG:    {&(RES0__INSTANCE0.MY_BAD_FIFO.BUFFER.value.table[2630]), INT_ENUM},*)
(*DBG:    {&(RES0__INSTANCE0.MY_BAD_FIFO.BUFFER.value.table[2631]), INT_ENUM},*)
(*DBG:    {&(RES0__INSTANCE0.MY_BAD_FIFO.BUFFER.value.table[2632]), INT_ENUM},*)
(*DBG:    {&(RES0__INSTANCE0.MY_BAD_FIFO.BUFFER.value.table[2633]), INT_ENUM},*)
(*DBG:    {&(RES0__INSTANCE0.MY_BAD_FIFO.BUFFER.value.table[2634]), INT_ENUM},*)
(*DBG:    {&(RES0__INSTANCE0.MY_BAD_FIFO.BUFFER.value.table[2635]), INT_ENUM},*)
(*DBG:    {&(RES0__INSTANCE0.MY_BAD_FIFO.BUFFER.value.table[2636]), INT_ENUM},*)
(*DBG:    {&(RES0__INSTANCE0.MY_BAD_FIFO.BUFFER.value.table[2637]), INT_ENUM},*)
(*DBG:    {&(RES0__INSTANCE0.MY_BAD_FIFO.BUFFER.value.table[2638]), INT_ENUM},*)
(*DBG:    {&(RES0__INSTANCE0.MY_BAD_FIFO.BUFFER.value.table[2639]), INT_ENUM},*)
(*DBG:    {&(RES0__INSTANCE0.MY_BAD_FIFO.BUFFER.value.table[2640]), INT_ENUM},*)
(*DBG:    {&(RES0__INSTANCE0.MY_BAD_FIFO.BUFFER.value.table[2641]), INT_ENUM},*)
(*DBG:    {&(RES0__INSTANCE0.MY_BAD_FIFO.BUFFER.value.table[2642]), INT_ENUM},*)
(*DBG:    {&(RES0__INSTANCE0.MY_BAD_FIFO.BUFFER.value.table[2643]), INT_ENUM},*)
(*DBG:    {&(RES0__INSTANCE0.MY_BAD_FIFO.BUFFER.value.table[2644]), INT_ENUM},*)
(*DBG:    {&(RES0__INSTANCE0.MY_BAD_FIFO.BUFFER.value.table[2645]), INT_ENUM},*)
(*DBG:    {&(RES0__INSTANCE0.MY_BAD_FIFO.BUFFER.value.table[2646]), INT_ENUM},*)
(*DBG:    {&(RES0__INSTANCE0.MY_BAD_FIFO.BUFFER.value.table[2647]), INT_ENUM},*)
(*DBG:    {&(RES0__INSTANCE0.MY_BAD_FIFO.BUFFER.value.table[2648]), INT_ENUM},*)
(*DBG:    {&(RES0__INSTANCE0.MY_BAD_FIFO.BUFFER.value.table[2649]), INT_ENUM},*)
(*DBG:    {&(RES0__INSTANCE0.MY_BAD_FIFO.BUFFER.value.table[2650]), INT_ENUM},*)
(*DBG:    {&(RES0__INSTANCE0.MY_BAD_FIFO.BUFFER.value.table[2651]), INT_ENUM},*)
(*DBG:    {&(RES0__INSTANCE0.MY_BAD_FIFO.BUFFER.value.table[2652]), INT_ENUM},*)
(*DBG:    {&(RES0__INSTANCE0.MY_BAD_FIFO.BUFFER.value.table[2653]), INT_ENUM},*)
(*DBG:    {&(RES0__INSTANCE0.MY_BAD_FIFO.BUFFER.value.table[2654]), INT_ENUM},*)
(*DBG:    {&(RES0__INSTANCE0.MY_BAD_FIFO.BUFFER.value.table[2655]), INT_ENUM},*)
(*DBG:    {&(RES0__INSTANCE0.MY_BAD_FIFO.BUFFER.value.table[2656]), INT_ENUM},*)
(*DBG:    {&(RES0__INSTANCE0.MY_BAD_FIFO.BUFFER.value.table[2657]), INT_ENUM},*)
(*DBG:    {&(RES0__INSTANCE0.MY_BAD_FIFO.BUFFER.value.table[2658]), INT_ENUM},*)
(*DBG:    {&(RES0__INSTANCE0.MY_BAD_FIFO.BUFFER.value.table[2659]), INT_ENUM},*)
(*DBG:    {&(RES0__INSTANCE0.MY_BAD_FIFO.BUFFER.value.table[2660]), INT_ENUM},*)
(*DBG:    {&(RES0__INSTANCE0.MY_BAD_FIFO.BUFFER.value.table[2661]), INT_ENUM},*)
(*DBG:    {&(RES0__INSTANCE0.MY_BAD_FIFO.BUFFER.value.table[2662]), INT_ENUM},*)
(*DBG:    {&(RES0__INSTANCE0.MY_BAD_FIFO.BUFFER.value.table[2663]), INT_ENUM},*)
(*DBG:    {&(RES0__INSTANCE0.MY_BAD_FIFO.BUFFER.value.table[2664]), INT_ENUM},*)
(*DBG:    {&(RES0__INSTANCE0.MY_BAD_FIFO.BUFFER.value.table[2665]), INT_ENUM},*)
(*DBG:    {&(RES0__INSTANCE0.MY_BAD_FIFO.BUFFER.value.table[2666]), INT_ENUM},*)
(*DBG:    {&(RES0__INSTANCE0.MY_BAD_FIFO.BUFFER.value.table[2667]), INT_ENUM},*)
(*DBG:    {&(RES0__INSTANCE0.MY_BAD_FIFO.BUFFER.value.table[2668]), INT_ENUM},*)
(*DBG:    {&(RES0__INSTANCE0.MY_BAD_FIFO.BUFFER.value.table[2669]), INT_ENUM},*)
(*DBG:    {&(RES0__INSTANCE0.MY_BAD_FIFO.BUFFER.value.table[2670]), INT_ENUM},*)
(*DBG:    {&(RES0__INSTANCE0.MY_BAD_FIFO.BUFFER.value.table[2671]), INT_ENUM},*)
(*DBG:    {&(RES0__INSTANCE0.MY_BAD_FIFO.BUFFER.value.table[2672]), INT_ENUM},*)
(*DBG:    {&(RES0__INSTANCE0.MY_BAD_FIFO.BUFFER.value.table[2673]), INT_ENUM},*)
(*DBG:    {&(RES0__INSTANCE0.MY_BAD_FIFO.BUFFER.value.table[2674]), INT_ENUM},*)
(*DBG:    {&(RES0__INSTANCE0.MY_BAD_FIFO.BUFFER.value.table[2675]), INT_ENUM},*)
(*DBG:    {&(RES0__INSTANCE0.MY_BAD_FIFO.BUFFER.value.table[2676]), INT_ENUM},*)
(*DBG:    {&(RES0__INSTANCE0.MY_BAD_FIFO.BUFFER.value.table[2677]), INT_ENUM},*)
(*DBG:    {&(RES0__INSTANCE0.MY_BAD_FIFO.BUFFER.value.table[2678]), INT_ENUM},*)
(*DBG:    {&(RES0__INSTANCE0.MY_BAD_FIFO.BUFFER.value.table[2679]), INT_ENUM},*)
(*DBG:    {&(RES0__INSTANCE0.MY_BAD_FIFO.BUFFER.value.table[2680]), INT_ENUM},*)
(*DBG:    {&(RES0__INSTANCE0.MY_BAD_FIFO.BUFFER.value.table[2681]), INT_ENUM},*)
(*DBG:    {&(RES0__INSTANCE0.MY_BAD_FIFO.BUFFER.value.table[2682]), INT_ENUM},*)
(*DBG:    {&(RES0__INSTANCE0.MY_BAD_FIFO.BUFFER.value.table[2683]), INT_ENUM},*)
(*DBG:    {&(RES0__INSTANCE0.MY_BAD_FIFO.BUFFER.value.table[2684]), INT_ENUM},*)
(*DBG:    {&(RES0__INSTANCE0.MY_BAD_FIFO.BUFFER.value.table[2685]), INT_ENUM},*)
(*DBG:    {&(RES0__INSTANCE0.MY_BAD_FIFO.BUFFER.value.table[2686]), INT_ENUM},*)
(*DBG:    {&(RES0__INSTANCE0.MY_BAD_FIFO.BUFFER.value.table[2687]), INT_ENUM},*)
(*DBG:    {&(RES0__INSTANCE0.MY_BAD_FIFO.BUFFER.value.table[2688]), INT_ENUM},*)
(*DBG:    {&(RES0__INSTANCE0.MY_BAD_FIFO.BUFFER.value.table[2689]), INT_ENUM},*)
(*DBG:    {&(RES0__INSTANCE0.MY_BAD_FIFO.BUFFER.value.table[2690]), INT_ENUM},*)
(*DBG:    {&(RES0__INSTANCE0.MY_BAD_FIFO.BUFFER.value.table[2691]), INT_ENUM},*)
(*DBG:    {&(RES0__INSTANCE0.MY_BAD_FIFO.BUFFER.value.table[2692]), INT_ENUM},*)
(*DBG:    {&(RES0__INSTANCE0.MY_BAD_FIFO.BUFFER.value.table[2693]), INT_ENUM},*)
(*DBG:    {&(RES0__INSTANCE0.MY_BAD_FIFO.BUFFER.value.table[2694]), INT_ENUM},*)
(*DBG:    {&(RES0__INSTANCE0.MY_BAD_FIFO.BUFFER.value.table[2695]), INT_ENUM},*)
(*DBG:    {&(RES0__INSTANCE0.MY_BAD_FIFO.BUFFER.value.table[2696]), INT_ENUM},*)
(*DBG:    {&(RES0__INSTANCE0.MY_BAD_FIFO.BUFFER.value.table[2697]), INT_ENUM},*)
(*DBG:    {&(RES0__INSTANCE0.MY_BAD_FIFO.BUFFER.value.table[2698]), INT_ENUM},*)
(*DBG:    {&(RES0__INSTANCE0.MY_BAD_FIFO.BUFFER.value.table[2699]), INT_ENUM},*)
(*DBG:    {&(RES0__INSTANCE0.MY_BAD_FIFO.BUFFER.value.table[2700]), INT_ENUM},*)
(*DBG:    {&(RES0__INSTANCE0.MY_BAD_FIFO.BUFFER.value.table[2701]), INT_ENUM},*)
(*DBG:    {&(RES0__INSTANCE0.MY_BAD_FIFO.BUFFER.value.table[2702]), INT_ENUM},*)
(*DBG:    {&(RES0__INSTANCE0.MY_BAD_FIFO.BUFFER.value.table[2703]), INT_ENUM},*)
(*DBG:    {&(RES0__INSTANCE0.MY_BAD_FIFO.BUFFER.value.table[2704]), INT_ENUM},*)
(*DBG:    {&(RES0__INSTANCE0.MY_BAD_FIFO.BUFFER.value.table[2705]), INT_ENUM},*)
(*DBG:    {&(RES0__INSTANCE0.MY_BAD_FIFO.BUFFER.value.table[2706]), INT_ENUM},*)
(*DBG:    {&(RES0__INSTANCE0.MY_BAD_FIFO.BUFFER.value.table[2707]), INT_ENUM},*)
(*DBG:    {&(RES0__INSTANCE0.MY_BAD_FIFO.BUFFER.value.table[2708]), INT_ENUM},*)
(*DBG:    {&(RES0__INSTANCE0.MY_BAD_FIFO.BUFFER.value.table[2709]), INT_ENUM},*)
(*DBG:    {&(RES0__INSTANCE0.MY_BAD_FIFO.BUFFER.value.table[2710]), INT_ENUM},*)
(*DBG:    {&(RES0__INSTANCE0.MY_BAD_FIFO.BUFFER.value.table[2711]), INT_ENUM},*)
(*DBG:    {&(RES0__INSTANCE0.MY_BAD_FIFO.BUFFER.value.table[2712]), INT_ENUM},*)
(*DBG:    {&(RES0__INSTANCE0.MY_BAD_FIFO.BUFFER.value.table[2713]), INT_ENUM},*)
(*DBG:    {&(RES0__INSTANCE0.MY_BAD_FIFO.BUFFER.value.table[2714]), INT_ENUM},*)
(*DBG:    {&(RES0__INSTANCE0.MY_BAD_FIFO.BUFFER.value.table[2715]), INT_ENUM},*)
(*DBG:    {&(RES0__INSTANCE0.MY_BAD_FIFO.BUFFER.value.table[2716]), INT_ENUM},*)
(*DBG:    {&(RES0__INSTANCE0.MY_BAD_FIFO.BUFFER.value.table[2717]), INT_ENUM},*)
(*DBG:    {&(RES0__INSTANCE0.MY_BAD_FIFO.BUFFER.value.table[2718]), INT_ENUM},*)
(*DBG:    {&(RES0__INSTANCE0.MY_BAD_FIFO.BUFFER.value.table[2719]), INT_ENUM},*)
(*DBG:    {&(RES0__INSTANCE0.MY_BAD_FIFO.BUFFER.value.table[2720]), INT_ENUM},*)
(*DBG:    {&(RES0__INSTANCE0.MY_BAD_FIFO.BUFFER.value.table[2721]), INT_ENUM},*)
(*DBG:    {&(RES0__INSTANCE0.MY_BAD_FIFO.BUFFER.value.table[2722]), INT_ENUM},*)
(*DBG:    {&(RES0__INSTANCE0.MY_BAD_FIFO.BUFFER.value.table[2723]), INT_ENUM},*)
(*DBG:    {&(RES0__INSTANCE0.MY_BAD_FIFO.BUFFER.value.table[2724]), INT_ENUM},*)
(*DBG:    {&(RES0__INSTANCE0.MY_BAD_FIFO.BUFFER.value.table[2725]), INT_ENUM},*)
(*DBG:    {&(RES0__INSTANCE0.MY_BAD_FIFO.BUFFER.value.table[2726]), INT_ENUM},*)
(*DBG:    {&(RES0__INSTANCE0.MY_BAD_FIFO.BUFFER.value.table[2727]), INT_ENUM},*)
(*DBG:    {&(RES0__INSTANCE0.MY_BAD_FIFO.BUFFER.value.table[2728]), INT_ENUM},*)
(*DBG:    {&(RES0__INSTANCE0.MY_BAD_FIFO.BUFFER.value.table[2729]), INT_ENUM},*)
(*DBG:    {&(RES0__INSTANCE0.MY_BAD_FIFO.BUFFER.value.table[2730]), INT_ENUM},*)
(*DBG:    {&(RES0__INSTANCE0.MY_BAD_FIFO.BUFFER.value.table[2731]), INT_ENUM},*)
(*DBG:    {&(RES0__INSTANCE0.MY_BAD_FIFO.BUFFER.value.table[2732]), INT_ENUM},*)
(*DBG:    {&(RES0__INSTANCE0.MY_BAD_FIFO.BUFFER.value.table[2733]), INT_ENUM},*)
(*DBG:    {&(RES0__INSTANCE0.MY_BAD_FIFO.BUFFER.value.table[2734]), INT_ENUM},*)
(*DBG:    {&(RES0__INSTANCE0.MY_BAD_FIFO.BUFFER.value.table[2735]), INT_ENUM},*)
(*DBG:    {&(RES0__INSTANCE0.MY_BAD_FIFO.BUFFER.value.table[2736]), INT_ENUM},*)
(*DBG:    {&(RES0__INSTANCE0.MY_BAD_FIFO.BUFFER.value.table[2737]), INT_ENUM},*)
(*DBG:    {&(RES0__INSTANCE0.MY_BAD_FIFO.BUFFER.value.table[2738]), INT_ENUM},*)
(*DBG:    {&(RES0__INSTANCE0.MY_BAD_FIFO.BUFFER.value.table[2739]), INT_ENUM},*)
(*DBG:    {&(RES0__INSTANCE0.MY_BAD_FIFO.BUFFER.value.table[2740]), INT_ENUM},*)
(*DBG:    {&(RES0__INSTANCE0.MY_BAD_FIFO.BUFFER.value.table[2741]), INT_ENUM},*)
(*DBG:    {&(RES0__INSTANCE0.MY_BAD_FIFO.BUFFER.value.table[2742]), INT_ENUM},*)
(*DBG:    {&(RES0__INSTANCE0.MY_BAD_FIFO.BUFFER.value.table[2743]), INT_ENUM},*)
(*DBG:    {&(RES0__INSTANCE0.MY_BAD_FIFO.BUFFER.value.table[2744]), INT_ENUM},*)
(*DBG:    {&(RES0__INSTANCE0.MY_BAD_FIFO.BUFFER.value.table[2745]), INT_ENUM},*)
(*DBG:    {&(RES0__INSTANCE0.MY_BAD_FIFO.BUFFER.value.table[2746]), INT_ENUM},*)
(*DBG:    {&(RES0__INSTANCE0.MY_BAD_FIFO.BUFFER.value.table[2747]), INT_ENUM},*)
(*DBG:    {&(RES0__INSTANCE0.MY_BAD_FIFO.BUFFER.value.table[2748]), INT_ENUM},*)
(*DBG:    {&(RES0__INSTANCE0.MY_BAD_FIFO.BUFFER.value.table[2749]), INT_ENUM},*)
(*DBG:    {&(RES0__INSTANCE0.MY_BAD_FIFO.BUFFER.value.table[2750]), INT_ENUM},*)
(*DBG:    {&(RES0__INSTANCE0.MY_BAD_FIFO.BUFFER.value.table[2751]), INT_ENUM},*)
(*DBG:    {&(RES0__INSTANCE0.MY_BAD_FIFO.BUFFER.value.table[2752]), INT_ENUM},*)
(*DBG:    {&(RES0__INSTANCE0.MY_BAD_FIFO.BUFFER.value.table[2753]), INT_ENUM},*)
(*DBG:    {&(RES0__INSTANCE0.MY_BAD_FIFO.BUFFER.value.table[2754]), INT_ENUM},*)
(*DBG:    {&(RES0__INSTANCE0.MY_BAD_FIFO.BUFFER.value.table[2755]), INT_ENUM},*)
(*DBG:    {&(RES0__INSTANCE0.MY_BAD_FIFO.BUFFER.value.table[2756]), INT_ENUM},*)
(*DBG:    {&(RES0__INSTANCE0.MY_BAD_FIFO.BUFFER.value.table[2757]), INT_ENUM},*)
(*DBG:    {&(RES0__INSTANCE0.MY_BAD_FIFO.BUFFER.value.table[2758]), INT_ENUM},*)
(*DBG:    {&(RES0__INSTANCE0.MY_BAD_FIFO.BUFFER.value.table[2759]), INT_ENUM},*)
(*DBG:    {&(RES0__INSTANCE0.MY_BAD_FIFO.BUFFER.value.table[2760]), INT_ENUM},*)
(*DBG:    {&(RES0__INSTANCE0.MY_BAD_FIFO.BUFFER.value.table[2761]), INT_ENUM},*)
(*DBG:    {&(RES0__INSTANCE0.MY_BAD_FIFO.BUFFER.value.table[2762]), INT_ENUM},*)
(*DBG:    {&(RES0__INSTANCE0.MY_BAD_FIFO.BUFFER.value.table[2763]), INT_ENUM},*)
(*DBG:    {&(RES0__INSTANCE0.MY_BAD_FIFO.BUFFER.value.table[2764]), INT_ENUM},*)
(*DBG:    {&(RES0__INSTANCE0.MY_BAD_FIFO.BUFFER.value.table[2765]), INT_ENUM},*)
(*DBG:    {&(RES0__INSTANCE0.MY_BAD_FIFO.BUFFER.value.table[2766]), INT_ENUM},*)
(*DBG:    {&(RES0__INSTANCE0.MY_BAD_FIFO.BUFFER.value.table[2767]), INT_ENUM},*)
(*DBG:    {&(RES0__INSTANCE0.MY_BAD_FIFO.BUFFER.value.table[2768]), INT_ENUM},*)
(*DBG:    {&(RES0__INSTANCE0.MY_BAD_FIFO.BUFFER.value.table[2769]), INT_ENUM},*)
(*DBG:    {&(RES0__INSTANCE0.MY_BAD_FIFO.BUFFER.value.table[2770]), INT_ENUM},*)
(*DBG:    {&(RES0__INSTANCE0.MY_BAD_FIFO.BUFFER.value.table[2771]), INT_ENUM},*)
(*DBG:    {&(RES0__INSTANCE0.MY_BAD_FIFO.BUFFER.value.table[2772]), INT_ENUM},*)
(*DBG:    {&(RES0__INSTANCE0.MY_BAD_FIFO.BUFFER.value.table[2773]), INT_ENUM},*)
(*DBG:    {&(RES0__INSTANCE0.MY_BAD_FIFO.BUFFER.value.table[2774]), INT_ENUM},*)
(*DBG:    {&(RES0__INSTANCE0.MY_BAD_FIFO.BUFFER.value.table[2775]), INT_ENUM},*)
(*DBG:    {&(RES0__INSTANCE0.MY_BAD_FIFO.BUFFER.value.table[2776]), INT_ENUM},*)
(*DBG:    {&(RES0__INSTANCE0.MY_BAD_FIFO.BUFFER.value.table[2777]), INT_ENUM},*)
(*DBG:    {&(RES0__INSTANCE0.MY_BAD_FIFO.BUFFER.value.table[2778]), INT_ENUM},*)
(*DBG:    {&(RES0__INSTANCE0.MY_BAD_FIFO.BUFFER.value.table[2779]), INT_ENUM},*)
(*DBG:    {&(RES0__INSTANCE0.MY_BAD_FIFO.BUFFER.value.table[2780]), INT_ENUM},*)
(*DBG:    {&(RES0__INSTANCE0.MY_BAD_FIFO.BUFFER.value.table[2781]), INT_ENUM},*)
(*DBG:    {&(RES0__INSTANCE0.MY_BAD_FIFO.BUFFER.value.table[2782]), INT_ENUM},*)
(*DBG:    {&(RES0__INSTANCE0.MY_BAD_FIFO.BUFFER.value.table[2783]), INT_ENUM},*)
(*DBG:    {&(RES0__INSTANCE0.MY_BAD_FIFO.BUFFER.value.table[2784]), INT_ENUM},*)
(*DBG:    {&(RES0__INSTANCE0.MY_BAD_FIFO.BUFFER.value.table[2785]), INT_ENUM},*)
(*DBG:    {&(RES0__INSTANCE0.MY_BAD_FIFO.BUFFER.value.table[2786]), INT_ENUM},*)
(*DBG:    {&(RES0__INSTANCE0.MY_BAD_FIFO.BUFFER.value.table[2787]), INT_ENUM},*)
(*DBG:    {&(RES0__INSTANCE0.MY_BAD_FIFO.BUFFER.value.table[2788]), INT_ENUM},*)
(*DBG:    {&(RES0__INSTANCE0.MY_BAD_FIFO.BUFFER.value.table[2789]), INT_ENUM},*)
(*DBG:    {&(RES0__INSTANCE0.MY_BAD_FIFO.BUFFER.value.table[2790]), INT_ENUM},*)
(*DBG:    {&(RES0__INSTANCE0.MY_BAD_FIFO.BUFFER.value.table[2791]), INT_ENUM},*)
(*DBG:    {&(RES0__INSTANCE0.MY_BAD_FIFO.BUFFER.value.table[2792]), INT_ENUM},*)
(*DBG:    {&(RES0__INSTANCE0.MY_BAD_FIFO.BUFFER.value.table[2793]), INT_ENUM},*)
(*DBG:    {&(RES0__INSTANCE0.MY_BAD_FIFO.BUFFER.value.table[2794]), INT_ENUM},*)
(*DBG:    {&(RES0__INSTANCE0.MY_BAD_FIFO.BUFFER.value.table[2795]), INT_ENUM},*)
(*DBG:    {&(RES0__INSTANCE0.MY_BAD_FIFO.BUFFER.value.table[2796]), INT_ENUM},*)
(*DBG:    {&(RES0__INSTANCE0.MY_BAD_FIFO.BUFFER.value.table[2797]), INT_ENUM},*)
(*DBG:    {&(RES0__INSTANCE0.MY_BAD_FIFO.BUFFER.value.table[2798]), INT_ENUM},*)
(*DBG:    {&(RES0__INSTANCE0.MY_BAD_FIFO.BUFFER.value.table[2799]), INT_ENUM},*)
(*DBG:    {&(RES0__INSTANCE0.MY_BAD_FIFO.BUFFER.value.table[2800]), INT_ENUM},*)
(*DBG:    {&(RES0__INSTANCE0.MY_BAD_FIFO.BUFFER.value.table[2801]), INT_ENUM},*)
(*DBG:    {&(RES0__INSTANCE0.MY_BAD_FIFO.BUFFER.value.table[2802]), INT_ENUM},*)
(*DBG:    {&(RES0__INSTANCE0.MY_BAD_FIFO.BUFFER.value.table[2803]), INT_ENUM},*)
(*DBG:    {&(RES0__INSTANCE0.MY_BAD_FIFO.BUFFER.value.table[2804]), INT_ENUM},*)
(*DBG:    {&(RES0__INSTANCE0.MY_BAD_FIFO.BUFFER.value.table[2805]), INT_ENUM},*)
(*DBG:    {&(RES0__INSTANCE0.MY_BAD_FIFO.BUFFER.value.table[2806]), INT_ENUM},*)
(*DBG:    {&(RES0__INSTANCE0.MY_BAD_FIFO.BUFFER.value.table[2807]), INT_ENUM},*)
(*DBG:    {&(RES0__INSTANCE0.MY_BAD_FIFO.BUFFER.value.table[2808]), INT_ENUM},*)
(*DBG:    {&(RES0__INSTANCE0.MY_BAD_FIFO.BUFFER.value.table[2809]), INT_ENUM},*)
(*DBG:    {&(RES0__INSTANCE0.MY_BAD_FIFO.BUFFER.value.table[2810]), INT_ENUM},*)
(*DBG:    {&(RES0__INSTANCE0.MY_BAD_FIFO.BUFFER.value.table[2811]), INT_ENUM},*)
(*DBG:    {&(RES0__INSTANCE0.MY_BAD_FIFO.BUFFER.value.table[2812]), INT_ENUM},*)
(*DBG:    {&(RES0__INSTANCE0.MY_BAD_FIFO.BUFFER.value.table[2813]), INT_ENUM},*)
(*DBG:    {&(RES0__INSTANCE0.MY_BAD_FIFO.BUFFER.value.table[2814]), INT_ENUM},*)
(*DBG:    {&(RES0__INSTANCE0.MY_BAD_FIFO.BUFFER.value.table[2815]), INT_ENUM},*)
(*DBG:    {&(RES0__INSTANCE0.MY_BAD_FIFO.BUFFER.value.table[2816]), INT_ENUM},*)
(*DBG:    {&(RES0__INSTANCE0.MY_BAD_FIFO.BUFFER.value.table[2817]), INT_ENUM},*)
(*DBG:    {&(RES0__INSTANCE0.MY_BAD_FIFO.BUFFER.value.table[2818]), INT_ENUM},*)
(*DBG:    {&(RES0__INSTANCE0.MY_BAD_FIFO.BUFFER.value.table[2819]), INT_ENUM},*)
(*DBG:    {&(RES0__INSTANCE0.MY_BAD_FIFO.BUFFER.value.table[2820]), INT_ENUM},*)
(*DBG:    {&(RES0__INSTANCE0.MY_BAD_FIFO.BUFFER.value.table[2821]), INT_ENUM},*)
(*DBG:    {&(RES0__INSTANCE0.MY_BAD_FIFO.BUFFER.value.table[2822]), INT_ENUM},*)
(*DBG:    {&(RES0__INSTANCE0.MY_BAD_FIFO.BUFFER.value.table[2823]), INT_ENUM},*)
(*DBG:    {&(RES0__INSTANCE0.MY_BAD_FIFO.BUFFER.value.table[2824]), INT_ENUM},*)
(*DBG:    {&(RES0__INSTANCE0.MY_BAD_FIFO.BUFFER.value.table[2825]), INT_ENUM},*)
(*DBG:    {&(RES0__INSTANCE0.MY_BAD_FIFO.BUFFER.value.table[2826]), INT_ENUM},*)
(*DBG:    {&(RES0__INSTANCE0.MY_BAD_FIFO.BUFFER.value.table[2827]), INT_ENUM},*)
(*DBG:    {&(RES0__INSTANCE0.MY_BAD_FIFO.BUFFER.value.table[2828]), INT_ENUM},*)
(*DBG:    {&(RES0__INSTANCE0.MY_BAD_FIFO.BUFFER.value.table[2829]), INT_ENUM},*)
(*DBG:    {&(RES0__INSTANCE0.MY_BAD_FIFO.BUFFER.value.table[2830]), INT_ENUM},*)
(*DBG:    {&(RES0__INSTANCE0.MY_BAD_FIFO.BUFFER.value.table[2831]), INT_ENUM},*)
(*DBG:    {&(RES0__INSTANCE0.MY_BAD_FIFO.BUFFER.value.table[2832]), INT_ENUM},*)
(*DBG:    {&(RES0__INSTANCE0.MY_BAD_FIFO.BUFFER.value.table[2833]), INT_ENUM},*)
(*DBG:    {&(RES0__INSTANCE0.MY_BAD_FIFO.BUFFER.value.table[2834]), INT_ENUM},*)
(*DBG:    {&(RES0__INSTANCE0.MY_BAD_FIFO.BUFFER.value.table[2835]), INT_ENUM},*)
(*DBG:    {&(RES0__INSTANCE0.MY_BAD_FIFO.BUFFER.value.table[2836]), INT_ENUM},*)
(*DBG:    {&(RES0__INSTANCE0.MY_BAD_FIFO.BUFFER.value.table[2837]), INT_ENUM},*)
(*DBG:    {&(RES0__INSTANCE0.MY_BAD_FIFO.BUFFER.value.table[2838]), INT_ENUM},*)
(*DBG:    {&(RES0__INSTANCE0.MY_BAD_FIFO.BUFFER.value.table[2839]), INT_ENUM},*)
(*DBG:    {&(RES0__INSTANCE0.MY_BAD_FIFO.BUFFER.value.table[2840]), INT_ENUM},*)
(*DBG:    {&(RES0__INSTANCE0.MY_BAD_FIFO.BUFFER.value.table[2841]), INT_ENUM},*)
(*DBG:    {&(RES0__INSTANCE0.MY_BAD_FIFO.BUFFER.value.table[2842]), INT_ENUM},*)
(*DBG:    {&(RES0__INSTANCE0.MY_BAD_FIFO.BUFFER.value.table[2843]), INT_ENUM},*)
(*DBG:    {&(RES0__INSTANCE0.MY_BAD_FIFO.BUFFER.value.table[2844]), INT_ENUM},*)
(*DBG:    {&(RES0__INSTANCE0.MY_BAD_FIFO.BUFFER.value.table[2845]), INT_ENUM},*)
(*DBG:    {&(RES0__INSTANCE0.MY_BAD_FIFO.BUFFER.value.table[2846]), INT_ENUM},*)
(*DBG:    {&(RES0__INSTANCE0.MY_BAD_FIFO.BUFFER.value.table[2847]), INT_ENUM},*)
(*DBG:    {&(RES0__INSTANCE0.MY_BAD_FIFO.BUFFER.value.table[2848]), INT_ENUM},*)
(*DBG:    {&(RES0__INSTANCE0.MY_BAD_FIFO.BUFFER.value.table[2849]), INT_ENUM},*)
(*DBG:    {&(RES0__INSTANCE0.MY_BAD_FIFO.BUFFER.value.table[2850]), INT_ENUM},*)
(*DBG:    {&(RES0__INSTANCE0.MY_BAD_FIFO.BUFFER.value.table[2851]), INT_ENUM},*)
(*DBG:    {&(RES0__INSTANCE0.MY_BAD_FIFO.BUFFER.value.table[2852]), INT_ENUM},*)
(*DBG:    {&(RES0__INSTANCE0.MY_BAD_FIFO.BUFFER.value.table[2853]), INT_ENUM},*)
(*DBG:    {&(RES0__INSTANCE0.MY_BAD_FIFO.BUFFER.value.table[2854]), INT_ENUM},*)
(*DBG:    {&(RES0__INSTANCE0.MY_BAD_FIFO.BUFFER.value.table[2855]), INT_ENUM},*)
(*DBG:    {&(RES0__INSTANCE0.MY_BAD_FIFO.BUFFER.value.table[2856]), INT_ENUM},*)
(*DBG:    {&(RES0__INSTANCE0.MY_BAD_FIFO.BUFFER.value.table[2857]), INT_ENUM},*)
(*DBG:    {&(RES0__INSTANCE0.MY_BAD_FIFO.BUFFER.value.table[2858]), INT_ENUM},*)
(*DBG:    {&(RES0__INSTANCE0.MY_BAD_FIFO.BUFFER.value.table[2859]), INT_ENUM},*)
(*DBG:    {&(RES0__INSTANCE0.MY_BAD_FIFO.BUFFER.value.table[2860]), INT_ENUM},*)
(*DBG:    {&(RES0__INSTANCE0.MY_BAD_FIFO.BUFFER.value.table[2861]), INT_ENUM},*)
(*DBG:    {&(RES0__INSTANCE0.MY_BAD_FIFO.BUFFER.value.table[2862]), INT_ENUM},*)
(*DBG:    {&(RES0__INSTANCE0.MY_BAD_FIFO.BUFFER.value.table[2863]), INT_ENUM},*)
(*DBG:    {&(RES0__INSTANCE0.MY_BAD_FIFO.BUFFER.value.table[2864]), INT_ENUM},*)
(*DBG:    {&(RES0__INSTANCE0.MY_BAD_FIFO.BUFFER.value.table[2865]), INT_ENUM},*)
(*DBG:    {&(RES0__INSTANCE0.MY_BAD_FIFO.BUFFER.value.table[2866]), INT_ENUM},*)
(*DBG:    {&(RES0__INSTANCE0.MY_BAD_FIFO.BUFFER.value.table[2867]), INT_ENUM},*)
(*DBG:    {&(RES0__INSTANCE0.MY_BAD_FIFO.BUFFER.value.table[2868]), INT_ENUM},*)
(*DBG:    {&(RES0__INSTANCE0.MY_BAD_FIFO.BUFFER.value.table[2869]), INT_ENUM},*)
(*DBG:    {&(RES0__INSTANCE0.MY_BAD_FIFO.BUFFER.value.table[2870]), INT_ENUM},*)
(*DBG:    {&(RES0__INSTANCE0.MY_BAD_FIFO.BUFFER.value.table[2871]), INT_ENUM},*)
(*DBG:    {&(RES0__INSTANCE0.MY_BAD_FIFO.BUFFER.value.table[2872]), INT_ENUM},*)
(*DBG:    {&(RES0__INSTANCE0.MY_BAD_FIFO.BUFFER.value.table[2873]), INT_ENUM},*)
(*DBG:    {&(RES0__INSTANCE0.MY_BAD_FIFO.BUFFER.value.table[2874]), INT_ENUM},*)
(*DBG:    {&(RES0__INSTANCE0.MY_BAD_FIFO.BUFFER.value.table[2875]), INT_ENUM},*)
(*DBG:    {&(RES0__INSTANCE0.MY_BAD_FIFO.BUFFER.value.table[2876]), INT_ENUM},*)
(*DBG:    {&(RES0__INSTANCE0.MY_BAD_FIFO.BUFFER.value.table[2877]), INT_ENUM},*)
(*DBG:    {&(RES0__INSTANCE0.MY_BAD_FIFO.BUFFER.value.table[2878]), INT_ENUM},*)
(*DBG:    {&(RES0__INSTANCE0.MY_BAD_FIFO.BUFFER.value.table[2879]), INT_ENUM},*)
(*DBG:    {&(RES0__INSTANCE0.MY_BAD_FIFO.BUFFER.value.table[2880]), INT_ENUM},*)
(*DBG:    {&(RES0__INSTANCE0.MY_BAD_FIFO.BUFFER.value.table[2881]), INT_ENUM},*)
(*DBG:    {&(RES0__INSTANCE0.MY_BAD_FIFO.BUFFER.value.table[2882]), INT_ENUM},*)
(*DBG:    {&(RES0__INSTANCE0.MY_BAD_FIFO.BUFFER.value.table[2883]), INT_ENUM},*)
(*DBG:    {&(RES0__INSTANCE0.MY_BAD_FIFO.BUFFER.value.table[2884]), INT_ENUM},*)
(*DBG:    {&(RES0__INSTANCE0.MY_BAD_FIFO.BUFFER.value.table[2885]), INT_ENUM},*)
(*DBG:    {&(RES0__INSTANCE0.MY_BAD_FIFO.BUFFER.value.table[2886]), INT_ENUM},*)
(*DBG:    {&(RES0__INSTANCE0.MY_BAD_FIFO.BUFFER.value.table[2887]), INT_ENUM},*)
(*DBG:    {&(RES0__INSTANCE0.MY_BAD_FIFO.BUFFER.value.table[2888]), INT_ENUM},*)
(*DBG:    {&(RES0__INSTANCE0.MY_BAD_FIFO.BUFFER.value.table[2889]), INT_ENUM},*)
(*DBG:    {&(RES0__INSTANCE0.MY_BAD_FIFO.BUFFER.value.table[2890]), INT_ENUM},*)
(*DBG:    {&(RES0__INSTANCE0.MY_BAD_FIFO.BUFFER.value.table[2891]), INT_ENUM},*)
(*DBG:    {&(RES0__INSTANCE0.MY_BAD_FIFO.BUFFER.value.table[2892]), INT_ENUM},*)
(*DBG:    {&(RES0__INSTANCE0.MY_BAD_FIFO.BUFFER.value.table[2893]), INT_ENUM},*)
(*DBG:    {&(RES0__INSTANCE0.MY_BAD_FIFO.BUFFER.value.table[2894]), INT_ENUM},*)
(*DBG:    {&(RES0__INSTANCE0.MY_BAD_FIFO.BUFFER.value.table[2895]), INT_ENUM},*)
(*DBG:    {&(RES0__INSTANCE0.MY_BAD_FIFO.BUFFER.value.table[2896]), INT_ENUM},*)
(*DBG:    {&(RES0__INSTANCE0.MY_BAD_FIFO.BUFFER.value.table[2897]), INT_ENUM},*)
(*DBG:    {&(RES0__INSTANCE0.MY_BAD_FIFO.BUFFER.value.table[2898]), INT_ENUM},*)
(*DBG:    {&(RES0__INSTANCE0.MY_BAD_FIFO.BUFFER.value.table[2899]), INT_ENUM},*)
(*DBG:    {&(RES0__INSTANCE0.MY_BAD_FIFO.BUFFER.value.table[2900]), INT_ENUM},*)
(*DBG:    {&(RES0__INSTANCE0.MY_BAD_FIFO.BUFFER.value.table[2901]), INT_ENUM},*)
(*DBG:    {&(RES0__INSTANCE0.MY_BAD_FIFO.BUFFER.value.table[2902]), INT_ENUM},*)
(*DBG:    {&(RES0__INSTANCE0.MY_BAD_FIFO.BUFFER.value.table[2903]), INT_ENUM},*)
(*DBG:    {&(RES0__INSTANCE0.MY_BAD_FIFO.BUFFER.value.table[2904]), INT_ENUM},*)
(*DBG:    {&(RES0__INSTANCE0.MY_BAD_FIFO.BUFFER.value.table[2905]), INT_ENUM},*)
(*DBG:    {&(RES0__INSTANCE0.MY_BAD_FIFO.BUFFER.value.table[2906]), INT_ENUM},*)
(*DBG:    {&(RES0__INSTANCE0.MY_BAD_FIFO.BUFFER.value.table[2907]), INT_ENUM},*)
(*DBG:    {&(RES0__INSTANCE0.MY_BAD_FIFO.BUFFER.value.table[2908]), INT_ENUM},*)
(*DBG:    {&(RES0__INSTANCE0.MY_BAD_FIFO.BUFFER.value.table[2909]), INT_ENUM},*)
(*DBG:    {&(RES0__INSTANCE0.MY_BAD_FIFO.BUFFER.value.table[2910]), INT_ENUM},*)
(*DBG:    {&(RES0__INSTANCE0.MY_BAD_FIFO.BUFFER.value.table[2911]), INT_ENUM},*)
(*DBG:    {&(RES0__INSTANCE0.MY_BAD_FIFO.BUFFER.value.table[2912]), INT_ENUM},*)
(*DBG:    {&(RES0__INSTANCE0.MY_BAD_FIFO.BUFFER.value.table[2913]), INT_ENUM},*)
(*DBG:    {&(RES0__INSTANCE0.MY_BAD_FIFO.BUFFER.value.table[2914]), INT_ENUM},*)
(*DBG:    {&(RES0__INSTANCE0.MY_BAD_FIFO.BUFFER.value.table[2915]), INT_ENUM},*)
(*DBG:    {&(RES0__INSTANCE0.MY_BAD_FIFO.BUFFER.value.table[2916]), INT_ENUM},*)
(*DBG:    {&(RES0__INSTANCE0.MY_BAD_FIFO.BUFFER.value.table[2917]), INT_ENUM},*)
(*DBG:    {&(RES0__INSTANCE0.MY_BAD_FIFO.BUFFER.value.table[2918]), INT_ENUM},*)
(*DBG:    {&(RES0__INSTANCE0.MY_BAD_FIFO.BUFFER.value.table[2919]), INT_ENUM},*)
(*DBG:    {&(RES0__INSTANCE0.MY_BAD_FIFO.BUFFER.value.table[2920]), INT_ENUM},*)
(*DBG:    {&(RES0__INSTANCE0.MY_BAD_FIFO.BUFFER.value.table[2921]), INT_ENUM},*)
(*DBG:    {&(RES0__INSTANCE0.MY_BAD_FIFO.BUFFER.value.table[2922]), INT_ENUM},*)
(*DBG:    {&(RES0__INSTANCE0.MY_BAD_FIFO.BUFFER.value.table[2923]), INT_ENUM},*)
(*DBG:    {&(RES0__INSTANCE0.MY_BAD_FIFO.BUFFER.value.table[2924]), INT_ENUM},*)
(*DBG:    {&(RES0__INSTANCE0.MY_BAD_FIFO.BUFFER.value.table[2925]), INT_ENUM},*)
(*DBG:    {&(RES0__INSTANCE0.MY_BAD_FIFO.BUFFER.value.table[2926]), INT_ENUM},*)
(*DBG:    {&(RES0__INSTANCE0.MY_BAD_FIFO.BUFFER.value.table[2927]), INT_ENUM},*)
(*DBG:    {&(RES0__INSTANCE0.MY_BAD_FIFO.BUFFER.value.table[2928]), INT_ENUM},*)
(*DBG:    {&(RES0__INSTANCE0.MY_BAD_FIFO.BUFFER.value.table[2929]), INT_ENUM},*)
(*DBG:    {&(RES0__INSTANCE0.MY_BAD_FIFO.BUFFER.value.table[2930]), INT_ENUM},*)
(*DBG:    {&(RES0__INSTANCE0.MY_BAD_FIFO.BUFFER.value.table[2931]), INT_ENUM},*)
(*DBG:    {&(RES0__INSTANCE0.MY_BAD_FIFO.BUFFER.value.table[2932]), INT_ENUM},*)
(*DBG:    {&(RES0__INSTANCE0.MY_BAD_FIFO.BUFFER.value.table[2933]), INT_ENUM},*)
(*DBG:    {&(RES0__INSTANCE0.MY_BAD_FIFO.BUFFER.value.table[2934]), INT_ENUM},*)
(*DBG:    {&(RES0__INSTANCE0.MY_BAD_FIFO.BUFFER.value.table[2935]), INT_ENUM},*)
(*DBG:    {&(RES0__INSTANCE0.MY_BAD_FIFO.BUFFER.value.table[2936]), INT_ENUM},*)
(*DBG:    {&(RES0__INSTANCE0.MY_BAD_FIFO.BUFFER.value.table[2937]), INT_ENUM},*)
(*DBG:    {&(RES0__INSTANCE0.MY_BAD_FIFO.BUFFER.value.table[2938]), INT_ENUM},*)
(*DBG:    {&(RES0__INSTANCE0.MY_BAD_FIFO.BUFFER.value.table[2939]), INT_ENUM},*)
(*DBG:    {&(RES0__INSTANCE0.MY_BAD_FIFO.BUFFER.value.table[2940]), INT_ENUM},*)
(*DBG:    {&(RES0__INSTANCE0.MY_BAD_FIFO.BUFFER.value.table[2941]), INT_ENUM},*)
(*DBG:    {&(RES0__INSTANCE0.MY_BAD_FIFO.BUFFER.value.table[2942]), INT_ENUM},*)
(*DBG:    {&(RES0__INSTANCE0.MY_BAD_FIFO.BUFFER.value.table[2943]), INT_ENUM},*)
(*DBG:    {&(RES0__INSTANCE0.MY_BAD_FIFO.BUFFER.value.table[2944]), INT_ENUM},*)
(*DBG:    {&(RES0__INSTANCE0.MY_BAD_FIFO.BUFFER.value.table[2945]), INT_ENUM},*)
(*DBG:    {&(RES0__INSTANCE0.MY_BAD_FIFO.BUFFER.value.table[2946]), INT_ENUM},*)
(*DBG:    {&(RES0__INSTANCE0.MY_BAD_FIFO.BUFFER.value.table[2947]), INT_ENUM},*)
(*DBG:    {&(RES0__INSTANCE0.MY_BAD_FIFO.BUFFER.value.table[2948]), INT_ENUM},*)
(*DBG:    {&(RES0__INSTANCE0.MY_BAD_FIFO.BUFFER.value.table[2949]), INT_ENUM},*)
(*DBG:    {&(RES0__INSTANCE0.MY_BAD_FIFO.BUFFER.value.table[2950]), INT_ENUM},*)
(*DBG:    {&(RES0__INSTANCE0.MY_BAD_FIFO.BUFFER.value.table[2951]), INT_ENUM},*)
(*DBG:    {&(RES0__INSTANCE0.MY_BAD_FIFO.BUFFER.value.table[2952]), INT_ENUM},*)
(*DBG:    {&(RES0__INSTANCE0.MY_BAD_FIFO.BUFFER.value.table[2953]), INT_ENUM},*)
(*DBG:    {&(RES0__INSTANCE0.MY_BAD_FIFO.BUFFER.value.table[2954]), INT_ENUM},*)
(*DBG:    {&(RES0__INSTANCE0.MY_BAD_FIFO.BUFFER.value.table[2955]), INT_ENUM},*)
(*DBG:    {&(RES0__INSTANCE0.MY_BAD_FIFO.BUFFER.value.table[2956]), INT_ENUM},*)
(*DBG:    {&(RES0__INSTANCE0.MY_BAD_FIFO.BUFFER.value.table[2957]), INT_ENUM},*)
(*DBG:    {&(RES0__INSTANCE0.MY_BAD_FIFO.BUFFER.value.table[2958]), INT_ENUM},*)
(*DBG:    {&(RES0__INSTANCE0.MY_BAD_FIFO.BUFFER.value.table[2959]), INT_ENUM},*)
(*DBG:    {&(RES0__INSTANCE0.MY_BAD_FIFO.BUFFER.value.table[2960]), INT_ENUM},*)
(*DBG:    {&(RES0__INSTANCE0.MY_BAD_FIFO.BUFFER.value.table[2961]), INT_ENUM},*)
(*DBG:    {&(RES0__INSTANCE0.MY_BAD_FIFO.BUFFER.value.table[2962]), INT_ENUM},*)
(*DBG:    {&(RES0__INSTANCE0.MY_BAD_FIFO.BUFFER.value.table[2963]), INT_ENUM},*)
(*DBG:    {&(RES0__INSTANCE0.MY_BAD_FIFO.BUFFER.value.table[2964]), INT_ENUM},*)
(*DBG:    {&(RES0__INSTANCE0.MY_BAD_FIFO.BUFFER.value.table[2965]), INT_ENUM},*)
(*DBG:    {&(RES0__INSTANCE0.MY_BAD_FIFO.BUFFER.value.table[2966]), INT_ENUM},*)
(*DBG:    {&(RES0__INSTANCE0.MY_BAD_FIFO.BUFFER.value.table[2967]), INT_ENUM},*)
(*DBG:    {&(RES0__INSTANCE0.MY_BAD_FIFO.BUFFER.value.table[2968]), INT_ENUM},*)
(*DBG:    {&(RES0__INSTANCE0.MY_BAD_FIFO.BUFFER.value.table[2969]), INT_ENUM},*)
(*DBG:    {&(RES0__INSTANCE0.MY_BAD_FIFO.BUFFER.value.table[2970]), INT_ENUM},*)
(*DBG:    {&(RES0__INSTANCE0.MY_BAD_FIFO.BUFFER.value.table[2971]), INT_ENUM},*)
(*DBG:    {&(RES0__INSTANCE0.MY_BAD_FIFO.BUFFER.value.table[2972]), INT_ENUM},*)
(*DBG:    {&(RES0__INSTANCE0.MY_BAD_FIFO.BUFFER.value.table[2973]), INT_ENUM},*)
(*DBG:    {&(RES0__INSTANCE0.MY_BAD_FIFO.BUFFER.value.table[2974]), INT_ENUM},*)
(*DBG:    {&(RES0__INSTANCE0.MY_BAD_FIFO.BUFFER.value.table[2975]), INT_ENUM},*)
(*DBG:    {&(RES0__INSTANCE0.MY_BAD_FIFO.BUFFER.value.table[2976]), INT_ENUM},*)
(*DBG:    {&(RES0__INSTANCE0.MY_BAD_FIFO.BUFFER.value.table[2977]), INT_ENUM},*)
(*DBG:    {&(RES0__INSTANCE0.MY_BAD_FIFO.BUFFER.value.table[2978]), INT_ENUM},*)
(*DBG:    {&(RES0__INSTANCE0.MY_BAD_FIFO.BUFFER.value.table[2979]), INT_ENUM},*)
(*DBG:    {&(RES0__INSTANCE0.MY_BAD_FIFO.BUFFER.value.table[2980]), INT_ENUM},*)
(*DBG:    {&(RES0__INSTANCE0.MY_BAD_FIFO.BUFFER.value.table[2981]), INT_ENUM},*)
(*DBG:    {&(RES0__INSTANCE0.MY_BAD_FIFO.BUFFER.value.table[2982]), INT_ENUM},*)
(*DBG:    {&(RES0__INSTANCE0.MY_BAD_FIFO.BUFFER.value.table[2983]), INT_ENUM},*)
(*DBG:    {&(RES0__INSTANCE0.MY_BAD_FIFO.BUFFER.value.table[2984]), INT_ENUM},*)
(*DBG:    {&(RES0__INSTANCE0.MY_BAD_FIFO.BUFFER.value.table[2985]), INT_ENUM},*)
(*DBG:    {&(RES0__INSTANCE0.MY_BAD_FIFO.BUFFER.value.table[2986]), INT_ENUM},*)
(*DBG:    {&(RES0__INSTANCE0.MY_BAD_FIFO.BUFFER.value.table[2987]), INT_ENUM},*)
(*DBG:    {&(RES0__INSTANCE0.MY_BAD_FIFO.BUFFER.value.table[2988]), INT_ENUM},*)
(*DBG:    {&(RES0__INSTANCE0.MY_BAD_FIFO.BUFFER.value.table[2989]), INT_ENUM},*)
(*DBG:    {&(RES0__INSTANCE0.MY_BAD_FIFO.BUFFER.value.table[2990]), INT_ENUM},*)
(*DBG:    {&(RES0__INSTANCE0.MY_BAD_FIFO.BUFFER.value.table[2991]), INT_ENUM},*)
(*DBG:    {&(RES0__INSTANCE0.MY_BAD_FIFO.BUFFER.value.table[2992]), INT_ENUM},*)
(*DBG:    {&(RES0__INSTANCE0.MY_BAD_FIFO.BUFFER.value.table[2993]), INT_ENUM},*)
(*DBG:    {&(RES0__INSTANCE0.MY_BAD_FIFO.BUFFER.value.table[2994]), INT_ENUM},*)
(*DBG:    {&(RES0__INSTANCE0.MY_BAD_FIFO.BUFFER.value.table[2995]), INT_ENUM},*)
(*DBG:    {&(RES0__INSTANCE0.MY_BAD_FIFO.BUFFER.value.table[2996]), INT_ENUM},*)
(*DBG:    {&(RES0__INSTANCE0.MY_BAD_FIFO.BUFFER.value.table[2997]), INT_ENUM},*)
(*DBG:    {&(RES0__INSTANCE0.MY_BAD_FIFO.BUFFER.value.table[2998]), INT_ENUM},*)
(*DBG:    {&(RES0__INSTANCE0.MY_BAD_FIFO.BUFFER.value.table[2999]), INT_ENUM},*)
(*DBG:    {&(RES0__INSTANCE0.MY_BAD_FIFO.BUFFER.value.table[3000]), INT_ENUM},*)
(*DBG:    {&(RES0__INSTANCE0.MY_BAD_FIFO.BUFFER.value.table[3001]), INT_ENUM},*)
(*DBG:    {&(RES0__INSTANCE0.MY_BAD_FIFO.BUFFER.value.table[3002]), INT_ENUM},*)
(*DBG:    {&(RES0__INSTANCE0.MY_BAD_FIFO.BUFFER.value.table[3003]), INT_ENUM},*)
(*DBG:    {&(RES0__INSTANCE0.MY_BAD_FIFO.BUFFER.value.table[3004]), INT_ENUM},*)
(*DBG:    {&(RES0__INSTANCE0.MY_BAD_FIFO.BUFFER.value.table[3005]), INT_ENUM},*)
(*DBG:    {&(RES0__INSTANCE0.MY_BAD_FIFO.BUFFER.value.table[3006]), INT_ENUM},*)
(*DBG:    {&(RES0__INSTANCE0.MY_BAD_FIFO.BUFFER.value.table[3007]), INT_ENUM},*)
(*DBG:    {&(RES0__INSTANCE0.MY_BAD_FIFO.BUFFER.value.table[3008]), INT_ENUM},*)
(*DBG:    {&(RES0__INSTANCE0.MY_BAD_FIFO.BUFFER.value.table[3009]), INT_ENUM},*)
(*DBG:    {&(RES0__INSTANCE0.MY_BAD_FIFO.BUFFER.value.table[3010]), INT_ENUM},*)
(*DBG:    {&(RES0__INSTANCE0.MY_BAD_FIFO.BUFFER.value.table[3011]), INT_ENUM},*)
(*DBG:    {&(RES0__INSTANCE0.MY_BAD_FIFO.BUFFER.value.table[3012]), INT_ENUM},*)
(*DBG:    {&(RES0__INSTANCE0.MY_BAD_FIFO.BUFFER.value.table[3013]), INT_ENUM},*)
(*DBG:    {&(RES0__INSTANCE0.MY_BAD_FIFO.BUFFER.value.table[3014]), INT_ENUM},*)
(*DBG:    {&(RES0__INSTANCE0.MY_BAD_FIFO.BUFFER.value.table[3015]), INT_ENUM},*)
(*DBG:    {&(RES0__INSTANCE0.MY_BAD_FIFO.BUFFER.value.table[3016]), INT_ENUM},*)
(*DBG:    {&(RES0__INSTANCE0.MY_BAD_FIFO.BUFFER.value.table[3017]), INT_ENUM},*)
(*DBG:    {&(RES0__INSTANCE0.MY_BAD_FIFO.BUFFER.value.table[3018]), INT_ENUM},*)
(*DBG:    {&(RES0__INSTANCE0.MY_BAD_FIFO.BUFFER.value.table[3019]), INT_ENUM},*)
(*DBG:    {&(RES0__INSTANCE0.MY_BAD_FIFO.BUFFER.value.table[3020]), INT_ENUM},*)
(*DBG:    {&(RES0__INSTANCE0.MY_BAD_FIFO.BUFFER.value.table[3021]), INT_ENUM},*)
(*DBG:    {&(RES0__INSTANCE0.MY_BAD_FIFO.BUFFER.value.table[3022]), INT_ENUM},*)
(*DBG:    {&(RES0__INSTANCE0.MY_BAD_FIFO.BUFFER.value.table[3023]), INT_ENUM},*)
(*DBG:    {&(RES0__INSTANCE0.MY_BAD_FIFO.BUFFER.value.table[3024]), INT_ENUM},*)
(*DBG:    {&(RES0__INSTANCE0.MY_BAD_FIFO.BUFFER.value.table[3025]), INT_ENUM},*)
(*DBG:    {&(RES0__INSTANCE0.MY_BAD_FIFO.BUFFER.value.table[3026]), INT_ENUM},*)
(*DBG:    {&(RES0__INSTANCE0.MY_BAD_FIFO.BUFFER.value.table[3027]), INT_ENUM},*)
(*DBG:    {&(RES0__INSTANCE0.MY_BAD_FIFO.BUFFER.value.table[3028]), INT_ENUM},*)
(*DBG:    {&(RES0__INSTANCE0.MY_BAD_FIFO.BUFFER.value.table[3029]), INT_ENUM},*)
(*DBG:    {&(RES0__INSTANCE0.MY_BAD_FIFO.BUFFER.value.table[3030]), INT_ENUM},*)
(*DBG:    {&(RES0__INSTANCE0.MY_BAD_FIFO.BUFFER.value.table[3031]), INT_ENUM},*)
(*DBG:    {&(RES0__INSTANCE0.MY_BAD_FIFO.BUFFER.value.table[3032]), INT_ENUM},*)
(*DBG:    {&(RES0__INSTANCE0.MY_BAD_FIFO.BUFFER.value.table[3033]), INT_ENUM},*)
(*DBG:    {&(RES0__INSTANCE0.MY_BAD_FIFO.BUFFER.value.table[3034]), INT_ENUM},*)
(*DBG:    {&(RES0__INSTANCE0.MY_BAD_FIFO.BUFFER.value.table[3035]), INT_ENUM},*)
(*DBG:    {&(RES0__INSTANCE0.MY_BAD_FIFO.BUFFER.value.table[3036]), INT_ENUM},*)
(*DBG:    {&(RES0__INSTANCE0.MY_BAD_FIFO.BUFFER.value.table[3037]), INT_ENUM},*)
(*DBG:    {&(RES0__INSTANCE0.MY_BAD_FIFO.BUFFER.value.table[3038]), INT_ENUM},*)
(*DBG:    {&(RES0__INSTANCE0.MY_BAD_FIFO.BUFFER.value.table[3039]), INT_ENUM},*)
(*DBG:    {&(RES0__INSTANCE0.MY_BAD_FIFO.BUFFER.value.table[3040]), INT_ENUM},*)
(*DBG:    {&(RES0__INSTANCE0.MY_BAD_FIFO.BUFFER.value.table[3041]), INT_ENUM},*)
(*DBG:    {&(RES0__INSTANCE0.MY_BAD_FIFO.BUFFER.value.table[3042]), INT_ENUM},*)
(*DBG:    {&(RES0__INSTANCE0.MY_BAD_FIFO.BUFFER.value.table[3043]), INT_ENUM},*)
(*DBG:    {&(RES0__INSTANCE0.MY_BAD_FIFO.BUFFER.value.table[3044]), INT_ENUM},*)
(*DBG:    {&(RES0__INSTANCE0.MY_BAD_FIFO.BUFFER.value.table[3045]), INT_ENUM},*)
(*DBG:    {&(RES0__INSTANCE0.MY_BAD_FIFO.BUFFER.value.table[3046]), INT_ENUM},*)
(*DBG:    {&(RES0__INSTANCE0.MY_BAD_FIFO.BUFFER.value.table[3047]), INT_ENUM},*)
(*DBG:    {&(RES0__INSTANCE0.MY_BAD_FIFO.BUFFER.value.table[3048]), INT_ENUM},*)
(*DBG:    {&(RES0__INSTANCE0.MY_BAD_FIFO.BUFFER.value.table[3049]), INT_ENUM},*)
(*DBG:    {&(RES0__INSTANCE0.MY_BAD_FIFO.BUFFER.value.table[3050]), INT_ENUM},*)
(*DBG:    {&(RES0__INSTANCE0.MY_BAD_FIFO.BUFFER.value.table[3051]), INT_ENUM},*)
(*DBG:    {&(RES0__INSTANCE0.MY_BAD_FIFO.BUFFER.value.table[3052]), INT_ENUM},*)
(*DBG:    {&(RES0__INSTANCE0.MY_BAD_FIFO.BUFFER.value.table[3053]), INT_ENUM},*)
(*DBG:    {&(RES0__INSTANCE0.MY_BAD_FIFO.BUFFER.value.table[3054]), INT_ENUM},*)
(*DBG:    {&(RES0__INSTANCE0.MY_BAD_FIFO.BUFFER.value.table[3055]), INT_ENUM},*)
(*DBG:    {&(RES0__INSTANCE0.MY_BAD_FIFO.BUFFER.value.table[3056]), INT_ENUM},*)
(*DBG:    {&(RES0__INSTANCE0.MY_BAD_FIFO.BUFFER.value.table[3057]), INT_ENUM},*)
(*DBG:    {&(RES0__INSTANCE0.MY_BAD_FIFO.BUFFER.value.table[3058]), INT_ENUM},*)
(*DBG:    {&(RES0__INSTANCE0.MY_BAD_FIFO.BUFFER.value.table[3059]), INT_ENUM},*)
(*DBG:    {&(RES0__INSTANCE0.MY_BAD_FIFO.BUFFER.value.table[3060]), INT_ENUM},*)
(*DBG:    {&(RES0__INSTANCE0.MY_BAD_FIFO.BUFFER.value.table[3061]), INT_ENUM},*)
(*DBG:    {&(RES0__INSTANCE0.MY_BAD_FIFO.BUFFER.value.table[3062]), INT_ENUM},*)
(*DBG:    {&(RES0__INSTANCE0.MY_BAD_FIFO.BUFFER.value.table[3063]), INT_ENUM},*)
(*DBG:    {&(RES0__INSTANCE0.MY_BAD_FIFO.BUFFER.value.table[3064]), INT_ENUM},*)
(*DBG:    {&(RES0__INSTANCE0.MY_BAD_FIFO.BUFFER.value.table[3065]), INT_ENUM},*)
(*DBG:    {&(RES0__INSTANCE0.MY_BAD_FIFO.BUFFER.value.table[3066]), INT_ENUM},*)
(*DBG:    {&(RES0__INSTANCE0.MY_BAD_FIFO.BUFFER.value.table[3067]), INT_ENUM},*)
(*DBG:    {&(RES0__INSTANCE0.MY_BAD_FIFO.BUFFER.value.table[3068]), INT_ENUM},*)
(*DBG:    {&(RES0__INSTANCE0.MY_BAD_FIFO.BUFFER.value.table[3069]), INT_ENUM},*)
(*DBG:    {&(RES0__INSTANCE0.MY_BAD_FIFO.BUFFER.value.table[3070]), INT_ENUM},*)
(*DBG:    {&(RES0__INSTANCE0.MY_BAD_FIFO.BUFFER.value.table[3071]), INT_ENUM},*)
(*DBG:    {&(RES0__INSTANCE0.MY_BAD_FIFO.BUFFER.value.table[3072]), INT_ENUM},*)
(*DBG:    {&(RES0__INSTANCE0.MY_BAD_FIFO.BUFFER.value.table[3073]), INT_ENUM},*)
(*DBG:    {&(RES0__INSTANCE0.MY_BAD_FIFO.BUFFER.value.table[3074]), INT_ENUM},*)
(*DBG:    {&(RES0__INSTANCE0.MY_BAD_FIFO.BUFFER.value.table[3075]), INT_ENUM},*)
(*DBG:    {&(RES0__INSTANCE0.MY_BAD_FIFO.BUFFER.value.table[3076]), INT_ENUM},*)
(*DBG:    {&(RES0__INSTANCE0.MY_BAD_FIFO.BUFFER.value.table[3077]), INT_ENUM},*)
(*DBG:    {&(RES0__INSTANCE0.MY_BAD_FIFO.BUFFER.value.table[3078]), INT_ENUM},*)
(*DBG:    {&(RES0__INSTANCE0.MY_BAD_FIFO.BUFFER.value.table[3079]), INT_ENUM},*)
(*DBG:    {&(RES0__INSTANCE0.MY_BAD_FIFO.BUFFER.value.table[3080]), INT_ENUM},*)
(*DBG:    {&(RES0__INSTANCE0.MY_BAD_FIFO.BUFFER.value.table[3081]), INT_ENUM},*)
(*DBG:    {&(RES0__INSTANCE0.MY_BAD_FIFO.BUFFER.value.table[3082]), INT_ENUM},*)
(*DBG:    {&(RES0__INSTANCE0.MY_BAD_FIFO.BUFFER.value.table[3083]), INT_ENUM},*)
(*DBG:    {&(RES0__INSTANCE0.MY_BAD_FIFO.BUFFER.value.table[3084]), INT_ENUM},*)
(*DBG:    {&(RES0__INSTANCE0.MY_BAD_FIFO.BUFFER.value.table[3085]), INT_ENUM},*)
(*DBG:    {&(RES0__INSTANCE0.MY_BAD_FIFO.BUFFER.value.table[3086]), INT_ENUM},*)
(*DBG:    {&(RES0__INSTANCE0.MY_BAD_FIFO.BUFFER.value.table[3087]), INT_ENUM},*)
(*DBG:    {&(RES0__INSTANCE0.MY_BAD_FIFO.BUFFER.value.table[3088]), INT_ENUM},*)
(*DBG:    {&(RES0__INSTANCE0.MY_BAD_FIFO.BUFFER.value.table[3089]), INT_ENUM},*)
(*DBG:    {&(RES0__INSTANCE0.MY_BAD_FIFO.BUFFER.value.table[3090]), INT_ENUM},*)
(*DBG:    {&(RES0__INSTANCE0.MY_BAD_FIFO.BUFFER.value.table[3091]), INT_ENUM},*)
(*DBG:    {&(RES0__INSTANCE0.MY_BAD_FIFO.BUFFER.value.table[3092]), INT_ENUM},*)
(*DBG:    {&(RES0__INSTANCE0.MY_BAD_FIFO.BUFFER.value.table[3093]), INT_ENUM},*)
(*DBG:    {&(RES0__INSTANCE0.MY_BAD_FIFO.BUFFER.value.table[3094]), INT_ENUM},*)
(*DBG:    {&(RES0__INSTANCE0.MY_BAD_FIFO.BUFFER.value.table[3095]), INT_ENUM},*)
(*DBG:    {&(RES0__INSTANCE0.MY_BAD_FIFO.BUFFER.value.table[3096]), INT_ENUM},*)
(*DBG:    {&(RES0__INSTANCE0.MY_BAD_FIFO.BUFFER.value.table[3097]), INT_ENUM},*)
(*DBG:    {&(RES0__INSTANCE0.MY_BAD_FIFO.BUFFER.value.table[3098]), INT_ENUM},*)
(*DBG:    {&(RES0__INSTANCE0.MY_BAD_FIFO.BUFFER.value.table[3099]), INT_ENUM},*)
(*DBG:    {&(RES0__INSTANCE0.MY_BAD_FIFO.BUFFER.value.table[3100]), INT_ENUM},*)
(*DBG:    {&(RES0__INSTANCE0.MY_BAD_FIFO.BUFFER.value.table[3101]), INT_ENUM},*)
(*DBG:    {&(RES0__INSTANCE0.MY_BAD_FIFO.BUFFER.value.table[3102]), INT_ENUM},*)
(*DBG:    {&(RES0__INSTANCE0.MY_BAD_FIFO.BUFFER.value.table[3103]), INT_ENUM},*)
(*DBG:    {&(RES0__INSTANCE0.MY_BAD_FIFO.BUFFER.value.table[3104]), INT_ENUM},*)
(*DBG:    {&(RES0__INSTANCE0.MY_BAD_FIFO.BUFFER.value.table[3105]), INT_ENUM},*)
(*DBG:    {&(RES0__INSTANCE0.MY_BAD_FIFO.BUFFER.value.table[3106]), INT_ENUM},*)
(*DBG:    {&(RES0__INSTANCE0.MY_BAD_FIFO.BUFFER.value.table[3107]), INT_ENUM},*)
(*DBG:    {&(RES0__INSTANCE0.MY_BAD_FIFO.BUFFER.value.table[3108]), INT_ENUM},*)
(*DBG:    {&(RES0__INSTANCE0.MY_BAD_FIFO.BUFFER.value.table[3109]), INT_ENUM},*)
(*DBG:    {&(RES0__INSTANCE0.MY_BAD_FIFO.BUFFER.value.table[3110]), INT_ENUM},*)
(*DBG:    {&(RES0__INSTANCE0.MY_BAD_FIFO.BUFFER.value.table[3111]), INT_ENUM},*)
(*DBG:    {&(RES0__INSTANCE0.MY_BAD_FIFO.BUFFER.value.table[3112]), INT_ENUM},*)
(*DBG:    {&(RES0__INSTANCE0.MY_BAD_FIFO.BUFFER.value.table[3113]), INT_ENUM},*)
(*DBG:    {&(RES0__INSTANCE0.MY_BAD_FIFO.BUFFER.value.table[3114]), INT_ENUM},*)
(*DBG:    {&(RES0__INSTANCE0.MY_BAD_FIFO.BUFFER.value.table[3115]), INT_ENUM},*)
(*DBG:    {&(RES0__INSTANCE0.MY_BAD_FIFO.BUFFER.value.table[3116]), INT_ENUM},*)
(*DBG:    {&(RES0__INSTANCE0.MY_BAD_FIFO.BUFFER.value.table[3117]), INT_ENUM},*)
(*DBG:    {&(RES0__INSTANCE0.MY_BAD_FIFO.BUFFER.value.table[3118]), INT_ENUM},*)
(*DBG:    {&(RES0__INSTANCE0.MY_BAD_FIFO.BUFFER.value.table[3119]), INT_ENUM},*)
(*DBG:    {&(RES0__INSTANCE0.MY_BAD_FIFO.BUFFER.value.table[3120]), INT_ENUM},*)
(*DBG:    {&(RES0__INSTANCE0.MY_BAD_FIFO.BUFFER.value.table[3121]), INT_ENUM},*)
(*DBG:    {&(RES0__INSTANCE0.MY_BAD_FIFO.BUFFER.value.table[3122]), INT_ENUM},*)
(*DBG:    {&(RES0__INSTANCE0.MY_BAD_FIFO.BUFFER.value.table[3123]), INT_ENUM},*)
(*DBG:    {&(RES0__INSTANCE0.MY_BAD_FIFO.BUFFER.value.table[3124]), INT_ENUM},*)
(*DBG:    {&(RES0__INSTANCE0.MY_BAD_FIFO.BUFFER.value.table[3125]), INT_ENUM},*)
(*DBG:    {&(RES0__INSTANCE0.MY_BAD_FIFO.BUFFER.value.table[3126]), INT_ENUM},*)
(*DBG:    {&(RES0__INSTANCE0.MY_BAD_FIFO.BUFFER.value.table[3127]), INT_ENUM},*)
(*DBG:    {&(RES0__INSTANCE0.MY_BAD_FIFO.BUFFER.value.table[3128]), INT_ENUM},*)
(*DBG:    {&(RES0__INSTANCE0.MY_BAD_FIFO.BUFFER.value.table[3129]), INT_ENUM},*)
(*DBG:    {&(RES0__INSTANCE0.MY_BAD_FIFO.BUFFER.value.table[3130]), INT_ENUM},*)
(*DBG:    {&(RES0__INSTANCE0.MY_BAD_FIFO.BUFFER.value.table[3131]), INT_ENUM},*)
(*DBG:    {&(RES0__INSTANCE0.MY_BAD_FIFO.BUFFER.value.table[3132]), INT_ENUM},*)
(*DBG:    {&(RES0__INSTANCE0.MY_BAD_FIFO.BUFFER.value.table[3133]), INT_ENUM},*)
(*DBG:    {&(RES0__INSTANCE0.MY_BAD_FIFO.BUFFER.value.table[3134]), INT_ENUM},*)
(*DBG:    {&(RES0__INSTANCE0.MY_BAD_FIFO.BUFFER.value.table[3135]), INT_ENUM},*)
(*DBG:    {&(RES0__INSTANCE0.MY_BAD_FIFO.BUFFER.value.table[3136]), INT_ENUM},*)
(*DBG:    {&(RES0__INSTANCE0.MY_BAD_FIFO.BUFFER.value.table[3137]), INT_ENUM},*)
(*DBG:    {&(RES0__INSTANCE0.MY_BAD_FIFO.BUFFER.value.table[3138]), INT_ENUM},*)
(*DBG:    {&(RES0__INSTANCE0.MY_BAD_FIFO.BUFFER.value.table[3139]), INT_ENUM},*)
(*DBG:    {&(RES0__INSTANCE0.MY_BAD_FIFO.BUFFER.value.table[3140]), INT_ENUM},*)
(*DBG:    {&(RES0__INSTANCE0.MY_BAD_FIFO.BUFFER.value.table[3141]), INT_ENUM},*)
(*DBG:    {&(RES0__INSTANCE0.MY_BAD_FIFO.BUFFER.value.table[3142]), INT_ENUM},*)
(*DBG:    {&(RES0__INSTANCE0.MY_BAD_FIFO.BUFFER.value.table[3143]), INT_ENUM},*)
(*DBG:    {&(RES0__INSTANCE0.MY_BAD_FIFO.BUFFER.value.table[3144]), INT_ENUM},*)
(*DBG:    {&(RES0__INSTANCE0.MY_BAD_FIFO.BUFFER.value.table[3145]), INT_ENUM},*)
(*DBG:    {&(RES0__INSTANCE0.MY_BAD_FIFO.BUFFER.value.table[3146]), INT_ENUM},*)
(*DBG:    {&(RES0__INSTANCE0.MY_BAD_FIFO.BUFFER.value.table[3147]), INT_ENUM},*)
(*DBG:    {&(RES0__INSTANCE0.MY_BAD_FIFO.BUFFER.value.table[3148]), INT_ENUM},*)
(*DBG:    {&(RES0__INSTANCE0.MY_BAD_FIFO.BUFFER.value.table[3149]), INT_ENUM},*)
(*DBG:    {&(RES0__INSTANCE0.MY_BAD_FIFO.BUFFER.value.table[3150]), INT_ENUM},*)
(*DBG:    {&(RES0__INSTANCE0.MY_BAD_FIFO.BUFFER.value.table[3151]), INT_ENUM},*)
(*DBG:    {&(RES0__INSTANCE0.MY_BAD_FIFO.BUFFER.value.table[3152]), INT_ENUM},*)
(*DBG:    {&(RES0__INSTANCE0.MY_BAD_FIFO.BUFFER.value.table[3153]), INT_ENUM},*)
(*DBG:    {&(RES0__INSTANCE0.MY_BAD_FIFO.BUFFER.value.table[3154]), INT_ENUM},*)
(*DBG:    {&(RES0__INSTANCE0.MY_BAD_FIFO.BUFFER.value.table[3155]), INT_ENUM},*)
(*DBG:    {&(RES0__INSTANCE0.MY_BAD_FIFO.BUFFER.value.table[3156]), INT_ENUM},*)
(*DBG:    {&(RES0__INSTANCE0.MY_BAD_FIFO.BUFFER.value.table[3157]), INT_ENUM},*)
(*DBG:    {&(RES0__INSTANCE0.MY_BAD_FIFO.BUFFER.value.table[3158]), INT_ENUM},*)
(*DBG:    {&(RES0__INSTANCE0.MY_BAD_FIFO.BUFFER.value.table[3159]), INT_ENUM},*)
(*DBG:    {&(RES0__INSTANCE0.MY_BAD_FIFO.BUFFER.value.table[3160]), INT_ENUM},*)
(*DBG:    {&(RES0__INSTANCE0.MY_BAD_FIFO.BUFFER.value.table[3161]), INT_ENUM},*)
(*DBG:    {&(RES0__INSTANCE0.MY_BAD_FIFO.BUFFER.value.table[3162]), INT_ENUM},*)
(*DBG:    {&(RES0__INSTANCE0.MY_BAD_FIFO.BUFFER.value.table[3163]), INT_ENUM},*)
(*DBG:    {&(RES0__INSTANCE0.MY_BAD_FIFO.BUFFER.value.table[3164]), INT_ENUM},*)
(*DBG:    {&(RES0__INSTANCE0.MY_BAD_FIFO.BUFFER.value.table[3165]), INT_ENUM},*)
(*DBG:    {&(RES0__INSTANCE0.MY_BAD_FIFO.BUFFER.value.table[3166]), INT_ENUM},*)
(*DBG:    {&(RES0__INSTANCE0.MY_BAD_FIFO.BUFFER.value.table[3167]), INT_ENUM},*)
(*DBG:    {&(RES0__INSTANCE0.MY_BAD_FIFO.BUFFER.value.table[3168]), INT_ENUM},*)
(*DBG:    {&(RES0__INSTANCE0.MY_BAD_FIFO.BUFFER.value.table[3169]), INT_ENUM},*)
(*DBG:    {&(RES0__INSTANCE0.MY_BAD_FIFO.BUFFER.value.table[3170]), INT_ENUM},*)
(*DBG:    {&(RES0__INSTANCE0.MY_BAD_FIFO.BUFFER.value.table[3171]), INT_ENUM},*)
(*DBG:    {&(RES0__INSTANCE0.MY_BAD_FIFO.BUFFER.value.table[3172]), INT_ENUM},*)
(*DBG:    {&(RES0__INSTANCE0.MY_BAD_FIFO.BUFFER.value.table[3173]), INT_ENUM},*)
(*DBG:    {&(RES0__INSTANCE0.MY_BAD_FIFO.BUFFER.value.table[3174]), INT_ENUM},*)
(*DBG:    {&(RES0__INSTANCE0.MY_BAD_FIFO.BUFFER.value.table[3175]), INT_ENUM},*)
(*DBG:    {&(RES0__INSTANCE0.MY_BAD_FIFO.BUFFER.value.table[3176]), INT_ENUM},*)
(*DBG:    {&(RES0__INSTANCE0.MY_BAD_FIFO.BUFFER.value.table[3177]), INT_ENUM},*)
(*DBG:    {&(RES0__INSTANCE0.MY_BAD_FIFO.BUFFER.value.table[3178]), INT_ENUM},*)
(*DBG:    {&(RES0__INSTANCE0.MY_BAD_FIFO.BUFFER.value.table[3179]), INT_ENUM},*)
(*DBG:    {&(RES0__INSTANCE0.MY_BAD_FIFO.BUFFER.value.table[3180]), INT_ENUM},*)
(*DBG:    {&(RES0__INSTANCE0.MY_BAD_FIFO.BUFFER.value.table[3181]), INT_ENUM},*)
(*DBG:    {&(RES0__INSTANCE0.MY_BAD_FIFO.BUFFER.value.table[3182]), INT_ENUM},*)
(*DBG:    {&(RES0__INSTANCE0.MY_BAD_FIFO.BUFFER.value.table[3183]), INT_ENUM},*)
(*DBG:    {&(RES0__INSTANCE0.MY_BAD_FIFO.BUFFER.value.table[3184]), INT_ENUM},*)
(*DBG:    {&(RES0__INSTANCE0.MY_BAD_FIFO.BUFFER.value.table[3185]), INT_ENUM},*)
(*DBG:    {&(RES0__INSTANCE0.MY_BAD_FIFO.BUFFER.value.table[3186]), INT_ENUM},*)
(*DBG:    {&(RES0__INSTANCE0.MY_BAD_FIFO.BUFFER.value.table[3187]), INT_ENUM},*)
(*DBG:    {&(RES0__INSTANCE0.MY_BAD_FIFO.BUFFER.value.table[3188]), INT_ENUM},*)
(*DBG:    {&(RES0__INSTANCE0.MY_BAD_FIFO.BUFFER.value.table[3189]), INT_ENUM},*)
(*DBG:    {&(RES0__INSTANCE0.MY_BAD_FIFO.BUFFER.value.table[3190]), INT_ENUM},*)
(*DBG:    {&(RES0__INSTANCE0.MY_BAD_FIFO.BUFFER.value.table[3191]), INT_ENUM},*)
(*DBG:    {&(RES0__INSTANCE0.MY_BAD_FIFO.BUFFER.value.table[3192]), INT_ENUM},*)
(*DBG:    {&(RES0__INSTANCE0.MY_BAD_FIFO.BUFFER.value.table[3193]), INT_ENUM},*)
(*DBG:    {&(RES0__INSTANCE0.MY_BAD_FIFO.BUFFER.value.table[3194]), INT_ENUM},*)
(*DBG:    {&(RES0__INSTANCE0.MY_BAD_FIFO.BUFFER.value.table[3195]), INT_ENUM},*)
(*DBG:    {&(RES0__INSTANCE0.MY_BAD_FIFO.BUFFER.value.table[3196]), INT_ENUM},*)
(*DBG:    {&(RES0__INSTANCE0.MY_BAD_FIFO.BUFFER.value.table[3197]), INT_ENUM},*)
(*DBG:    {&(RES0__INSTANCE0.MY_BAD_FIFO.BUFFER.value.table[3198]), INT_ENUM},*)
(*DBG:    {&(RES0__INSTANCE0.MY_BAD_FIFO.BUFFER.value.table[3199]), INT_ENUM},*)
(*DBG:    {&(RES0__INSTANCE0.MY_BAD_FIFO.BUFFER.value.table[3200]), INT_ENUM},*)
(*DBG:    {&(RES0__INSTANCE0.MY_BAD_FIFO.BUFFER.value.table[3201]), INT_ENUM},*)
(*DBG:    {&(RES0__INSTANCE0.MY_BAD_FIFO.BUFFER.value.table[3202]), INT_ENUM},*)
(*DBG:    {&(RES0__INSTANCE0.MY_BAD_FIFO.BUFFER.value.table[3203]), INT_ENUM},*)
(*DBG:    {&(RES0__INSTANCE0.MY_BAD_FIFO.BUFFER.value.table[3204]), INT_ENUM},*)
(*DBG:    {&(RES0__INSTANCE0.MY_BAD_FIFO.BUFFER.value.table[3205]), INT_ENUM},*)
(*DBG:    {&(RES0__INSTANCE0.MY_BAD_FIFO.BUFFER.value.table[3206]), INT_ENUM},*)
(*DBG:    {&(RES0__INSTANCE0.MY_BAD_FIFO.BUFFER.value.table[3207]), INT_ENUM},*)
(*DBG:    {&(RES0__INSTANCE0.MY_BAD_FIFO.BUFFER.value.table[3208]), INT_ENUM},*)
(*DBG:    {&(RES0__INSTANCE0.MY_BAD_FIFO.BUFFER.value.table[3209]), INT_ENUM},*)
(*DBG:    {&(RES0__INSTANCE0.MY_BAD_FIFO.BUFFER.value.table[3210]), INT_ENUM},*)
(*DBG:    {&(RES0__INSTANCE0.MY_BAD_FIFO.BUFFER.value.table[3211]), INT_ENUM},*)
(*DBG:    {&(RES0__INSTANCE0.MY_BAD_FIFO.BUFFER.value.table[3212]), INT_ENUM},*)
(*DBG:    {&(RES0__INSTANCE0.MY_BAD_FIFO.BUFFER.value.table[3213]), INT_ENUM},*)
(*DBG:    {&(RES0__INSTANCE0.MY_BAD_FIFO.BUFFER.value.table[3214]), INT_ENUM},*)
(*DBG:    {&(RES0__INSTANCE0.MY_BAD_FIFO.BUFFER.value.table[3215]), INT_ENUM},*)
(*DBG:    {&(RES0__INSTANCE0.MY_BAD_FIFO.BUFFER.value.table[3216]), INT_ENUM},*)
(*DBG:    {&(RES0__INSTANCE0.MY_BAD_FIFO.BUFFER.value.table[3217]), INT_ENUM},*)
(*DBG:    {&(RES0__INSTANCE0.MY_BAD_FIFO.BUFFER.value.table[3218]), INT_ENUM},*)
(*DBG:    {&(RES0__INSTANCE0.MY_BAD_FIFO.BUFFER.value.table[3219]), INT_ENUM},*)
(*DBG:    {&(RES0__INSTANCE0.MY_BAD_FIFO.BUFFER.value.table[3220]), INT_ENUM},*)
(*DBG:    {&(RES0__INSTANCE0.MY_BAD_FIFO.BUFFER.value.table[3221]), INT_ENUM},*)
(*DBG:    {&(RES0__INSTANCE0.MY_BAD_FIFO.BUFFER.value.table[3222]), INT_ENUM},*)
(*DBG:    {&(RES0__INSTANCE0.MY_BAD_FIFO.BUFFER.value.table[3223]), INT_ENUM},*)
(*DBG:    {&(RES0__INSTANCE0.MY_BAD_FIFO.BUFFER.value.table[3224]), INT_ENUM},*)
(*DBG:    {&(RES0__INSTANCE0.MY_BAD_FIFO.BUFFER.value.table[3225]), INT_ENUM},*)
(*DBG:    {&(RES0__INSTANCE0.MY_BAD_FIFO.BUFFER.value.table[3226]), INT_ENUM},*)
(*DBG:    {&(RES0__INSTANCE0.MY_BAD_FIFO.BUFFER.value.table[3227]), INT_ENUM},*)
(*DBG:    {&(RES0__INSTANCE0.MY_BAD_FIFO.BUFFER.value.table[3228]), INT_ENUM},*)
(*DBG:    {&(RES0__INSTANCE0.MY_BAD_FIFO.BUFFER.value.table[3229]), INT_ENUM},*)
(*DBG:    {&(RES0__INSTANCE0.MY_BAD_FIFO.BUFFER.value.table[3230]), INT_ENUM},*)
(*DBG:    {&(RES0__INSTANCE0.MY_BAD_FIFO.BUFFER.value.table[3231]), INT_ENUM},*)
(*DBG:    {&(RES0__INSTANCE0.MY_BAD_FIFO.BUFFER.value.table[3232]), INT_ENUM},*)
(*DBG:    {&(RES0__INSTANCE0.MY_BAD_FIFO.BUFFER.value.table[3233]), INT_ENUM},*)
(*DBG:    {&(RES0__INSTANCE0.MY_BAD_FIFO.BUFFER.value.table[3234]), INT_ENUM},*)
(*DBG:    {&(RES0__INSTANCE0.MY_BAD_FIFO.BUFFER.value.table[3235]), INT_ENUM},*)
(*DBG:    {&(RES0__INSTANCE0.MY_BAD_FIFO.BUFFER.value.table[3236]), INT_ENUM},*)
(*DBG:    {&(RES0__INSTANCE0.MY_BAD_FIFO.BUFFER.value.table[3237]), INT_ENUM},*)
(*DBG:    {&(RES0__INSTANCE0.MY_BAD_FIFO.BUFFER.value.table[3238]), INT_ENUM},*)
(*DBG:    {&(RES0__INSTANCE0.MY_BAD_FIFO.BUFFER.value.table[3239]), INT_ENUM},*)
(*DBG:    {&(RES0__INSTANCE0.MY_BAD_FIFO.BUFFER.value.table[3240]), INT_ENUM},*)
(*DBG:    {&(RES0__INSTANCE0.MY_BAD_FIFO.BUFFER.value.table[3241]), INT_ENUM},*)
(*DBG:    {&(RES0__INSTANCE0.MY_BAD_FIFO.BUFFER.value.table[3242]), INT_ENUM},*)
(*DBG:    {&(RES0__INSTANCE0.MY_BAD_FIFO.BUFFER.value.table[3243]), INT_ENUM},*)
(*DBG:    {&(RES0__INSTANCE0.MY_BAD_FIFO.BUFFER.value.table[3244]), INT_ENUM},*)
(*DBG:    {&(RES0__INSTANCE0.MY_BAD_FIFO.BUFFER.value.table[3245]), INT_ENUM},*)
(*DBG:    {&(RES0__INSTANCE0.MY_BAD_FIFO.BUFFER.value.table[3246]), INT_ENUM},*)
(*DBG:    {&(RES0__INSTANCE0.MY_BAD_FIFO.BUFFER.value.table[3247]), INT_ENUM},*)
(*DBG:    {&(RES0__INSTANCE0.MY_BAD_FIFO.BUFFER.value.table[3248]), INT_ENUM},*)
(*DBG:    {&(RES0__INSTANCE0.MY_BAD_FIFO.BUFFER.value.table[3249]), INT_ENUM},*)
(*DBG:    {&(RES0__INSTANCE0.MY_BAD_FIFO.BUFFER.value.table[3250]), INT_ENUM},*)
(*DBG:    {&(RES0__INSTANCE0.MY_BAD_FIFO.BUFFER.value.table[3251]), INT_ENUM},*)
(*DBG:    {&(RES0__INSTANCE0.MY_BAD_FIFO.BUFFER.value.table[3252]), INT_ENUM},*)
(*DBG:    {&(RES0__INSTANCE0.MY_BAD_FIFO.BUFFER.value.table[3253]), INT_ENUM},*)
(*DBG:    {&(RES0__INSTANCE0.MY_BAD_FIFO.BUFFER.value.table[3254]), INT_ENUM},*)
(*DBG:    {&(RES0__INSTANCE0.MY_BAD_FIFO.BUFFER.value.table[3255]), INT_ENUM},*)
(*DBG:    {&(RES0__INSTANCE0.MY_BAD_FIFO.BUFFER.value.table[3256]), INT_ENUM},*)
(*DBG:    {&(RES0__INSTANCE0.MY_BAD_FIFO.BUFFER.value.table[3257]), INT_ENUM},*)
(*DBG:    {&(RES0__INSTANCE0.MY_BAD_FIFO.BUFFER.value.table[3258]), INT_ENUM},*)
(*DBG:    {&(RES0__INSTANCE0.MY_BAD_FIFO.BUFFER.value.table[3259]), INT_ENUM},*)
(*DBG:    {&(RES0__INSTANCE0.MY_BAD_FIFO.BUFFER.value.table[3260]), INT_ENUM},*)
(*DBG:    {&(RES0__INSTANCE0.MY_BAD_FIFO.BUFFER.value.table[3261]), INT_ENUM},*)
(*DBG:    {&(RES0__INSTANCE0.MY_BAD_FIFO.BUFFER.value.table[3262]), INT_ENUM},*)
(*DBG:    {&(RES0__INSTANCE0.MY_BAD_FIFO.BUFFER.value.table[3263]), INT_ENUM},*)
(*DBG:    {&(RES0__INSTANCE0.MY_BAD_FIFO.BUFFER.value.table[3264]), INT_ENUM},*)
(*DBG:    {&(RES0__INSTANCE0.MY_BAD_FIFO.BUFFER.value.table[3265]), INT_ENUM},*)
(*DBG:    {&(RES0__INSTANCE0.MY_BAD_FIFO.BUFFER.value.table[3266]), INT_ENUM},*)
(*DBG:    {&(RES0__INSTANCE0.MY_BAD_FIFO.BUFFER.value.table[3267]), INT_ENUM},*)
(*DBG:    {&(RES0__INSTANCE0.MY_BAD_FIFO.BUFFER.value.table[3268]), INT_ENUM},*)
(*DBG:    {&(RES0__INSTANCE0.MY_BAD_FIFO.BUFFER.value.table[3269]), INT_ENUM},*)
(*DBG:    {&(RES0__INSTANCE0.MY_BAD_FIFO.BUFFER.value.table[3270]), INT_ENUM},*)
(*DBG:    {&(RES0__INSTANCE0.MY_BAD_FIFO.BUFFER.value.table[3271]), INT_ENUM},*)
(*DBG:    {&(RES0__INSTANCE0.MY_BAD_FIFO.BUFFER.value.table[3272]), INT_ENUM},*)
(*DBG:    {&(RES0__INSTANCE0.MY_BAD_FIFO.BUFFER.value.table[3273]), INT_ENUM},*)
(*DBG:    {&(RES0__INSTANCE0.MY_BAD_FIFO.BUFFER.value.table[3274]), INT_ENUM},*)
(*DBG:    {&(RES0__INSTANCE0.MY_BAD_FIFO.BUFFER.value.table[3275]), INT_ENUM},*)
(*DBG:    {&(RES0__INSTANCE0.MY_BAD_FIFO.BUFFER.value.table[3276]), INT_ENUM},*)
(*DBG:    {&(RES0__INSTANCE0.MY_BAD_FIFO.BUFFER.value.table[3277]), INT_ENUM},*)
(*DBG:    {&(RES0__INSTANCE0.MY_BAD_FIFO.BUFFER.value.table[3278]), INT_ENUM},*)
(*DBG:    {&(RES0__INSTANCE0.MY_BAD_FIFO.BUFFER.value.table[3279]), INT_ENUM},*)
(*DBG:    {&(RES0__INSTANCE0.MY_BAD_FIFO.BUFFER.value.table[3280]), INT_ENUM},*)
(*DBG:    {&(RES0__INSTANCE0.MY_BAD_FIFO.BUFFER.value.table[3281]), INT_ENUM},*)
(*DBG:    {&(RES0__INSTANCE0.MY_BAD_FIFO.BUFFER.value.table[3282]), INT_ENUM},*)
(*DBG:    {&(RES0__INSTANCE0.MY_BAD_FIFO.BUFFER.value.table[3283]), INT_ENUM},*)
(*DBG:    {&(RES0__INSTANCE0.MY_BAD_FIFO.BUFFER.value.table[3284]), INT_ENUM},*)
(*DBG:    {&(RES0__INSTANCE0.MY_BAD_FIFO.BUFFER.value.table[3285]), INT_ENUM},*)
(*DBG:    {&(RES0__INSTANCE0.MY_BAD_FIFO.BUFFER.value.table[3286]), INT_ENUM},*)
(*DBG:    {&(RES0__INSTANCE0.MY_BAD_FIFO.BUFFER.value.table[3287]), INT_ENUM},*)
(*DBG:    {&(RES0__INSTANCE0.MY_BAD_FIFO.BUFFER.value.table[3288]), INT_ENUM},*)
(*DBG:    {&(RES0__INSTANCE0.MY_BAD_FIFO.BUFFER.value.table[3289]), INT_ENUM},*)
(*DBG:    {&(RES0__INSTANCE0.MY_BAD_FIFO.BUFFER.value.table[3290]), INT_ENUM},*)
(*DBG:    {&(RES0__INSTANCE0.MY_BAD_FIFO.BUFFER.value.table[3291]), INT_ENUM},*)
(*DBG:    {&(RES0__INSTANCE0.MY_BAD_FIFO.BUFFER.value.table[3292]), INT_ENUM},*)
(*DBG:    {&(RES0__INSTANCE0.MY_BAD_FIFO.BUFFER.value.table[3293]), INT_ENUM},*)
(*DBG:    {&(RES0__INSTANCE0.MY_BAD_FIFO.BUFFER.value.table[3294]), INT_ENUM},*)
(*DBG:    {&(RES0__INSTANCE0.MY_BAD_FIFO.BUFFER.value.table[3295]), INT_ENUM},*)
(*DBG:    {&(RES0__INSTANCE0.MY_BAD_FIFO.BUFFER.value.table[3296]), INT_ENUM},*)
(*DBG:    {&(RES0__INSTANCE0.MY_BAD_FIFO.BUFFER.value.table[3297]), INT_ENUM},*)
(*DBG:    {&(RES0__INSTANCE0.MY_BAD_FIFO.BUFFER.value.table[3298]), INT_ENUM},*)
(*DBG:    {&(RES0__INSTANCE0.MY_BAD_FIFO.BUFFER.value.table[3299]), INT_ENUM},*)
(*DBG:    {&(RES0__INSTANCE0.MY_BAD_FIFO.BUFFER.value.table[3300]), INT_ENUM},*)
(*DBG:    {&(RES0__INSTANCE0.MY_BAD_FIFO.BUFFER.value.table[3301]), INT_ENUM},*)
(*DBG:    {&(RES0__INSTANCE0.MY_BAD_FIFO.BUFFER.value.table[3302]), INT_ENUM},*)
(*DBG:    {&(RES0__INSTANCE0.MY_BAD_FIFO.BUFFER.value.table[3303]), INT_ENUM},*)
(*DBG:    {&(RES0__INSTANCE0.MY_BAD_FIFO.BUFFER.value.table[3304]), INT_ENUM},*)
(*DBG:    {&(RES0__INSTANCE0.MY_BAD_FIFO.BUFFER.value.table[3305]), INT_ENUM},*)
(*DBG:    {&(RES0__INSTANCE0.MY_BAD_FIFO.BUFFER.value.table[3306]), INT_ENUM},*)
(*DBG:    {&(RES0__INSTANCE0.MY_BAD_FIFO.BUFFER.value.table[3307]), INT_ENUM},*)
(*DBG:    {&(RES0__INSTANCE0.MY_BAD_FIFO.BUFFER.value.table[3308]), INT_ENUM},*)
(*DBG:    {&(RES0__INSTANCE0.MY_BAD_FIFO.BUFFER.value.table[3309]), INT_ENUM},*)
(*DBG:    {&(RES0__INSTANCE0.MY_BAD_FIFO.BUFFER.value.table[3310]), INT_ENUM},*)
(*DBG:    {&(RES0__INSTANCE0.MY_BAD_FIFO.BUFFER.value.table[3311]), INT_ENUM},*)
(*DBG:    {&(RES0__INSTANCE0.MY_BAD_FIFO.BUFFER.value.table[3312]), INT_ENUM},*)
(*DBG:    {&(RES0__INSTANCE0.MY_BAD_FIFO.BUFFER.value.table[3313]), INT_ENUM},*)
(*DBG:    {&(RES0__INSTANCE0.MY_BAD_FIFO.BUFFER.value.table[3314]), INT_ENUM},*)
(*DBG:    {&(RES0__INSTANCE0.MY_BAD_FIFO.BUFFER.value.table[3315]), INT_ENUM},*)
(*DBG:    {&(RES0__INSTANCE0.MY_BAD_FIFO.BUFFER.value.table[3316]), INT_ENUM},*)
(*DBG:    {&(RES0__INSTANCE0.MY_BAD_FIFO.BUFFER.value.table[3317]), INT_ENUM},*)
(*DBG:    {&(RES0__INSTANCE0.MY_BAD_FIFO.BUFFER.value.table[3318]), INT_ENUM},*)
(*DBG:    {&(RES0__INSTANCE0.MY_BAD_FIFO.BUFFER.value.table[3319]), INT_ENUM},*)
(*DBG:    {&(RES0__INSTANCE0.MY_BAD_FIFO.BUFFER.value.table[3320]), INT_ENUM},*)
(*DBG:    {&(RES0__INSTANCE0.MY_BAD_FIFO.BUFFER.value.table[3321]), INT_ENUM},*)
(*DBG:    {&(RES0__INSTANCE0.MY_BAD_FIFO.BUFFER.value.table[3322]), INT_ENUM},*)
(*DBG:    {&(RES0__INSTANCE0.MY_BAD_FIFO.BUFFER.value.table[3323]), INT_ENUM},*)
(*DBG:    {&(RES0__INSTANCE0.MY_BAD_FIFO.BUFFER.value.table[3324]), INT_ENUM},*)
(*DBG:    {&(RES0__INSTANCE0.MY_BAD_FIFO.BUFFER.value.table[3325]), INT_ENUM},*)
(*DBG:    {&(RES0__INSTANCE0.MY_BAD_FIFO.BUFFER.value.table[3326]), INT_ENUM},*)
(*DBG:    {&(RES0__INSTANCE0.MY_BAD_FIFO.BUFFER.value.table[3327]), INT_ENUM},*)
(*DBG:    {&(RES0__INSTANCE0.MY_BAD_FIFO.BUFFER.value.table[3328]), INT_ENUM},*)
(*DBG:    {&(RES0__INSTANCE0.MY_BAD_FIFO.BUFFER.value.table[3329]), INT_ENUM},*)
(*DBG:    {&(RES0__INSTANCE0.MY_BAD_FIFO.BUFFER.value.table[3330]), INT_ENUM},*)
(*DBG:    {&(RES0__INSTANCE0.MY_BAD_FIFO.BUFFER.value.table[3331]), INT_ENUM},*)
(*DBG:    {&(RES0__INSTANCE0.MY_BAD_FIFO.BUFFER.value.table[3332]), INT_ENUM},*)
(*DBG:    {&(RES0__INSTANCE0.MY_BAD_FIFO.BUFFER.value.table[3333]), INT_ENUM},*)
(*DBG:    {&(RES0__INSTANCE0.MY_BAD_FIFO.BUFFER.value.table[3334]), INT_ENUM},*)
(*DBG:    {&(RES0__INSTANCE0.MY_BAD_FIFO.BUFFER.value.table[3335]), INT_ENUM},*)
(*DBG:    {&(RES0__INSTANCE0.MY_BAD_FIFO.BUFFER.value.table[3336]), INT_ENUM},*)
(*DBG:    {&(RES0__INSTANCE0.MY_BAD_FIFO.BUFFER.value.table[3337]), INT_ENUM},*)
(*DBG:    {&(RES0__INSTANCE0.MY_BAD_FIFO.BUFFER.value.table[3338]), INT_ENUM},*)
(*DBG:    {&(RES0__INSTANCE0.MY_BAD_FIFO.BUFFER.value.table[3339]), INT_ENUM},*)
(*DBG:    {&(RES0__INSTANCE0.MY_BAD_FIFO.BUFFER.value.table[3340]), INT_ENUM},*)
(*DBG:    {&(RES0__INSTANCE0.MY_BAD_FIFO.BUFFER.value.table[3341]), INT_ENUM},*)
(*DBG:    {&(RES0__INSTANCE0.MY_BAD_FIFO.BUFFER.value.table[3342]), INT_ENUM},*)
(*DBG:    {&(RES0__INSTANCE0.MY_BAD_FIFO.BUFFER.value.table[3343]), INT_ENUM},*)
(*DBG:    {&(RES0__INSTANCE0.MY_BAD_FIFO.BUFFER.value.table[3344]), INT_ENUM},*)
(*DBG:    {&(RES0__INSTANCE0.MY_BAD_FIFO.BUFFER.value.table[3345]), INT_ENUM},*)
(*DBG:    {&(RES0__INSTANCE0.MY_BAD_FIFO.BUFFER.value.table[3346]), INT_ENUM},*)
(*DBG:    {&(RES0__INSTANCE0.MY_BAD_FIFO.BUFFER.value.table[3347]), INT_ENUM},*)
(*DBG:    {&(RES0__INSTANCE0.MY_BAD_FIFO.BUFFER.value.table[3348]), INT_ENUM},*)
(*DBG:    {&(RES0__INSTANCE0.MY_BAD_FIFO.BUFFER.value.table[3349]), INT_ENUM},*)
(*DBG:    {&(RES0__INSTANCE0.MY_BAD_FIFO.BUFFER.value.table[3350]), INT_ENUM},*)
(*DBG:    {&(RES0__INSTANCE0.MY_BAD_FIFO.BUFFER.value.table[3351]), INT_ENUM},*)
(*DBG:    {&(RES0__INSTANCE0.MY_BAD_FIFO.BUFFER.value.table[3352]), INT_ENUM},*)
(*DBG:    {&(RES0__INSTANCE0.MY_BAD_FIFO.BUFFER.value.table[3353]), INT_ENUM},*)
(*DBG:    {&(RES0__INSTANCE0.MY_BAD_FIFO.BUFFER.value.table[3354]), INT_ENUM},*)
(*DBG:    {&(RES0__INSTANCE0.MY_BAD_FIFO.BUFFER.value.table[3355]), INT_ENUM},*)
(*DBG:    {&(RES0__INSTANCE0.MY_BAD_FIFO.BUFFER.value.table[3356]), INT_ENUM},*)
(*DBG:    {&(RES0__INSTANCE0.MY_BAD_FIFO.BUFFER.value.table[3357]), INT_ENUM},*)
(*DBG:    {&(RES0__INSTANCE0.MY_BAD_FIFO.BUFFER.value.table[3358]), INT_ENUM},*)
(*DBG:    {&(RES0__INSTANCE0.MY_BAD_FIFO.BUFFER.value.table[3359]), INT_ENUM},*)
(*DBG:    {&(RES0__INSTANCE0.MY_BAD_FIFO.BUFFER.value.table[3360]), INT_ENUM},*)
(*DBG:    {&(RES0__INSTANCE0.MY_BAD_FIFO.BUFFER.value.table[3361]), INT_ENUM},*)
(*DBG:    {&(RES0__INSTANCE0.MY_BAD_FIFO.BUFFER.value.table[3362]), INT_ENUM},*)
(*DBG:    {&(RES0__INSTANCE0.MY_BAD_FIFO.BUFFER.value.table[3363]), INT_ENUM},*)
(*DBG:    {&(RES0__INSTANCE0.MY_BAD_FIFO.BUFFER.value.table[3364]), INT_ENUM},*)
(*DBG:    {&(RES0__INSTANCE0.MY_BAD_FIFO.BUFFER.value.table[3365]), INT_ENUM},*)
(*DBG:    {&(RES0__INSTANCE0.MY_BAD_FIFO.BUFFER.value.table[3366]), INT_ENUM},*)
(*DBG:    {&(RES0__INSTANCE0.MY_BAD_FIFO.BUFFER.value.table[3367]), INT_ENUM},*)
(*DBG:    {&(RES0__INSTANCE0.MY_BAD_FIFO.BUFFER.value.table[3368]), INT_ENUM},*)
(*DBG:    {&(RES0__INSTANCE0.MY_BAD_FIFO.BUFFER.value.table[3369]), INT_ENUM},*)
(*DBG:    {&(RES0__INSTANCE0.MY_BAD_FIFO.BUFFER.value.table[3370]), INT_ENUM},*)
(*DBG:    {&(RES0__INSTANCE0.MY_BAD_FIFO.BUFFER.value.table[3371]), INT_ENUM},*)
(*DBG:    {&(RES0__INSTANCE0.MY_BAD_FIFO.BUFFER.value.table[3372]), INT_ENUM},*)
(*DBG:    {&(RES0__INSTANCE0.MY_BAD_FIFO.BUFFER.value.table[3373]), INT_ENUM},*)
(*DBG:    {&(RES0__INSTANCE0.MY_BAD_FIFO.BUFFER.value.table[3374]), INT_ENUM},*)
(*DBG:    {&(RES0__INSTANCE0.MY_BAD_FIFO.BUFFER.value.table[3375]), INT_ENUM},*)
(*DBG:    {&(RES0__INSTANCE0.MY_BAD_FIFO.BUFFER.value.table[3376]), INT_ENUM},*)
(*DBG:    {&(RES0__INSTANCE0.MY_BAD_FIFO.BUFFER.value.table[3377]), INT_ENUM},*)
(*DBG:    {&(RES0__INSTANCE0.MY_BAD_FIFO.BUFFER.value.table[3378]), INT_ENUM},*)
(*DBG:    {&(RES0__INSTANCE0.MY_BAD_FIFO.BUFFER.value.table[3379]), INT_ENUM},*)
(*DBG:    {&(RES0__INSTANCE0.MY_BAD_FIFO.BUFFER.value.table[3380]), INT_ENUM},*)
(*DBG:    {&(RES0__INSTANCE0.MY_BAD_FIFO.BUFFER.value.table[3381]), INT_ENUM},*)
(*DBG:    {&(RES0__INSTANCE0.MY_BAD_FIFO.BUFFER.value.table[3382]), INT_ENUM},*)
(*DBG:    {&(RES0__INSTANCE0.MY_BAD_FIFO.BUFFER.value.table[3383]), INT_ENUM},*)
(*DBG:    {&(RES0__INSTANCE0.MY_BAD_FIFO.BUFFER.value.table[3384]), INT_ENUM},*)
(*DBG:    {&(RES0__INSTANCE0.MY_BAD_FIFO.BUFFER.value.table[3385]), INT_ENUM},*)
(*DBG:    {&(RES0__INSTANCE0.MY_BAD_FIFO.BUFFER.value.table[3386]), INT_ENUM},*)
(*DBG:    {&(RES0__INSTANCE0.MY_BAD_FIFO.BUFFER.value.table[3387]), INT_ENUM},*)
(*DBG:    {&(RES0__INSTANCE0.MY_BAD_FIFO.BUFFER.value.table[3388]), INT_ENUM},*)
(*DBG:    {&(RES0__INSTANCE0.MY_BAD_FIFO.BUFFER.value.table[3389]), INT_ENUM},*)
(*DBG:    {&(RES0__INSTANCE0.MY_BAD_FIFO.BUFFER.value.table[3390]), INT_ENUM},*)
(*DBG:    {&(RES0__INSTANCE0.MY_BAD_FIFO.BUFFER.value.table[3391]), INT_ENUM},*)
(*DBG:    {&(RES0__INSTANCE0.MY_BAD_FIFO.BUFFER.value.table[3392]), INT_ENUM},*)
(*DBG:    {&(RES0__INSTANCE0.MY_BAD_FIFO.BUFFER.value.table[3393]), INT_ENUM},*)
(*DBG:    {&(RES0__INSTANCE0.MY_BAD_FIFO.BUFFER.value.table[3394]), INT_ENUM},*)
(*DBG:    {&(RES0__INSTANCE0.MY_BAD_FIFO.BUFFER.value.table[3395]), INT_ENUM},*)
(*DBG:    {&(RES0__INSTANCE0.MY_BAD_FIFO.BUFFER.value.table[3396]), INT_ENUM},*)
(*DBG:    {&(RES0__INSTANCE0.MY_BAD_FIFO.BUFFER.value.table[3397]), INT_ENUM},*)
(*DBG:    {&(RES0__INSTANCE0.MY_BAD_FIFO.BUFFER.value.table[3398]), INT_ENUM},*)
(*DBG:    {&(RES0__INSTANCE0.MY_BAD_FIFO.BUFFER.value.table[3399]), INT_ENUM},*)
(*DBG:    {&(RES0__INSTANCE0.MY_BAD_FIFO.BUFFER.value.table[3400]), INT_ENUM},*)
(*DBG:    {&(RES0__INSTANCE0.MY_BAD_FIFO.BUFFER.value.table[3401]), INT_ENUM},*)
(*DBG:    {&(RES0__INSTANCE0.MY_BAD_FIFO.BUFFER.value.table[3402]), INT_ENUM},*)
(*DBG:    {&(RES0__INSTANCE0.MY_BAD_FIFO.BUFFER.value.table[3403]), INT_ENUM},*)
(*DBG:    {&(RES0__INSTANCE0.MY_BAD_FIFO.BUFFER.value.table[3404]), INT_ENUM},*)
(*DBG:    {&(RES0__INSTANCE0.MY_BAD_FIFO.BUFFER.value.table[3405]), INT_ENUM},*)
(*DBG:    {&(RES0__INSTANCE0.MY_BAD_FIFO.BUFFER.value.table[3406]), INT_ENUM},*)
(*DBG:    {&(RES0__INSTANCE0.MY_BAD_FIFO.BUFFER.value.table[3407]), INT_ENUM},*)
(*DBG:    {&(RES0__INSTANCE0.MY_BAD_FIFO.BUFFER.value.table[3408]), INT_ENUM},*)
(*DBG:    {&(RES0__INSTANCE0.MY_BAD_FIFO.BUFFER.value.table[3409]), INT_ENUM},*)
(*DBG:    {&(RES0__INSTANCE0.MY_BAD_FIFO.BUFFER.value.table[3410]), INT_ENUM},*)
(*DBG:    {&(RES0__INSTANCE0.MY_BAD_FIFO.BUFFER.value.table[3411]), INT_ENUM},*)
(*DBG:    {&(RES0__INSTANCE0.MY_BAD_FIFO.BUFFER.value.table[3412]), INT_ENUM},*)
(*DBG:    {&(RES0__INSTANCE0.MY_BAD_FIFO.BUFFER.value.table[3413]), INT_ENUM},*)
(*DBG:    {&(RES0__INSTANCE0.MY_BAD_FIFO.BUFFER.value.table[3414]), INT_ENUM},*)
(*DBG:    {&(RES0__INSTANCE0.MY_BAD_FIFO.BUFFER.value.table[3415]), INT_ENUM},*)
(*DBG:    {&(RES0__INSTANCE0.MY_BAD_FIFO.BUFFER.value.table[3416]), INT_ENUM},*)
(*DBG:    {&(RES0__INSTANCE0.MY_BAD_FIFO.BUFFER.value.table[3417]), INT_ENUM},*)
(*DBG:    {&(RES0__INSTANCE0.MY_BAD_FIFO.BUFFER.value.table[3418]), INT_ENUM},*)
(*DBG:    {&(RES0__INSTANCE0.MY_BAD_FIFO.BUFFER.value.table[3419]), INT_ENUM},*)
(*DBG:    {&(RES0__INSTANCE0.MY_BAD_FIFO.BUFFER.value.table[3420]), INT_ENUM},*)
(*DBG:    {&(RES0__INSTANCE0.MY_BAD_FIFO.BUFFER.value.table[3421]), INT_ENUM},*)
(*DBG:    {&(RES0__INSTANCE0.MY_BAD_FIFO.BUFFER.value.table[3422]), INT_ENUM},*)
(*DBG:    {&(RES0__INSTANCE0.MY_BAD_FIFO.BUFFER.value.table[3423]), INT_ENUM},*)
(*DBG:    {&(RES0__INSTANCE0.MY_BAD_FIFO.BUFFER.value.table[3424]), INT_ENUM},*)
(*DBG:    {&(RES0__INSTANCE0.MY_BAD_FIFO.BUFFER.value.table[3425]), INT_ENUM},*)
(*DBG:    {&(RES0__INSTANCE0.MY_BAD_FIFO.BUFFER.value.table[3426]), INT_ENUM},*)
(*DBG:    {&(RES0__INSTANCE0.MY_BAD_FIFO.BUFFER.value.table[3427]), INT_ENUM},*)
(*DBG:    {&(RES0__INSTANCE0.MY_BAD_FIFO.BUFFER.value.table[3428]), INT_ENUM},*)
(*DBG:    {&(RES0__INSTANCE0.MY_BAD_FIFO.BUFFER.value.table[3429]), INT_ENUM},*)
(*DBG:    {&(RES0__INSTANCE0.MY_BAD_FIFO.BUFFER.value.table[3430]), INT_ENUM},*)
(*DBG:    {&(RES0__INSTANCE0.MY_BAD_FIFO.BUFFER.value.table[3431]), INT_ENUM},*)
(*DBG:    {&(RES0__INSTANCE0.MY_BAD_FIFO.BUFFER.value.table[3432]), INT_ENUM},*)
(*DBG:    {&(RES0__INSTANCE0.MY_BAD_FIFO.BUFFER.value.table[3433]), INT_ENUM},*)
(*DBG:    {&(RES0__INSTANCE0.MY_BAD_FIFO.BUFFER.value.table[3434]), INT_ENUM},*)
(*DBG:    {&(RES0__INSTANCE0.MY_BAD_FIFO.BUFFER.value.table[3435]), INT_ENUM},*)
(*DBG:    {&(RES0__INSTANCE0.MY_BAD_FIFO.BUFFER.value.table[3436]), INT_ENUM},*)
(*DBG:    {&(RES0__INSTANCE0.MY_BAD_FIFO.BUFFER.value.table[3437]), INT_ENUM},*)
(*DBG:    {&(RES0__INSTANCE0.MY_BAD_FIFO.BUFFER.value.table[3438]), INT_ENUM},*)
(*DBG:    {&(RES0__INSTANCE0.MY_BAD_FIFO.BUFFER.value.table[3439]), INT_ENUM},*)
(*DBG:    {&(RES0__INSTANCE0.MY_BAD_FIFO.BUFFER.value.table[3440]), INT_ENUM},*)
(*DBG:    {&(RES0__INSTANCE0.MY_BAD_FIFO.BUFFER.value.table[3441]), INT_ENUM},*)
(*DBG:    {&(RES0__INSTANCE0.MY_BAD_FIFO.BUFFER.value.table[3442]), INT_ENUM},*)
(*DBG:    {&(RES0__INSTANCE0.MY_BAD_FIFO.BUFFER.value.table[3443]), INT_ENUM},*)
(*DBG:    {&(RES0__INSTANCE0.MY_BAD_FIFO.BUFFER.value.table[3444]), INT_ENUM},*)
(*DBG:    {&(RES0__INSTANCE0.MY_BAD_FIFO.BUFFER.value.table[3445]), INT_ENUM},*)
(*DBG:    {&(RES0__INSTANCE0.MY_BAD_FIFO.BUFFER.value.table[3446]), INT_ENUM},*)
(*DBG:    {&(RES0__INSTANCE0.MY_BAD_FIFO.BUFFER.value.table[3447]), INT_ENUM},*)
(*DBG:    {&(RES0__INSTANCE0.MY_BAD_FIFO.BUFFER.value.table[3448]), INT_ENUM},*)
(*DBG:    {&(RES0__INSTANCE0.MY_BAD_FIFO.BUFFER.value.table[3449]), INT_ENUM},*)
(*DBG:    {&(RES0__INSTANCE0.MY_BAD_FIFO.BUFFER.value.table[3450]), INT_ENUM},*)
(*DBG:    {&(RES0__INSTANCE0.MY_BAD_FIFO.BUFFER.value.table[3451]), INT_ENUM},*)
(*DBG:    {&(RES0__INSTANCE0.MY_BAD_FIFO.BUFFER.value.table[3452]), INT_ENUM},*)
(*DBG:    {&(RES0__INSTANCE0.MY_BAD_FIFO.BUFFER.value.table[3453]), INT_ENUM},*)
(*DBG:    {&(RES0__INSTANCE0.MY_BAD_FIFO.BUFFER.value.table[3454]), INT_ENUM},*)
(*DBG:    {&(RES0__INSTANCE0.MY_BAD_FIFO.BUFFER.value.table[3455]), INT_ENUM},*)
(*DBG:    {&(RES0__INSTANCE0.MY_BAD_FIFO.BUFFER.value.table[3456]), INT_ENUM},*)
(*DBG:    {&(RES0__INSTANCE0.MY_BAD_FIFO.BUFFER.value.table[3457]), INT_ENUM},*)
(*DBG:    {&(RES0__INSTANCE0.MY_BAD_FIFO.BUFFER.value.table[3458]), INT_ENUM},*)
(*DBG:    {&(RES0__INSTANCE0.MY_BAD_FIFO.BUFFER.value.table[3459]), INT_ENUM},*)
(*DBG:    {&(RES0__INSTANCE0.MY_BAD_FIFO.BUFFER.value.table[3460]), INT_ENUM},*)
(*DBG:    {&(RES0__INSTANCE0.MY_BAD_FIFO.BUFFER.value.table[3461]), INT_ENUM},*)
(*DBG:    {&(RES0__INSTANCE0.MY_BAD_FIFO.BUFFER.value.table[3462]), INT_ENUM},*)
(*DBG:    {&(RES0__INSTANCE0.MY_BAD_FIFO.BUFFER.value.table[3463]), INT_ENUM},*)
(*DBG:    {&(RES0__INSTANCE0.MY_BAD_FIFO.BUFFER.value.table[3464]), INT_ENUM},*)
(*DBG:    {&(RES0__INSTANCE0.MY_BAD_FIFO.BUFFER.value.table[3465]), INT_ENUM},*)
(*DBG:    {&(RES0__INSTANCE0.MY_BAD_FIFO.BUFFER.value.table[3466]), INT_ENUM},*)
(*DBG:    {&(RES0__INSTANCE0.MY_BAD_FIFO.BUFFER.value.table[3467]), INT_ENUM},*)
(*DBG:    {&(RES0__INSTANCE0.MY_BAD_FIFO.BUFFER.value.table[3468]), INT_ENUM},*)
(*DBG:    {&(RES0__INSTANCE0.MY_BAD_FIFO.BUFFER.value.table[3469]), INT_ENUM},*)
(*DBG:    {&(RES0__INSTANCE0.MY_BAD_FIFO.BUFFER.value.table[3470]), INT_ENUM},*)
(*DBG:    {&(RES0__INSTANCE0.MY_BAD_FIFO.BUFFER.value.table[3471]), INT_ENUM},*)
(*DBG:    {&(RES0__INSTANCE0.MY_BAD_FIFO.BUFFER.value.table[3472]), INT_ENUM},*)
(*DBG:    {&(RES0__INSTANCE0.MY_BAD_FIFO.BUFFER.value.table[3473]), INT_ENUM},*)
(*DBG:    {&(RES0__INSTANCE0.MY_BAD_FIFO.BUFFER.value.table[3474]), INT_ENUM},*)
(*DBG:    {&(RES0__INSTANCE0.MY_BAD_FIFO.BUFFER.value.table[3475]), INT_ENUM},*)
(*DBG:    {&(RES0__INSTANCE0.MY_BAD_FIFO.BUFFER.value.table[3476]), INT_ENUM},*)
(*DBG:    {&(RES0__INSTANCE0.MY_BAD_FIFO.BUFFER.value.table[3477]), INT_ENUM},*)
(*DBG:    {&(RES0__INSTANCE0.MY_BAD_FIFO.BUFFER.value.table[3478]), INT_ENUM},*)
(*DBG:    {&(RES0__INSTANCE0.MY_BAD_FIFO.BUFFER.value.table[3479]), INT_ENUM},*)
(*DBG:    {&(RES0__INSTANCE0.MY_BAD_FIFO.BUFFER.value.table[3480]), INT_ENUM},*)
(*DBG:    {&(RES0__INSTANCE0.MY_BAD_FIFO.BUFFER.value.table[3481]), INT_ENUM},*)
(*DBG:    {&(RES0__INSTANCE0.MY_BAD_FIFO.BUFFER.value.table[3482]), INT_ENUM},*)
(*DBG:    {&(RES0__INSTANCE0.MY_BAD_FIFO.BUFFER.value.table[3483]), INT_ENUM},*)
(*DBG:    {&(RES0__INSTANCE0.MY_BAD_FIFO.BUFFER.value.table[3484]), INT_ENUM},*)
(*DBG:    {&(RES0__INSTANCE0.MY_BAD_FIFO.BUFFER.value.table[3485]), INT_ENUM},*)
(*DBG:    {&(RES0__INSTANCE0.MY_BAD_FIFO.BUFFER.value.table[3486]), INT_ENUM},*)
(*DBG:    {&(RES0__INSTANCE0.MY_BAD_FIFO.BUFFER.value.table[3487]), INT_ENUM},*)
(*DBG:    {&(RES0__INSTANCE0.MY_BAD_FIFO.BUFFER.value.table[3488]), INT_ENUM},*)
(*DBG:    {&(RES0__INSTANCE0.MY_BAD_FIFO.BUFFER.value.table[3489]), INT_ENUM},*)
(*DBG:    {&(RES0__INSTANCE0.MY_BAD_FIFO.BUFFER.value.table[3490]), INT_ENUM},*)
(*DBG:    {&(RES0__INSTANCE0.MY_BAD_FIFO.BUFFER.value.table[3491]), INT_ENUM},*)
(*DBG:    {&(RES0__INSTANCE0.MY_BAD_FIFO.BUFFER.value.table[3492]), INT_ENUM},*)
(*DBG:    {&(RES0__INSTANCE0.MY_BAD_FIFO.BUFFER.value.table[3493]), INT_ENUM},*)
(*DBG:    {&(RES0__INSTANCE0.MY_BAD_FIFO.BUFFER.value.table[3494]), INT_ENUM},*)
(*DBG:    {&(RES0__INSTANCE0.MY_BAD_FIFO.BUFFER.value.table[3495]), INT_ENUM},*)
(*DBG:    {&(RES0__INSTANCE0.MY_BAD_FIFO.BUFFER.value.table[3496]), INT_ENUM},*)
(*DBG:    {&(RES0__INSTANCE0.MY_BAD_FIFO.BUFFER.value.table[3497]), INT_ENUM},*)
(*DBG:    {&(RES0__INSTANCE0.MY_BAD_FIFO.BUFFER.value.table[3498]), INT_ENUM},*)
(*DBG:    {&(RES0__INSTANCE0.MY_BAD_FIFO.BUFFER.value.table[3499]), INT_ENUM},*)
(*DBG:    {&(RES0__INSTANCE0.MY_BAD_FIFO.BUFFER.value.table[3500]), INT_ENUM},*)
(*DBG:    {&(RES0__INSTANCE0.MY_BAD_FIFO.BUFFER.value.table[3501]), INT_ENUM},*)
(*DBG:    {&(RES0__INSTANCE0.MY_BAD_FIFO.BUFFER.value.table[3502]), INT_ENUM},*)
(*DBG:    {&(RES0__INSTANCE0.MY_BAD_FIFO.BUFFER.value.table[3503]), INT_ENUM},*)
(*DBG:    {&(RES0__INSTANCE0.MY_BAD_FIFO.BUFFER.value.table[3504]), INT_ENUM},*)
(*DBG:    {&(RES0__INSTANCE0.MY_BAD_FIFO.BUFFER.value.table[3505]), INT_ENUM},*)
(*DBG:    {&(RES0__INSTANCE0.MY_BAD_FIFO.BUFFER.value.table[3506]), INT_ENUM},*)
(*DBG:    {&(RES0__INSTANCE0.MY_BAD_FIFO.BUFFER.value.table[3507]), INT_ENUM},*)
(*DBG:    {&(RES0__INSTANCE0.MY_BAD_FIFO.BUFFER.value.table[3508]), INT_ENUM},*)
(*DBG:    {&(RES0__INSTANCE0.MY_BAD_FIFO.BUFFER.value.table[3509]), INT_ENUM},*)
(*DBG:    {&(RES0__INSTANCE0.MY_BAD_FIFO.BUFFER.value.table[3510]), INT_ENUM},*)
(*DBG:    {&(RES0__INSTANCE0.MY_BAD_FIFO.BUFFER.value.table[3511]), INT_ENUM},*)
(*DBG:    {&(RES0__INSTANCE0.MY_BAD_FIFO.BUFFER.value.table[3512]), INT_ENUM},*)
(*DBG:    {&(RES0__INSTANCE0.MY_BAD_FIFO.BUFFER.value.table[3513]), INT_ENUM},*)
(*DBG:    {&(RES0__INSTANCE0.MY_BAD_FIFO.BUFFER.value.table[3514]), INT_ENUM},*)
(*DBG:    {&(RES0__INSTANCE0.MY_BAD_FIFO.BUFFER.value.table[3515]), INT_ENUM},*)
(*DBG:    {&(RES0__INSTANCE0.MY_BAD_FIFO.BUFFER.value.table[3516]), INT_ENUM},*)
(*DBG:    {&(RES0__INSTANCE0.MY_BAD_FIFO.BUFFER.value.table[3517]), INT_ENUM},*)
(*DBG:    {&(RES0__INSTANCE0.MY_BAD_FIFO.BUFFER.value.table[3518]), INT_ENUM},*)
(*DBG:    {&(RES0__INSTANCE0.MY_BAD_FIFO.BUFFER.value.table[3519]), INT_ENUM},*)
(*DBG:    {&(RES0__INSTANCE0.MY_BAD_FIFO.BUFFER.value.table[3520]), INT_ENUM},*)
(*DBG:    {&(RES0__INSTANCE0.MY_BAD_FIFO.BUFFER.value.table[3521]), INT_ENUM},*)
(*DBG:    {&(RES0__INSTANCE0.MY_BAD_FIFO.BUFFER.value.table[3522]), INT_ENUM},*)
(*DBG:    {&(RES0__INSTANCE0.MY_BAD_FIFO.BUFFER.value.table[3523]), INT_ENUM},*)
(*DBG:    {&(RES0__INSTANCE0.MY_BAD_FIFO.BUFFER.value.table[3524]), INT_ENUM},*)
(*DBG:    {&(RES0__INSTANCE0.MY_BAD_FIFO.BUFFER.value.table[3525]), INT_ENUM},*)
(*DBG:    {&(RES0__INSTANCE0.MY_BAD_FIFO.BUFFER.value.table[3526]), INT_ENUM},*)
(*DBG:    {&(RES0__INSTANCE0.MY_BAD_FIFO.BUFFER.value.table[3527]), INT_ENUM},*)
(*DBG:    {&(RES0__INSTANCE0.MY_BAD_FIFO.BUFFER.value.table[3528]), INT_ENUM},*)
(*DBG:    {&(RES0__INSTANCE0.MY_BAD_FIFO.BUFFER.value.table[3529]), INT_ENUM},*)
(*DBG:    {&(RES0__INSTANCE0.MY_BAD_FIFO.BUFFER.value.table[3530]), INT_ENUM},*)
(*DBG:    {&(RES0__INSTANCE0.MY_BAD_FIFO.BUFFER.value.table[3531]), INT_ENUM},*)
(*DBG:    {&(RES0__INSTANCE0.MY_BAD_FIFO.BUFFER.value.table[3532]), INT_ENUM},*)
(*DBG:    {&(RES0__INSTANCE0.MY_BAD_FIFO.BUFFER.value.table[3533]), INT_ENUM},*)
(*DBG:    {&(RES0__INSTANCE0.MY_BAD_FIFO.BUFFER.value.table[3534]), INT_ENUM},*)
(*DBG:    {&(RES0__INSTANCE0.MY_BAD_FIFO.BUFFER.value.table[3535]), INT_ENUM},*)
(*DBG:    {&(RES0__INSTANCE0.MY_BAD_FIFO.BUFFER.value.table[3536]), INT_ENUM},*)
(*DBG:    {&(RES0__INSTANCE0.MY_BAD_FIFO.BUFFER.value.table[3537]), INT_ENUM},*)
(*DBG:    {&(RES0__INSTANCE0.MY_BAD_FIFO.BUFFER.value.table[3538]), INT_ENUM},*)
(*DBG:    {&(RES0__INSTANCE0.MY_BAD_FIFO.BUFFER.value.table[3539]), INT_ENUM},*)
(*DBG:    {&(RES0__INSTANCE0.MY_BAD_FIFO.BUFFER.value.table[3540]), INT_ENUM},*)
(*DBG:    {&(RES0__INSTANCE0.MY_BAD_FIFO.BUFFER.value.table[3541]), INT_ENUM},*)
(*DBG:    {&(RES0__INSTANCE0.MY_BAD_FIFO.BUFFER.value.table[3542]), INT_ENUM},*)
(*DBG:    {&(RES0__INSTANCE0.MY_BAD_FIFO.BUFFER.value.table[3543]), INT_ENUM},*)
(*DBG:    {&(RES0__INSTANCE0.MY_BAD_FIFO.BUFFER.value.table[3544]), INT_ENUM},*)
(*DBG:    {&(RES0__INSTANCE0.MY_BAD_FIFO.BUFFER.value.table[3545]), INT_ENUM},*)
(*DBG:    {&(RES0__INSTANCE0.MY_BAD_FIFO.BUFFER.value.table[3546]), INT_ENUM},*)
(*DBG:    {&(RES0__INSTANCE0.MY_BAD_FIFO.BUFFER.value.table[3547]), INT_ENUM},*)
(*DBG:    {&(RES0__INSTANCE0.MY_BAD_FIFO.BUFFER.value.table[3548]), INT_ENUM},*)
(*DBG:    {&(RES0__INSTANCE0.MY_BAD_FIFO.BUFFER.value.table[3549]), INT_ENUM},*)
(*DBG:    {&(RES0__INSTANCE0.MY_BAD_FIFO.BUFFER.value.table[3550]), INT_ENUM},*)
(*DBG:    {&(RES0__INSTANCE0.MY_BAD_FIFO.BUFFER.value.table[3551]), INT_ENUM},*)
(*DBG:    {&(RES0__INSTANCE0.MY_BAD_FIFO.BUFFER.value.table[3552]), INT_ENUM},*)
(*DBG:    {&(RES0__INSTANCE0.MY_BAD_FIFO.BUFFER.value.table[3553]), INT_ENUM},*)
(*DBG:    {&(RES0__INSTANCE0.MY_BAD_FIFO.BUFFER.value.table[3554]), INT_ENUM},*)
(*DBG:    {&(RES0__INSTANCE0.MY_BAD_FIFO.BUFFER.value.table[3555]), INT_ENUM},*)
(*DBG:    {&(RES0__INSTANCE0.MY_BAD_FIFO.BUFFER.value.table[3556]), INT_ENUM},*)
(*DBG:    {&(RES0__INSTANCE0.MY_BAD_FIFO.BUFFER.value.table[3557]), INT_ENUM},*)
(*DBG:    {&(RES0__INSTANCE0.MY_BAD_FIFO.BUFFER.value.table[3558]), INT_ENUM},*)
(*DBG:    {&(RES0__INSTANCE0.MY_BAD_FIFO.BUFFER.value.table[3559]), INT_ENUM},*)
(*DBG:    {&(RES0__INSTANCE0.MY_BAD_FIFO.BUFFER.value.table[3560]), INT_ENUM},*)
(*DBG:    {&(RES0__INSTANCE0.MY_BAD_FIFO.BUFFER.value.table[3561]), INT_ENUM},*)
(*DBG:    {&(RES0__INSTANCE0.MY_BAD_FIFO.BUFFER.value.table[3562]), INT_ENUM},*)
(*DBG:    {&(RES0__INSTANCE0.MY_BAD_FIFO.BUFFER.value.table[3563]), INT_ENUM},*)
(*DBG:    {&(RES0__INSTANCE0.MY_BAD_FIFO.BUFFER.value.table[3564]), INT_ENUM},*)
(*DBG:    {&(RES0__INSTANCE0.MY_BAD_FIFO.BUFFER.value.table[3565]), INT_ENUM},*)
(*DBG:    {&(RES0__INSTANCE0.MY_BAD_FIFO.BUFFER.value.table[3566]), INT_ENUM},*)
(*DBG:    {&(RES0__INSTANCE0.MY_BAD_FIFO.BUFFER.value.table[3567]), INT_ENUM},*)
(*DBG:    {&(RES0__INSTANCE0.MY_BAD_FIFO.BUFFER.value.table[3568]), INT_ENUM},*)
(*DBG:    {&(RES0__INSTANCE0.MY_BAD_FIFO.BUFFER.value.table[3569]), INT_ENUM},*)
(*DBG:    {&(RES0__INSTANCE0.MY_BAD_FIFO.BUFFER.value.table[3570]), INT_ENUM},*)
(*DBG:    {&(RES0__INSTANCE0.MY_BAD_FIFO.BUFFER.value.table[3571]), INT_ENUM},*)
(*DBG:    {&(RES0__INSTANCE0.MY_BAD_FIFO.BUFFER.value.table[3572]), INT_ENUM},*)
(*DBG:    {&(RES0__INSTANCE0.MY_BAD_FIFO.BUFFER.value.table[3573]), INT_ENUM},*)
(*DBG:    {&(RES0__INSTANCE0.MY_BAD_FIFO.BUFFER.value.table[3574]), INT_ENUM},*)
(*DBG:    {&(RES0__INSTANCE0.MY_BAD_FIFO.BUFFER.value.table[3575]), INT_ENUM},*)
(*DBG:    {&(RES0__INSTANCE0.MY_BAD_FIFO.BUFFER.value.table[3576]), INT_ENUM},*)
(*DBG:    {&(RES0__INSTANCE0.MY_BAD_FIFO.BUFFER.value.table[3577]), INT_ENUM},*)
(*DBG:    {&(RES0__INSTANCE0.MY_BAD_FIFO.BUFFER.value.table[3578]), INT_ENUM},*)
(*DBG:    {&(RES0__INSTANCE0.MY_BAD_FIFO.BUFFER.value.table[3579]), INT_ENUM},*)
(*DBG:    {&(RES0__INSTANCE0.MY_BAD_FIFO.BUFFER.value.table[3580]), INT_ENUM},*)
(*DBG:    {&(RES0__INSTANCE0.MY_BAD_FIFO.BUFFER.value.table[3581]), INT_ENUM},*)
(*DBG:    {&(RES0__INSTANCE0.MY_BAD_FIFO.BUFFER.value.table[3582]), INT_ENUM},*)
(*DBG:    {&(RES0__INSTANCE0.MY_BAD_FIFO.BUFFER.value.table[3583]), INT_ENUM},*)
(*DBG:    {&(RES0__INSTANCE0.MY_BAD_FIFO.BUFFER.value.table[3584]), INT_ENUM},*)
(*DBG:    {&(RES0__INSTANCE0.MY_BAD_FIFO.BUFFER.value.table[3585]), INT_ENUM},*)
(*DBG:    {&(RES0__INSTANCE0.MY_BAD_FIFO.BUFFER.value.table[3586]), INT_ENUM},*)
(*DBG:    {&(RES0__INSTANCE0.MY_BAD_FIFO.BUFFER.value.table[3587]), INT_ENUM},*)
(*DBG:    {&(RES0__INSTANCE0.MY_BAD_FIFO.BUFFER.value.table[3588]), INT_ENUM},*)
(*DBG:    {&(RES0__INSTANCE0.MY_BAD_FIFO.BUFFER.value.table[3589]), INT_ENUM},*)
(*DBG:    {&(RES0__INSTANCE0.MY_BAD_FIFO.BUFFER.value.table[3590]), INT_ENUM},*)
(*DBG:    {&(RES0__INSTANCE0.MY_BAD_FIFO.BUFFER.value.table[3591]), INT_ENUM},*)
(*DBG:    {&(RES0__INSTANCE0.MY_BAD_FIFO.BUFFER.value.table[3592]), INT_ENUM},*)
(*DBG:    {&(RES0__INSTANCE0.MY_BAD_FIFO.BUFFER.value.table[3593]), INT_ENUM},*)
(*DBG:    {&(RES0__INSTANCE0.MY_BAD_FIFO.BUFFER.value.table[3594]), INT_ENUM},*)
(*DBG:    {&(RES0__INSTANCE0.MY_BAD_FIFO.BUFFER.value.table[3595]), INT_ENUM},*)
(*DBG:    {&(RES0__INSTANCE0.MY_BAD_FIFO.BUFFER.value.table[3596]), INT_ENUM},*)
(*DBG:    {&(RES0__INSTANCE0.MY_BAD_FIFO.BUFFER.value.table[3597]), INT_ENUM},*)
(*DBG:    {&(RES0__INSTANCE0.MY_BAD_FIFO.BUFFER.value.table[3598]), INT_ENUM},*)
(*DBG:    {&(RES0__INSTANCE0.MY_BAD_FIFO.BUFFER.value.table[3599]), INT_ENUM},*)
(*DBG:    {&(RES0__INSTANCE0.MY_BAD_FIFO.BUFFER.value.table[3600]), INT_ENUM},*)
(*DBG:    {&(RES0__INSTANCE0.MY_BAD_FIFO.BUFFER.value.table[3601]), INT_ENUM},*)
(*DBG:    {&(RES0__INSTANCE0.MY_BAD_FIFO.BUFFER.value.table[3602]), INT_ENUM},*)
(*DBG:    {&(RES0__INSTANCE0.MY_BAD_FIFO.BUFFER.value.table[3603]), INT_ENUM},*)
(*DBG:    {&(RES0__INSTANCE0.MY_BAD_FIFO.BUFFER.value.table[3604]), INT_ENUM},*)
(*DBG:    {&(RES0__INSTANCE0.MY_BAD_FIFO.BUFFER.value.table[3605]), INT_ENUM},*)
(*DBG:    {&(RES0__INSTANCE0.MY_BAD_FIFO.BUFFER.value.table[3606]), INT_ENUM},*)
(*DBG:    {&(RES0__INSTANCE0.MY_BAD_FIFO.BUFFER.value.table[3607]), INT_ENUM},*)
(*DBG:    {&(RES0__INSTANCE0.MY_BAD_FIFO.BUFFER.value.table[3608]), INT_ENUM},*)
(*DBG:    {&(RES0__INSTANCE0.MY_BAD_FIFO.BUFFER.value.table[3609]), INT_ENUM},*)
(*DBG:    {&(RES0__INSTANCE0.MY_BAD_FIFO.BUFFER.value.table[3610]), INT_ENUM},*)
(*DBG:    {&(RES0__INSTANCE0.MY_BAD_FIFO.BUFFER.value.table[3611]), INT_ENUM},*)
(*DBG:    {&(RES0__INSTANCE0.MY_BAD_FIFO.BUFFER.value.table[3612]), INT_ENUM},*)
(*DBG:    {&(RES0__INSTANCE0.MY_BAD_FIFO.BUFFER.value.table[3613]), INT_ENUM},*)
(*DBG:    {&(RES0__INSTANCE0.MY_BAD_FIFO.BUFFER.value.table[3614]), INT_ENUM},*)
(*DBG:    {&(RES0__INSTANCE0.MY_BAD_FIFO.BUFFER.value.table[3615]), INT_ENUM},*)
(*DBG:    {&(RES0__INSTANCE0.MY_BAD_FIFO.BUFFER.value.table[3616]), INT_ENUM},*)
(*DBG:    {&(RES0__INSTANCE0.MY_BAD_FIFO.BUFFER.value.table[3617]), INT_ENUM},*)
(*DBG:    {&(RES0__INSTANCE0.MY_BAD_FIFO.BUFFER.value.table[3618]), INT_ENUM},*)
(*DBG:    {&(RES0__INSTANCE0.MY_BAD_FIFO.BUFFER.value.table[3619]), INT_ENUM},*)
(*DBG:    {&(RES0__INSTANCE0.MY_BAD_FIFO.BUFFER.value.table[3620]), INT_ENUM},*)
(*DBG:    {&(RES0__INSTANCE0.MY_BAD_FIFO.BUFFER.value.table[3621]), INT_ENUM},*)
(*DBG:    {&(RES0__INSTANCE0.MY_BAD_FIFO.BUFFER.value.table[3622]), INT_ENUM},*)
(*DBG:    {&(RES0__INSTANCE0.MY_BAD_FIFO.BUFFER.value.table[3623]), INT_ENUM},*)
(*DBG:    {&(RES0__INSTANCE0.MY_BAD_FIFO.BUFFER.value.table[3624]), INT_ENUM},*)
(*DBG:    {&(RES0__INSTANCE0.MY_BAD_FIFO.BUFFER.value.table[3625]), INT_ENUM},*)
(*DBG:    {&(RES0__INSTANCE0.MY_BAD_FIFO.BUFFER.value.table[3626]), INT_ENUM},*)
(*DBG:    {&(RES0__INSTANCE0.MY_BAD_FIFO.BUFFER.value.table[3627]), INT_ENUM},*)
(*DBG:    {&(RES0__INSTANCE0.MY_BAD_FIFO.BUFFER.value.table[3628]), INT_ENUM},*)
(*DBG:    {&(RES0__INSTANCE0.MY_BAD_FIFO.BUFFER.value.table[3629]), INT_ENUM},*)
(*DBG:    {&(RES0__INSTANCE0.MY_BAD_FIFO.BUFFER.value.table[3630]), INT_ENUM},*)
(*DBG:    {&(RES0__INSTANCE0.MY_BAD_FIFO.BUFFER.value.table[3631]), INT_ENUM},*)
(*DBG:    {&(RES0__INSTANCE0.MY_BAD_FIFO.BUFFER.value.table[3632]), INT_ENUM},*)
(*DBG:    {&(RES0__INSTANCE0.MY_BAD_FIFO.BUFFER.value.table[3633]), INT_ENUM},*)
(*DBG:    {&(RES0__INSTANCE0.MY_BAD_FIFO.BUFFER.value.table[3634]), INT_ENUM},*)
(*DBG:    {&(RES0__INSTANCE0.MY_BAD_FIFO.BUFFER.value.table[3635]), INT_ENUM},*)
(*DBG:    {&(RES0__INSTANCE0.MY_BAD_FIFO.BUFFER.value.table[3636]), INT_ENUM},*)
(*DBG:    {&(RES0__INSTANCE0.MY_BAD_FIFO.BUFFER.value.table[3637]), INT_ENUM},*)
(*DBG:    {&(RES0__INSTANCE0.MY_BAD_FIFO.BUFFER.value.table[3638]), INT_ENUM},*)
(*DBG:    {&(RES0__INSTANCE0.MY_BAD_FIFO.BUFFER.value.table[3639]), INT_ENUM},*)
(*DBG:    {&(RES0__INSTANCE0.MY_BAD_FIFO.BUFFER.value.table[3640]), INT_ENUM},*)
(*DBG:    {&(RES0__INSTANCE0.MY_BAD_FIFO.BUFFER.value.table[3641]), INT_ENUM},*)
(*DBG:    {&(RES0__INSTANCE0.MY_BAD_FIFO.BUFFER.value.table[3642]), INT_ENUM},*)
(*DBG:    {&(RES0__INSTANCE0.MY_BAD_FIFO.BUFFER.value.table[3643]), INT_ENUM},*)
(*DBG:    {&(RES0__INSTANCE0.MY_BAD_FIFO.BUFFER.value.table[3644]), INT_ENUM},*)
(*DBG:    {&(RES0__INSTANCE0.MY_BAD_FIFO.BUFFER.value.table[3645]), INT_ENUM},*)
(*DBG:    {&(RES0__INSTANCE0.MY_BAD_FIFO.BUFFER.value.table[3646]), INT_ENUM},*)
(*DBG:    {&(RES0__INSTANCE0.MY_BAD_FIFO.BUFFER.value.table[3647]), INT_ENUM},*)
(*DBG:    {&(RES0__INSTANCE0.MY_BAD_FIFO.BUFFER.value.table[3648]), INT_ENUM},*)
(*DBG:    {&(RES0__INSTANCE0.MY_BAD_FIFO.BUFFER.value.table[3649]), INT_ENUM},*)
(*DBG:    {&(RES0__INSTANCE0.MY_BAD_FIFO.BUFFER.value.table[3650]), INT_ENUM},*)
(*DBG:    {&(RES0__INSTANCE0.MY_BAD_FIFO.BUFFER.value.table[3651]), INT_ENUM},*)
(*DBG:    {&(RES0__INSTANCE0.MY_BAD_FIFO.BUFFER.value.table[3652]), INT_ENUM},*)
(*DBG:    {&(RES0__INSTANCE0.MY_BAD_FIFO.BUFFER.value.table[3653]), INT_ENUM},*)
(*DBG:    {&(RES0__INSTANCE0.MY_BAD_FIFO.BUFFER.value.table[3654]), INT_ENUM},*)
(*DBG:    {&(RES0__INSTANCE0.MY_BAD_FIFO.BUFFER.value.table[3655]), INT_ENUM},*)
(*DBG:    {&(RES0__INSTANCE0.MY_BAD_FIFO.BUFFER.value.table[3656]), INT_ENUM},*)
(*DBG:    {&(RES0__INSTANCE0.MY_BAD_FIFO.BUFFER.value.table[3657]), INT_ENUM},*)
(*DBG:    {&(RES0__INSTANCE0.MY_BAD_FIFO.BUFFER.value.table[3658]), INT_ENUM},*)
(*DBG:    {&(RES0__INSTANCE0.MY_BAD_FIFO.BUFFER.value.table[3659]), INT_ENUM},*)
(*DBG:    {&(RES0__INSTANCE0.MY_BAD_FIFO.BUFFER.value.table[3660]), INT_ENUM},*)
(*DBG:    {&(RES0__INSTANCE0.MY_BAD_FIFO.BUFFER.value.table[3661]), INT_ENUM},*)
(*DBG:    {&(RES0__INSTANCE0.MY_BAD_FIFO.BUFFER.value.table[3662]), INT_ENUM},*)
(*DBG:    {&(RES0__INSTANCE0.MY_BAD_FIFO.BUFFER.value.table[3663]), INT_ENUM},*)
(*DBG:    {&(RES0__INSTANCE0.MY_BAD_FIFO.BUFFER.value.table[3664]), INT_ENUM},*)
(*DBG:    {&(RES0__INSTANCE0.MY_BAD_FIFO.BUFFER.value.table[3665]), INT_ENUM},*)
(*DBG:    {&(RES0__INSTANCE0.MY_BAD_FIFO.BUFFER.value.table[3666]), INT_ENUM},*)
(*DBG:    {&(RES0__INSTANCE0.MY_BAD_FIFO.BUFFER.value.table[3667]), INT_ENUM},*)
(*DBG:    {&(RES0__INSTANCE0.MY_BAD_FIFO.BUFFER.value.table[3668]), INT_ENUM},*)
(*DBG:    {&(RES0__INSTANCE0.MY_BAD_FIFO.BUFFER.value.table[3669]), INT_ENUM},*)
(*DBG:    {&(RES0__INSTANCE0.MY_BAD_FIFO.BUFFER.value.table[3670]), INT_ENUM},*)
(*DBG:    {&(RES0__INSTANCE0.MY_BAD_FIFO.BUFFER.value.table[3671]), INT_ENUM},*)
(*DBG:    {&(RES0__INSTANCE0.MY_BAD_FIFO.BUFFER.value.table[3672]), INT_ENUM},*)
(*DBG:    {&(RES0__INSTANCE0.MY_BAD_FIFO.BUFFER.value.table[3673]), INT_ENUM},*)
(*DBG:    {&(RES0__INSTANCE0.MY_BAD_FIFO.BUFFER.value.table[3674]), INT_ENUM},*)
(*DBG:    {&(RES0__INSTANCE0.MY_BAD_FIFO.BUFFER.value.table[3675]), INT_ENUM},*)
(*DBG:    {&(RES0__INSTANCE0.MY_BAD_FIFO.BUFFER.value.table[3676]), INT_ENUM},*)
(*DBG:    {&(RES0__INSTANCE0.MY_BAD_FIFO.BUFFER.value.table[3677]), INT_ENUM},*)
(*DBG:    {&(RES0__INSTANCE0.MY_BAD_FIFO.BUFFER.value.table[3678]), INT_ENUM},*)
(*DBG:    {&(RES0__INSTANCE0.MY_BAD_FIFO.BUFFER.value.table[3679]), INT_ENUM},*)
(*DBG:    {&(RES0__INSTANCE0.MY_BAD_FIFO.BUFFER.value.table[3680]), INT_ENUM},*)
(*DBG:    {&(RES0__INSTANCE0.MY_BAD_FIFO.BUFFER.value.table[3681]), INT_ENUM},*)
(*DBG:    {&(RES0__INSTANCE0.MY_BAD_FIFO.BUFFER.value.table[3682]), INT_ENUM},*)
(*DBG:    {&(RES0__INSTANCE0.MY_BAD_FIFO.BUFFER.value.table[3683]), INT_ENUM},*)
(*DBG:    {&(RES0__INSTANCE0.MY_BAD_FIFO.BUFFER.value.table[3684]), INT_ENUM},*)
(*DBG:    {&(RES0__INSTANCE0.MY_BAD_FIFO.BUFFER.value.table[3685]), INT_ENUM},*)
(*DBG:    {&(RES0__INSTANCE0.MY_BAD_FIFO.BUFFER.value.table[3686]), INT_ENUM},*)
(*DBG:    {&(RES0__INSTANCE0.MY_BAD_FIFO.BUFFER.value.table[3687]), INT_ENUM},*)
(*DBG:    {&(RES0__INSTANCE0.MY_BAD_FIFO.BUFFER.value.table[3688]), INT_ENUM},*)
(*DBG:    {&(RES0__INSTANCE0.MY_BAD_FIFO.BUFFER.value.table[3689]), INT_ENUM},*)
(*DBG:    {&(RES0__INSTANCE0.MY_BAD_FIFO.BUFFER.value.table[3690]), INT_ENUM},*)
(*DBG:    {&(RES0__INSTANCE0.MY_BAD_FIFO.BUFFER.value.table[3691]), INT_ENUM},*)
(*DBG:    {&(RES0__INSTANCE0.MY_BAD_FIFO.BUFFER.value.table[3692]), INT_ENUM},*)
(*DBG:    {&(RES0__INSTANCE0.MY_BAD_FIFO.BUFFER.value.table[3693]), INT_ENUM},*)
(*DBG:    {&(RES0__INSTANCE0.MY_BAD_FIFO.BUFFER.value.table[3694]), INT_ENUM},*)
(*DBG:    {&(RES0__INSTANCE0.MY_BAD_FIFO.BUFFER.value.table[3695]), INT_ENUM},*)
(*DBG:    {&(RES0__INSTANCE0.MY_BAD_FIFO.BUFFER.value.table[3696]), INT_ENUM},*)
(*DBG:    {&(RES0__INSTANCE0.MY_BAD_FIFO.BUFFER.value.table[3697]), INT_ENUM},*)
(*DBG:    {&(RES0__INSTANCE0.MY_BAD_FIFO.BUFFER.value.table[3698]), INT_ENUM},*)
(*DBG:    {&(RES0__INSTANCE0.MY_BAD_FIFO.BUFFER.value.table[3699]), INT_ENUM},*)
(*DBG:    {&(RES0__INSTANCE0.MY_BAD_FIFO.BUFFER.value.table[3700]), INT_ENUM},*)
(*DBG:    {&(RES0__INSTANCE0.MY_BAD_FIFO.BUFFER.value.table[3701]), INT_ENUM},*)
(*DBG:    {&(RES0__INSTANCE0.MY_BAD_FIFO.BUFFER.value.table[3702]), INT_ENUM},*)
(*DBG:    {&(RES0__INSTANCE0.MY_BAD_FIFO.BUFFER.value.table[3703]), INT_ENUM},*)
(*DBG:    {&(RES0__INSTANCE0.MY_BAD_FIFO.BUFFER.value.table[3704]), INT_ENUM},*)
(*DBG:    {&(RES0__INSTANCE0.MY_BAD_FIFO.BUFFER.value.table[3705]), INT_ENUM},*)
(*DBG:    {&(RES0__INSTANCE0.MY_BAD_FIFO.BUFFER.value.table[3706]), INT_ENUM},*)
(*DBG:    {&(RES0__INSTANCE0.MY_BAD_FIFO.BUFFER.value.table[3707]), INT_ENUM},*)
(*DBG:    {&(RES0__INSTANCE0.MY_BAD_FIFO.BUFFER.value.table[3708]), INT_ENUM},*)
(*DBG:    {&(RES0__INSTANCE0.MY_BAD_FIFO.BUFFER.value.table[3709]), INT_ENUM},*)
(*DBG:    {&(RES0__INSTANCE0.MY_BAD_FIFO.BUFFER.value.table[3710]), INT_ENUM},*)
(*DBG:    {&(RES0__INSTANCE0.MY_BAD_FIFO.BUFFER.value.table[3711]), INT_ENUM},*)
(*DBG:    {&(RES0__INSTANCE0.MY_BAD_FIFO.BUFFER.value.table[3712]), INT_ENUM},*)
(*DBG:    {&(RES0__INSTANCE0.MY_BAD_FIFO.BUFFER.value.table[3713]), INT_ENUM},*)
(*DBG:    {&(RES0__INSTANCE0.MY_BAD_FIFO.BUFFER.value.table[3714]), INT_ENUM},*)
(*DBG:    {&(RES0__INSTANCE0.MY_BAD_FIFO.BUFFER.value.table[3715]), INT_ENUM},*)
(*DBG:    {&(RES0__INSTANCE0.MY_BAD_FIFO.BUFFER.value.table[3716]), INT_ENUM},*)
(*DBG:    {&(RES0__INSTANCE0.MY_BAD_FIFO.BUFFER.value.table[3717]), INT_ENUM},*)
(*DBG:    {&(RES0__INSTANCE0.MY_BAD_FIFO.BUFFER.value.table[3718]), INT_ENUM},*)
(*DBG:    {&(RES0__INSTANCE0.MY_BAD_FIFO.BUFFER.value.table[3719]), INT_ENUM},*)
(*DBG:    {&(RES0__INSTANCE0.MY_BAD_FIFO.BUFFER.value.table[3720]), INT_ENUM},*)
(*DBG:    {&(RES0__INSTANCE0.MY_BAD_FIFO.BUFFER.value.table[3721]), INT_ENUM},*)
(*DBG:    {&(RES0__INSTANCE0.MY_BAD_FIFO.BUFFER.value.table[3722]), INT_ENUM},*)
(*DBG:    {&(RES0__INSTANCE0.MY_BAD_FIFO.BUFFER.value.table[3723]), INT_ENUM},*)
(*DBG:    {&(RES0__INSTANCE0.MY_BAD_FIFO.BUFFER.value.table[3724]), INT_ENUM},*)
(*DBG:    {&(RES0__INSTANCE0.MY_BAD_FIFO.BUFFER.value.table[3725]), INT_ENUM},*)
(*DBG:    {&(RES0__INSTANCE0.MY_BAD_FIFO.BUFFER.value.table[3726]), INT_ENUM},*)
(*DBG:    {&(RES0__INSTANCE0.MY_BAD_FIFO.BUFFER.value.table[3727]), INT_ENUM},*)
(*DBG:    {&(RES0__INSTANCE0.MY_BAD_FIFO.BUFFER.value.table[3728]), INT_ENUM},*)
(*DBG:    {&(RES0__INSTANCE0.MY_BAD_FIFO.BUFFER.value.table[3729]), INT_ENUM},*)
(*DBG:    {&(RES0__INSTANCE0.MY_BAD_FIFO.BUFFER.value.table[3730]), INT_ENUM},*)
(*DBG:    {&(RES0__INSTANCE0.MY_BAD_FIFO.BUFFER.value.table[3731]), INT_ENUM},*)
(*DBG:    {&(RES0__INSTANCE0.MY_BAD_FIFO.BUFFER.value.table[3732]), INT_ENUM},*)
(*DBG:    {&(RES0__INSTANCE0.MY_BAD_FIFO.BUFFER.value.table[3733]), INT_ENUM},*)
(*DBG:    {&(RES0__INSTANCE0.MY_BAD_FIFO.BUFFER.value.table[3734]), INT_ENUM},*)
(*DBG:    {&(RES0__INSTANCE0.MY_BAD_FIFO.BUFFER.value.table[3735]), INT_ENUM},*)
(*DBG:    {&(RES0__INSTANCE0.MY_BAD_FIFO.BUFFER.value.table[3736]), INT_ENUM},*)
(*DBG:    {&(RES0__INSTANCE0.MY_BAD_FIFO.BUFFER.value.table[3737]), INT_ENUM},*)
(*DBG:    {&(RES0__INSTANCE0.MY_BAD_FIFO.BUFFER.value.table[3738]), INT_ENUM},*)
(*DBG:    {&(RES0__INSTANCE0.MY_BAD_FIFO.BUFFER.value.table[3739]), INT_ENUM},*)
(*DBG:    {&(RES0__INSTANCE0.MY_BAD_FIFO.BUFFER.value.table[3740]), INT_ENUM},*)
(*DBG:    {&(RES0__INSTANCE0.MY_BAD_FIFO.BUFFER.value.table[3741]), INT_ENUM},*)
(*DBG:    {&(RES0__INSTANCE0.MY_BAD_FIFO.BUFFER.value.table[3742]), INT_ENUM},*)
(*DBG:    {&(RES0__INSTANCE0.MY_BAD_FIFO.BUFFER.value.table[3743]), INT_ENUM},*)
(*DBG:    {&(RES0__INSTANCE0.MY_BAD_FIFO.BUFFER.value.table[3744]), INT_ENUM},*)
(*DBG:    {&(RES0__INSTANCE0.MY_BAD_FIFO.BUFFER.value.table[3745]), INT_ENUM},*)
(*DBG:    {&(RES0__INSTANCE0.MY_BAD_FIFO.BUFFER.value.table[3746]), INT_ENUM},*)
(*DBG:    {&(RES0__INSTANCE0.MY_BAD_FIFO.BUFFER.value.table[3747]), INT_ENUM},*)
(*DBG:    {&(RES0__INSTANCE0.MY_BAD_FIFO.BUFFER.value.table[3748]), INT_ENUM},*)
(*DBG:    {&(RES0__INSTANCE0.MY_BAD_FIFO.BUFFER.value.table[3749]), INT_ENUM},*)
(*DBG:    {&(RES0__INSTANCE0.MY_BAD_FIFO.BUFFER.value.table[3750]), INT_ENUM},*)
(*DBG:    {&(RES0__INSTANCE0.MY_BAD_FIFO.BUFFER.value.table[3751]), INT_ENUM},*)
(*DBG:    {&(RES0__INSTANCE0.MY_BAD_FIFO.BUFFER.value.table[3752]), INT_ENUM},*)
(*DBG:    {&(RES0__INSTANCE0.MY_BAD_FIFO.BUFFER.value.table[3753]), INT_ENUM},*)
(*DBG:    {&(RES0__INSTANCE0.MY_BAD_FIFO.BUFFER.value.table[3754]), INT_ENUM},*)
(*DBG:    {&(RES0__INSTANCE0.MY_BAD_FIFO.BUFFER.value.table[3755]), INT_ENUM},*)
(*DBG:    {&(RES0__INSTANCE0.MY_BAD_FIFO.BUFFER.value.table[3756]), INT_ENUM},*)
(*DBG:    {&(RES0__INSTANCE0.MY_BAD_FIFO.BUFFER.value.table[3757]), INT_ENUM},*)
(*DBG:    {&(RES0__INSTANCE0.MY_BAD_FIFO.BUFFER.value.table[3758]), INT_ENUM},*)
(*DBG:    {&(RES0__INSTANCE0.MY_BAD_FIFO.BUFFER.value.table[3759]), INT_ENUM},*)
(*DBG:    {&(RES0__INSTANCE0.MY_BAD_FIFO.BUFFER.value.table[3760]), INT_ENUM},*)
(*DBG:    {&(RES0__INSTANCE0.MY_BAD_FIFO.BUFFER.value.table[3761]), INT_ENUM},*)
(*DBG:    {&(RES0__INSTANCE0.MY_BAD_FIFO.BUFFER.value.table[3762]), INT_ENUM},*)
(*DBG:    {&(RES0__INSTANCE0.MY_BAD_FIFO.BUFFER.value.table[3763]), INT_ENUM},*)
(*DBG:    {&(RES0__INSTANCE0.MY_BAD_FIFO.BUFFER.value.table[3764]), INT_ENUM},*)
(*DBG:    {&(RES0__INSTANCE0.MY_BAD_FIFO.BUFFER.value.table[3765]), INT_ENUM},*)
(*DBG:    {&(RES0__INSTANCE0.MY_BAD_FIFO.BUFFER.value.table[3766]), INT_ENUM},*)
(*DBG:    {&(RES0__INSTANCE0.MY_BAD_FIFO.BUFFER.value.table[3767]), INT_ENUM},*)
(*DBG:    {&(RES0__INSTANCE0.MY_BAD_FIFO.BUFFER.value.table[3768]), INT_ENUM},*)
(*DBG:    {&(RES0__INSTANCE0.MY_BAD_FIFO.BUFFER.value.table[3769]), INT_ENUM},*)
(*DBG:    {&(RES0__INSTANCE0.MY_BAD_FIFO.BUFFER.value.table[3770]), INT_ENUM},*)
(*DBG:    {&(RES0__INSTANCE0.MY_BAD_FIFO.BUFFER.value.table[3771]), INT_ENUM},*)
(*DBG:    {&(RES0__INSTANCE0.MY_BAD_FIFO.BUFFER.value.table[3772]), INT_ENUM},*)
(*DBG:    {&(RES0__INSTANCE0.MY_BAD_FIFO.BUFFER.value.table[3773]), INT_ENUM},*)
(*DBG:    {&(RES0__INSTANCE0.MY_BAD_FIFO.BUFFER.value.table[3774]), INT_ENUM},*)
(*DBG:    {&(RES0__INSTANCE0.MY_BAD_FIFO.BUFFER.value.table[3775]), INT_ENUM},*)
(*DBG:    {&(RES0__INSTANCE0.MY_BAD_FIFO.BUFFER.value.table[3776]), INT_ENUM},*)
(*DBG:    {&(RES0__INSTANCE0.MY_BAD_FIFO.BUFFER.value.table[3777]), INT_ENUM},*)
(*DBG:    {&(RES0__INSTANCE0.MY_BAD_FIFO.BUFFER.value.table[3778]), INT_ENUM},*)
(*DBG:    {&(RES0__INSTANCE0.MY_BAD_FIFO.BUFFER.value.table[3779]), INT_ENUM},*)
(*DBG:    {&(RES0__INSTANCE0.MY_BAD_FIFO.BUFFER.value.table[3780]), INT_ENUM},*)
(*DBG:    {&(RES0__INSTANCE0.MY_BAD_FIFO.BUFFER.value.table[3781]), INT_ENUM},*)
(*DBG:    {&(RES0__INSTANCE0.MY_BAD_FIFO.BUFFER.value.table[3782]), INT_ENUM},*)
(*DBG:    {&(RES0__INSTANCE0.MY_BAD_FIFO.BUFFER.value.table[3783]), INT_ENUM},*)
(*DBG:    {&(RES0__INSTANCE0.MY_BAD_FIFO.BUFFER.value.table[3784]), INT_ENUM},*)
(*DBG:    {&(RES0__INSTANCE0.MY_BAD_FIFO.BUFFER.value.table[3785]), INT_ENUM},*)
(*DBG:    {&(RES0__INSTANCE0.MY_BAD_FIFO.BUFFER.value.table[3786]), INT_ENUM},*)
(*DBG:    {&(RES0__INSTANCE0.MY_BAD_FIFO.BUFFER.value.table[3787]), INT_ENUM},*)
(*DBG:    {&(RES0__INSTANCE0.MY_BAD_FIFO.BUFFER.value.table[3788]), INT_ENUM},*)
(*DBG:    {&(RES0__INSTANCE0.MY_BAD_FIFO.BUFFER.value.table[3789]), INT_ENUM},*)
(*DBG:    {&(RES0__INSTANCE0.MY_BAD_FIFO.BUFFER.value.table[3790]), INT_ENUM},*)
(*DBG:    {&(RES0__INSTANCE0.MY_BAD_FIFO.BUFFER.value.table[3791]), INT_ENUM},*)
(*DBG:    {&(RES0__INSTANCE0.MY_BAD_FIFO.BUFFER.value.table[3792]), INT_ENUM},*)
(*DBG:    {&(RES0__INSTANCE0.MY_BAD_FIFO.BUFFER.value.table[3793]), INT_ENUM},*)
(*DBG:    {&(RES0__INSTANCE0.MY_BAD_FIFO.BUFFER.value.table[3794]), INT_ENUM},*)
(*DBG:    {&(RES0__INSTANCE0.MY_BAD_FIFO.BUFFER.value.table[3795]), INT_ENUM},*)
(*DBG:    {&(RES0__INSTANCE0.MY_BAD_FIFO.BUFFER.value.table[3796]), INT_ENUM},*)
(*DBG:    {&(RES0__INSTANCE0.MY_BAD_FIFO.BUFFER.value.table[3797]), INT_ENUM},*)
(*DBG:    {&(RES0__INSTANCE0.MY_BAD_FIFO.BUFFER.value.table[3798]), INT_ENUM},*)
(*DBG:    {&(RES0__INSTANCE0.MY_BAD_FIFO.BUFFER.value.table[3799]), INT_ENUM},*)
(*DBG:    {&(RES0__INSTANCE0.MY_BAD_FIFO.BUFFER.value.table[3800]), INT_ENUM},*)
(*DBG:    {&(RES0__INSTANCE0.MY_BAD_FIFO.BUFFER.value.table[3801]), INT_ENUM},*)
(*DBG:    {&(RES0__INSTANCE0.MY_BAD_FIFO.BUFFER.value.table[3802]), INT_ENUM},*)
(*DBG:    {&(RES0__INSTANCE0.MY_BAD_FIFO.BUFFER.value.table[3803]), INT_ENUM},*)
(*DBG:    {&(RES0__INSTANCE0.MY_BAD_FIFO.BUFFER.value.table[3804]), INT_ENUM},*)
(*DBG:    {&(RES0__INSTANCE0.MY_BAD_FIFO.BUFFER.value.table[3805]), INT_ENUM},*)
(*DBG:    {&(RES0__INSTANCE0.MY_BAD_FIFO.BUFFER.value.table[3806]), INT_ENUM},*)
(*DBG:    {&(RES0__INSTANCE0.MY_BAD_FIFO.BUFFER.value.table[3807]), INT_ENUM},*)
(*DBG:    {&(RES0__INSTANCE0.MY_BAD_FIFO.BUFFER.value.table[3808]), INT_ENUM},*)
(*DBG:    {&(RES0__INSTANCE0.MY_BAD_FIFO.BUFFER.value.table[3809]), INT_ENUM},*)
(*DBG:    {&(RES0__INSTANCE0.MY_BAD_FIFO.BUFFER.value.table[3810]), INT_ENUM},*)
(*DBG:    {&(RES0__INSTANCE0.MY_BAD_FIFO.BUFFER.value.table[3811]), INT_ENUM},*)
(*DBG:    {&(RES0__INSTANCE0.MY_BAD_FIFO.BUFFER.value.table[3812]), INT_ENUM},*)
(*DBG:    {&(RES0__INSTANCE0.MY_BAD_FIFO.BUFFER.value.table[3813]), INT_ENUM},*)
(*DBG:    {&(RES0__INSTANCE0.MY_BAD_FIFO.BUFFER.value.table[3814]), INT_ENUM},*)
(*DBG:    {&(RES0__INSTANCE0.MY_BAD_FIFO.BUFFER.value.table[3815]), INT_ENUM},*)
(*DBG:    {&(RES0__INSTANCE0.MY_BAD_FIFO.BUFFER.value.table[3816]), INT_ENUM},*)
(*DBG:    {&(RES0__INSTANCE0.MY_BAD_FIFO.BUFFER.value.table[3817]), INT_ENUM},*)
(*DBG:    {&(RES0__INSTANCE0.MY_BAD_FIFO.BUFFER.value.table[3818]), INT_ENUM},*)
(*DBG:    {&(RES0__INSTANCE0.MY_BAD_FIFO.BUFFER.value.table[3819]), INT_ENUM},*)
(*DBG:    {&(RES0__INSTANCE0.MY_BAD_FIFO.BUFFER.value.table[3820]), INT_ENUM},*)
(*DBG:    {&(RES0__INSTANCE0.MY_BAD_FIFO.BUFFER.value.table[3821]), INT_ENUM},*)
(*DBG:    {&(RES0__INSTANCE0.MY_BAD_FIFO.BUFFER.value.table[3822]), INT_ENUM},*)
(*DBG:    {&(RES0__INSTANCE0.MY_BAD_FIFO.BUFFER.value.table[3823]), INT_ENUM},*)
(*DBG:    {&(RES0__INSTANCE0.MY_BAD_FIFO.BUFFER.value.table[3824]), INT_ENUM},*)
(*DBG:    {&(RES0__INSTANCE0.MY_BAD_FIFO.BUFFER.value.table[3825]), INT_ENUM},*)
(*DBG:    {&(RES0__INSTANCE0.MY_BAD_FIFO.BUFFER.value.table[3826]), INT_ENUM},*)
(*DBG:    {&(RES0__INSTANCE0.MY_BAD_FIFO.BUFFER.value.table[3827]), INT_ENUM},*)
(*DBG:    {&(RES0__INSTANCE0.MY_BAD_FIFO.BUFFER.value.table[3828]), INT_ENUM},*)
(*DBG:    {&(RES0__INSTANCE0.MY_BAD_FIFO.BUFFER.value.table[3829]), INT_ENUM},*)
(*DBG:    {&(RES0__INSTANCE0.MY_BAD_FIFO.BUFFER.value.table[3830]), INT_ENUM},*)
(*DBG:    {&(RES0__INSTANCE0.MY_BAD_FIFO.BUFFER.value.table[3831]), INT_ENUM},*)
(*DBG:    {&(RES0__INSTANCE0.MY_BAD_FIFO.BUFFER.value.table[3832]), INT_ENUM},*)
(*DBG:    {&(RES0__INSTANCE0.MY_BAD_FIFO.BUFFER.value.table[3833]), INT_ENUM},*)
(*DBG:    {&(RES0__INSTANCE0.MY_BAD_FIFO.BUFFER.value.table[3834]), INT_ENUM},*)
(*DBG:    {&(RES0__INSTANCE0.MY_BAD_FIFO.BUFFER.value.table[3835]), INT_ENUM},*)
(*DBG:    {&(RES0__INSTANCE0.MY_BAD_FIFO.BUFFER.value.table[3836]), INT_ENUM},*)
(*DBG:    {&(RES0__INSTANCE0.MY_BAD_FIFO.BUFFER.value.table[3837]), INT_ENUM},*)
(*DBG:    {&(RES0__INSTANCE0.MY_BAD_FIFO.BUFFER.value.table[3838]), INT_ENUM},*)
(*DBG:    {&(RES0__INSTANCE0.MY_BAD_FIFO.BUFFER.value.table[3839]), INT_ENUM},*)
(*DBG:    {&(RES0__INSTANCE0.MY_BAD_FIFO.BUFFER.value.table[3840]), INT_ENUM},*)
(*DBG:    {&(RES0__INSTANCE0.MY_BAD_FIFO.BUFFER.value.table[3841]), INT_ENUM},*)
(*DBG:    {&(RES0__INSTANCE0.MY_BAD_FIFO.BUFFER.value.table[3842]), INT_ENUM},*)
(*DBG:    {&(RES0__INSTANCE0.MY_BAD_FIFO.BUFFER.value.table[3843]), INT_ENUM},*)
(*DBG:    {&(RES0__INSTANCE0.MY_BAD_FIFO.BUFFER.value.table[3844]), INT_ENUM},*)
(*DBG:    {&(RES0__INSTANCE0.MY_BAD_FIFO.BUFFER.value.table[3845]), INT_ENUM},*)
(*DBG:    {&(RES0__INSTANCE0.MY_BAD_FIFO.BUFFER.value.table[3846]), INT_ENUM},*)
(*DBG:    {&(RES0__INSTANCE0.MY_BAD_FIFO.BUFFER.value.table[3847]), INT_ENUM},*)
(*DBG:    {&(RES0__INSTANCE0.MY_BAD_FIFO.BUFFER.value.table[3848]), INT_ENUM},*)
(*DBG:    {&(RES0__INSTANCE0.MY_BAD_FIFO.BUFFER.value.table[3849]), INT_ENUM},*)
(*DBG:    {&(RES0__INSTANCE0.MY_BAD_FIFO.BUFFER.value.table[3850]), INT_ENUM},*)
(*DBG:    {&(RES0__INSTANCE0.MY_BAD_FIFO.BUFFER.value.table[3851]), INT_ENUM},*)
(*DBG:    {&(RES0__INSTANCE0.MY_BAD_FIFO.BUFFER.value.table[3852]), INT_ENUM},*)
(*DBG:    {&(RES0__INSTANCE0.MY_BAD_FIFO.BUFFER.value.table[3853]), INT_ENUM},*)
(*DBG:    {&(RES0__INSTANCE0.MY_BAD_FIFO.BUFFER.value.table[3854]), INT_ENUM},*)
(*DBG:    {&(RES0__INSTANCE0.MY_BAD_FIFO.BUFFER.value.table[3855]), INT_ENUM},*)
(*DBG:    {&(RES0__INSTANCE0.MY_BAD_FIFO.BUFFER.value.table[3856]), INT_ENUM},*)
(*DBG:    {&(RES0__INSTANCE0.MY_BAD_FIFO.BUFFER.value.table[3857]), INT_ENUM},*)
(*DBG:    {&(RES0__INSTANCE0.MY_BAD_FIFO.BUFFER.value.table[3858]), INT_ENUM},*)
(*DBG:    {&(RES0__INSTANCE0.MY_BAD_FIFO.BUFFER.value.table[3859]), INT_ENUM},*)
(*DBG:    {&(RES0__INSTANCE0.MY_BAD_FIFO.BUFFER.value.table[3860]), INT_ENUM},*)
(*DBG:    {&(RES0__INSTANCE0.MY_BAD_FIFO.BUFFER.value.table[3861]), INT_ENUM},*)
(*DBG:    {&(RES0__INSTANCE0.MY_BAD_FIFO.BUFFER.value.table[3862]), INT_ENUM},*)
(*DBG:    {&(RES0__INSTANCE0.MY_BAD_FIFO.BUFFER.value.table[3863]), INT_ENUM},*)
(*DBG:    {&(RES0__INSTANCE0.MY_BAD_FIFO.BUFFER.value.table[3864]), INT_ENUM},*)
(*DBG:    {&(RES0__INSTANCE0.MY_BAD_FIFO.BUFFER.value.table[3865]), INT_ENUM},*)
(*DBG:    {&(RES0__INSTANCE0.MY_BAD_FIFO.BUFFER.value.table[3866]), INT_ENUM},*)
(*DBG:    {&(RES0__INSTANCE0.MY_BAD_FIFO.BUFFER.value.table[3867]), INT_ENUM},*)
(*DBG:    {&(RES0__INSTANCE0.MY_BAD_FIFO.BUFFER.value.table[3868]), INT_ENUM},*)
(*DBG:    {&(RES0__INSTANCE0.MY_BAD_FIFO.BUFFER.value.table[3869]), INT_ENUM},*)
(*DBG:    {&(RES0__INSTANCE0.MY_BAD_FIFO.BUFFER.value.table[3870]), INT_ENUM},*)
(*DBG:    {&(RES0__INSTANCE0.MY_BAD_FIFO.BUFFER.value.table[3871]), INT_ENUM},*)
(*DBG:    {&(RES0__INSTANCE0.MY_BAD_FIFO.BUFFER.value.table[3872]), INT_ENUM},*)
(*DBG:    {&(RES0__INSTANCE0.MY_BAD_FIFO.BUFFER.value.table[3873]), INT_ENUM},*)
(*DBG:    {&(RES0__INSTANCE0.MY_BAD_FIFO.BUFFER.value.table[3874]), INT_ENUM},*)
(*DBG:    {&(RES0__INSTANCE0.MY_BAD_FIFO.BUFFER.value.table[3875]), INT_ENUM},*)
(*DBG:    {&(RES0__INSTANCE0.MY_BAD_FIFO.BUFFER.value.table[3876]), INT_ENUM},*)
(*DBG:    {&(RES0__INSTANCE0.MY_BAD_FIFO.BUFFER.value.table[3877]), INT_ENUM},*)
(*DBG:    {&(RES0__INSTANCE0.MY_BAD_FIFO.BUFFER.value.table[3878]), INT_ENUM},*)
(*DBG:    {&(RES0__INSTANCE0.MY_BAD_FIFO.BUFFER.value.table[3879]), INT_ENUM},*)
(*DBG:    {&(RES0__INSTANCE0.MY_BAD_FIFO.BUFFER.value.table[3880]), INT_ENUM},*)
(*DBG:    {&(RES0__INSTANCE0.MY_BAD_FIFO.BUFFER.value.table[3881]), INT_ENUM},*)
(*DBG:    {&(RES0__INSTANCE0.MY_BAD_FIFO.BUFFER.value.table[3882]), INT_ENUM},*)
(*DBG:    {&(RES0__INSTANCE0.MY_BAD_FIFO.BUFFER.value.table[3883]), INT_ENUM},*)
(*DBG:    {&(RES0__INSTANCE0.MY_BAD_FIFO.BUFFER.value.table[3884]), INT_ENUM},*)
(*DBG:    {&(RES0__INSTANCE0.MY_BAD_FIFO.BUFFER.value.table[3885]), INT_ENUM},*)
(*DBG:    {&(RES0__INSTANCE0.MY_BAD_FIFO.BUFFER.value.table[3886]), INT_ENUM},*)
(*DBG:    {&(RES0__INSTANCE0.MY_BAD_FIFO.BUFFER.value.table[3887]), INT_ENUM},*)
(*DBG:    {&(RES0__INSTANCE0.MY_BAD_FIFO.BUFFER.value.table[3888]), INT_ENUM},*)
(*DBG:    {&(RES0__INSTANCE0.MY_BAD_FIFO.BUFFER.value.table[3889]), INT_ENUM},*)
(*DBG:    {&(RES0__INSTANCE0.MY_BAD_FIFO.BUFFER.value.table[3890]), INT_ENUM},*)
(*DBG:    {&(RES0__INSTANCE0.MY_BAD_FIFO.BUFFER.value.table[3891]), INT_ENUM},*)
(*DBG:    {&(RES0__INSTANCE0.MY_BAD_FIFO.BUFFER.value.table[3892]), INT_ENUM},*)
(*DBG:    {&(RES0__INSTANCE0.MY_BAD_FIFO.BUFFER.value.table[3893]), INT_ENUM},*)
(*DBG:    {&(RES0__INSTANCE0.MY_BAD_FIFO.BUFFER.value.table[3894]), INT_ENUM},*)
(*DBG:    {&(RES0__INSTANCE0.MY_BAD_FIFO.BUFFER.value.table[3895]), INT_ENUM},*)
(*DBG:    {&(RES0__INSTANCE0.MY_BAD_FIFO.BUFFER.value.table[3896]), INT_ENUM},*)
(*DBG:    {&(RES0__INSTANCE0.MY_BAD_FIFO.BUFFER.value.table[3897]), INT_ENUM},*)
(*DBG:    {&(RES0__INSTANCE0.MY_BAD_FIFO.BUFFER.value.table[3898]), INT_ENUM},*)
(*DBG:    {&(RES0__INSTANCE0.MY_BAD_FIFO.BUFFER.value.table[3899]), INT_ENUM},*)
(*DBG:    {&(RES0__INSTANCE0.MY_BAD_FIFO.BUFFER.value.table[3900]), INT_ENUM},*)
(*DBG:    {&(RES0__INSTANCE0.MY_BAD_FIFO.BUFFER.value.table[3901]), INT_ENUM},*)
(*DBG:    {&(RES0__INSTANCE0.MY_BAD_FIFO.BUFFER.value.table[3902]), INT_ENUM},*)
(*DBG:    {&(RES0__INSTANCE0.MY_BAD_FIFO.BUFFER.value.table[3903]), INT_ENUM},*)
(*DBG:    {&(RES0__INSTANCE0.MY_BAD_FIFO.BUFFER.value.table[3904]), INT_ENUM},*)
(*DBG:    {&(RES0__INSTANCE0.MY_BAD_FIFO.BUFFER.value.table[3905]), INT_ENUM},*)
(*DBG:    {&(RES0__INSTANCE0.MY_BAD_FIFO.BUFFER.value.table[3906]), INT_ENUM},*)
(*DBG:    {&(RES0__INSTANCE0.MY_BAD_FIFO.BUFFER.value.table[3907]), INT_ENUM},*)
(*DBG:    {&(RES0__INSTANCE0.MY_BAD_FIFO.BUFFER.value.table[3908]), INT_ENUM},*)
(*DBG:    {&(RES0__INSTANCE0.MY_BAD_FIFO.BUFFER.value.table[3909]), INT_ENUM},*)
(*DBG:    {&(RES0__INSTANCE0.MY_BAD_FIFO.BUFFER.value.table[3910]), INT_ENUM},*)
(*DBG:    {&(RES0__INSTANCE0.MY_BAD_FIFO.BUFFER.value.table[3911]), INT_ENUM},*)
(*DBG:    {&(RES0__INSTANCE0.MY_BAD_FIFO.BUFFER.value.table[3912]), INT_ENUM},*)
(*DBG:    {&(RES0__INSTANCE0.MY_BAD_FIFO.BUFFER.value.table[3913]), INT_ENUM},*)
(*DBG:    {&(RES0__INSTANCE0.MY_BAD_FIFO.BUFFER.value.table[3914]), INT_ENUM},*)
(*DBG:    {&(RES0__INSTANCE0.MY_BAD_FIFO.BUFFER.value.table[3915]), INT_ENUM},*)
(*DBG:    {&(RES0__INSTANCE0.MY_BAD_FIFO.BUFFER.value.table[3916]), INT_ENUM},*)
(*DBG:    {&(RES0__INSTANCE0.MY_BAD_FIFO.BUFFER.value.table[3917]), INT_ENUM},*)
(*DBG:    {&(RES0__INSTANCE0.MY_BAD_FIFO.BUFFER.value.table[3918]), INT_ENUM},*)
(*DBG:    {&(RES0__INSTANCE0.MY_BAD_FIFO.BUFFER.value.table[3919]), INT_ENUM},*)
(*DBG:    {&(RES0__INSTANCE0.MY_BAD_FIFO.BUFFER.value.table[3920]), INT_ENUM},*)
(*DBG:    {&(RES0__INSTANCE0.MY_BAD_FIFO.BUFFER.value.table[3921]), INT_ENUM},*)
(*DBG:    {&(RES0__INSTANCE0.MY_BAD_FIFO.BUFFER.value.table[3922]), INT_ENUM},*)
(*DBG:    {&(RES0__INSTANCE0.MY_BAD_FIFO.BUFFER.value.table[3923]), INT_ENUM},*)
(*DBG:    {&(RES0__INSTANCE0.MY_BAD_FIFO.BUFFER.value.table[3924]), INT_ENUM},*)
(*DBG:    {&(RES0__INSTANCE0.MY_BAD_FIFO.BUFFER.value.table[3925]), INT_ENUM},*)
(*DBG:    {&(RES0__INSTANCE0.MY_BAD_FIFO.BUFFER.value.table[3926]), INT_ENUM},*)
(*DBG:    {&(RES0__INSTANCE0.MY_BAD_FIFO.BUFFER.value.table[3927]), INT_ENUM},*)
(*DBG:    {&(RES0__INSTANCE0.MY_BAD_FIFO.BUFFER.value.table[3928]), INT_ENUM},*)
(*DBG:    {&(RES0__INSTANCE0.MY_BAD_FIFO.BUFFER.value.table[3929]), INT_ENUM},*)
(*DBG:    {&(RES0__INSTANCE0.MY_BAD_FIFO.BUFFER.value.table[3930]), INT_ENUM},*)
(*DBG:    {&(RES0__INSTANCE0.MY_BAD_FIFO.BUFFER.value.table[3931]), INT_ENUM},*)
(*DBG:    {&(RES0__INSTANCE0.MY_BAD_FIFO.BUFFER.value.table[3932]), INT_ENUM},*)
(*DBG:    {&(RES0__INSTANCE0.MY_BAD_FIFO.BUFFER.value.table[3933]), INT_ENUM},*)
(*DBG:    {&(RES0__INSTANCE0.MY_BAD_FIFO.BUFFER.value.table[3934]), INT_ENUM},*)
(*DBG:    {&(RES0__INSTANCE0.MY_BAD_FIFO.BUFFER.value.table[3935]), INT_ENUM},*)
(*DBG:    {&(RES0__INSTANCE0.MY_BAD_FIFO.BUFFER.value.table[3936]), INT_ENUM},*)
(*DBG:    {&(RES0__INSTANCE0.MY_BAD_FIFO.BUFFER.value.table[3937]), INT_ENUM},*)
(*DBG:    {&(RES0__INSTANCE0.MY_BAD_FIFO.BUFFER.value.table[3938]), INT_ENUM},*)
(*DBG:    {&(RES0__INSTANCE0.MY_BAD_FIFO.BUFFER.value.table[3939]), INT_ENUM},*)
(*DBG:    {&(RES0__INSTANCE0.MY_BAD_FIFO.BUFFER.value.table[3940]), INT_ENUM},*)
(*DBG:    {&(RES0__INSTANCE0.MY_BAD_FIFO.BUFFER.value.table[3941]), INT_ENUM},*)
(*DBG:    {&(RES0__INSTANCE0.MY_BAD_FIFO.BUFFER.value.table[3942]), INT_ENUM},*)
(*DBG:    {&(RES0__INSTANCE0.MY_BAD_FIFO.BUFFER.value.table[3943]), INT_ENUM},*)
(*DBG:    {&(RES0__INSTANCE0.MY_BAD_FIFO.BUFFER.value.table[3944]), INT_ENUM},*)
(*DBG:    {&(RES0__INSTANCE0.MY_BAD_FIFO.BUFFER.value.table[3945]), INT_ENUM},*)
(*DBG:    {&(RES0__INSTANCE0.MY_BAD_FIFO.BUFFER.value.table[3946]), INT_ENUM},*)
(*DBG:    {&(RES0__INSTANCE0.MY_BAD_FIFO.BUFFER.value.table[3947]), INT_ENUM},*)
(*DBG:    {&(RES0__INSTANCE0.MY_BAD_FIFO.BUFFER.value.table[3948]), INT_ENUM},*)
(*DBG:    {&(RES0__INSTANCE0.MY_BAD_FIFO.BUFFER.value.table[3949]), INT_ENUM},*)
(*DBG:    {&(RES0__INSTANCE0.MY_BAD_FIFO.BUFFER.value.table[3950]), INT_ENUM},*)
(*DBG:    {&(RES0__INSTANCE0.MY_BAD_FIFO.BUFFER.value.table[3951]), INT_ENUM},*)
(*DBG:    {&(RES0__INSTANCE0.MY_BAD_FIFO.BUFFER.value.table[3952]), INT_ENUM},*)
(*DBG:    {&(RES0__INSTANCE0.MY_BAD_FIFO.BUFFER.value.table[3953]), INT_ENUM},*)
(*DBG:    {&(RES0__INSTANCE0.MY_BAD_FIFO.BUFFER.value.table[3954]), INT_ENUM},*)
(*DBG:    {&(RES0__INSTANCE0.MY_BAD_FIFO.BUFFER.value.table[3955]), INT_ENUM},*)
(*DBG:    {&(RES0__INSTANCE0.MY_BAD_FIFO.BUFFER.value.table[3956]), INT_ENUM},*)
(*DBG:    {&(RES0__INSTANCE0.MY_BAD_FIFO.BUFFER.value.table[3957]), INT_ENUM},*)
(*DBG:    {&(RES0__INSTANCE0.MY_BAD_FIFO.BUFFER.value.table[3958]), INT_ENUM},*)
(*DBG:    {&(RES0__INSTANCE0.MY_BAD_FIFO.BUFFER.value.table[3959]), INT_ENUM},*)
(*DBG:    {&(RES0__INSTANCE0.MY_BAD_FIFO.BUFFER.value.table[3960]), INT_ENUM},*)
(*DBG:    {&(RES0__INSTANCE0.MY_BAD_FIFO.BUFFER.value.table[3961]), INT_ENUM},*)
(*DBG:    {&(RES0__INSTANCE0.MY_BAD_FIFO.BUFFER.value.table[3962]), INT_ENUM},*)
(*DBG:    {&(RES0__INSTANCE0.MY_BAD_FIFO.BUFFER.value.table[3963]), INT_ENUM},*)
(*DBG:    {&(RES0__INSTANCE0.MY_BAD_FIFO.BUFFER.value.table[3964]), INT_ENUM},*)
(*DBG:    {&(RES0__INSTANCE0.MY_BAD_FIFO.BUFFER.value.table[3965]), INT_ENUM},*)
(*DBG:    {&(RES0__INSTANCE0.MY_BAD_FIFO.BUFFER.value.table[3966]), INT_ENUM},*)
(*DBG:    {&(RES0__INSTANCE0.MY_BAD_FIFO.BUFFER.value.table[3967]), INT_ENUM},*)
(*DBG:    {&(RES0__INSTANCE0.MY_BAD_FIFO.BUFFER.value.table[3968]), INT_ENUM},*)
(*DBG:    {&(RES0__INSTANCE0.MY_BAD_FIFO.BUFFER.value.table[3969]), INT_ENUM},*)
(*DBG:    {&(RES0__INSTANCE0.MY_BAD_FIFO.BUFFER.value.table[3970]), INT_ENUM},*)
(*DBG:    {&(RES0__INSTANCE0.MY_BAD_FIFO.BUFFER.value.table[3971]), INT_ENUM},*)
(*DBG:    {&(RES0__INSTANCE0.MY_BAD_FIFO.BUFFER.value.table[3972]), INT_ENUM},*)
(*DBG:    {&(RES0__INSTANCE0.MY_BAD_FIFO.BUFFER.value.table[3973]), INT_ENUM},*)
(*DBG:    {&(RES0__INSTANCE0.MY_BAD_FIFO.BUFFER.value.table[3974]), INT_ENUM},*)
(*DBG:    {&(RES0__INSTANCE0.MY_BAD_FIFO.BUFFER.value.table[3975]), INT_ENUM},*)
(*DBG:    {&(RES0__INSTANCE0.MY_BAD_FIFO.BUFFER.value.table[3976]), INT_ENUM},*)
(*DBG:    {&(RES0__INSTANCE0.MY_BAD_FIFO.BUFFER.value.table[3977]), INT_ENUM},*)
(*DBG:    {&(RES0__INSTANCE0.MY_BAD_FIFO.BUFFER.value.table[3978]), INT_ENUM},*)
(*DBG:    {&(RES0__INSTANCE0.MY_BAD_FIFO.BUFFER.value.table[3979]), INT_ENUM},*)
(*DBG:    {&(RES0__INSTANCE0.MY_BAD_FIFO.BUFFER.value.table[3980]), INT_ENUM},*)
(*DBG:    {&(RES0__INSTANCE0.MY_BAD_FIFO.BUFFER.value.table[3981]), INT_ENUM},*)
(*DBG:    {&(RES0__INSTANCE0.MY_BAD_FIFO.BUFFER.value.table[3982]), INT_ENUM},*)
(*DBG:    {&(RES0__INSTANCE0.MY_BAD_FIFO.BUFFER.value.table[3983]), INT_ENUM},*)
(*DBG:    {&(RES0__INSTANCE0.MY_BAD_FIFO.BUFFER.value.table[3984]), INT_ENUM},*)
(*DBG:    {&(RES0__INSTANCE0.MY_BAD_FIFO.BUFFER.value.table[3985]), INT_ENUM},*)
(*DBG:    {&(RES0__INSTANCE0.MY_BAD_FIFO.BUFFER.value.table[3986]), INT_ENUM},*)
(*DBG:    {&(RES0__INSTANCE0.MY_BAD_FIFO.BUFFER.value.table[3987]), INT_ENUM},*)
(*DBG:    {&(RES0__INSTANCE0.MY_BAD_FIFO.BUFFER.value.table[3988]), INT_ENUM},*)
(*DBG:    {&(RES0__INSTANCE0.MY_BAD_FIFO.BUFFER.value.table[3989]), INT_ENUM},*)
(*DBG:    {&(RES0__INSTANCE0.MY_BAD_FIFO.BUFFER.value.table[3990]), INT_ENUM},*)
(*DBG:    {&(RES0__INSTANCE0.MY_BAD_FIFO.BUFFER.value.table[3991]), INT_ENUM},*)
(*DBG:    {&(RES0__INSTANCE0.MY_BAD_FIFO.BUFFER.value.table[3992]), INT_ENUM},*)
(*DBG:    {&(RES0__INSTANCE0.MY_BAD_FIFO.BUFFER.value.table[3993]), INT_ENUM},*)
(*DBG:    {&(RES0__INSTANCE0.MY_BAD_FIFO.BUFFER.value.table[3994]), INT_ENUM},*)
(*DBG:    {&(RES0__INSTANCE0.MY_BAD_FIFO.BUFFER.value.table[3995]), INT_ENUM},*)
(*DBG:    {&(RES0__INSTANCE0.MY_BAD_FIFO.BUFFER.value.table[3996]), INT_ENUM},*)
(*DBG:    {&(RES0__INSTANCE0.MY_BAD_FIFO.BUFFER.value.table[3997]), INT_ENUM},*)
(*DBG:    {&(RES0__INSTANCE0.MY_BAD_FIFO.BUFFER.value.table[3998]), INT_ENUM},*)
(*DBG:    {&(RES0__INSTANCE0.MY_BAD_FIFO.BUFFER.value.table[3999]), INT_ENUM},*)
(*DBG:    {&(RES0__INSTANCE0.MY_BAD_FIFO.BUFFER.value.table[4000]), INT_ENUM},*)
(*DBG:    {&(RES0__INSTANCE0.MY_BAD_FIFO.BUFFER.value.table[4001]), INT_ENUM},*)
(*DBG:    {&(RES0__INSTANCE0.MY_BAD_FIFO.BUFFER.value.table[4002]), INT_ENUM},*)
(*DBG:    {&(RES0__INSTANCE0.MY_BAD_FIFO.BUFFER.value.table[4003]), INT_ENUM},*)
(*DBG:    {&(RES0__INSTANCE0.MY_BAD_FIFO.BUFFER.value.table[4004]), INT_ENUM},*)
(*DBG:    {&(RES0__INSTANCE0.MY_BAD_FIFO.BUFFER.value.table[4005]), INT_ENUM},*)
(*DBG:    {&(RES0__INSTANCE0.MY_BAD_FIFO.BUFFER.value.table[4006]), INT_ENUM},*)
(*DBG:    {&(RES0__INSTANCE0.MY_BAD_FIFO.BUFFER.value.table[4007]), INT_ENUM},*)
(*DBG:    {&(RES0__INSTANCE0.MY_BAD_FIFO.BUFFER.value.table[4008]), INT_ENUM},*)
(*DBG:    {&(RES0__INSTANCE0.MY_BAD_FIFO.BUFFER.value.table[4009]), INT_ENUM},*)
(*DBG:    {&(RES0__INSTANCE0.MY_BAD_FIFO.BUFFER.value.table[4010]), INT_ENUM},*)
(*DBG:    {&(RES0__INSTANCE0.MY_BAD_FIFO.BUFFER.value.table[4011]), INT_ENUM},*)
(*DBG:    {&(RES0__INSTANCE0.MY_BAD_FIFO.BUFFER.value.table[4012]), INT_ENUM},*)
(*DBG:    {&(RES0__INSTANCE0.MY_BAD_FIFO.BUFFER.value.table[4013]), INT_ENUM},*)
(*DBG:    {&(RES0__INSTANCE0.MY_BAD_FIFO.BUFFER.value.table[4014]), INT_ENUM},*)
(*DBG:    {&(RES0__INSTANCE0.MY_BAD_FIFO.BUFFER.value.table[4015]), INT_ENUM},*)
(*DBG:    {&(RES0__INSTANCE0.MY_BAD_FIFO.BUFFER.value.table[4016]), INT_ENUM},*)
(*DBG:    {&(RES0__INSTANCE0.MY_BAD_FIFO.BUFFER.value.table[4017]), INT_ENUM},*)
(*DBG:    {&(RES0__INSTANCE0.MY_BAD_FIFO.BUFFER.value.table[4018]), INT_ENUM},*)
(*DBG:    {&(RES0__INSTANCE0.MY_BAD_FIFO.BUFFER.value.table[4019]), INT_ENUM},*)
(*DBG:    {&(RES0__INSTANCE0.MY_BAD_FIFO.BUFFER.value.table[4020]), INT_ENUM},*)
(*DBG:    {&(RES0__INSTANCE0.MY_BAD_FIFO.BUFFER.value.table[4021]), INT_ENUM},*)
(*DBG:    {&(RES0__INSTANCE0.MY_BAD_FIFO.BUFFER.value.table[4022]), INT_ENUM},*)
(*DBG:    {&(RES0__INSTANCE0.MY_BAD_FIFO.BUFFER.value.table[4023]), INT_ENUM},*)
(*DBG:    {&(RES0__INSTANCE0.MY_BAD_FIFO.BUFFER.value.table[4024]), INT_ENUM},*)
(*DBG:    {&(RES0__INSTANCE0.MY_BAD_FIFO.BUFFER.value.table[4025]), INT_ENUM},*)
(*DBG:    {&(RES0__INSTANCE0.MY_BAD_FIFO.BUFFER.value.table[4026]), INT_ENUM},*)
(*DBG:    {&(RES0__INSTANCE0.MY_BAD_FIFO.BUFFER.value.table[4027]), INT_ENUM},*)
(*DBG:    {&(RES0__INSTANCE0.MY_BAD_FIFO.BUFFER.value.table[4028]), INT_ENUM},*)
(*DBG:    {&(RES0__INSTANCE0.MY_BAD_FIFO.BUFFER.value.table[4029]), INT_ENUM},*)
(*DBG:    {&(RES0__INSTANCE0.MY_BAD_FIFO.BUFFER.value.table[4030]), INT_ENUM},*)
(*DBG:    {&(RES0__INSTANCE0.MY_BAD_FIFO.BUFFER.value.table[4031]), INT_ENUM},*)
(*DBG:    {&(RES0__INSTANCE0.MY_BAD_FIFO.BUFFER.value.table[4032]), INT_ENUM},*)
(*DBG:    {&(RES0__INSTANCE0.MY_BAD_FIFO.BUFFER.value.table[4033]), INT_ENUM},*)
(*DBG:    {&(RES0__INSTANCE0.MY_BAD_FIFO.BUFFER.value.table[4034]), INT_ENUM},*)
(*DBG:    {&(RES0__INSTANCE0.MY_BAD_FIFO.BUFFER.value.table[4035]), INT_ENUM},*)
(*DBG:    {&(RES0__INSTANCE0.MY_BAD_FIFO.BUFFER.value.table[4036]), INT_ENUM},*)
(*DBG:    {&(RES0__INSTANCE0.MY_BAD_FIFO.BUFFER.value.table[4037]), INT_ENUM},*)
(*DBG:    {&(RES0__INSTANCE0.MY_BAD_FIFO.BUFFER.value.table[4038]), INT_ENUM},*)
(*DBG:    {&(RES0__INSTANCE0.MY_BAD_FIFO.BUFFER.value.table[4039]), INT_ENUM},*)
(*DBG:    {&(RES0__INSTANCE0.MY_BAD_FIFO.BUFFER.value.table[4040]), INT_ENUM},*)
(*DBG:    {&(RES0__INSTANCE0.MY_BAD_FIFO.BUFFER.value.table[4041]), INT_ENUM},*)
(*DBG:    {&(RES0__INSTANCE0.MY_BAD_FIFO.BUFFER.value.table[4042]), INT_ENUM},*)
(*DBG:    {&(RES0__INSTANCE0.MY_BAD_FIFO.BUFFER.value.table[4043]), INT_ENUM},*)
(*DBG:    {&(RES0__INSTANCE0.MY_BAD_FIFO.BUFFER.value.table[4044]), INT_ENUM},*)
(*DBG:    {&(RES0__INSTANCE0.MY_BAD_FIFO.BUFFER.value.table[4045]), INT_ENUM},*)
(*DBG:    {&(RES0__INSTANCE0.MY_BAD_FIFO.BUFFER.value.table[4046]), INT_ENUM},*)
(*DBG:    {&(RES0__INSTANCE0.MY_BAD_FIFO.BUFFER.value.table[4047]), INT_ENUM},*)
(*DBG:    {&(RES0__INSTANCE0.MY_BAD_FIFO.BUFFER.value.table[4048]), INT_ENUM},*)
(*DBG:    {&(RES0__INSTANCE0.MY_BAD_FIFO.BUFFER.value.table[4049]), INT_ENUM},*)
(*DBG:    {&(RES0__INSTANCE0.MY_BAD_FIFO.BUFFER.value.table[4050]), INT_ENUM},*)
(*DBG:    {&(RES0__INSTANCE0.MY_BAD_FIFO.BUFFER.value.table[4051]), INT_ENUM},*)
(*DBG:    {&(RES0__INSTANCE0.MY_BAD_FIFO.BUFFER.value.table[4052]), INT_ENUM},*)
(*DBG:    {&(RES0__INSTANCE0.MY_BAD_FIFO.BUFFER.value.table[4053]), INT_ENUM},*)
(*DBG:    {&(RES0__INSTANCE0.MY_BAD_FIFO.BUFFER.value.table[4054]), INT_ENUM},*)
(*DBG:    {&(RES0__INSTANCE0.MY_BAD_FIFO.BUFFER.value.table[4055]), INT_ENUM},*)
(*DBG:    {&(RES0__INSTANCE0.MY_BAD_FIFO.BUFFER.value.table[4056]), INT_ENUM},*)
(*DBG:    {&(RES0__INSTANCE0.MY_BAD_FIFO.BUFFER.value.table[4057]), INT_ENUM},*)
(*DBG:    {&(RES0__INSTANCE0.MY_BAD_FIFO.BUFFER.value.table[4058]), INT_ENUM},*)
(*DBG:    {&(RES0__INSTANCE0.MY_BAD_FIFO.BUFFER.value.table[4059]), INT_ENUM},*)
(*DBG:    {&(RES0__INSTANCE0.MY_BAD_FIFO.BUFFER.value.table[4060]), INT_ENUM},*)
(*DBG:    {&(RES0__INSTANCE0.MY_BAD_FIFO.BUFFER.value.table[4061]), INT_ENUM},*)
(*DBG:    {&(RES0__INSTANCE0.MY_BAD_FIFO.BUFFER.value.table[4062]), INT_ENUM},*)
(*DBG:    {&(RES0__INSTANCE0.MY_BAD_FIFO.BUFFER.value.table[4063]), INT_ENUM},*)
(*DBG:    {&(RES0__INSTANCE0.MY_BAD_FIFO.BUFFER.value.table[4064]), INT_ENUM},*)
(*DBG:    {&(RES0__INSTANCE0.MY_BAD_FIFO.BUFFER.value.table[4065]), INT_ENUM},*)
(*DBG:    {&(RES0__INSTANCE0.MY_BAD_FIFO.BUFFER.value.table[4066]), INT_ENUM},*)
(*DBG:    {&(RES0__INSTANCE0.MY_BAD_FIFO.BUFFER.value.table[4067]), INT_ENUM},*)
(*DBG:    {&(RES0__INSTANCE0.MY_BAD_FIFO.BUFFER.value.table[4068]), INT_ENUM},*)
(*DBG:    {&(RES0__INSTANCE0.MY_BAD_FIFO.BUFFER.value.table[4069]), INT_ENUM},*)
(*DBG:    {&(RES0__INSTANCE0.MY_BAD_FIFO.BUFFER.value.table[4070]), INT_ENUM},*)
(*DBG:    {&(RES0__INSTANCE0.MY_BAD_FIFO.BUFFER.value.table[4071]), INT_ENUM},*)
(*DBG:    {&(RES0__INSTANCE0.MY_BAD_FIFO.BUFFER.value.table[4072]), INT_ENUM},*)
(*DBG:    {&(RES0__INSTANCE0.MY_BAD_FIFO.BUFFER.value.table[4073]), INT_ENUM},*)
(*DBG:    {&(RES0__INSTANCE0.MY_BAD_FIFO.BUFFER.value.table[4074]), INT_ENUM},*)
(*DBG:    {&(RES0__INSTANCE0.MY_BAD_FIFO.BUFFER.value.table[4075]), INT_ENUM},*)
(*DBG:    {&(RES0__INSTANCE0.MY_BAD_FIFO.BUFFER.value.table[4076]), INT_ENUM},*)
(*DBG:    {&(RES0__INSTANCE0.MY_BAD_FIFO.BUFFER.value.table[4077]), INT_ENUM},*)
(*DBG:    {&(RES0__INSTANCE0.MY_BAD_FIFO.BUFFER.value.table[4078]), INT_ENUM},*)
(*DBG:    {&(RES0__INSTANCE0.MY_BAD_FIFO.BUFFER.value.table[4079]), INT_ENUM},*)
(*DBG:    {&(RES0__INSTANCE0.MY_BAD_FIFO.BUFFER.value.table[4080]), INT_ENUM},*)
(*DBG:    {&(RES0__INSTANCE0.MY_BAD_FIFO.BUFFER.value.table[4081]), INT_ENUM},*)
(*DBG:    {&(RES0__INSTANCE0.MY_BAD_FIFO.BUFFER.value.table[4082]), INT_ENUM},*)
(*DBG:    {&(RES0__INSTANCE0.MY_BAD_FIFO.BUFFER.value.table[4083]), INT_ENUM},*)
(*DBG:    {&(RES0__INSTANCE0.MY_BAD_FIFO.BUFFER.value.table[4084]), INT_ENUM},*)
(*DBG:    {&(RES0__INSTANCE0.MY_BAD_FIFO.BUFFER.value.table[4085]), INT_ENUM},*)
(*DBG:    {&(RES0__INSTANCE0.MY_BAD_FIFO.BUFFER.value.table[4086]), INT_ENUM},*)
(*DBG:    {&(RES0__INSTANCE0.MY_BAD_FIFO.BUFFER.value.table[4087]), INT_ENUM},*)
(*DBG:    {&(RES0__INSTANCE0.MY_BAD_FIFO.BUFFER.value.table[4088]), INT_ENUM},*)
(*DBG:    {&(RES0__INSTANCE0.MY_BAD_FIFO.BUFFER.value.table[4089]), INT_ENUM},*)
(*DBG:    {&(RES0__INSTANCE0.MY_BAD_FIFO.BUFFER.value.table[4090]), INT_ENUM},*)
(*DBG:    {&(RES0__INSTANCE0.MY_BAD_FIFO.BUFFER.value.table[4091]), INT_ENUM},*)
(*DBG:    {&(RES0__INSTANCE0.MY_BAD_FIFO.BUFFER.value.table[4092]), INT_ENUM},*)
(*DBG:    {&(RES0__INSTANCE0.MY_BAD_FIFO.BUFFER.value.table[4093]), INT_ENUM},*)
(*DBG:    {&(RES0__INSTANCE0.MY_BAD_FIFO.BUFFER.value.table[4094]), INT_ENUM},*)
(*DBG:    {&(RES0__INSTANCE0.MY_BAD_FIFO.BUFFER.value.table[4095]), INT_ENUM},*)
(*DBG:    {&(RES0__INSTANCE0.MY_BAD_FIFO.BUFFER.value.table[4096]), INT_ENUM},*)
(*DBG:    {&(RES0__INSTANCE0.MY_BAD_FIFO.BUFFER.value.table[4097]), INT_ENUM},*)
(*DBG:    {&(RES0__INSTANCE0.MY_BAD_FIFO.BUFFER.value.table[4098]), INT_ENUM},*)
(*DBG:    {&(RES0__INSTANCE0.MY_BAD_FIFO.BUFFER.value.table[4099]), INT_ENUM},*)
(*DBG:    {&(RES0__INSTANCE0.MY_BAD_FIFO.BUFFER.value.table[4100]), INT_ENUM},*)
(*DBG:    {&(RES0__INSTANCE0.MY_BAD_FIFO.BUFFER.value.table[4101]), INT_ENUM},*)
(*DBG:    {&(RES0__INSTANCE0.MY_BAD_FIFO.BUFFER.value.table[4102]), INT_ENUM},*)
(*DBG:    {&(RES0__INSTANCE0.MY_BAD_FIFO.BUFFER.value.table[4103]), INT_ENUM},*)
(*DBG:    {&(RES0__INSTANCE0.MY_BAD_FIFO.BUFFER.value.table[4104]), INT_ENUM},*)
(*DBG:    {&(RES0__INSTANCE0.MY_BAD_FIFO.BUFFER.value.table[4105]), INT_ENUM},*)
(*DBG:    {&(RES0__INSTANCE0.MY_BAD_FIFO.BUFFER.value.table[4106]), INT_ENUM},*)
(*DBG:    {&(RES0__INSTANCE0.MY_BAD_FIFO.BUFFER.value.table[4107]), INT_ENUM},*)
(*DBG:    {&(RES0__INSTANCE0.MY_BAD_FIFO.BUFFER.value.table[4108]), INT_ENUM},*)
(*DBG:    {&(RES0__INSTANCE0.MY_BAD_FIFO.BUFFER.value.table[4109]), INT_ENUM},*)
(*DBG:    {&(RES0__INSTANCE0.MY_BAD_FIFO.BUFFER.value.table[4110]), INT_ENUM},*)
(*DBG:    {&(RES0__INSTANCE0.MY_BAD_FIFO.BUFFER.value.table[4111]), INT_ENUM},*)
(*DBG:    {&(RES0__INSTANCE0.MY_BAD_FIFO.BUFFER.value.table[4112]), INT_ENUM},*)
(*DBG:    {&(RES0__INSTANCE0.MY_BAD_FIFO.BUFFER.value.table[4113]), INT_ENUM},*)
(*DBG:    {&(RES0__INSTANCE0.MY_BAD_FIFO.BUFFER.value.table[4114]), INT_ENUM},*)
(*DBG:    {&(RES0__INSTANCE0.MY_BAD_FIFO.BUFFER.value.table[4115]), INT_ENUM},*)
(*DBG:    {&(RES0__INSTANCE0.MY_BAD_FIFO.BUFFER.value.table[4116]), INT_ENUM},*)
(*DBG:    {&(RES0__INSTANCE0.MY_BAD_FIFO.BUFFER.value.table[4117]), INT_ENUM},*)
(*DBG:    {&(RES0__INSTANCE0.MY_BAD_FIFO.BUFFER.value.table[4118]), INT_ENUM},*)
(*DBG:    {&(RES0__INSTANCE0.MY_BAD_FIFO.BUFFER.value.table[4119]), INT_ENUM},*)
(*DBG:    {&(RES0__INSTANCE0.MY_BAD_FIFO.BUFFER.value.table[4120]), INT_ENUM},*)
(*DBG:    {&(RES0__INSTANCE0.MY_BAD_FIFO.BUFFER.value.table[4121]), INT_ENUM},*)
(*DBG:    {&(RES0__INSTANCE0.MY_BAD_FIFO.BUFFER.value.table[4122]), INT_ENUM},*)
(*DBG:    {&(RES0__INSTANCE0.MY_BAD_FIFO.BUFFER.value.table[4123]), INT_ENUM},*)
(*DBG:    {&(RES0__INSTANCE0.MY_BAD_FIFO.BUFFER.value.table[4124]), INT_ENUM},*)
(*DBG:    {&(RES0__INSTANCE0.MY_BAD_FIFO.BUFFER.value.table[4125]), INT_ENUM},*)
(*DBG:    {&(RES0__INSTANCE0.MY_BAD_FIFO.BUFFER.value.table[4126]), INT_ENUM},*)
(*DBG:    {&(RES0__INSTANCE0.MY_BAD_FIFO.BUFFER.value.table[4127]), INT_ENUM},*)
(*DBG:    {&(RES0__INSTANCE0.MY_BAD_FIFO.BUFFER.value.table[4128]), INT_ENUM},*)
(*DBG:    {&(RES0__INSTANCE0.MY_BAD_FIFO.BUFFER.value.table[4129]), INT_ENUM},*)
(*DBG:    {&(RES0__INSTANCE0.MY_BAD_FIFO.BUFFER.value.table[4130]), INT_ENUM},*)
(*DBG:    {&(RES0__INSTANCE0.MY_BAD_FIFO.BUFFER.value.table[4131]), INT_ENUM},*)
(*DBG:    {&(RES0__INSTANCE0.MY_BAD_FIFO.BUFFER.value.table[4132]), INT_ENUM},*)
(*DBG:    {&(RES0__INSTANCE0.MY_BAD_FIFO.BUFFER.value.table[4133]), INT_ENUM},*)
(*DBG:    {&(RES0__INSTANCE0.MY_BAD_FIFO.BUFFER.value.table[4134]), INT_ENUM},*)
(*DBG:    {&(RES0__INSTANCE0.MY_BAD_FIFO.BUFFER.value.table[4135]), INT_ENUM},*)
(*DBG:    {&(RES0__INSTANCE0.MY_BAD_FIFO.BUFFER.value.table[4136]), INT_ENUM},*)
(*DBG:    {&(RES0__INSTANCE0.MY_BAD_FIFO.BUFFER.value.table[4137]), INT_ENUM},*)
(*DBG:    {&(RES0__INSTANCE0.MY_BAD_FIFO.BUFFER.value.table[4138]), INT_ENUM},*)
(*DBG:    {&(RES0__INSTANCE0.MY_BAD_FIFO.BUFFER.value.table[4139]), INT_ENUM},*)
(*DBG:    {&(RES0__INSTANCE0.MY_BAD_FIFO.BUFFER.value.table[4140]), INT_ENUM},*)
(*DBG:    {&(RES0__INSTANCE0.MY_BAD_FIFO.BUFFER.value.table[4141]), INT_ENUM},*)
(*DBG:    {&(RES0__INSTANCE0.MY_BAD_FIFO.BUFFER.value.table[4142]), INT_ENUM},*)
(*DBG:    {&(RES0__INSTANCE0.MY_BAD_FIFO.BUFFER.value.table[4143]), INT_ENUM},*)
(*DBG:    {&(RES0__INSTANCE0.MY_BAD_FIFO.BUFFER.value.table[4144]), INT_ENUM},*)
(*DBG:    {&(RES0__INSTANCE0.MY_BAD_FIFO.BUFFER.value.table[4145]), INT_ENUM},*)
(*DBG:    {&(RES0__INSTANCE0.MY_BAD_FIFO.BUFFER.value.table[4146]), INT_ENUM},*)
(*DBG:    {&(RES0__INSTANCE0.MY_BAD_FIFO.BUFFER.value.table[4147]), INT_ENUM},*)
(*DBG:    {&(RES0__INSTANCE0.MY_BAD_FIFO.BUFFER.value.table[4148]), INT_ENUM},*)
(*DBG:    {&(RES0__INSTANCE0.MY_BAD_FIFO.BUFFER.value.table[4149]), INT_ENUM},*)
(*DBG:    {&(RES0__INSTANCE0.MY_BAD_FIFO.BUFFER.value.table[4150]), INT_ENUM},*)
(*DBG:    {&(RES0__INSTANCE0.MY_BAD_FIFO.BUFFER.value.table[4151]), INT_ENUM},*)
(*DBG:    {&(RES0__INSTANCE0.MY_BAD_FIFO.BUFFER.value.table[4152]), INT_ENUM},*)
(*DBG:    {&(RES0__INSTANCE0.MY_BAD_FIFO.BUFFER.value.table[4153]), INT_ENUM},*)
(*DBG:    {&(RES0__INSTANCE0.MY_BAD_FIFO.BUFFER.value.table[4154]), INT_ENUM},*)
(*DBG:    {&(RES0__INSTANCE0.MY_BAD_FIFO.BUFFER.value.table[4155]), INT_ENUM},*)
(*DBG:    {&(RES0__INSTANCE0.MY_BAD_FIFO.BUFFER.value.table[4156]), INT_ENUM},*)
(*DBG:    {&(RES0__INSTANCE0.MY_BAD_FIFO.BUFFER.value.table[4157]), INT_ENUM},*)
(*DBG:    {&(RES0__INSTANCE0.MY_BAD_FIFO.BUFFER.value.table[4158]), INT_ENUM},*)
(*DBG:    {&(RES0__INSTANCE0.MY_BAD_FIFO.BUFFER.value.table[4159]), INT_ENUM},*)
(*DBG:    {&(RES0__INSTANCE0.MY_BAD_FIFO.BUFFER.value.table[4160]), INT_ENUM},*)
(*DBG:    {&(RES0__INSTANCE0.MY_BAD_FIFO.BUFFER.value.table[4161]), INT_ENUM},*)
(*DBG:    {&(RES0__INSTANCE0.MY_BAD_FIFO.BUFFER.value.table[4162]), INT_ENUM},*)
(*DBG:    {&(RES0__INSTANCE0.MY_BAD_FIFO.BUFFER.value.table[4163]), INT_ENUM},*)
(*DBG:    {&(RES0__INSTANCE0.MY_BAD_FIFO.BUFFER.value.table[4164]), INT_ENUM},*)
(*DBG:    {&(RES0__INSTANCE0.MY_BAD_FIFO.BUFFER.value.table[4165]), INT_ENUM},*)
(*DBG:    {&(RES0__INSTANCE0.MY_BAD_FIFO.BUFFER.value.table[4166]), INT_ENUM},*)
(*DBG:    {&(RES0__INSTANCE0.MY_BAD_FIFO.BUFFER.value.table[4167]), INT_ENUM},*)
(*DBG:    {&(RES0__INSTANCE0.MY_BAD_FIFO.BUFFER.value.table[4168]), INT_ENUM},*)
(*DBG:    {&(RES0__INSTANCE0.MY_BAD_FIFO.BUFFER.value.table[4169]), INT_ENUM},*)
(*DBG:    {&(RES0__INSTANCE0.MY_BAD_FIFO.BUFFER.value.table[4170]), INT_ENUM},*)
(*DBG:    {&(RES0__INSTANCE0.MY_BAD_FIFO.BUFFER.value.table[4171]), INT_ENUM},*)
(*DBG:    {&(RES0__INSTANCE0.MY_BAD_FIFO.BUFFER.value.table[4172]), INT_ENUM},*)
(*DBG:    {&(RES0__INSTANCE0.MY_BAD_FIFO.BUFFER.value.table[4173]), INT_ENUM},*)
(*DBG:    {&(RES0__INSTANCE0.MY_BAD_FIFO.BUFFER.value.table[4174]), INT_ENUM},*)
(*DBG:    {&(RES0__INSTANCE0.MY_BAD_FIFO.BUFFER.value.table[4175]), INT_ENUM},*)
(*DBG:    {&(RES0__INSTANCE0.MY_BAD_FIFO.BUFFER.value.table[4176]), INT_ENUM},*)
(*DBG:    {&(RES0__INSTANCE0.MY_BAD_FIFO.BUFFER.value.table[4177]), INT_ENUM},*)
(*DBG:    {&(RES0__INSTANCE0.MY_BAD_FIFO.BUFFER.value.table[4178]), INT_ENUM},*)
(*DBG:    {&(RES0__INSTANCE0.MY_BAD_FIFO.BUFFER.value.table[4179]), INT_ENUM},*)
(*DBG:    {&(RES0__INSTANCE0.MY_BAD_FIFO.BUFFER.value.table[4180]), INT_ENUM},*)
(*DBG:    {&(RES0__INSTANCE0.MY_BAD_FIFO.BUFFER.value.table[4181]), INT_ENUM},*)
(*DBG:    {&(RES0__INSTANCE0.MY_BAD_FIFO.BUFFER.value.table[4182]), INT_ENUM},*)
(*DBG:    {&(RES0__INSTANCE0.MY_BAD_FIFO.BUFFER.value.table[4183]), INT_ENUM},*)
(*DBG:    {&(RES0__INSTANCE0.MY_BAD_FIFO.BUFFER.value.table[4184]), INT_ENUM},*)
(*DBG:    {&(RES0__INSTANCE0.MY_BAD_FIFO.BUFFER.value.table[4185]), INT_ENUM},*)
(*DBG:    {&(RES0__INSTANCE0.MY_BAD_FIFO.BUFFER.value.table[4186]), INT_ENUM},*)
(*DBG:    {&(RES0__INSTANCE0.MY_BAD_FIFO.BUFFER.value.table[4187]), INT_ENUM},*)
(*DBG:    {&(RES0__INSTANCE0.MY_BAD_FIFO.BUFFER.value.table[4188]), INT_ENUM},*)
(*DBG:    {&(RES0__INSTANCE0.MY_BAD_FIFO.BUFFER.value.table[4189]), INT_ENUM},*)
(*DBG:    {&(RES0__INSTANCE0.MY_BAD_FIFO.BUFFER.value.table[4190]), INT_ENUM},*)
(*DBG:    {&(RES0__INSTANCE0.MY_BAD_FIFO.BUFFER.value.table[4191]), INT_ENUM},*)
(*DBG:    {&(RES0__INSTANCE0.MY_BAD_FIFO.BUFFER.value.table[4192]), INT_ENUM},*)
(*DBG:    {&(RES0__INSTANCE0.MY_BAD_FIFO.BUFFER.value.table[4193]), INT_ENUM},*)
(*DBG:    {&(RES0__INSTANCE0.MY_BAD_FIFO.BUFFER.value.table[4194]), INT_ENUM},*)
(*DBG:    {&(RES0__INSTANCE0.MY_BAD_FIFO.BUFFER.value.table[4195]), INT_ENUM},*)
(*DBG:    {&(RES0__INSTANCE0.MY_BAD_FIFO.BUFFER.value.table[4196]), INT_ENUM},*)
(*DBG:    {&(RES0__INSTANCE0.MY_BAD_FIFO.BUFFER.value.table[4197]), INT_ENUM},*)
(*DBG:    {&(RES0__INSTANCE0.MY_BAD_FIFO.BUFFER.value.table[4198]), INT_ENUM},*)
(*DBG:    {&(RES0__INSTANCE0.MY_BAD_FIFO.BUFFER.value.table[4199]), INT_ENUM},*)
(*DBG:    {&(RES0__INSTANCE0.MY_BAD_FIFO.BUFFER.value.table[4200]), INT_ENUM},*)
(*DBG:    {&(RES0__INSTANCE0.MY_BAD_FIFO.BUFFER.value.table[4201]), INT_ENUM},*)
(*DBG:    {&(RES0__INSTANCE0.MY_BAD_FIFO.BUFFER.value.table[4202]), INT_ENUM},*)
(*DBG:    {&(RES0__INSTANCE0.MY_BAD_FIFO.BUFFER.value.table[4203]), INT_ENUM},*)
(*DBG:    {&(RES0__INSTANCE0.MY_BAD_FIFO.BUFFER.value.table[4204]), INT_ENUM},*)
(*DBG:    {&(RES0__INSTANCE0.MY_BAD_FIFO.BUFFER.value.table[4205]), INT_ENUM},*)
(*DBG:    {&(RES0__INSTANCE0.MY_BAD_FIFO.BUFFER.value.table[4206]), INT_ENUM},*)
(*DBG:    {&(RES0__INSTANCE0.MY_BAD_FIFO.BUFFER.value.table[4207]), INT_ENUM},*)
(*DBG:    {&(RES0__INSTANCE0.MY_BAD_FIFO.BUFFER.value.table[4208]), INT_ENUM},*)
(*DBG:    {&(RES0__INSTANCE0.MY_BAD_FIFO.BUFFER.value.table[4209]), INT_ENUM},*)
(*DBG:    {&(RES0__INSTANCE0.MY_BAD_FIFO.BUFFER.value.table[4210]), INT_ENUM},*)
(*DBG:    {&(RES0__INSTANCE0.MY_BAD_FIFO.BUFFER.value.table[4211]), INT_ENUM},*)
(*DBG:    {&(RES0__INSTANCE0.MY_BAD_FIFO.BUFFER.value.table[4212]), INT_ENUM},*)
(*DBG:    {&(RES0__INSTANCE0.MY_BAD_FIFO.BUFFER.value.table[4213]), INT_ENUM},*)
(*DBG:    {&(RES0__INSTANCE0.MY_BAD_FIFO.BUFFER.value.table[4214]), INT_ENUM},*)
(*DBG:    {&(RES0__INSTANCE0.MY_BAD_FIFO.BUFFER.value.table[4215]), INT_ENUM},*)
(*DBG:    {&(RES0__INSTANCE0.MY_BAD_FIFO.BUFFER.value.table[4216]), INT_ENUM},*)
(*DBG:    {&(RES0__INSTANCE0.MY_BAD_FIFO.BUFFER.value.table[4217]), INT_ENUM},*)
(*DBG:    {&(RES0__INSTANCE0.MY_BAD_FIFO.BUFFER.value.table[4218]), INT_ENUM},*)
(*DBG:    {&(RES0__INSTANCE0.MY_BAD_FIFO.BUFFER.value.table[4219]), INT_ENUM},*)
(*DBG:    {&(RES0__INSTANCE0.MY_BAD_FIFO.BUFFER.value.table[4220]), INT_ENUM},*)
(*DBG:    {&(RES0__INSTANCE0.MY_BAD_FIFO.BUFFER.value.table[4221]), INT_ENUM},*)
(*DBG:    {&(RES0__INSTANCE0.MY_BAD_FIFO.BUFFER.value.table[4222]), INT_ENUM},*)
(*DBG:    {&(RES0__INSTANCE0.MY_BAD_FIFO.BUFFER.value.table[4223]), INT_ENUM},*)
(*DBG:    {&(RES0__INSTANCE0.MY_BAD_FIFO.BUFFER.value.table[4224]), INT_ENUM},*)
(*DBG:    {&(RES0__INSTANCE0.MY_BAD_FIFO.BUFFER.value.table[4225]), INT_ENUM},*)
(*DBG:    {&(RES0__INSTANCE0.MY_BAD_FIFO.BUFFER.value.table[4226]), INT_ENUM},*)
(*DBG:    {&(RES0__INSTANCE0.MY_BAD_FIFO.BUFFER.value.table[4227]), INT_ENUM},*)
(*DBG:    {&(RES0__INSTANCE0.MY_BAD_FIFO.BUFFER.value.table[4228]), INT_ENUM},*)
(*DBG:    {&(RES0__INSTANCE0.MY_BAD_FIFO.BUFFER.value.table[4229]), INT_ENUM},*)
(*DBG:    {&(RES0__INSTANCE0.MY_BAD_FIFO.BUFFER.value.table[4230]), INT_ENUM},*)
(*DBG:    {&(RES0__INSTANCE0.MY_BAD_FIFO.BUFFER.value.table[4231]), INT_ENUM},*)
(*DBG:    {&(RES0__INSTANCE0.MY_BAD_FIFO.BUFFER.value.table[4232]), INT_ENUM},*)
(*DBG:    {&(RES0__INSTANCE0.MY_BAD_FIFO.BUFFER.value.table[4233]), INT_ENUM},*)
(*DBG:    {&(RES0__INSTANCE0.MY_BAD_FIFO.BUFFER.value.table[4234]), INT_ENUM},*)
(*DBG:    {&(RES0__INSTANCE0.MY_BAD_FIFO.BUFFER.value.table[4235]), INT_ENUM},*)
(*DBG:    {&(RES0__INSTANCE0.MY_BAD_FIFO.BUFFER.value.table[4236]), INT_ENUM},*)
(*DBG:    {&(RES0__INSTANCE0.MY_BAD_FIFO.BUFFER.value.table[4237]), INT_ENUM},*)
(*DBG:    {&(RES0__INSTANCE0.MY_BAD_FIFO.BUFFER.value.table[4238]), INT_ENUM},*)
(*DBG:    {&(RES0__INSTANCE0.MY_BAD_FIFO.BUFFER.value.table[4239]), INT_ENUM},*)
(*DBG:    {&(RES0__INSTANCE0.MY_BAD_FIFO.BUFFER.value.table[4240]), INT_ENUM},*)
(*DBG:    {&(RES0__INSTANCE0.MY_BAD_FIFO.BUFFER.value.table[4241]), INT_ENUM},*)
(*DBG:    {&(RES0__INSTANCE0.MY_BAD_FIFO.BUFFER.value.table[4242]), INT_ENUM},*)
(*DBG:    {&(RES0__INSTANCE0.MY_BAD_FIFO.BUFFER.value.table[4243]), INT_ENUM},*)
(*DBG:    {&(RES0__INSTANCE0.MY_BAD_FIFO.BUFFER.value.table[4244]), INT_ENUM},*)
(*DBG:    {&(RES0__INSTANCE0.MY_BAD_FIFO.BUFFER.value.table[4245]), INT_ENUM},*)
(*DBG:    {&(RES0__INSTANCE0.MY_BAD_FIFO.BUFFER.value.table[4246]), INT_ENUM},*)
(*DBG:    {&(RES0__INSTANCE0.MY_BAD_FIFO.BUFFER.value.table[4247]), INT_ENUM},*)
(*DBG:    {&(RES0__INSTANCE0.MY_BAD_FIFO.BUFFER.value.table[4248]), INT_ENUM},*)
(*DBG:    {&(RES0__INSTANCE0.MY_BAD_FIFO.BUFFER.value.table[4249]), INT_ENUM},*)
(*DBG:    {&(RES0__INSTANCE0.MY_BAD_FIFO.BUFFER.value.table[4250]), INT_ENUM},*)
(*DBG:    {&(RES0__INSTANCE0.MY_BAD_FIFO.BUFFER.value.table[4251]), INT_ENUM},*)
(*DBG:    {&(RES0__INSTANCE0.MY_BAD_FIFO.BUFFER.value.table[4252]), INT_ENUM},*)
(*DBG:    {&(RES0__INSTANCE0.MY_BAD_FIFO.BUFFER.value.table[4253]), INT_ENUM},*)
(*DBG:    {&(RES0__INSTANCE0.MY_BAD_FIFO.BUFFER.value.table[4254]), INT_ENUM},*)
(*DBG:    {&(RES0__INSTANCE0.MY_BAD_FIFO.BUFFER.value.table[4255]), INT_ENUM},*)
(*DBG:    {&(RES0__INSTANCE0.MY_BAD_FIFO.BUFFER.value.table[4256]), INT_ENUM},*)
(*DBG:    {&(RES0__INSTANCE0.MY_BAD_FIFO.BUFFER.value.table[4257]), INT_ENUM},*)
(*DBG:    {&(RES0__INSTANCE0.MY_BAD_FIFO.BUFFER.value.table[4258]), INT_ENUM},*)
(*DBG:    {&(RES0__INSTANCE0.MY_BAD_FIFO.BUFFER.value.table[4259]), INT_ENUM},*)
(*DBG:    {&(RES0__INSTANCE0.MY_BAD_FIFO.BUFFER.value.table[4260]), INT_ENUM},*)
(*DBG:    {&(RES0__INSTANCE0.MY_BAD_FIFO.BUFFER.value.table[4261]), INT_ENUM},*)
(*DBG:    {&(RES0__INSTANCE0.MY_BAD_FIFO.BUFFER.value.table[4262]), INT_ENUM},*)
(*DBG:    {&(RES0__INSTANCE0.MY_BAD_FIFO.BUFFER.value.table[4263]), INT_ENUM},*)
(*DBG:    {&(RES0__INSTANCE0.MY_BAD_FIFO.BUFFER.value.table[4264]), INT_ENUM},*)
(*DBG:    {&(RES0__INSTANCE0.MY_BAD_FIFO.BUFFER.value.table[4265]), INT_ENUM},*)
(*DBG:    {&(RES0__INSTANCE0.MY_BAD_FIFO.BUFFER.value.table[4266]), INT_ENUM},*)
(*DBG:    {&(RES0__INSTANCE0.MY_BAD_FIFO.BUFFER.value.table[4267]), INT_ENUM},*)
(*DBG:    {&(RES0__INSTANCE0.MY_BAD_FIFO.BUFFER.value.table[4268]), INT_ENUM},*)
(*DBG:    {&(RES0__INSTANCE0.MY_BAD_FIFO.BUFFER.value.table[4269]), INT_ENUM},*)
(*DBG:    {&(RES0__INSTANCE0.MY_BAD_FIFO.BUFFER.value.table[4270]), INT_ENUM},*)
(*DBG:    {&(RES0__INSTANCE0.MY_BAD_FIFO.BUFFER.value.table[4271]), INT_ENUM},*)
(*DBG:    {&(RES0__INSTANCE0.MY_BAD_FIFO.BUFFER.value.table[4272]), INT_ENUM},*)
(*DBG:    {&(RES0__INSTANCE0.MY_BAD_FIFO.BUFFER.value.table[4273]), INT_ENUM},*)
(*DBG:    {&(RES0__INSTANCE0.MY_BAD_FIFO.BUFFER.value.table[4274]), INT_ENUM},*)
(*DBG:    {&(RES0__INSTANCE0.MY_BAD_FIFO.BUFFER.value.table[4275]), INT_ENUM},*)
(*DBG:    {&(RES0__INSTANCE0.MY_BAD_FIFO.BUFFER.value.table[4276]), INT_ENUM},*)
(*DBG:    {&(RES0__INSTANCE0.MY_BAD_FIFO.BUFFER.value.table[4277]), INT_ENUM},*)
(*DBG:    {&(RES0__INSTANCE0.MY_BAD_FIFO.BUFFER.value.table[4278]), INT_ENUM},*)
(*DBG:    {&(RES0__INSTANCE0.MY_BAD_FIFO.BUFFER.value.table[4279]), INT_ENUM},*)
(*DBG:    {&(RES0__INSTANCE0.MY_BAD_FIFO.BUFFER.value.table[4280]), INT_ENUM},*)
(*DBG:    {&(RES0__INSTANCE0.MY_BAD_FIFO.BUFFER.value.table[4281]), INT_ENUM},*)
(*DBG:    {&(RES0__INSTANCE0.MY_BAD_FIFO.BUFFER.value.table[4282]), INT_ENUM},*)
(*DBG:    {&(RES0__INSTANCE0.MY_BAD_FIFO.BUFFER.value.table[4283]), INT_ENUM},*)
(*DBG:    {&(RES0__INSTANCE0.MY_BAD_FIFO.BUFFER.value.table[4284]), INT_ENUM},*)
(*DBG:    {&(RES0__INSTANCE0.MY_BAD_FIFO.BUFFER.value.table[4285]), INT_ENUM},*)
(*DBG:    {&(RES0__INSTANCE0.MY_BAD_FIFO.BUFFER.value.table[4286]), INT_ENUM},*)
(*DBG:    {&(RES0__INSTANCE0.MY_BAD_FIFO.BUFFER.value.table[4287]), INT_ENUM},*)
(*DBG:    {&(RES0__INSTANCE0.MY_BAD_FIFO.BUFFER.value.table[4288]), INT_ENUM},*)
(*DBG:    {&(RES0__INSTANCE0.MY_BAD_FIFO.BUFFER.value.table[4289]), INT_ENUM},*)
(*DBG:    {&(RES0__INSTANCE0.MY_BAD_FIFO.BUFFER.value.table[4290]), INT_ENUM},*)
(*DBG:    {&(RES0__INSTANCE0.MY_BAD_FIFO.BUFFER.value.table[4291]), INT_ENUM},*)
(*DBG:    {&(RES0__INSTANCE0.MY_BAD_FIFO.BUFFER.value.table[4292]), INT_ENUM},*)
(*DBG:    {&(RES0__INSTANCE0.MY_BAD_FIFO.BUFFER.value.table[4293]), INT_ENUM},*)
(*DBG:    {&(RES0__INSTANCE0.MY_BAD_FIFO.BUFFER.value.table[4294]), INT_ENUM},*)
(*DBG:    {&(RES0__INSTANCE0.MY_BAD_FIFO.BUFFER.value.table[4295]), INT_ENUM},*)
(*DBG:    {&(RES0__INSTANCE0.MY_BAD_FIFO.BUFFER.value.table[4296]), INT_ENUM},*)
(*DBG:    {&(RES0__INSTANCE0.MY_BAD_FIFO.BUFFER.value.table[4297]), INT_ENUM},*)
(*DBG:    {&(RES0__INSTANCE0.MY_BAD_FIFO.BUFFER.value.table[4298]), INT_ENUM},*)
(*DBG:    {&(RES0__INSTANCE0.MY_BAD_FIFO.BUFFER.value.table[4299]), INT_ENUM},*)
(*DBG:    {&(RES0__INSTANCE0.MY_BAD_FIFO.BUFFER.value.table[4300]), INT_ENUM},*)
(*DBG:    {&(RES0__INSTANCE0.MY_BAD_FIFO.BUFFER.value.table[4301]), INT_ENUM},*)
(*DBG:    {&(RES0__INSTANCE0.MY_BAD_FIFO.BUFFER.value.table[4302]), INT_ENUM},*)
(*DBG:    {&(RES0__INSTANCE0.MY_BAD_FIFO.BUFFER.value.table[4303]), INT_ENUM},*)
(*DBG:    {&(RES0__INSTANCE0.MY_BAD_FIFO.BUFFER.value.table[4304]), INT_ENUM},*)
(*DBG:    {&(RES0__INSTANCE0.MY_BAD_FIFO.BUFFER.value.table[4305]), INT_ENUM},*)
(*DBG:    {&(RES0__INSTANCE0.MY_BAD_FIFO.BUFFER.value.table[4306]), INT_ENUM},*)
(*DBG:    {&(RES0__INSTANCE0.MY_BAD_FIFO.BUFFER.value.table[4307]), INT_ENUM},*)
(*DBG:    {&(RES0__INSTANCE0.MY_BAD_FIFO.BUFFER.value.table[4308]), INT_ENUM},*)
(*DBG:    {&(RES0__INSTANCE0.MY_BAD_FIFO.BUFFER.value.table[4309]), INT_ENUM},*)
(*DBG:    {&(RES0__INSTANCE0.MY_BAD_FIFO.BUFFER.value.table[4310]), INT_ENUM},*)
(*DBG:    {&(RES0__INSTANCE0.MY_BAD_FIFO.BUFFER.value.table[4311]), INT_ENUM},*)
(*DBG:    {&(RES0__INSTANCE0.MY_BAD_FIFO.BUFFER.value.table[4312]), INT_ENUM},*)
(*DBG:    {&(RES0__INSTANCE0.MY_BAD_FIFO.BUFFER.value.table[4313]), INT_ENUM},*)
(*DBG:    {&(RES0__INSTANCE0.MY_BAD_FIFO.BUFFER.value.table[4314]), INT_ENUM},*)
(*DBG:    {&(RES0__INSTANCE0.MY_BAD_FIFO.BUFFER.value.table[4315]), INT_ENUM},*)
(*DBG:    {&(RES0__INSTANCE0.MY_BAD_FIFO.BUFFER.value.table[4316]), INT_ENUM},*)
(*DBG:    {&(RES0__INSTANCE0.MY_BAD_FIFO.BUFFER.value.table[4317]), INT_ENUM},*)
(*DBG:    {&(RES0__INSTANCE0.MY_BAD_FIFO.BUFFER.value.table[4318]), INT_ENUM},*)
(*DBG:    {&(RES0__INSTANCE0.MY_BAD_FIFO.BUFFER.value.table[4319]), INT_ENUM},*)
(*DBG:    {&(RES0__INSTANCE0.MY_BAD_FIFO.BUFFER.value.table[4320]), INT_ENUM},*)
(*DBG:    {&(RES0__INSTANCE0.MY_BAD_FIFO.BUFFER.value.table[4321]), INT_ENUM},*)
(*DBG:    {&(RES0__INSTANCE0.MY_BAD_FIFO.BUFFER.value.table[4322]), INT_ENUM},*)
(*DBG:    {&(RES0__INSTANCE0.MY_BAD_FIFO.BUFFER.value.table[4323]), INT_ENUM},*)
(*DBG:    {&(RES0__INSTANCE0.MY_BAD_FIFO.BUFFER.value.table[4324]), INT_ENUM},*)
(*DBG:    {&(RES0__INSTANCE0.MY_BAD_FIFO.BUFFER.value.table[4325]), INT_ENUM},*)
(*DBG:    {&(RES0__INSTANCE0.MY_BAD_FIFO.BUFFER.value.table[4326]), INT_ENUM},*)
(*DBG:    {&(RES0__INSTANCE0.MY_BAD_FIFO.BUFFER.value.table[4327]), INT_ENUM},*)
(*DBG:    {&(RES0__INSTANCE0.MY_BAD_FIFO.BUFFER.value.table[4328]), INT_ENUM},*)
(*DBG:    {&(RES0__INSTANCE0.MY_BAD_FIFO.BUFFER.value.table[4329]), INT_ENUM},*)
(*DBG:    {&(RES0__INSTANCE0.MY_BAD_FIFO.BUFFER.value.table[4330]), INT_ENUM},*)
(*DBG:    {&(RES0__INSTANCE0.MY_BAD_FIFO.BUFFER.value.table[4331]), INT_ENUM},*)
(*DBG:    {&(RES0__INSTANCE0.MY_BAD_FIFO.BUFFER.value.table[4332]), INT_ENUM},*)
(*DBG:    {&(RES0__INSTANCE0.MY_BAD_FIFO.BUFFER.value.table[4333]), INT_ENUM},*)
(*DBG:    {&(RES0__INSTANCE0.MY_BAD_FIFO.BUFFER.value.table[4334]), INT_ENUM},*)
(*DBG:    {&(RES0__INSTANCE0.MY_BAD_FIFO.BUFFER.value.table[4335]), INT_ENUM},*)
(*DBG:    {&(RES0__INSTANCE0.MY_BAD_FIFO.BUFFER.value.table[4336]), INT_ENUM},*)
(*DBG:    {&(RES0__INSTANCE0.MY_BAD_FIFO.BUFFER.value.table[4337]), INT_ENUM},*)
(*DBG:    {&(RES0__INSTANCE0.MY_BAD_FIFO.BUFFER.value.table[4338]), INT_ENUM},*)
(*DBG:    {&(RES0__INSTANCE0.MY_BAD_FIFO.BUFFER.value.table[4339]), INT_ENUM},*)
(*DBG:    {&(RES0__INSTANCE0.MY_BAD_FIFO.BUFFER.value.table[4340]), INT_ENUM},*)
(*DBG:    {&(RES0__INSTANCE0.MY_BAD_FIFO.BUFFER.value.table[4341]), INT_ENUM},*)
(*DBG:    {&(RES0__INSTANCE0.MY_BAD_FIFO.BUFFER.value.table[4342]), INT_ENUM},*)
(*DBG:    {&(RES0__INSTANCE0.MY_BAD_FIFO.BUFFER.value.table[4343]), INT_ENUM},*)
(*DBG:    {&(RES0__INSTANCE0.MY_BAD_FIFO.BUFFER.value.table[4344]), INT_ENUM},*)
(*DBG:    {&(RES0__INSTANCE0.MY_BAD_FIFO.BUFFER.value.table[4345]), INT_ENUM},*)
(*DBG:    {&(RES0__INSTANCE0.MY_BAD_FIFO.BUFFER.value.table[4346]), INT_ENUM},*)
(*DBG:    {&(RES0__INSTANCE0.MY_BAD_FIFO.BUFFER.value.table[4347]), INT_ENUM},*)
(*DBG:    {&(RES0__INSTANCE0.MY_BAD_FIFO.BUFFER.value.table[4348]), INT_ENUM},*)
(*DBG:    {&(RES0__INSTANCE0.MY_BAD_FIFO.BUFFER.value.table[4349]), INT_ENUM},*)
(*DBG:    {&(RES0__INSTANCE0.MY_BAD_FIFO.BUFFER.value.table[4350]), INT_ENUM},*)
(*DBG:    {&(RES0__INSTANCE0.MY_BAD_FIFO.BUFFER.value.table[4351]), INT_ENUM},*)
(*DBG:    {&(RES0__INSTANCE0.MY_BAD_FIFO.BUFFER.value.table[4352]), INT_ENUM},*)
(*DBG:    {&(RES0__INSTANCE0.MY_BAD_FIFO.BUFFER.value.table[4353]), INT_ENUM},*)
(*DBG:    {&(RES0__INSTANCE0.MY_BAD_FIFO.BUFFER.value.table[4354]), INT_ENUM},*)
(*DBG:    {&(RES0__INSTANCE0.MY_BAD_FIFO.BUFFER.value.table[4355]), INT_ENUM},*)
(*DBG:    {&(RES0__INSTANCE0.MY_BAD_FIFO.BUFFER.value.table[4356]), INT_ENUM},*)
(*DBG:    {&(RES0__INSTANCE0.MY_BAD_FIFO.BUFFER.value.table[4357]), INT_ENUM},*)
(*DBG:    {&(RES0__INSTANCE0.MY_BAD_FIFO.BUFFER.value.table[4358]), INT_ENUM},*)
(*DBG:    {&(RES0__INSTANCE0.MY_BAD_FIFO.BUFFER.value.table[4359]), INT_ENUM},*)
(*DBG:    {&(RES0__INSTANCE0.MY_BAD_FIFO.BUFFER.value.table[4360]), INT_ENUM},*)
(*DBG:    {&(RES0__INSTANCE0.MY_BAD_FIFO.BUFFER.value.table[4361]), INT_ENUM},*)
(*DBG:    {&(RES0__INSTANCE0.MY_BAD_FIFO.BUFFER.value.table[4362]), INT_ENUM},*)
(*DBG:    {&(RES0__INSTANCE0.MY_BAD_FIFO.BUFFER.value.table[4363]), INT_ENUM},*)
(*DBG:    {&(RES0__INSTANCE0.MY_BAD_FIFO.BUFFER.value.table[4364]), INT_ENUM},*)
(*DBG:    {&(RES0__INSTANCE0.MY_BAD_FIFO.BUFFER.value.table[4365]), INT_ENUM},*)
(*DBG:    {&(RES0__INSTANCE0.MY_BAD_FIFO.BUFFER.value.table[4366]), INT_ENUM},*)
(*DBG:    {&(RES0__INSTANCE0.MY_BAD_FIFO.BUFFER.value.table[4367]), INT_ENUM},*)
(*DBG:    {&(RES0__INSTANCE0.MY_BAD_FIFO.BUFFER.value.table[4368]), INT_ENUM},*)
(*DBG:    {&(RES0__INSTANCE0.MY_BAD_FIFO.BUFFER.value.table[4369]), INT_ENUM},*)
(*DBG:    {&(RES0__INSTANCE0.MY_BAD_FIFO.BUFFER.value.table[4370]), INT_ENUM},*)
(*DBG:    {&(RES0__INSTANCE0.MY_BAD_FIFO.BUFFER.value.table[4371]), INT_ENUM},*)
(*DBG:    {&(RES0__INSTANCE0.MY_BAD_FIFO.BUFFER.value.table[4372]), INT_ENUM},*)
(*DBG:    {&(RES0__INSTANCE0.MY_BAD_FIFO.BUFFER.value.table[4373]), INT_ENUM},*)
(*DBG:    {&(RES0__INSTANCE0.MY_BAD_FIFO.BUFFER.value.table[4374]), INT_ENUM},*)
(*DBG:    {&(RES0__INSTANCE0.MY_BAD_FIFO.BUFFER.value.table[4375]), INT_ENUM},*)
(*DBG:    {&(RES0__INSTANCE0.MY_BAD_FIFO.BUFFER.value.table[4376]), INT_ENUM},*)
(*DBG:    {&(RES0__INSTANCE0.MY_BAD_FIFO.BUFFER.value.table[4377]), INT_ENUM},*)
(*DBG:    {&(RES0__INSTANCE0.MY_BAD_FIFO.BUFFER.value.table[4378]), INT_ENUM},*)
(*DBG:    {&(RES0__INSTANCE0.MY_BAD_FIFO.BUFFER.value.table[4379]), INT_ENUM},*)
(*DBG:    {&(RES0__INSTANCE0.MY_BAD_FIFO.BUFFER.value.table[4380]), INT_ENUM},*)
(*DBG:    {&(RES0__INSTANCE0.MY_BAD_FIFO.BUFFER.value.table[4381]), INT_ENUM},*)
(*DBG:    {&(RES0__INSTANCE0.MY_BAD_FIFO.BUFFER.value.table[4382]), INT_ENUM},*)
(*DBG:    {&(RES0__INSTANCE0.MY_BAD_FIFO.BUFFER.value.table[4383]), INT_ENUM},*)
(*DBG:    {&(RES0__INSTANCE0.MY_BAD_FIFO.BUFFER.value.table[4384]), INT_ENUM},*)
(*DBG:    {&(RES0__INSTANCE0.MY_BAD_FIFO.BUFFER.value.table[4385]), INT_ENUM},*)
(*DBG:    {&(RES0__INSTANCE0.MY_BAD_FIFO.BUFFER.value.table[4386]), INT_ENUM},*)
(*DBG:    {&(RES0__INSTANCE0.MY_BAD_FIFO.BUFFER.value.table[4387]), INT_ENUM},*)
(*DBG:    {&(RES0__INSTANCE0.MY_BAD_FIFO.BUFFER.value.table[4388]), INT_ENUM},*)
(*DBG:    {&(RES0__INSTANCE0.MY_BAD_FIFO.BUFFER.value.table[4389]), INT_ENUM},*)
(*DBG:    {&(RES0__INSTANCE0.MY_BAD_FIFO.BUFFER.value.table[4390]), INT_ENUM},*)
(*DBG:    {&(RES0__INSTANCE0.MY_BAD_FIFO.BUFFER.value.table[4391]), INT_ENUM},*)
(*DBG:    {&(RES0__INSTANCE0.MY_BAD_FIFO.BUFFER.value.table[4392]), INT_ENUM},*)
(*DBG:    {&(RES0__INSTANCE0.MY_BAD_FIFO.BUFFER.value.table[4393]), INT_ENUM},*)
(*DBG:    {&(RES0__INSTANCE0.MY_BAD_FIFO.BUFFER.value.table[4394]), INT_ENUM},*)
(*DBG:    {&(RES0__INSTANCE0.MY_BAD_FIFO.BUFFER.value.table[4395]), INT_ENUM},*)
(*DBG:    {&(RES0__INSTANCE0.MY_BAD_FIFO.BUFFER.value.table[4396]), INT_ENUM},*)
(*DBG:    {&(RES0__INSTANCE0.MY_BAD_FIFO.BUFFER.value.table[4397]), INT_ENUM},*)
(*DBG:    {&(RES0__INSTANCE0.MY_BAD_FIFO.BUFFER.value.table[4398]), INT_ENUM},*)
(*DBG:    {&(RES0__INSTANCE0.MY_BAD_FIFO.BUFFER.value.table[4399]), INT_ENUM},*)
(*DBG:    {&(RES0__INSTANCE0.MY_BAD_FIFO.BUFFER.value.table[4400]), INT_ENUM},*)
(*DBG:    {&(RES0__INSTANCE0.MY_BAD_FIFO.BUFFER.value.table[4401]), INT_ENUM},*)
(*DBG:    {&(RES0__INSTANCE0.MY_BAD_FIFO.BUFFER.value.table[4402]), INT_ENUM},*)
(*DBG:    {&(RES0__INSTANCE0.MY_BAD_FIFO.BUFFER.value.table[4403]), INT_ENUM},*)
(*DBG:    {&(RES0__INSTANCE0.MY_BAD_FIFO.BUFFER.value.table[4404]), INT_ENUM},*)
(*DBG:    {&(RES0__INSTANCE0.MY_BAD_FIFO.BUFFER.value.table[4405]), INT_ENUM},*)
(*DBG:    {&(RES0__INSTANCE0.MY_BAD_FIFO.BUFFER.value.table[4406]), INT_ENUM},*)
(*DBG:    {&(RES0__INSTANCE0.MY_BAD_FIFO.BUFFER.value.table[4407]), INT_ENUM},*)
(*DBG:    {&(RES0__INSTANCE0.MY_BAD_FIFO.BUFFER.value.table[4408]), INT_ENUM},*)
(*DBG:    {&(RES0__INSTANCE0.MY_BAD_FIFO.BUFFER.value.table[4409]), INT_ENUM},*)
(*DBG:    {&(RES0__INSTANCE0.MY_BAD_FIFO.BUFFER.value.table[4410]), INT_ENUM},*)
(*DBG:    {&(RES0__INSTANCE0.MY_BAD_FIFO.BUFFER.value.table[4411]), INT_ENUM},*)
(*DBG:    {&(RES0__INSTANCE0.MY_BAD_FIFO.BUFFER.value.table[4412]), INT_ENUM},*)
(*DBG:    {&(RES0__INSTANCE0.MY_BAD_FIFO.BUFFER.value.table[4413]), INT_ENUM},*)
(*DBG:    {&(RES0__INSTANCE0.MY_BAD_FIFO.BUFFER.value.table[4414]), INT_ENUM},*)
(*DBG:    {&(RES0__INSTANCE0.MY_BAD_FIFO.BUFFER.value.table[4415]), INT_ENUM},*)
(*DBG:    {&(RES0__INSTANCE0.MY_BAD_FIFO.BUFFER.value.table[4416]), INT_ENUM},*)
(*DBG:    {&(RES0__INSTANCE0.MY_BAD_FIFO.BUFFER.value.table[4417]), INT_ENUM},*)
(*DBG:    {&(RES0__INSTANCE0.MY_BAD_FIFO.BUFFER.value.table[4418]), INT_ENUM},*)
(*DBG:    {&(RES0__INSTANCE0.MY_BAD_FIFO.BUFFER.value.table[4419]), INT_ENUM},*)
(*DBG:    {&(RES0__INSTANCE0.MY_BAD_FIFO.BUFFER.value.table[4420]), INT_ENUM},*)
(*DBG:    {&(RES0__INSTANCE0.MY_BAD_FIFO.BUFFER.value.table[4421]), INT_ENUM},*)
(*DBG:    {&(RES0__INSTANCE0.MY_BAD_FIFO.BUFFER.value.table[4422]), INT_ENUM},*)
(*DBG:    {&(RES0__INSTANCE0.MY_BAD_FIFO.BUFFER.value.table[4423]), INT_ENUM},*)
(*DBG:    {&(RES0__INSTANCE0.MY_BAD_FIFO.BUFFER.value.table[4424]), INT_ENUM},*)
(*DBG:    {&(RES0__INSTANCE0.MY_BAD_FIFO.BUFFER.value.table[4425]), INT_ENUM},*)
(*DBG:    {&(RES0__INSTANCE0.MY_BAD_FIFO.BUFFER.value.table[4426]), INT_ENUM},*)
(*DBG:    {&(RES0__INSTANCE0.MY_BAD_FIFO.BUFFER.value.table[4427]), INT_ENUM},*)
(*DBG:    {&(RES0__INSTANCE0.MY_BAD_FIFO.BUFFER.value.table[4428]), INT_ENUM},*)
(*DBG:    {&(RES0__INSTANCE0.MY_BAD_FIFO.BUFFER.value.table[4429]), INT_ENUM},*)
(*DBG:    {&(RES0__INSTANCE0.MY_BAD_FIFO.BUFFER.value.table[4430]), INT_ENUM},*)
(*DBG:    {&(RES0__INSTANCE0.MY_BAD_FIFO.BUFFER.value.table[4431]), INT_ENUM},*)
(*DBG:    {&(RES0__INSTANCE0.MY_BAD_FIFO.BUFFER.value.table[4432]), INT_ENUM},*)
(*DBG:    {&(RES0__INSTANCE0.MY_BAD_FIFO.BUFFER.value.table[4433]), INT_ENUM},*)
(*DBG:    {&(RES0__INSTANCE0.MY_BAD_FIFO.BUFFER.value.table[4434]), INT_ENUM},*)
(*DBG:    {&(RES0__INSTANCE0.MY_BAD_FIFO.BUFFER.value.table[4435]), INT_ENUM},*)
(*DBG:    {&(RES0__INSTANCE0.MY_BAD_FIFO.BUFFER.value.table[4436]), INT_ENUM},*)
(*DBG:    {&(RES0__INSTANCE0.MY_BAD_FIFO.BUFFER.value.table[4437]), INT_ENUM},*)
(*DBG:    {&(RES0__INSTANCE0.MY_BAD_FIFO.BUFFER.value.table[4438]), INT_ENUM},*)
(*DBG:    {&(RES0__INSTANCE0.MY_BAD_FIFO.BUFFER.value.table[4439]), INT_ENUM},*)
(*DBG:    {&(RES0__INSTANCE0.MY_BAD_FIFO.BUFFER.value.table[4440]), INT_ENUM},*)
(*DBG:    {&(RES0__INSTANCE0.MY_BAD_FIFO.BUFFER.value.table[4441]), INT_ENUM},*)
(*DBG:    {&(RES0__INSTANCE0.MY_BAD_FIFO.BUFFER.value.table[4442]), INT_ENUM},*)
(*DBG:    {&(RES0__INSTANCE0.MY_BAD_FIFO.BUFFER.value.table[4443]), INT_ENUM},*)
(*DBG:    {&(RES0__INSTANCE0.MY_BAD_FIFO.BUFFER.value.table[4444]), INT_ENUM},*)
(*DBG:    {&(RES0__INSTANCE0.MY_BAD_FIFO.BUFFER.value.table[4445]), INT_ENUM},*)
(*DBG:    {&(RES0__INSTANCE0.MY_BAD_FIFO.BUFFER.value.table[4446]), INT_ENUM},*)
(*DBG:    {&(RES0__INSTANCE0.MY_BAD_FIFO.BUFFER.value.table[4447]), INT_ENUM},*)
(*DBG:    {&(RES0__INSTANCE0.MY_BAD_FIFO.BUFFER.value.table[4448]), INT_ENUM},*)
(*DBG:    {&(RES0__INSTANCE0.MY_BAD_FIFO.BUFFER.value.table[4449]), INT_ENUM},*)
(*DBG:    {&(RES0__INSTANCE0.MY_BAD_FIFO.BUFFER.value.table[4450]), INT_ENUM},*)
(*DBG:    {&(RES0__INSTANCE0.MY_BAD_FIFO.BUFFER.value.table[4451]), INT_ENUM},*)
(*DBG:    {&(RES0__INSTANCE0.MY_BAD_FIFO.BUFFER.value.table[4452]), INT_ENUM},*)
(*DBG:    {&(RES0__INSTANCE0.MY_BAD_FIFO.BUFFER.value.table[4453]), INT_ENUM},*)
(*DBG:    {&(RES0__INSTANCE0.MY_BAD_FIFO.BUFFER.value.table[4454]), INT_ENUM},*)
(*DBG:    {&(RES0__INSTANCE0.MY_BAD_FIFO.BUFFER.value.table[4455]), INT_ENUM},*)
(*DBG:    {&(RES0__INSTANCE0.MY_BAD_FIFO.BUFFER.value.table[4456]), INT_ENUM},*)
(*DBG:    {&(RES0__INSTANCE0.MY_BAD_FIFO.BUFFER.value.table[4457]), INT_ENUM},*)
(*DBG:    {&(RES0__INSTANCE0.MY_BAD_FIFO.BUFFER.value.table[4458]), INT_ENUM},*)
(*DBG:    {&(RES0__INSTANCE0.MY_BAD_FIFO.BUFFER.value.table[4459]), INT_ENUM},*)
(*DBG:    {&(RES0__INSTANCE0.MY_BAD_FIFO.BUFFER.value.table[4460]), INT_ENUM},*)
(*DBG:    {&(RES0__INSTANCE0.MY_BAD_FIFO.BUFFER.value.table[4461]), INT_ENUM},*)
(*DBG:    {&(RES0__INSTANCE0.MY_BAD_FIFO.BUFFER.value.table[4462]), INT_ENUM},*)
(*DBG:    {&(RES0__INSTANCE0.MY_BAD_FIFO.BUFFER.value.table[4463]), INT_ENUM},*)
(*DBG:    {&(RES0__INSTANCE0.MY_BAD_FIFO.BUFFER.value.table[4464]), INT_ENUM},*)
(*DBG:    {&(RES0__INSTANCE0.MY_BAD_FIFO.BUFFER.value.table[4465]), INT_ENUM},*)
(*DBG:    {&(RES0__INSTANCE0.MY_BAD_FIFO.BUFFER.value.table[4466]), INT_ENUM},*)
(*DBG:    {&(RES0__INSTANCE0.MY_BAD_FIFO.BUFFER.value.table[4467]), INT_ENUM},*)
(*DBG:    {&(RES0__INSTANCE0.MY_BAD_FIFO.BUFFER.value.table[4468]), INT_ENUM},*)
(*DBG:    {&(RES0__INSTANCE0.MY_BAD_FIFO.BUFFER.value.table[4469]), INT_ENUM},*)
(*DBG:    {&(RES0__INSTANCE0.MY_BAD_FIFO.BUFFER.value.table[4470]), INT_ENUM},*)
(*DBG:    {&(RES0__INSTANCE0.MY_BAD_FIFO.BUFFER.value.table[4471]), INT_ENUM},*)
(*DBG:    {&(RES0__INSTANCE0.MY_BAD_FIFO.BUFFER.value.table[4472]), INT_ENUM},*)
(*DBG:    {&(RES0__INSTANCE0.MY_BAD_FIFO.BUFFER.value.table[4473]), INT_ENUM},*)
(*DBG:    {&(RES0__INSTANCE0.MY_BAD_FIFO.BUFFER.value.table[4474]), INT_ENUM},*)
(*DBG:    {&(RES0__INSTANCE0.MY_BAD_FIFO.BUFFER.value.table[4475]), INT_ENUM},*)
(*DBG:    {&(RES0__INSTANCE0.MY_BAD_FIFO.BUFFER.value.table[4476]), INT_ENUM},*)
(*DBG:    {&(RES0__INSTANCE0.MY_BAD_FIFO.BUFFER.value.table[4477]), INT_ENUM},*)
(*DBG:    {&(RES0__INSTANCE0.MY_BAD_FIFO.BUFFER.value.table[4478]), INT_ENUM},*)
(*DBG:    {&(RES0__INSTANCE0.MY_BAD_FIFO.BUFFER.value.table[4479]), INT_ENUM},*)
(*DBG:    {&(RES0__INSTANCE0.MY_BAD_FIFO.BUFFER.value.table[4480]), INT_ENUM},*)
(*DBG:    {&(RES0__INSTANCE0.MY_BAD_FIFO.BUFFER.value.table[4481]), INT_ENUM},*)
(*DBG:    {&(RES0__INSTANCE0.MY_BAD_FIFO.BUFFER.value.table[4482]), INT_ENUM},*)
(*DBG:    {&(RES0__INSTANCE0.MY_BAD_FIFO.BUFFER.value.table[4483]), INT_ENUM},*)
(*DBG:    {&(RES0__INSTANCE0.MY_BAD_FIFO.BUFFER.value.table[4484]), INT_ENUM},*)
(*DBG:    {&(RES0__INSTANCE0.MY_BAD_FIFO.BUFFER.value.table[4485]), INT_ENUM},*)
(*DBG:    {&(RES0__INSTANCE0.MY_BAD_FIFO.BUFFER.value.table[4486]), INT_ENUM},*)
(*DBG:    {&(RES0__INSTANCE0.MY_BAD_FIFO.BUFFER.value.table[4487]), INT_ENUM},*)
(*DBG:    {&(RES0__INSTANCE0.MY_BAD_FIFO.BUFFER.value.table[4488]), INT_ENUM},*)
(*DBG:    {&(RES0__INSTANCE0.MY_BAD_FIFO.BUFFER.value.table[4489]), INT_ENUM},*)
(*DBG:    {&(RES0__INSTANCE0.MY_BAD_FIFO.BUFFER.value.table[4490]), INT_ENUM},*)
(*DBG:    {&(RES0__INSTANCE0.MY_BAD_FIFO.BUFFER.value.table[4491]), INT_ENUM},*)
(*DBG:    {&(RES0__INSTANCE0.MY_BAD_FIFO.BUFFER.value.table[4492]), INT_ENUM},*)
(*DBG:    {&(RES0__INSTANCE0.MY_BAD_FIFO.BUFFER.value.table[4493]), INT_ENUM},*)
(*DBG:    {&(RES0__INSTANCE0.MY_BAD_FIFO.BUFFER.value.table[4494]), INT_ENUM},*)
(*DBG:    {&(RES0__INSTANCE0.MY_BAD_FIFO.BUFFER.value.table[4495]), INT_ENUM},*)
(*DBG:    {&(RES0__INSTANCE0.MY_BAD_FIFO.BUFFER.value.table[4496]), INT_ENUM},*)
(*DBG:    {&(RES0__INSTANCE0.MY_BAD_FIFO.BUFFER.value.table[4497]), INT_ENUM},*)
(*DBG:    {&(RES0__INSTANCE0.MY_BAD_FIFO.BUFFER.value.table[4498]), INT_ENUM},*)
(*DBG:    {&(RES0__INSTANCE0.MY_BAD_FIFO.BUFFER.value.table[4499]), INT_ENUM},*)
(*DBG:    {&(RES0__INSTANCE0.MY_BAD_FIFO.BUFFER.value.table[4500]), INT_ENUM},*)
(*DBG:    {&(RES0__INSTANCE0.MY_BAD_FIFO.BUFFER.value.table[4501]), INT_ENUM},*)
(*DBG:    {&(RES0__INSTANCE0.MY_BAD_FIFO.BUFFER.value.table[4502]), INT_ENUM},*)
(*DBG:    {&(RES0__INSTANCE0.MY_BAD_FIFO.BUFFER.value.table[4503]), INT_ENUM},*)
(*DBG:    {&(RES0__INSTANCE0.MY_BAD_FIFO.BUFFER.value.table[4504]), INT_ENUM},*)
(*DBG:    {&(RES0__INSTANCE0.MY_BAD_FIFO.BUFFER.value.table[4505]), INT_ENUM},*)
(*DBG:    {&(RES0__INSTANCE0.MY_BAD_FIFO.BUFFER.value.table[4506]), INT_ENUM},*)
(*DBG:    {&(RES0__INSTANCE0.MY_BAD_FIFO.BUFFER.value.table[4507]), INT_ENUM},*)
(*DBG:    {&(RES0__INSTANCE0.MY_BAD_FIFO.BUFFER.value.table[4508]), INT_ENUM},*)
(*DBG:    {&(RES0__INSTANCE0.MY_BAD_FIFO.BUFFER.value.table[4509]), INT_ENUM},*)
(*DBG:    {&(RES0__INSTANCE0.MY_BAD_FIFO.BUFFER.value.table[4510]), INT_ENUM},*)
(*DBG:    {&(RES0__INSTANCE0.MY_BAD_FIFO.BUFFER.value.table[4511]), INT_ENUM},*)
(*DBG:    {&(RES0__INSTANCE0.MY_BAD_FIFO.BUFFER.value.table[4512]), INT_ENUM},*)
(*DBG:    {&(RES0__INSTANCE0.MY_BAD_FIFO.BUFFER.value.table[4513]), INT_ENUM},*)
(*DBG:    {&(RES0__INSTANCE0.MY_BAD_FIFO.BUFFER.value.table[4514]), INT_ENUM},*)
(*DBG:    {&(RES0__INSTANCE0.MY_BAD_FIFO.BUFFER.value.table[4515]), INT_ENUM},*)
(*DBG:    {&(RES0__INSTANCE0.MY_BAD_FIFO.BUFFER.value.table[4516]), INT_ENUM},*)
(*DBG:    {&(RES0__INSTANCE0.MY_BAD_FIFO.BUFFER.value.table[4517]), INT_ENUM},*)
(*DBG:    {&(RES0__INSTANCE0.MY_BAD_FIFO.BUFFER.value.table[4518]), INT_ENUM},*)
(*DBG:    {&(RES0__INSTANCE0.MY_BAD_FIFO.BUFFER.value.table[4519]), INT_ENUM},*)
(*DBG:    {&(RES0__INSTANCE0.MY_BAD_FIFO.BUFFER.value.table[4520]), INT_ENUM},*)
(*DBG:    {&(RES0__INSTANCE0.MY_BAD_FIFO.BUFFER.value.table[4521]), INT_ENUM},*)
(*DBG:    {&(RES0__INSTANCE0.MY_BAD_FIFO.BUFFER.value.table[4522]), INT_ENUM},*)
(*DBG:    {&(RES0__INSTANCE0.MY_BAD_FIFO.BUFFER.value.table[4523]), INT_ENUM},*)
(*DBG:    {&(RES0__INSTANCE0.MY_BAD_FIFO.BUFFER.value.table[4524]), INT_ENUM},*)
(*DBG:    {&(RES0__INSTANCE0.MY_BAD_FIFO.BUFFER.value.table[4525]), INT_ENUM},*)
(*DBG:    {&(RES0__INSTANCE0.MY_BAD_FIFO.BUFFER.value.table[4526]), INT_ENUM},*)
(*DBG:    {&(RES0__INSTANCE0.MY_BAD_FIFO.BUFFER.value.table[4527]), INT_ENUM},*)
(*DBG:    {&(RES0__INSTANCE0.MY_BAD_FIFO.BUFFER.value.table[4528]), INT_ENUM},*)
(*DBG:    {&(RES0__INSTANCE0.MY_BAD_FIFO.BUFFER.value.table[4529]), INT_ENUM},*)
(*DBG:    {&(RES0__INSTANCE0.MY_BAD_FIFO.BUFFER.value.table[4530]), INT_ENUM},*)
(*DBG:    {&(RES0__INSTANCE0.MY_BAD_FIFO.BUFFER.value.table[4531]), INT_ENUM},*)
(*DBG:    {&(RES0__INSTANCE0.MY_BAD_FIFO.BUFFER.value.table[4532]), INT_ENUM},*)
(*DBG:    {&(RES0__INSTANCE0.MY_BAD_FIFO.BUFFER.value.table[4533]), INT_ENUM},*)
(*DBG:    {&(RES0__INSTANCE0.MY_BAD_FIFO.BUFFER.value.table[4534]), INT_ENUM},*)
(*DBG:    {&(RES0__INSTANCE0.MY_BAD_FIFO.BUFFER.value.table[4535]), INT_ENUM},*)
(*DBG:    {&(RES0__INSTANCE0.MY_BAD_FIFO.BUFFER.value.table[4536]), INT_ENUM},*)
(*DBG:    {&(RES0__INSTANCE0.MY_BAD_FIFO.BUFFER.value.table[4537]), INT_ENUM},*)
(*DBG:    {&(RES0__INSTANCE0.MY_BAD_FIFO.BUFFER.value.table[4538]), INT_ENUM},*)
(*DBG:    {&(RES0__INSTANCE0.MY_BAD_FIFO.BUFFER.value.table[4539]), INT_ENUM},*)
(*DBG:    {&(RES0__INSTANCE0.MY_BAD_FIFO.BUFFER.value.table[4540]), INT_ENUM},*)
(*DBG:    {&(RES0__INSTANCE0.MY_BAD_FIFO.BUFFER.value.table[4541]), INT_ENUM},*)
(*DBG:    {&(RES0__INSTANCE0.MY_BAD_FIFO.BUFFER.value.table[4542]), INT_ENUM},*)
(*DBG:    {&(RES0__INSTANCE0.MY_BAD_FIFO.BUFFER.value.table[4543]), INT_ENUM},*)
(*DBG:    {&(RES0__INSTANCE0.MY_BAD_FIFO.BUFFER.value.table[4544]), INT_ENUM},*)
(*DBG:    {&(RES0__INSTANCE0.MY_BAD_FIFO.BUFFER.value.table[4545]), INT_ENUM},*)
(*DBG:    {&(RES0__INSTANCE0.MY_BAD_FIFO.BUFFER.value.table[4546]), INT_ENUM},*)
(*DBG:    {&(RES0__INSTANCE0.MY_BAD_FIFO.BUFFER.value.table[4547]), INT_ENUM},*)
(*DBG:    {&(RES0__INSTANCE0.MY_BAD_FIFO.BUFFER.value.table[4548]), INT_ENUM},*)
(*DBG:    {&(RES0__INSTANCE0.MY_BAD_FIFO.BUFFER.value.table[4549]), INT_ENUM},*)
(*DBG:    {&(RES0__INSTANCE0.MY_BAD_FIFO.BUFFER.value.table[4550]), INT_ENUM},*)
(*DBG:    {&(RES0__INSTANCE0.MY_BAD_FIFO.BUFFER.value.table[4551]), INT_ENUM},*)
(*DBG:    {&(RES0__INSTANCE0.MY_BAD_FIFO.BUFFER.value.table[4552]), INT_ENUM},*)
(*DBG:    {&(RES0__INSTANCE0.MY_BAD_FIFO.BUFFER.value.table[4553]), INT_ENUM},*)
(*DBG:    {&(RES0__INSTANCE0.MY_BAD_FIFO.BUFFER.value.table[4554]), INT_ENUM},*)
(*DBG:    {&(RES0__INSTANCE0.MY_BAD_FIFO.BUFFER.value.table[4555]), INT_ENUM},*)
(*DBG:    {&(RES0__INSTANCE0.MY_BAD_FIFO.BUFFER.value.table[4556]), INT_ENUM},*)
(*DBG:    {&(RES0__INSTANCE0.MY_BAD_FIFO.BUFFER.value.table[4557]), INT_ENUM},*)
(*DBG:    {&(RES0__INSTANCE0.MY_BAD_FIFO.BUFFER.value.table[4558]), INT_ENUM},*)
(*DBG:    {&(RES0__INSTANCE0.MY_BAD_FIFO.BUFFER.value.table[4559]), INT_ENUM},*)
(*DBG:    {&(RES0__INSTANCE0.MY_BAD_FIFO.BUFFER.value.table[4560]), INT_ENUM},*)
(*DBG:    {&(RES0__INSTANCE0.MY_BAD_FIFO.BUFFER.value.table[4561]), INT_ENUM},*)
(*DBG:    {&(RES0__INSTANCE0.MY_BAD_FIFO.BUFFER.value.table[4562]), INT_ENUM},*)
(*DBG:    {&(RES0__INSTANCE0.MY_BAD_FIFO.BUFFER.value.table[4563]), INT_ENUM},*)
(*DBG:    {&(RES0__INSTANCE0.MY_BAD_FIFO.BUFFER.value.table[4564]), INT_ENUM},*)
(*DBG:    {&(RES0__INSTANCE0.MY_BAD_FIFO.BUFFER.value.table[4565]), INT_ENUM},*)
(*DBG:    {&(RES0__INSTANCE0.MY_BAD_FIFO.BUFFER.value.table[4566]), INT_ENUM},*)
(*DBG:    {&(RES0__INSTANCE0.MY_BAD_FIFO.BUFFER.value.table[4567]), INT_ENUM},*)
(*DBG:    {&(RES0__INSTANCE0.MY_BAD_FIFO.BUFFER.value.table[4568]), INT_ENUM},*)
(*DBG:    {&(RES0__INSTANCE0.MY_BAD_FIFO.BUFFER.value.table[4569]), INT_ENUM},*)
(*DBG:    {&(RES0__INSTANCE0.MY_BAD_FIFO.BUFFER.value.table[4570]), INT_ENUM},*)
(*DBG:    {&(RES0__INSTANCE0.MY_BAD_FIFO.BUFFER.value.table[4571]), INT_ENUM},*)
(*DBG:    {&(RES0__INSTANCE0.MY_BAD_FIFO.BUFFER.value.table[4572]), INT_ENUM},*)
(*DBG:    {&(RES0__INSTANCE0.MY_BAD_FIFO.BUFFER.value.table[4573]), INT_ENUM},*)
(*DBG:    {&(RES0__INSTANCE0.MY_BAD_FIFO.BUFFER.value.table[4574]), INT_ENUM},*)
(*DBG:    {&(RES0__INSTANCE0.MY_BAD_FIFO.BUFFER.value.table[4575]), INT_ENUM},*)
(*DBG:    {&(RES0__INSTANCE0.MY_BAD_FIFO.BUFFER.value.table[4576]), INT_ENUM},*)
(*DBG:    {&(RES0__INSTANCE0.MY_BAD_FIFO.BUFFER.value.table[4577]), INT_ENUM},*)
(*DBG:    {&(RES0__INSTANCE0.MY_BAD_FIFO.BUFFER.value.table[4578]), INT_ENUM},*)
(*DBG:    {&(RES0__INSTANCE0.MY_BAD_FIFO.BUFFER.value.table[4579]), INT_ENUM},*)
(*DBG:    {&(RES0__INSTANCE0.MY_BAD_FIFO.BUFFER.value.table[4580]), INT_ENUM},*)
(*DBG:    {&(RES0__INSTANCE0.MY_BAD_FIFO.BUFFER.value.table[4581]), INT_ENUM},*)
(*DBG:    {&(RES0__INSTANCE0.MY_BAD_FIFO.BUFFER.value.table[4582]), INT_ENUM},*)
(*DBG:    {&(RES0__INSTANCE0.MY_BAD_FIFO.BUFFER.value.table[4583]), INT_ENUM},*)
(*DBG:    {&(RES0__INSTANCE0.MY_BAD_FIFO.BUFFER.value.table[4584]), INT_ENUM},*)
(*DBG:    {&(RES0__INSTANCE0.MY_BAD_FIFO.BUFFER.value.table[4585]), INT_ENUM},*)
(*DBG:    {&(RES0__INSTANCE0.MY_BAD_FIFO.BUFFER.value.table[4586]), INT_ENUM},*)
(*DBG:    {&(RES0__INSTANCE0.MY_BAD_FIFO.BUFFER.value.table[4587]), INT_ENUM},*)
(*DBG:    {&(RES0__INSTANCE0.MY_BAD_FIFO.BUFFER.value.table[4588]), INT_ENUM},*)
(*DBG:    {&(RES0__INSTANCE0.MY_BAD_FIFO.BUFFER.value.table[4589]), INT_ENUM},*)
(*DBG:    {&(RES0__INSTANCE0.MY_BAD_FIFO.BUFFER.value.table[4590]), INT_ENUM},*)
(*DBG:    {&(RES0__INSTANCE0.MY_BAD_FIFO.BUFFER.value.table[4591]), INT_ENUM},*)
(*DBG:    {&(RES0__INSTANCE0.MY_BAD_FIFO.BUFFER.value.table[4592]), INT_ENUM},*)
(*DBG:    {&(RES0__INSTANCE0.MY_BAD_FIFO.BUFFER.value.table[4593]), INT_ENUM},*)
(*DBG:    {&(RES0__INSTANCE0.MY_BAD_FIFO.BUFFER.value.table[4594]), INT_ENUM},*)
(*DBG:    {&(RES0__INSTANCE0.MY_BAD_FIFO.BUFFER.value.table[4595]), INT_ENUM},*)
(*DBG:    {&(RES0__INSTANCE0.MY_BAD_FIFO.BUFFER.value.table[4596]), INT_ENUM},*)
(*DBG:    {&(RES0__INSTANCE0.MY_BAD_FIFO.BUFFER.value.table[4597]), INT_ENUM},*)
(*DBG:    {&(RES0__INSTANCE0.MY_BAD_FIFO.BUFFER.value.table[4598]), INT_ENUM},*)
(*DBG:    {&(RES0__INSTANCE0.MY_BAD_FIFO.BUFFER.value.table[4599]), INT_ENUM},*)
(*DBG:    {&(RES0__INSTANCE0.MY_BAD_FIFO.BUFFER.value.table[4600]), INT_ENUM},*)
(*DBG:    {&(RES0__INSTANCE0.MY_BAD_FIFO.BUFFER.value.table[4601]), INT_ENUM},*)
(*DBG:    {&(RES0__INSTANCE0.MY_BAD_FIFO.BUFFER.value.table[4602]), INT_ENUM},*)
(*DBG:    {&(RES0__INSTANCE0.MY_BAD_FIFO.BUFFER.value.table[4603]), INT_ENUM},*)
(*DBG:    {&(RES0__INSTANCE0.MY_BAD_FIFO.BUFFER.value.table[4604]), INT_ENUM},*)
(*DBG:    {&(RES0__INSTANCE0.MY_BAD_FIFO.BUFFER.value.table[4605]), INT_ENUM},*)
(*DBG:    {&(RES0__INSTANCE0.MY_BAD_FIFO.BUFFER.value.table[4606]), INT_ENUM},*)
(*DBG:    {&(RES0__INSTANCE0.MY_BAD_FIFO.BUFFER.value.table[4607]), INT_ENUM},*)
(*DBG:    {&(RES0__INSTANCE0.MY_BAD_FIFO.BUFFER.value.table[4608]), INT_ENUM},*)
(*DBG:    {&(RES0__INSTANCE0.MY_BAD_FIFO.BUFFER.value.table[4609]), INT_ENUM},*)
(*DBG:    {&(RES0__INSTANCE0.MY_BAD_FIFO.BUFFER.value.table[4610]), INT_ENUM},*)
(*DBG:    {&(RES0__INSTANCE0.MY_BAD_FIFO.BUFFER.value.table[4611]), INT_ENUM},*)
(*DBG:    {&(RES0__INSTANCE0.MY_BAD_FIFO.BUFFER.value.table[4612]), INT_ENUM},*)
(*DBG:    {&(RES0__INSTANCE0.MY_BAD_FIFO.BUFFER.value.table[4613]), INT_ENUM},*)
(*DBG:    {&(RES0__INSTANCE0.MY_BAD_FIFO.BUFFER.value.table[4614]), INT_ENUM},*)
(*DBG:    {&(RES0__INSTANCE0.MY_BAD_FIFO.BUFFER.value.table[4615]), INT_ENUM},*)
(*DBG:    {&(RES0__INSTANCE0.MY_BAD_FIFO.BUFFER.value.table[4616]), INT_ENUM},*)
(*DBG:    {&(RES0__INSTANCE0.MY_BAD_FIFO.BUFFER.value.table[4617]), INT_ENUM},*)
(*DBG:    {&(RES0__INSTANCE0.MY_BAD_FIFO.BUFFER.value.table[4618]), INT_ENUM},*)
(*DBG:    {&(RES0__INSTANCE0.MY_BAD_FIFO.BUFFER.value.table[4619]), INT_ENUM},*)
(*DBG:    {&(RES0__INSTANCE0.MY_BAD_FIFO.BUFFER.value.table[4620]), INT_ENUM},*)
(*DBG:    {&(RES0__INSTANCE0.MY_BAD_FIFO.BUFFER.value.table[4621]), INT_ENUM},*)
(*DBG:    {&(RES0__INSTANCE0.MY_BAD_FIFO.BUFFER.value.table[4622]), INT_ENUM},*)
(*DBG:    {&(RES0__INSTANCE0.MY_BAD_FIFO.BUFFER.value.table[4623]), INT_ENUM},*)
(*DBG:    {&(RES0__INSTANCE0.MY_BAD_FIFO.BUFFER.value.table[4624]), INT_ENUM},*)
(*DBG:    {&(RES0__INSTANCE0.MY_BAD_FIFO.BUFFER.value.table[4625]), INT_ENUM},*)
(*DBG:    {&(RES0__INSTANCE0.MY_BAD_FIFO.BUFFER.value.table[4626]), INT_ENUM},*)
(*DBG:    {&(RES0__INSTANCE0.MY_BAD_FIFO.BUFFER.value.table[4627]), INT_ENUM},*)
(*DBG:    {&(RES0__INSTANCE0.MY_BAD_FIFO.BUFFER.value.table[4628]), INT_ENUM},*)
(*DBG:    {&(RES0__INSTANCE0.MY_BAD_FIFO.BUFFER.value.table[4629]), INT_ENUM},*)
(*DBG:    {&(RES0__INSTANCE0.MY_BAD_FIFO.BUFFER.value.table[4630]), INT_ENUM},*)
(*DBG:    {&(RES0__INSTANCE0.MY_BAD_FIFO.BUFFER.value.table[4631]), INT_ENUM},*)
(*DBG:    {&(RES0__INSTANCE0.MY_BAD_FIFO.BUFFER.value.table[4632]), INT_ENUM},*)
(*DBG:    {&(RES0__INSTANCE0.MY_BAD_FIFO.BUFFER.value.table[4633]), INT_ENUM},*)
(*DBG:    {&(RES0__INSTANCE0.MY_BAD_FIFO.BUFFER.value.table[4634]), INT_ENUM},*)
(*DBG:    {&(RES0__INSTANCE0.MY_BAD_FIFO.BUFFER.value.table[4635]), INT_ENUM},*)
(*DBG:    {&(RES0__INSTANCE0.MY_BAD_FIFO.BUFFER.value.table[4636]), INT_ENUM},*)
(*DBG:    {&(RES0__INSTANCE0.MY_BAD_FIFO.BUFFER.value.table[4637]), INT_ENUM},*)
(*DBG:    {&(RES0__INSTANCE0.MY_BAD_FIFO.BUFFER.value.table[4638]), INT_ENUM},*)
(*DBG:    {&(RES0__INSTANCE0.MY_BAD_FIFO.BUFFER.value.table[4639]), INT_ENUM},*)
(*DBG:    {&(RES0__INSTANCE0.MY_BAD_FIFO.BUFFER.value.table[4640]), INT_ENUM},*)
(*DBG:    {&(RES0__INSTANCE0.MY_BAD_FIFO.BUFFER.value.table[4641]), INT_ENUM},*)
(*DBG:    {&(RES0__INSTANCE0.MY_BAD_FIFO.BUFFER.value.table[4642]), INT_ENUM},*)
(*DBG:    {&(RES0__INSTANCE0.MY_BAD_FIFO.BUFFER.value.table[4643]), INT_ENUM},*)
(*DBG:    {&(RES0__INSTANCE0.MY_BAD_FIFO.BUFFER.value.table[4644]), INT_ENUM},*)
(*DBG:    {&(RES0__INSTANCE0.MY_BAD_FIFO.BUFFER.value.table[4645]), INT_ENUM},*)
(*DBG:    {&(RES0__INSTANCE0.MY_BAD_FIFO.BUFFER.value.table[4646]), INT_ENUM},*)
(*DBG:    {&(RES0__INSTANCE0.MY_BAD_FIFO.BUFFER.value.table[4647]), INT_ENUM},*)
(*DBG:    {&(RES0__INSTANCE0.MY_BAD_FIFO.BUFFER.value.table[4648]), INT_ENUM},*)
(*DBG:    {&(RES0__INSTANCE0.MY_BAD_FIFO.BUFFER.value.table[4649]), INT_ENUM},*)
(*DBG:    {&(RES0__INSTANCE0.MY_BAD_FIFO.BUFFER.value.table[4650]), INT_ENUM},*)
(*DBG:    {&(RES0__INSTANCE0.MY_BAD_FIFO.BUFFER.value.table[4651]), INT_ENUM},*)
(*DBG:    {&(RES0__INSTANCE0.MY_BAD_FIFO.BUFFER.value.table[4652]), INT_ENUM},*)
(*DBG:    {&(RES0__INSTANCE0.MY_BAD_FIFO.BUFFER.value.table[4653]), INT_ENUM},*)
(*DBG:    {&(RES0__INSTANCE0.MY_BAD_FIFO.BUFFER.value.table[4654]), INT_ENUM},*)
(*DBG:    {&(RES0__INSTANCE0.MY_BAD_FIFO.BUFFER.value.table[4655]), INT_ENUM},*)
(*DBG:    {&(RES0__INSTANCE0.MY_BAD_FIFO.BUFFER.value.table[4656]), INT_ENUM},*)
(*DBG:    {&(RES0__INSTANCE0.MY_BAD_FIFO.BUFFER.value.table[4657]), INT_ENUM},*)
(*DBG:    {&(RES0__INSTANCE0.MY_BAD_FIFO.BUFFER.value.table[4658]), INT_ENUM},*)
(*DBG:    {&(RES0__INSTANCE0.MY_BAD_FIFO.BUFFER.value.table[4659]), INT_ENUM},*)
(*DBG:    {&(RES0__INSTANCE0.MY_BAD_FIFO.BUFFER.value.table[4660]), INT_ENUM},*)
(*DBG:    {&(RES0__INSTANCE0.MY_BAD_FIFO.BUFFER.value.table[4661]), INT_ENUM},*)
(*DBG:    {&(RES0__INSTANCE0.MY_BAD_FIFO.BUFFER.value.table[4662]), INT_ENUM},*)
(*DBG:    {&(RES0__INSTANCE0.MY_BAD_FIFO.BUFFER.value.table[4663]), INT_ENUM},*)
(*DBG:    {&(RES0__INSTANCE0.MY_BAD_FIFO.BUFFER.value.table[4664]), INT_ENUM},*)
(*DBG:    {&(RES0__INSTANCE0.MY_BAD_FIFO.BUFFER.value.table[4665]), INT_ENUM},*)
(*DBG:    {&(RES0__INSTANCE0.MY_BAD_FIFO.BUFFER.value.table[4666]), INT_ENUM},*)
(*DBG:    {&(RES0__INSTANCE0.MY_BAD_FIFO.BUFFER.value.table[4667]), INT_ENUM},*)
(*DBG:    {&(RES0__INSTANCE0.MY_BAD_FIFO.BUFFER.value.table[4668]), INT_ENUM},*)
(*DBG:    {&(RES0__INSTANCE0.MY_BAD_FIFO.BUFFER.value.table[4669]), INT_ENUM},*)
(*DBG:    {&(RES0__INSTANCE0.MY_BAD_FIFO.BUFFER.value.table[4670]), INT_ENUM},*)
(*DBG:    {&(RES0__INSTANCE0.MY_BAD_FIFO.BUFFER.value.table[4671]), INT_ENUM},*)
(*DBG:    {&(RES0__INSTANCE0.MY_BAD_FIFO.BUFFER.value.table[4672]), INT_ENUM},*)
(*DBG:    {&(RES0__INSTANCE0.MY_BAD_FIFO.BUFFER.value.table[4673]), INT_ENUM},*)
(*DBG:    {&(RES0__INSTANCE0.MY_BAD_FIFO.BUFFER.value.table[4674]), INT_ENUM},*)
(*DBG:    {&(RES0__INSTANCE0.MY_BAD_FIFO.BUFFER.value.table[4675]), INT_ENUM},*)
(*DBG:    {&(RES0__INSTANCE0.MY_BAD_FIFO.BUFFER.value.table[4676]), INT_ENUM},*)
(*DBG:    {&(RES0__INSTANCE0.MY_BAD_FIFO.BUFFER.value.table[4677]), INT_ENUM},*)
(*DBG:    {&(RES0__INSTANCE0.MY_BAD_FIFO.BUFFER.value.table[4678]), INT_ENUM},*)
(*DBG:    {&(RES0__INSTANCE0.MY_BAD_FIFO.BUFFER.value.table[4679]), INT_ENUM},*)
(*DBG:    {&(RES0__INSTANCE0.MY_BAD_FIFO.BUFFER.value.table[4680]), INT_ENUM},*)
(*DBG:    {&(RES0__INSTANCE0.MY_BAD_FIFO.BUFFER.value.table[4681]), INT_ENUM},*)
(*DBG:    {&(RES0__INSTANCE0.MY_BAD_FIFO.BUFFER.value.table[4682]), INT_ENUM},*)
(*DBG:    {&(RES0__INSTANCE0.MY_BAD_FIFO.BUFFER.value.table[4683]), INT_ENUM},*)
(*DBG:    {&(RES0__INSTANCE0.MY_BAD_FIFO.BUFFER.value.table[4684]), INT_ENUM},*)
(*DBG:    {&(RES0__INSTANCE0.MY_BAD_FIFO.BUFFER.value.table[4685]), INT_ENUM},*)
(*DBG:    {&(RES0__INSTANCE0.MY_BAD_FIFO.BUFFER.value.table[4686]), INT_ENUM},*)
(*DBG:    {&(RES0__INSTANCE0.MY_BAD_FIFO.BUFFER.value.table[4687]), INT_ENUM},*)
(*DBG:    {&(RES0__INSTANCE0.MY_BAD_FIFO.BUFFER.value.table[4688]), INT_ENUM},*)
(*DBG:    {&(RES0__INSTANCE0.MY_BAD_FIFO.BUFFER.value.table[4689]), INT_ENUM},*)
(*DBG:    {&(RES0__INSTANCE0.MY_BAD_FIFO.BUFFER.value.table[4690]), INT_ENUM},*)
(*DBG:    {&(RES0__INSTANCE0.MY_BAD_FIFO.BUFFER.value.table[4691]), INT_ENUM},*)
(*DBG:    {&(RES0__INSTANCE0.MY_BAD_FIFO.BUFFER.value.table[4692]), INT_ENUM},*)
(*DBG:    {&(RES0__INSTANCE0.MY_BAD_FIFO.BUFFER.value.table[4693]), INT_ENUM},*)
(*DBG:    {&(RES0__INSTANCE0.MY_BAD_FIFO.BUFFER.value.table[4694]), INT_ENUM},*)
(*DBG:    {&(RES0__INSTANCE0.MY_BAD_FIFO.BUFFER.value.table[4695]), INT_ENUM},*)
(*DBG:    {&(RES0__INSTANCE0.MY_BAD_FIFO.BUFFER.value.table[4696]), INT_ENUM},*)
(*DBG:    {&(RES0__INSTANCE0.MY_BAD_FIFO.BUFFER.value.table[4697]), INT_ENUM},*)
(*DBG:    {&(RES0__INSTANCE0.MY_BAD_FIFO.BUFFER.value.table[4698]), INT_ENUM},*)
(*DBG:    {&(RES0__INSTANCE0.MY_BAD_FIFO.BUFFER.value.table[4699]), INT_ENUM},*)
(*DBG:    {&(RES0__INSTANCE0.MY_BAD_FIFO.BUFFER.value.table[4700]), INT_ENUM},*)
(*DBG:    {&(RES0__INSTANCE0.MY_BAD_FIFO.BUFFER.value.table[4701]), INT_ENUM},*)
(*DBG:    {&(RES0__INSTANCE0.MY_BAD_FIFO.BUFFER.value.table[4702]), INT_ENUM},*)
(*DBG:    {&(RES0__INSTANCE0.MY_BAD_FIFO.BUFFER.value.table[4703]), INT_ENUM},*)
(*DBG:    {&(RES0__INSTANCE0.MY_BAD_FIFO.BUFFER.value.table[4704]), INT_ENUM},*)
(*DBG:    {&(RES0__INSTANCE0.MY_BAD_FIFO.BUFFER.value.table[4705]), INT_ENUM},*)
(*DBG:    {&(RES0__INSTANCE0.MY_BAD_FIFO.BUFFER.value.table[4706]), INT_ENUM},*)
(*DBG:    {&(RES0__INSTANCE0.MY_BAD_FIFO.BUFFER.value.table[4707]), INT_ENUM},*)
(*DBG:    {&(RES0__INSTANCE0.MY_BAD_FIFO.BUFFER.value.table[4708]), INT_ENUM},*)
(*DBG:    {&(RES0__INSTANCE0.MY_BAD_FIFO.BUFFER.value.table[4709]), INT_ENUM},*)
(*DBG:    {&(RES0__INSTANCE0.MY_BAD_FIFO.BUFFER.value.table[4710]), INT_ENUM},*)
(*DBG:    {&(RES0__INSTANCE0.MY_BAD_FIFO.BUFFER.value.table[4711]), INT_ENUM},*)
(*DBG:    {&(RES0__INSTANCE0.MY_BAD_FIFO.BUFFER.value.table[4712]), INT_ENUM},*)
(*DBG:    {&(RES0__INSTANCE0.MY_BAD_FIFO.BUFFER.value.table[4713]), INT_ENUM},*)
(*DBG:    {&(RES0__INSTANCE0.MY_BAD_FIFO.BUFFER.value.table[4714]), INT_ENUM},*)
(*DBG:    {&(RES0__INSTANCE0.MY_BAD_FIFO.BUFFER.value.table[4715]), INT_ENUM},*)
(*DBG:    {&(RES0__INSTANCE0.MY_BAD_FIFO.BUFFER.value.table[4716]), INT_ENUM},*)
(*DBG:    {&(RES0__INSTANCE0.MY_BAD_FIFO.BUFFER.value.table[4717]), INT_ENUM},*)
(*DBG:    {&(RES0__INSTANCE0.MY_BAD_FIFO.BUFFER.value.table[4718]), INT_ENUM},*)
(*DBG:    {&(RES0__INSTANCE0.MY_BAD_FIFO.BUFFER.value.table[4719]), INT_ENUM},*)
(*DBG:    {&(RES0__INSTANCE0.MY_BAD_FIFO.BUFFER.value.table[4720]), INT_ENUM},*)
(*DBG:    {&(RES0__INSTANCE0.MY_BAD_FIFO.BUFFER.value.table[4721]), INT_ENUM},*)
(*DBG:    {&(RES0__INSTANCE0.MY_BAD_FIFO.BUFFER.value.table[4722]), INT_ENUM},*)
(*DBG:    {&(RES0__INSTANCE0.MY_BAD_FIFO.BUFFER.value.table[4723]), INT_ENUM},*)
(*DBG:    {&(RES0__INSTANCE0.MY_BAD_FIFO.BUFFER.value.table[4724]), INT_ENUM},*)
(*DBG:    {&(RES0__INSTANCE0.MY_BAD_FIFO.BUFFER.value.table[4725]), INT_ENUM},*)
(*DBG:    {&(RES0__INSTANCE0.MY_BAD_FIFO.BUFFER.value.table[4726]), INT_ENUM},*)
(*DBG:    {&(RES0__INSTANCE0.MY_BAD_FIFO.BUFFER.value.table[4727]), INT_ENUM},*)
(*DBG:    {&(RES0__INSTANCE0.MY_BAD_FIFO.BUFFER.value.table[4728]), INT_ENUM},*)
(*DBG:    {&(RES0__INSTANCE0.MY_BAD_FIFO.BUFFER.value.table[4729]), INT_ENUM},*)
(*DBG:    {&(RES0__INSTANCE0.MY_BAD_FIFO.BUFFER.value.table[4730]), INT_ENUM},*)
(*DBG:    {&(RES0__INSTANCE0.MY_BAD_FIFO.BUFFER.value.table[4731]), INT_ENUM},*)
(*DBG:    {&(RES0__INSTANCE0.MY_BAD_FIFO.BUFFER.value.table[4732]), INT_ENUM},*)
(*DBG:    {&(RES0__INSTANCE0.MY_BAD_FIFO.BUFFER.value.table[4733]), INT_ENUM},*)
(*DBG:    {&(RES0__INSTANCE0.MY_BAD_FIFO.BUFFER.value.table[4734]), INT_ENUM},*)
(*DBG:    {&(RES0__INSTANCE0.MY_BAD_FIFO.BUFFER.value.table[4735]), INT_ENUM},*)
(*DBG:    {&(RES0__INSTANCE0.MY_BAD_FIFO.BUFFER.value.table[4736]), INT_ENUM},*)
(*DBG:    {&(RES0__INSTANCE0.MY_BAD_FIFO.BUFFER.value.table[4737]), INT_ENUM},*)
(*DBG:    {&(RES0__INSTANCE0.MY_BAD_FIFO.BUFFER.value.table[4738]), INT_ENUM},*)
(*DBG:    {&(RES0__INSTANCE0.MY_BAD_FIFO.BUFFER.value.table[4739]), INT_ENUM},*)
(*DBG:    {&(RES0__INSTANCE0.MY_BAD_FIFO.BUFFER.value.table[4740]), INT_ENUM},*)
(*DBG:    {&(RES0__INSTANCE0.MY_BAD_FIFO.BUFFER.value.table[4741]), INT_ENUM},*)
(*DBG:    {&(RES0__INSTANCE0.MY_BAD_FIFO.BUFFER.value.table[4742]), INT_ENUM},*)
(*DBG:    {&(RES0__INSTANCE0.MY_BAD_FIFO.BUFFER.value.table[4743]), INT_ENUM},*)
(*DBG:    {&(RES0__INSTANCE0.MY_BAD_FIFO.BUFFER.value.table[4744]), INT_ENUM},*)
(*DBG:    {&(RES0__INSTANCE0.MY_BAD_FIFO.BUFFER.value.table[4745]), INT_ENUM},*)
(*DBG:    {&(RES0__INSTANCE0.MY_BAD_FIFO.BUFFER.value.table[4746]), INT_ENUM},*)
(*DBG:    {&(RES0__INSTANCE0.MY_BAD_FIFO.BUFFER.value.table[4747]), INT_ENUM},*)
(*DBG:    {&(RES0__INSTANCE0.MY_BAD_FIFO.BUFFER.value.table[4748]), INT_ENUM},*)
(*DBG:    {&(RES0__INSTANCE0.MY_BAD_FIFO.BUFFER.value.table[4749]), INT_ENUM},*)
(*DBG:    {&(RES0__INSTANCE0.MY_BAD_FIFO.BUFFER.value.table[4750]), INT_ENUM},*)
(*DBG:    {&(RES0__INSTANCE0.MY_BAD_FIFO.BUFFER.value.table[4751]), INT_ENUM},*)
(*DBG:    {&(RES0__INSTANCE0.MY_BAD_FIFO.BUFFER.value.table[4752]), INT_ENUM},*)
(*DBG:    {&(RES0__INSTANCE0.MY_BAD_FIFO.BUFFER.value.table[4753]), INT_ENUM},*)
(*DBG:    {&(RES0__INSTANCE0.MY_BAD_FIFO.BUFFER.value.table[4754]), INT_ENUM},*)
(*DBG:    {&(RES0__INSTANCE0.MY_BAD_FIFO.BUFFER.value.table[4755]), INT_ENUM},*)
(*DBG:    {&(RES0__INSTANCE0.MY_BAD_FIFO.BUFFER.value.table[4756]), INT_ENUM},*)
(*DBG:    {&(RES0__INSTANCE0.MY_BAD_FIFO.BUFFER.value.table[4757]), INT_ENUM},*)
(*DBG:    {&(RES0__INSTANCE0.MY_BAD_FIFO.BUFFER.value.table[4758]), INT_ENUM},*)
(*DBG:    {&(RES0__INSTANCE0.MY_BAD_FIFO.BUFFER.value.table[4759]), INT_ENUM},*)
(*DBG:    {&(RES0__INSTANCE0.MY_BAD_FIFO.BUFFER.value.table[4760]), INT_ENUM},*)
(*DBG:    {&(RES0__INSTANCE0.MY_BAD_FIFO.BUFFER.value.table[4761]), INT_ENUM},*)
(*DBG:    {&(RES0__INSTANCE0.MY_BAD_FIFO.BUFFER.value.table[4762]), INT_ENUM},*)
(*DBG:    {&(RES0__INSTANCE0.MY_BAD_FIFO.BUFFER.value.table[4763]), INT_ENUM},*)
(*DBG:    {&(RES0__INSTANCE0.MY_BAD_FIFO.BUFFER.value.table[4764]), INT_ENUM},*)
(*DBG:    {&(RES0__INSTANCE0.MY_BAD_FIFO.BUFFER.value.table[4765]), INT_ENUM},*)
(*DBG:    {&(RES0__INSTANCE0.MY_BAD_FIFO.BUFFER.value.table[4766]), INT_ENUM},*)
(*DBG:    {&(RES0__INSTANCE0.MY_BAD_FIFO.BUFFER.value.table[4767]), INT_ENUM},*)
(*DBG:    {&(RES0__INSTANCE0.MY_BAD_FIFO.BUFFER.value.table[4768]), INT_ENUM},*)
(*DBG:    {&(RES0__INSTANCE0.MY_BAD_FIFO.BUFFER.value.table[4769]), INT_ENUM},*)
(*DBG:    {&(RES0__INSTANCE0.MY_BAD_FIFO.BUFFER.value.table[4770]), INT_ENUM},*)
(*DBG:    {&(RES0__INSTANCE0.MY_BAD_FIFO.BUFFER.value.table[4771]), INT_ENUM},*)
(*DBG:    {&(RES0__INSTANCE0.MY_BAD_FIFO.BUFFER.value.table[4772]), INT_ENUM},*)
(*DBG:    {&(RES0__INSTANCE0.MY_BAD_FIFO.BUFFER.value.table[4773]), INT_ENUM},*)
(*DBG:    {&(RES0__INSTANCE0.MY_BAD_FIFO.BUFFER.value.table[4774]), INT_ENUM},*)
(*DBG:    {&(RES0__INSTANCE0.MY_BAD_FIFO.BUFFER.value.table[4775]), INT_ENUM},*)
(*DBG:    {&(RES0__INSTANCE0.MY_BAD_FIFO.BUFFER.value.table[4776]), INT_ENUM},*)
(*DBG:    {&(RES0__INSTANCE0.MY_BAD_FIFO.BUFFER.value.table[4777]), INT_ENUM},*)
(*DBG:    {&(RES0__INSTANCE0.MY_BAD_FIFO.BUFFER.value.table[4778]), INT_ENUM},*)
(*DBG:    {&(RES0__INSTANCE0.MY_BAD_FIFO.BUFFER.value.table[4779]), INT_ENUM},*)
(*DBG:    {&(RES0__INSTANCE0.MY_BAD_FIFO.BUFFER.value.table[4780]), INT_ENUM},*)
(*DBG:    {&(RES0__INSTANCE0.MY_BAD_FIFO.BUFFER.value.table[4781]), INT_ENUM},*)
(*DBG:    {&(RES0__INSTANCE0.MY_BAD_FIFO.BUFFER.value.table[4782]), INT_ENUM},*)
(*DBG:    {&(RES0__INSTANCE0.MY_BAD_FIFO.BUFFER.value.table[4783]), INT_ENUM},*)
(*DBG:    {&(RES0__INSTANCE0.MY_BAD_FIFO.BUFFER.value.table[4784]), INT_ENUM},*)
(*DBG:    {&(RES0__INSTANCE0.MY_BAD_FIFO.BUFFER.value.table[4785]), INT_ENUM},*)
(*DBG:    {&(RES0__INSTANCE0.MY_BAD_FIFO.BUFFER.value.table[4786]), INT_ENUM},*)
(*DBG:    {&(RES0__INSTANCE0.MY_BAD_FIFO.BUFFER.value.table[4787]), INT_ENUM},*)
(*DBG:    {&(RES0__INSTANCE0.MY_BAD_FIFO.BUFFER.value.table[4788]), INT_ENUM},*)
(*DBG:    {&(RES0__INSTANCE0.MY_BAD_FIFO.BUFFER.value.table[4789]), INT_ENUM},*)
(*DBG:    {&(RES0__INSTANCE0.MY_BAD_FIFO.BUFFER.value.table[4790]), INT_ENUM},*)
(*DBG:    {&(RES0__INSTANCE0.MY_BAD_FIFO.BUFFER.value.table[4791]), INT_ENUM},*)
(*DBG:    {&(RES0__INSTANCE0.MY_BAD_FIFO.BUFFER.value.table[4792]), INT_ENUM},*)
(*DBG:    {&(RES0__INSTANCE0.MY_BAD_FIFO.BUFFER.value.table[4793]), INT_ENUM},*)
(*DBG:    {&(RES0__INSTANCE0.MY_BAD_FIFO.BUFFER.value.table[4794]), INT_ENUM},*)
(*DBG:    {&(RES0__INSTANCE0.MY_BAD_FIFO.BUFFER.value.table[4795]), INT_ENUM},*)
(*DBG:    {&(RES0__INSTANCE0.MY_BAD_FIFO.BUFFER.value.table[4796]), INT_ENUM},*)
(*DBG:    {&(RES0__INSTANCE0.MY_BAD_FIFO.BUFFER.value.table[4797]), INT_ENUM},*)
(*DBG:    {&(RES0__INSTANCE0.MY_BAD_FIFO.BUFFER.value.table[4798]), INT_ENUM},*)
(*DBG:    {&(RES0__INSTANCE0.MY_BAD_FIFO.BUFFER.value.table[4799]), INT_ENUM},*)
(*DBG:    {&(RES0__INSTANCE0.MY_BAD_FIFO.BUFFER.value.table[4800]), INT_ENUM},*)
(*DBG:    {&(RES0__INSTANCE0.MY_BAD_FIFO.BUFFER.value.table[4801]), INT_ENUM},*)
(*DBG:    {&(RES0__INSTANCE0.MY_BAD_FIFO.BUFFER.value.table[4802]), INT_ENUM},*)
(*DBG:    {&(RES0__INSTANCE0.MY_BAD_FIFO.BUFFER.value.table[4803]), INT_ENUM},*)
(*DBG:    {&(RES0__INSTANCE0.MY_BAD_FIFO.BUFFER.value.table[4804]), INT_ENUM},*)
(*DBG:    {&(RES0__INSTANCE0.MY_BAD_FIFO.BUFFER.value.table[4805]), INT_ENUM},*)
(*DBG:    {&(RES0__INSTANCE0.MY_BAD_FIFO.BUFFER.value.table[4806]), INT_ENUM},*)
(*DBG:    {&(RES0__INSTANCE0.MY_BAD_FIFO.BUFFER.value.table[4807]), INT_ENUM},*)
(*DBG:    {&(RES0__INSTANCE0.MY_BAD_FIFO.BUFFER.value.table[4808]), INT_ENUM},*)
(*DBG:    {&(RES0__INSTANCE0.MY_BAD_FIFO.BUFFER.value.table[4809]), INT_ENUM},*)
(*DBG:    {&(RES0__INSTANCE0.MY_BAD_FIFO.BUFFER.value.table[4810]), INT_ENUM},*)
(*DBG:    {&(RES0__INSTANCE0.MY_BAD_FIFO.BUFFER.value.table[4811]), INT_ENUM},*)
(*DBG:    {&(RES0__INSTANCE0.MY_BAD_FIFO.BUFFER.value.table[4812]), INT_ENUM},*)
(*DBG:    {&(RES0__INSTANCE0.MY_BAD_FIFO.BUFFER.value.table[4813]), INT_ENUM},*)
(*DBG:    {&(RES0__INSTANCE0.MY_BAD_FIFO.BUFFER.value.table[4814]), INT_ENUM},*)
(*DBG:    {&(RES0__INSTANCE0.MY_BAD_FIFO.BUFFER.value.table[4815]), INT_ENUM},*)
(*DBG:    {&(RES0__INSTANCE0.MY_BAD_FIFO.BUFFER.value.table[4816]), INT_ENUM},*)
(*DBG:    {&(RES0__INSTANCE0.MY_BAD_FIFO.BUFFER.value.table[4817]), INT_ENUM},*)
(*DBG:    {&(RES0__INSTANCE0.MY_BAD_FIFO.BUFFER.value.table[4818]), INT_ENUM},*)
(*DBG:    {&(RES0__INSTANCE0.MY_BAD_FIFO.BUFFER.value.table[4819]), INT_ENUM},*)
(*DBG:    {&(RES0__INSTANCE0.MY_BAD_FIFO.BUFFER.value.table[4820]), INT_ENUM},*)
(*DBG:    {&(RES0__INSTANCE0.MY_BAD_FIFO.BUFFER.value.table[4821]), INT_ENUM},*)
(*DBG:    {&(RES0__INSTANCE0.MY_BAD_FIFO.BUFFER.value.table[4822]), INT_ENUM},*)
(*DBG:    {&(RES0__INSTANCE0.MY_BAD_FIFO.BUFFER.value.table[4823]), INT_ENUM},*)
(*DBG:    {&(RES0__INSTANCE0.MY_BAD_FIFO.BUFFER.value.table[4824]), INT_ENUM},*)
(*DBG:    {&(RES0__INSTANCE0.MY_BAD_FIFO.BUFFER.value.table[4825]), INT_ENUM},*)
(*DBG:    {&(RES0__INSTANCE0.MY_BAD_FIFO.BUFFER.value.table[4826]), INT_ENUM},*)
(*DBG:    {&(RES0__INSTANCE0.MY_BAD_FIFO.BUFFER.value.table[4827]), INT_ENUM},*)
(*DBG:    {&(RES0__INSTANCE0.MY_BAD_FIFO.BUFFER.value.table[4828]), INT_ENUM},*)
(*DBG:    {&(RES0__INSTANCE0.MY_BAD_FIFO.BUFFER.value.table[4829]), INT_ENUM},*)
(*DBG:    {&(RES0__INSTANCE0.MY_BAD_FIFO.BUFFER.value.table[4830]), INT_ENUM},*)
(*DBG:    {&(RES0__INSTANCE0.MY_BAD_FIFO.BUFFER.value.table[4831]), INT_ENUM},*)
(*DBG:    {&(RES0__INSTANCE0.MY_BAD_FIFO.BUFFER.value.table[4832]), INT_ENUM},*)
(*DBG:    {&(RES0__INSTANCE0.MY_BAD_FIFO.BUFFER.value.table[4833]), INT_ENUM},*)
(*DBG:    {&(RES0__INSTANCE0.MY_BAD_FIFO.BUFFER.value.table[4834]), INT_ENUM},*)
(*DBG:    {&(RES0__INSTANCE0.MY_BAD_FIFO.BUFFER.value.table[4835]), INT_ENUM},*)
(*DBG:    {&(RES0__INSTANCE0.MY_BAD_FIFO.BUFFER.value.table[4836]), INT_ENUM},*)
(*DBG:    {&(RES0__INSTANCE0.MY_BAD_FIFO.BUFFER.value.table[4837]), INT_ENUM},*)
(*DBG:    {&(RES0__INSTANCE0.MY_BAD_FIFO.BUFFER.value.table[4838]), INT_ENUM},*)
(*DBG:    {&(RES0__INSTANCE0.MY_BAD_FIFO.BUFFER.value.table[4839]), INT_ENUM},*)
(*DBG:    {&(RES0__INSTANCE0.MY_BAD_FIFO.BUFFER.value.table[4840]), INT_ENUM},*)
(*DBG:    {&(RES0__INSTANCE0.MY_BAD_FIFO.BUFFER.value.table[4841]), INT_ENUM},*)
(*DBG:    {&(RES0__INSTANCE0.MY_BAD_FIFO.BUFFER.value.table[4842]), INT_ENUM},*)
(*DBG:    {&(RES0__INSTANCE0.MY_BAD_FIFO.BUFFER.value.table[4843]), INT_ENUM},*)
(*DBG:    {&(RES0__INSTANCE0.MY_BAD_FIFO.BUFFER.value.table[4844]), INT_ENUM},*)
(*DBG:    {&(RES0__INSTANCE0.MY_BAD_FIFO.BUFFER.value.table[4845]), INT_ENUM},*)
(*DBG:    {&(RES0__INSTANCE0.MY_BAD_FIFO.BUFFER.value.table[4846]), INT_ENUM},*)
(*DBG:    {&(RES0__INSTANCE0.MY_BAD_FIFO.BUFFER.value.table[4847]), INT_ENUM},*)
(*DBG:    {&(RES0__INSTANCE0.MY_BAD_FIFO.BUFFER.value.table[4848]), INT_ENUM},*)
(*DBG:    {&(RES0__INSTANCE0.MY_BAD_FIFO.BUFFER.value.table[4849]), INT_ENUM},*)
(*DBG:    {&(RES0__INSTANCE0.MY_BAD_FIFO.BUFFER.value.table[4850]), INT_ENUM},*)
(*DBG:    {&(RES0__INSTANCE0.MY_BAD_FIFO.BUFFER.value.table[4851]), INT_ENUM},*)
(*DBG:    {&(RES0__INSTANCE0.MY_BAD_FIFO.BUFFER.value.table[4852]), INT_ENUM},*)
(*DBG:    {&(RES0__INSTANCE0.MY_BAD_FIFO.BUFFER.value.table[4853]), INT_ENUM},*)
(*DBG:    {&(RES0__INSTANCE0.MY_BAD_FIFO.BUFFER.value.table[4854]), INT_ENUM},*)
(*DBG:    {&(RES0__INSTANCE0.MY_BAD_FIFO.BUFFER.value.table[4855]), INT_ENUM},*)
(*DBG:    {&(RES0__INSTANCE0.MY_BAD_FIFO.BUFFER.value.table[4856]), INT_ENUM},*)
(*DBG:    {&(RES0__INSTANCE0.MY_BAD_FIFO.BUFFER.value.table[4857]), INT_ENUM},*)
(*DBG:    {&(RES0__INSTANCE0.MY_BAD_FIFO.BUFFER.value.table[4858]), INT_ENUM},*)
(*DBG:    {&(RES0__INSTANCE0.MY_B